(* IEC 61131-3 sources: volt/packages/volt-lsp-iec/test-corpus/lenze-mid/Device/Plc Logic/Application/Library Manager/(unresolved)/cmpopcuastack interfaces (part 2) *)

(* ---- OPCUA_NODEIDS.dut ---- *)
TYPE OPCUA_NODEIDS :
(
	OPCUAID_BASEDATATYPE := 24,
	OPCUAID_NUMBER := 26,
	OPCUAID_INTEGER := 27,
	OPCUAID_UINTEGER := 28,
	OPCUAID_ENUMERATION := 29,
	OPCUAID_BOOLEAN := 1,
	OPCUAID_SBYTE := 2,
	OPCUAID_BYTE := 3,
	OPCUAID_INT16 := 4,
	OPCUAID_UINT16 := 5,
	OPCUAID_INT32 := 6,
	OPCUAID_UINT32 := 7,
	OPCUAID_INT64 := 8,
	OPCUAID_UINT64 := 9,
	OPCUAID_FLOAT := 10,
	OPCUAID_DOUBLE := 11,
	OPCUAID_STRING := 12,
	OPCUAID_DATETIME := 13,
	OPCUAID_GUID := 14,
	OPCUAID_BYTESTRING := 15,
	OPCUAID_XMLELEMENT := 16,
	OPCUAID_NODEID := 17,
	OPCUAID_EXPANDEDNODEID := 18,
	OPCUAID_STATUSCODE := 19,
	OPCUAID_QUALIFIEDNAME := 20,
	OPCUAID_LOCALIZEDTEXT := 21,
	OPCUAID_STRUCTURE := 22,
	OPCUAID_DATAVALUE := 23,
	OPCUAID_DIAGNOSTICINFO := 25,
	OPCUAID_IMAGE := 30,
	OPCUAID_DECIMAL := 50,
	OPCUAID_NAMINGRULETYPE := 120,
	OPCUAID_IMAGEBMP := 2000,
	OPCUAID_IMAGEGIF := 2001,
	OPCUAID_IMAGEJPG := 2002,
	OPCUAID_IMAGEPNG := 2003,
	OPCUAID_AUDIODATATYPE := 16307,
	OPCUAID_BITFIELDMASKDATATYPE := 11737,
	OPCUAID_KEYVALUEPAIR := 14533,
	OPCUAID_ENDPOINTTYPE := 15528,
	OPCUAID_OPENFILEMODE := 11939,
	OPCUAID_IDENTITYCRITERIATYPE := 15632,
	OPCUAID_IDENTITYMAPPINGRULETYPE := 15634,
	OPCUAID_TRUSTLISTMASKS := 12552,
	OPCUAID_TRUSTLISTDATATYPE := 12554,
	OPCUAID_DECIMALDATATYPE := 17861,
	OPCUAID_DATATYPESCHEMAHEADER := 15534,
	OPCUAID_DATATYPEDESCRIPTION := 14525,
	OPCUAID_STRUCTUREDESCRIPTION := 15487,
	OPCUAID_ENUMDESCRIPTION := 15488,
	OPCUAID_SIMPLETYPEDESCRIPTION := 15005,
	OPCUAID_UABINARYFILEDATATYPE := 15006,
	OPCUAID_PUBSUBSTATE := 14647,
	OPCUAID_DATASETMETADATATYPE := 14523,
	OPCUAID_FIELDMETADATA := 14524,
	OPCUAID_DATASETFIELDFLAGS := 15904,
	OPCUAID_CONFIGURATIONVERSIONDATATYPE := 14593,
	OPCUAID_PUBLISHEDDATASETDATATYPE := 15578,
	OPCUAID_PUBLISHEDDATASETSOURCEDATATYPE := 15580,
	OPCUAID_PUBLISHEDVARIABLEDATATYPE := 14273,
	OPCUAID_PUBLISHEDDATAITEMSDATATYPE := 15581,
	OPCUAID_PUBLISHEDEVENTSDATATYPE := 15582,
	OPCUAID_DATASETFIELDCONTENTMASK := 15583,
	OPCUAID_DATASETWRITERDATATYPE := 15597,
	OPCUAID_DATASETWRITERTRANSPORTDATATYPE := 15598,
	OPCUAID_DATASETWRITERMESSAGEDATATYPE := 15605,
	OPCUAID_PUBSUBGROUPDATATYPE := 15609,
	OPCUAID_WRITERGROUPDATATYPE := 15480,
	OPCUAID_WRITERGROUPTRANSPORTDATATYPE := 15611,
	OPCUAID_WRITERGROUPMESSAGEDATATYPE := 15616,
	OPCUAID_PUBSUBCONNECTIONDATATYPE := 15617,
	OPCUAID_CONNECTIONTRANSPORTDATATYPE := 15618,
	OPCUAID_NETWORKADDRESSDATATYPE := 15502,
	OPCUAID_NETWORKADDRESSURLDATATYPE := 15510,
	OPCUAID_READERGROUPDATATYPE := 15520,
	OPCUAID_READERGROUPTRANSPORTDATATYPE := 15621,
	OPCUAID_READERGROUPMESSAGEDATATYPE := 15622,
	OPCUAID_DATASETREADERDATATYPE := 15623,
	OPCUAID_DATASETREADERTRANSPORTDATATYPE := 15628,
	OPCUAID_DATASETREADERMESSAGEDATATYPE := 15629,
	OPCUAID_SUBSCRIBEDDATASETDATATYPE := 15630,
	OPCUAID_TARGETVARIABLESDATATYPE := 15631,
	OPCUAID_FIELDTARGETDATATYPE := 14744,
	OPCUAID_OVERRIDEVALUEHANDLING := 15874,
	OPCUAID_SUBSCRIBEDDATASETMIRRORDATATYPE := 15635,
	OPCUAID_PUBSUBCONFIGURATIONDATATYPE := 15530,
	OPCUAID_DATASETORDERINGTYPE := 20408,
	OPCUAID_UADPNETWORKMESSAGECONTENTMASK := 15642,
	OPCUAID_UADPWRITERGROUPMESSAGEDATATYPE := 15645,
	OPCUAID_UADPDATASETMESSAGECONTENTMASK := 15646,
	OPCUAID_UADPDATASETWRITERMESSAGEDATATYPE := 15652,
	OPCUAID_UADPDATASETREADERMESSAGEDATATYPE := 15653,
	OPCUAID_JSONNETWORKMESSAGECONTENTMASK := 15654,
	OPCUAID_JSONWRITERGROUPMESSAGEDATATYPE := 15657,
	OPCUAID_JSONDATASETMESSAGECONTENTMASK := 15658,
	OPCUAID_JSONDATASETWRITERMESSAGEDATATYPE := 15664,
	OPCUAID_JSONDATASETREADERMESSAGEDATATYPE := 15665,
	OPCUAID_DATAGRAMCONNECTIONTRANSPORTDATATYPE := 17467,
	OPCUAID_DATAGRAMWRITERGROUPTRANSPORTDATATYPE := 15532,
	OPCUAID_BROKERCONNECTIONTRANSPORTDATATYPE := 15007,
	OPCUAID_BROKERTRANSPORTQUALITYOFSERVICE := 15008,
	OPCUAID_BROKERWRITERGROUPTRANSPORTDATATYPE := 15667,
	OPCUAID_BROKERDATASETWRITERTRANSPORTDATATYPE := 15669,
	OPCUAID_BROKERDATASETREADERTRANSPORTDATATYPE := 15670,
	OPCUAID_DIAGNOSTICSLEVEL := 19723,
	OPCUAID_PUBSUBDIAGNOSTICSCOUNTERCLASSIFICATION := 19730,
	OPCUAID_IDTYPE := 256,
	OPCUAID_NODECLASS := 257,
	OPCUAID_PERMISSIONTYPE := 94,
	OPCUAID_ACCESSLEVELTYPE := 15031,
	OPCUAID_ACCESSLEVELEXTYPE := 15406,
	OPCUAID_EVENTNOTIFIERTYPE := 15033,
	OPCUAID_ACCESSRESTRICTIONTYPE := 95,
	OPCUAID_ROLEPERMISSIONTYPE := 96,
	OPCUAID_DATATYPEDEFINITION := 97,
	OPCUAID_STRUCTURETYPE := 98,
	OPCUAID_STRUCTUREFIELD := 101,
	OPCUAID_STRUCTUREDEFINITION := 99,
	OPCUAID_ENUMDEFINITION := 100,
	OPCUAID_NODE := 258,
	OPCUAID_INSTANCENODE := 11879,
	OPCUAID_TYPENODE := 11880,
	OPCUAID_OBJECTNODE := 261,
	OPCUAID_OBJECTTYPENODE := 264,
	OPCUAID_VARIABLENODE := 267,
	OPCUAID_VARIABLETYPENODE := 270,
	OPCUAID_REFERENCETYPENODE := 273,
	OPCUAID_METHODNODE := 276,
	OPCUAID_VIEWNODE := 279,
	OPCUAID_DATATYPENODE := 282,
	OPCUAID_REFERENCENODE := 285,
	OPCUAID_ARGUMENT := 296,
	OPCUAID_ENUMVALUETYPE := 7594,
	OPCUAID_ENUMFIELD := 102,
	OPCUAID_OPTIONSET := 12755,
	OPCUAID_UNION := 12756,
	OPCUAID_NORMALIZEDSTRING := 12877,
	OPCUAID_DECIMALSTRING := 12878,
	OPCUAID_DURATIONSTRING := 12879,
	OPCUAID_TIMESTRING := 12880,
	OPCUAID_DATESTRING := 12881,
	OPCUAID_DURATION := 290,
	OPCUAID_UTCTIME := 294,
	OPCUAID_LOCALEID := 295,
	OPCUAID_TIMEZONEDATATYPE := 8912,
	OPCUAID_INTEGERID := 288,
	OPCUAID_APPLICATIONTYPE := 307,
	OPCUAID_APPLICATIONDESCRIPTION := 308,
	OPCUAID_REQUESTHEADER := 389,
	OPCUAID_RESPONSEHEADER := 392,
	OPCUAID_VERSIONTIME := 20998,
	OPCUAID_SERVICEFAULT := 395,
	OPCUAID_SESSIONLESSINVOKEREQUESTTYPE := 15901,
	OPCUAID_SESSIONLESSINVOKERESPONSETYPE := 20999,
	OPCUAID_FINDSERVERSREQUEST := 420,
	OPCUAID_FINDSERVERSRESPONSE := 423,
	OPCUAID_SERVERONNETWORK := 12189,
	OPCUAID_FINDSERVERSONNETWORKREQUEST := 12190,
	OPCUAID_FINDSERVERSONNETWORKRESPONSE := 12191,
	OPCUAID_APPLICATIONINSTANCECERTIFICATE := 311,
	OPCUAID_MESSAGESECURITYMODE := 302,
	OPCUAID_USERTOKENTYPE := 303,
	OPCUAID_USERTOKENPOLICY := 304,
	OPCUAID_ENDPOINTDESCRIPTION := 312,
	OPCUAID_GETENDPOINTSREQUEST := 426,
	OPCUAID_GETENDPOINTSRESPONSE := 429,
	OPCUAID_REGISTEREDSERVER := 432,
	OPCUAID_REGISTERSERVERREQUEST := 435,
	OPCUAID_REGISTERSERVERRESPONSE := 438,
	OPCUAID_DISCOVERYCONFIGURATION := 12890,
	OPCUAID_MDNSDISCOVERYCONFIGURATION := 12891,
	OPCUAID_REGISTERSERVER2REQUEST := 12193,
	OPCUAID_REGISTERSERVER2RESPONSE := 12194,
	OPCUAID_SECURITYTOKENREQUESTTYPE := 315,
	OPCUAID_CHANNELSECURITYTOKEN := 441,
	OPCUAID_OPENSECURECHANNELREQUEST := 444,
	OPCUAID_OPENSECURECHANNELRESPONSE := 447,
	OPCUAID_CLOSESECURECHANNELREQUEST := 450,
	OPCUAID_CLOSESECURECHANNELRESPONSE := 453,
	OPCUAID_SIGNEDSOFTWARECERTIFICATE := 344,
	OPCUAID_SESSIONAUTHENTICATIONTOKEN := 388,
	OPCUAID_SIGNATUREDATA := 456,
	OPCUAID_CREATESESSIONREQUEST := 459,
	OPCUAID_CREATESESSIONRESPONSE := 462,
	OPCUAID_USERIDENTITYTOKEN := 316,
	OPCUAID_ANONYMOUSIDENTITYTOKEN := 319,
	OPCUAID_USERNAMEIDENTITYTOKEN := 322,
	OPCUAID_X509IDENTITYTOKEN := 325,
	OPCUAID_ISSUEDIDENTITYTOKEN := 938,
	OPCUAID_ACTIVATESESSIONREQUEST := 465,
	OPCUAID_ACTIVATESESSIONRESPONSE := 468,
	OPCUAID_CLOSESESSIONREQUEST := 471,
	OPCUAID_CLOSESESSIONRESPONSE := 474,
	OPCUAID_CANCELREQUEST := 477,
	OPCUAID_CANCELRESPONSE := 480,
	OPCUAID_NODEATTRIBUTESMASK := 348,
	OPCUAID_NODEATTRIBUTES := 349,
	OPCUAID_OBJECTATTRIBUTES := 352,
	OPCUAID_VARIABLEATTRIBUTES := 355,
	OPCUAID_METHODATTRIBUTES := 358,
	OPCUAID_OBJECTTYPEATTRIBUTES := 361,
	OPCUAID_VARIABLETYPEATTRIBUTES := 364,
	OPCUAID_REFERENCETYPEATTRIBUTES := 367,
	OPCUAID_DATATYPEATTRIBUTES := 370,
	OPCUAID_VIEWATTRIBUTES := 373,
	OPCUAID_GENERICATTRIBUTEVALUE := 17606,
	OPCUAID_GENERICATTRIBUTES := 17607,
	OPCUAID_ADDNODESITEM := 376,
	OPCUAID_ADDNODESRESULT := 483,
	OPCUAID_ADDNODESREQUEST := 486,
	OPCUAID_ADDNODESRESPONSE := 489,
	OPCUAID_ADDREFERENCESITEM := 379,
	OPCUAID_ADDREFERENCESREQUEST := 492,
	OPCUAID_ADDREFERENCESRESPONSE := 495,
	OPCUAID_DELETENODESITEM := 382,
	OPCUAID_DELETENODESREQUEST := 498,
	OPCUAID_DELETENODESRESPONSE := 501,
	OPCUAID_DELETEREFERENCESITEM := 385,
	OPCUAID_DELETEREFERENCESREQUEST := 504,
	OPCUAID_DELETEREFERENCESRESPONSE := 507,
	OPCUAID_ATTRIBUTEWRITEMASK := 347,
	OPCUAID_BROWSEDIRECTION := 510,
	OPCUAID_VIEWDESCRIPTION := 511,
	OPCUAID_BROWSEDESCRIPTION := 514,
	OPCUAID_BROWSERESULTMASK := 517,
	OPCUAID_REFERENCEDESCRIPTION := 518,
	OPCUAID_CONTINUATIONPOINT := 521,
	OPCUAID_BROWSERESULT := 522,
	OPCUAID_BROWSEREQUEST := 525,
	OPCUAID_BROWSERESPONSE := 528,
	OPCUAID_BROWSENEXTREQUEST := 531,
	OPCUAID_BROWSENEXTRESPONSE := 534,
	OPCUAID_RELATIVEPATHELEMENT := 537,
	OPCUAID_RELATIVEPATH := 540,
	OPCUAID_BROWSEPATH := 543,
	OPCUAID_BROWSEPATHTARGET := 546,
	OPCUAID_BROWSEPATHRESULT := 549,
	OPCUAID_TRANSLATEBROWSEPATHSTONODEIDSREQUEST := 552,
	OPCUAID_TRANSLATEBROWSEPATHSTONODEIDSRESPONSE := 555,
	OPCUAID_REGISTERNODESREQUEST := 558,
	OPCUAID_REGISTERNODESRESPONSE := 561,
	OPCUAID_UNREGISTERNODESREQUEST := 564,
	OPCUAID_UNREGISTERNODESRESPONSE := 567,
	OPCUAID_COUNTER := 289,
	OPCUAID_NUMERICRANGE := 291,
	OPCUAID_TIME := 292,
	OPCUAID_DATE := 293,
	OPCUAID_ENDPOINTCONFIGURATION := 331,
	OPCUAID_QUERYDATADESCRIPTION := 570,
	OPCUAID_NODETYPEDESCRIPTION := 573,
	OPCUAID_FILTEROPERATOR := 576,
	OPCUAID_QUERYDATASET := 577,
	OPCUAID_NODEREFERENCE := 580,
	OPCUAID_CONTENTFILTERELEMENT := 583,
	OPCUAID_CONTENTFILTER := 586,
	OPCUAID_FILTEROPERAND := 589,
	OPCUAID_ELEMENTOPERAND := 592,
	OPCUAID_LITERALOPERAND := 595,
	OPCUAID_ATTRIBUTEOPERAND := 598,
	OPCUAID_SIMPLEATTRIBUTEOPERAND := 601,
	OPCUAID_CONTENTFILTERELEMENTRESULT := 604,
	OPCUAID_CONTENTFILTERRESULT := 607,
	OPCUAID_PARSINGRESULT := 610,
	OPCUAID_QUERYFIRSTREQUEST := 613,
	OPCUAID_QUERYFIRSTRESPONSE := 616,
	OPCUAID_QUERYNEXTREQUEST := 619,
	OPCUAID_QUERYNEXTRESPONSE := 622,
	OPCUAID_TIMESTAMPSTORETURN := 625,
	OPCUAID_READVALUEID := 626,
	OPCUAID_READREQUEST := 629,
	OPCUAID_READRESPONSE := 632,
	OPCUAID_HISTORYREADVALUEID := 635,
	OPCUAID_HISTORYREADRESULT := 638,
	OPCUAID_HISTORYREADDETAILS := 641,
	OPCUAID_READEVENTDETAILS := 644,
	OPCUAID_READRAWMODIFIEDDETAILS := 647,
	OPCUAID_READPROCESSEDDETAILS := 650,
	OPCUAID_READATTIMEDETAILS := 653,
	OPCUAID_HISTORYDATA := 656,
	OPCUAID_MODIFICATIONINFO := 11216,
	OPCUAID_HISTORYMODIFIEDDATA := 11217,
	OPCUAID_HISTORYEVENT := 659,
	OPCUAID_HISTORYREADREQUEST := 662,
	OPCUAID_HISTORYREADRESPONSE := 665,
	OPCUAID_WRITEVALUE := 668,
	OPCUAID_WRITEREQUEST := 671,
	OPCUAID_WRITERESPONSE := 674,
	OPCUAID_HISTORYUPDATEDETAILS := 677,
	OPCUAID_HISTORYUPDATETYPE := 11234,
	OPCUAID_PERFORMUPDATETYPE := 11293,
	OPCUAID_UPDATEDATADETAILS := 680,
	OPCUAID_UPDATESTRUCTUREDATADETAILS := 11295,
	OPCUAID_UPDATEEVENTDETAILS := 683,
	OPCUAID_DELETERAWMODIFIEDDETAILS := 686,
	OPCUAID_DELETEATTIMEDETAILS := 689,
	OPCUAID_DELETEEVENTDETAILS := 692,
	OPCUAID_HISTORYUPDATERESULT := 695,
	OPCUAID_HISTORYUPDATEREQUEST := 698,
	OPCUAID_HISTORYUPDATERESPONSE := 701,
	OPCUAID_CALLMETHODREQUEST := 704,
	OPCUAID_CALLMETHODRESULT := 707,
	OPCUAID_CALLREQUEST := 710,
	OPCUAID_CALLRESPONSE := 713,
	OPCUAID_MONITORINGMODE := 716,
	OPCUAID_DATACHANGETRIGGER := 717,
	OPCUAID_DEADBANDTYPE := 718,
	OPCUAID_MONITORINGFILTER := 719,
	OPCUAID_DATACHANGEFILTER := 722,
	OPCUAID_EVENTFILTER := 725,
	OPCUAID_AGGREGATECONFIGURATION := 948,
	OPCUAID_AGGREGATEFILTER := 728,
	OPCUAID_MONITORINGFILTERRESULT := 731,
	OPCUAID_EVENTFILTERRESULT := 734,
	OPCUAID_AGGREGATEFILTERRESULT := 737,
	OPCUAID_MONITORINGPARAMETERS := 740,
	OPCUAID_MONITOREDITEMCREATEREQUEST := 743,
	OPCUAID_MONITOREDITEMCREATERESULT := 746,
	OPCUAID_CREATEMONITOREDITEMSREQUEST := 749,
	OPCUAID_CREATEMONITOREDITEMSRESPONSE := 752,
	OPCUAID_MONITOREDITEMMODIFYREQUEST := 755,
	OPCUAID_MONITOREDITEMMODIFYRESULT := 758,
	OPCUAID_MODIFYMONITOREDITEMSREQUEST := 761,
	OPCUAID_MODIFYMONITOREDITEMSRESPONSE := 764,
	OPCUAID_SETMONITORINGMODEREQUEST := 767,
	OPCUAID_SETMONITORINGMODERESPONSE := 770,
	OPCUAID_SETTRIGGERINGREQUEST := 773,
	OPCUAID_SETTRIGGERINGRESPONSE := 776,
	OPCUAID_DELETEMONITOREDITEMSREQUEST := 779,
	OPCUAID_DELETEMONITOREDITEMSRESPONSE := 782,
	OPCUAID_CREATESUBSCRIPTIONREQUEST := 785,
	OPCUAID_CREATESUBSCRIPTIONRESPONSE := 788,
	OPCUAID_MODIFYSUBSCRIPTIONREQUEST := 791,
	OPCUAID_MODIFYSUBSCRIPTIONRESPONSE := 794,
	OPCUAID_SETPUBLISHINGMODEREQUEST := 797,
	OPCUAID_SETPUBLISHINGMODERESPONSE := 800,
	OPCUAID_NOTIFICATIONMESSAGE := 803,
	OPCUAID_NOTIFICATIONDATA := 945,
	OPCUAID_DATACHANGENOTIFICATION := 809,
	OPCUAID_MONITOREDITEMNOTIFICATION := 806,
	OPCUAID_EVENTNOTIFICATIONLIST := 914,
	OPCUAID_EVENTFIELDLIST := 917,
	OPCUAID_HISTORYEVENTFIELDLIST := 920,
	OPCUAID_STATUSCHANGENOTIFICATION := 818,
	OPCUAID_SUBSCRIPTIONACKNOWLEDGEMENT := 821,
	OPCUAID_PUBLISHREQUEST := 824,
	OPCUAID_PUBLISHRESPONSE := 827,
	OPCUAID_REPUBLISHREQUEST := 830,
	OPCUAID_REPUBLISHRESPONSE := 833,
	OPCUAID_TRANSFERRESULT := 836,
	OPCUAID_TRANSFERSUBSCRIPTIONSREQUEST := 839,
	OPCUAID_TRANSFERSUBSCRIPTIONSRESPONSE := 842,
	OPCUAID_DELETESUBSCRIPTIONSREQUEST := 845,
	OPCUAID_DELETESUBSCRIPTIONSRESPONSE := 848,
	OPCUAID_BUILDINFO := 338,
	OPCUAID_REDUNDANCYSUPPORT := 851,
	OPCUAID_SERVERSTATE := 852,
	OPCUAID_REDUNDANTSERVERDATATYPE := 853,
	OPCUAID_ENDPOINTURLLISTDATATYPE := 11943,
	OPCUAID_NETWORKGROUPDATATYPE := 11944,
	OPCUAID_SAMPLINGINTERVALDIAGNOSTICSDATATYPE := 856,
	OPCUAID_SERVERDIAGNOSTICSSUMMARYDATATYPE := 859,
	OPCUAID_SERVERSTATUSDATATYPE := 862,
	OPCUAID_SESSIONDIAGNOSTICSDATATYPE := 865,
	OPCUAID_SESSIONSECURITYDIAGNOSTICSDATATYPE := 868,
	OPCUAID_SERVICECOUNTERDATATYPE := 871,
	OPCUAID_STATUSRESULT := 299,
	OPCUAID_SUBSCRIPTIONDIAGNOSTICSDATATYPE := 874,
	OPCUAID_MODELCHANGESTRUCTUREVERBMASK := 11941,
	OPCUAID_MODELCHANGESTRUCTUREDATATYPE := 877,
	OPCUAID_SEMANTICCHANGESTRUCTUREDATATYPE := 897,
	OPCUAID_RANGE := 884,
	OPCUAID_EUINFORMATION := 887,
	OPCUAID_AXISSCALEENUMERATION := 12077,
	OPCUAID_COMPLEXNUMBERTYPE := 12171,
	OPCUAID_DOUBLECOMPLEXNUMBERTYPE := 12172,
	OPCUAID_AXISINFORMATION := 12079,
	OPCUAID_XVTYPE := 12080,
	OPCUAID_PROGRAMDIAGNOSTICDATATYPE := 894,
	OPCUAID_PROGRAMDIAGNOSTIC2DATATYPE := 15396,
	OPCUAID_ANNOTATION := 891,
	OPCUAID_EXCEPTIONDEVIATIONFORMAT := 890,
	OPCUAID_OPCUANAMESPACEMETADATA_NAMESPACEFILE_OPEN := 15971,
	OPCUAID_OPCUANAMESPACEMETADATA_NAMESPACEFILE_CLOSE := 15974,
	OPCUAID_OPCUANAMESPACEMETADATA_NAMESPACEFILE_READ := 15976,
	OPCUAID_OPCUANAMESPACEMETADATA_NAMESPACEFILE_WRITE := 15979,
	OPCUAID_OPCUANAMESPACEMETADATA_NAMESPACEFILE_GETPOSITION := 15981,
	OPCUAID_OPCUANAMESPACEMETADATA_NAMESPACEFILE_SETPOSITION := 15984,
	OPCUAID_SERVERTYPE_SERVERCAPABILITIES_ROLESET_ADDROLE := 16290,
	OPCUAID_SERVERTYPE_SERVERCAPABILITIES_ROLESET_REMOVEROLE := 16293,
	OPCUAID_SERVERTYPE_GETMONITOREDITEMS := 11489,
	OPCUAID_SERVERTYPE_RESENDDATA := 12871,
	OPCUAID_SERVERTYPE_SETSUBSCRIPTIONDURABLE := 12746,
	OPCUAID_SERVERTYPE_REQUESTSERVERSTATECHANGE := 12883,
	OPCUAID_SERVERCAPABILITIESTYPE_ROLESET_ADDROLE := 16296,
	OPCUAID_SERVERCAPABILITIESTYPE_ROLESET_REMOVEROLE := 16299,
	OPCUAID_FILETYPE_OPEN := 11580,
	OPCUAID_FILETYPE_CLOSE := 11583,
	OPCUAID_FILETYPE_READ := 11585,
	OPCUAID_FILETYPE_WRITE := 11588,
	OPCUAID_FILETYPE_GETPOSITION := 11590,
	OPCUAID_FILETYPE_SETPOSITION := 11593,
	OPCUAID_ADDRESSSPACEFILETYPE_EXPORTNAMESPACE := 11615,
	OPCUAID_NAMESPACEMETADATATYPE_NAMESPACEFILE_OPEN := 11629,
	OPCUAID_NAMESPACEMETADATATYPE_NAMESPACEFILE_CLOSE := 11632,
	OPCUAID_NAMESPACEMETADATATYPE_NAMESPACEFILE_READ := 11634,
	OPCUAID_NAMESPACEMETADATATYPE_NAMESPACEFILE_WRITE := 11637,
	OPCUAID_NAMESPACEMETADATATYPE_NAMESPACEFILE_GETPOSITION := 11639,
	OPCUAID_NAMESPACEMETADATATYPE_NAMESPACEFILE_SETPOSITION := 11642,
	OPCUAID_NAMESPACESTYPE_NAMESPACEIDENTIFIER_PLACEHOLDER_NAMESPACEFILE_OPEN := 11659,
	OPCUAID_NAMESPACESTYPE_NAMESPACEIDENTIFIER_PLACEHOLDER_NAMESPACEFILE_CLOSE := 11662,
	OPCUAID_NAMESPACESTYPE_NAMESPACEIDENTIFIER_PLACEHOLDER_NAMESPACEFILE_READ := 11664,
	OPCUAID_NAMESPACESTYPE_NAMESPACEIDENTIFIER_PLACEHOLDER_NAMESPACEFILE_WRITE := 11667,
	OPCUAID_NAMESPACESTYPE_NAMESPACEIDENTIFIER_PLACEHOLDER_NAMESPACEFILE_GETPOSITION := 11669,
	OPCUAID_NAMESPACESTYPE_NAMESPACEIDENTIFIER_PLACEHOLDER_NAMESPACEFILE_SETPOSITION := 11672,
	OPCUAID_SERVER_SERVERCAPABILITIES_ROLESET_ADDROLE := 16301,
	OPCUAID_SERVER_SERVERCAPABILITIES_ROLESET_REMOVEROLE := 16304,
	OPCUAID_SERVER_GETMONITOREDITEMS := 11492,
	OPCUAID_SERVER_RESENDDATA := 12873,
	OPCUAID_SERVER_SETSUBSCRIPTIONDURABLE := 12749,
	OPCUAID_SERVER_REQUESTSERVERSTATECHANGE := 12886,
	OPCUAID_FILEDIRECTORYTYPE_FILEDIRECTORYNAME_PLACEHOLDER_CREATEDIRECTORY := 13355,
	OPCUAID_FILEDIRECTORYTYPE_FILEDIRECTORYNAME_PLACEHOLDER_CREATEFILE := 13358,
	OPCUAID_FILEDIRECTORYTYPE_FILEDIRECTORYNAME_PLACEHOLDER_DELETEFILESYSTEMOBJECT := 17718,
	OPCUAID_FILEDIRECTORYTYPE_FILEDIRECTORYNAME_PLACEHOLDER_MOVEORCOPY := 13363,
	OPCUAID_FILEDIRECTORYTYPE_FILENAME_PLACEHOLDER_OPEN := 13372,
	OPCUAID_FILEDIRECTORYTYPE_FILENAME_PLACEHOLDER_CLOSE := 13375,
	OPCUAID_FILEDIRECTORYTYPE_FILENAME_PLACEHOLDER_READ := 13377,
	OPCUAID_FILEDIRECTORYTYPE_FILENAME_PLACEHOLDER_WRITE := 13380,
	OPCUAID_FILEDIRECTORYTYPE_FILENAME_PLACEHOLDER_GETPOSITION := 13382,
	OPCUAID_FILEDIRECTORYTYPE_FILENAME_PLACEHOLDER_SETPOSITION := 13385,
	OPCUAID_FILEDIRECTORYTYPE_CREATEDIRECTORY := 13387,
	OPCUAID_FILEDIRECTORYTYPE_CREATEFILE := 13390,
	OPCUAID_FILEDIRECTORYTYPE_DELETEFILESYSTEMOBJECT := 13393,
	OPCUAID_FILEDIRECTORYTYPE_MOVEORCOPY := 13395,
	OPCUAID_FILESYSTEM_FILEDIRECTORYNAME_PLACEHOLDER_CREATEDIRECTORY := 16316,
	OPCUAID_FILESYSTEM_FILEDIRECTORYNAME_PLACEHOLDER_CREATEFILE := 16319,
	OPCUAID_FILESYSTEM_FILEDIRECTORYNAME_PLACEHOLDER_DELETEFILESYSTEMOBJECT := 17722,
	OPCUAID_FILESYSTEM_FILEDIRECTORYNAME_PLACEHOLDER_MOVEORCOPY := 16324,
	OPCUAID_FILESYSTEM_FILENAME_PLACEHOLDER_OPEN := 16333,
	OPCUAID_FILESYSTEM_FILENAME_PLACEHOLDER_CLOSE := 16336,
	OPCUAID_FILESYSTEM_FILENAME_PLACEHOLDER_READ := 16338,
	OPCUAID_FILESYSTEM_FILENAME_PLACEHOLDER_WRITE := 16341,
	OPCUAID_FILESYSTEM_FILENAME_PLACEHOLDER_GETPOSITION := 16343,
	OPCUAID_FILESYSTEM_FILENAME_PLACEHOLDER_SETPOSITION := 16346,
	OPCUAID_FILESYSTEM_CREATEDIRECTORY := 16348,
	OPCUAID_FILESYSTEM_CREATEFILE := 16351,
	OPCUAID_FILESYSTEM_DELETEFILESYSTEMOBJECT := 16354,
	OPCUAID_FILESYSTEM_MOVEORCOPY := 16356,
	OPCUAID_TEMPORARYFILETRANSFERTYPE_GENERATEFILEFORREAD := 15746,
	OPCUAID_TEMPORARYFILETRANSFERTYPE_GENERATEFILEFORWRITE := 15749,
	OPCUAID_TEMPORARYFILETRANSFERTYPE_CLOSEANDCOMMIT := 15751,
	OPCUAID_TEMPORARYFILETRANSFERTYPE_TRANSFERSTATE_PLACEHOLDER_RESET := 15794,
	OPCUAID_FILETRANSFERSTATEMACHINETYPE_RESET := 15843,
	OPCUAID_ROLESETTYPE_ADDROLE := 15997,
	OPCUAID_ROLESETTYPE_REMOVEROLE := 16000,
	OPCUAID_ROLETYPE_ADDIDENTITY := 15624,
	OPCUAID_ROLETYPE_REMOVEIDENTITY := 15626,
	OPCUAID_ROLETYPE_ADDAPPLICATION := 16176,
	OPCUAID_ROLETYPE_REMOVEAPPLICATION := 16178,
	OPCUAID_ROLETYPE_ADDENDPOINT := 16180,
	OPCUAID_ROLETYPE_REMOVEENDPOINT := 16182,
	OPCUAID_WELLKNOWNROLE_ANONYMOUS_ADDIDENTITY := 15648,
	OPCUAID_WELLKNOWNROLE_ANONYMOUS_REMOVEIDENTITY := 15650,
	OPCUAID_WELLKNOWNROLE_ANONYMOUS_ADDAPPLICATION := 16195,
	OPCUAID_WELLKNOWNROLE_ANONYMOUS_REMOVEAPPLICATION := 16197,
	OPCUAID_WELLKNOWNROLE_ANONYMOUS_ADDENDPOINT := 16199,
	OPCUAID_WELLKNOWNROLE_ANONYMOUS_REMOVEENDPOINT := 16201,
	OPCUAID_WELLKNOWNROLE_AUTHENTICATEDUSER_ADDIDENTITY := 15660,
	OPCUAID_WELLKNOWNROLE_AUTHENTICATEDUSER_REMOVEIDENTITY := 15662,
	OPCUAID_WELLKNOWNROLE_AUTHENTICATEDUSER_ADDAPPLICATION := 16206,
	OPCUAID_WELLKNOWNROLE_AUTHENTICATEDUSER_REMOVEAPPLICATION := 16208,
	OPCUAID_WELLKNOWNROLE_AUTHENTICATEDUSER_ADDENDPOINT := 16210,
	OPCUAID_WELLKNOWNROLE_AUTHENTICATEDUSER_REMOVEENDPOINT := 16212,
	OPCUAID_WELLKNOWNROLE_OBSERVER_ADDIDENTITY := 15672,
	OPCUAID_WELLKNOWNROLE_OBSERVER_REMOVEIDENTITY := 15674,
	OPCUAID_WELLKNOWNROLE_OBSERVER_ADDAPPLICATION := 16217,
	OPCUAID_WELLKNOWNROLE_OBSERVER_REMOVEAPPLICATION := 16219,
	OPCUAID_WELLKNOWNROLE_OBSERVER_ADDENDPOINT := 16221,
	OPCUAID_WELLKNOWNROLE_OBSERVER_REMOVEENDPOINT := 16223,
	OPCUAID_WELLKNOWNROLE_OPERATOR_ADDIDENTITY := 15684,
	OPCUAID_WELLKNOWNROLE_OPERATOR_REMOVEIDENTITY := 15686,
	OPCUAID_WELLKNOWNROLE_OPERATOR_ADDAPPLICATION := 16228,
	OPCUAID_WELLKNOWNROLE_OPERATOR_REMOVEAPPLICATION := 16230,
	OPCUAID_WELLKNOWNROLE_OPERATOR_ADDENDPOINT := 16232,
	OPCUAID_WELLKNOWNROLE_OPERATOR_REMOVEENDPOINT := 16234,
	OPCUAID_WELLKNOWNROLE_ENGINEER_ADDIDENTITY := 16041,
	OPCUAID_WELLKNOWNROLE_ENGINEER_REMOVEIDENTITY := 16043,
	OPCUAID_WELLKNOWNROLE_ENGINEER_ADDAPPLICATION := 16239,
	OPCUAID_WELLKNOWNROLE_ENGINEER_REMOVEAPPLICATION := 16241,
	OPCUAID_WELLKNOWNROLE_ENGINEER_ADDENDPOINT := 16243,
	OPCUAID_WELLKNOWNROLE_ENGINEER_REMOVEENDPOINT := 16245,
	OPCUAID_WELLKNOWNROLE_SUPERVISOR_ADDIDENTITY := 15696,
	OPCUAID_WELLKNOWNROLE_SUPERVISOR_REMOVEIDENTITY := 15698,
	OPCUAID_WELLKNOWNROLE_SUPERVISOR_ADDAPPLICATION := 16250,
	OPCUAID_WELLKNOWNROLE_SUPERVISOR_REMOVEAPPLICATION := 16252,
	OPCUAID_WELLKNOWNROLE_SUPERVISOR_ADDENDPOINT := 16254,
	OPCUAID_WELLKNOWNROLE_SUPERVISOR_REMOVEENDPOINT := 16256,
	OPCUAID_WELLKNOWNROLE_CONFIGUREADMIN_ADDIDENTITY := 15720,
	OPCUAID_WELLKNOWNROLE_CONFIGUREADMIN_REMOVEIDENTITY := 15722,
	OPCUAID_WELLKNOWNROLE_CONFIGUREADMIN_ADDAPPLICATION := 16272,
	OPCUAID_WELLKNOWNROLE_CONFIGUREADMIN_REMOVEAPPLICATION := 16274,
	OPCUAID_WELLKNOWNROLE_CONFIGUREADMIN_ADDENDPOINT := 16276,
	OPCUAID_WELLKNOWNROLE_CONFIGUREADMIN_REMOVEENDPOINT := 16278,
	OPCUAID_WELLKNOWNROLE_SECURITYADMIN_ADDIDENTITY := 15708,
	OPCUAID_WELLKNOWNROLE_SECURITYADMIN_REMOVEIDENTITY := 15710,
	OPCUAID_WELLKNOWNROLE_SECURITYADMIN_ADDAPPLICATION := 16261,
	OPCUAID_WELLKNOWNROLE_SECURITYADMIN_REMOVEAPPLICATION := 16263,
	OPCUAID_WELLKNOWNROLE_SECURITYADMIN_ADDENDPOINT := 16265,
	OPCUAID_WELLKNOWNROLE_SECURITYADMIN_REMOVEENDPOINT := 16267,
	OPCUAID_CONDITIONTYPE_DISABLE := 9028,
	OPCUAID_CONDITIONTYPE_ENABLE := 9027,
	OPCUAID_CONDITIONTYPE_ADDCOMMENT := 9029,
	OPCUAID_CONDITIONTYPE_CONDITIONREFRESH := 3875,
	OPCUAID_CONDITIONTYPE_CONDITIONREFRESH2 := 12912,
	OPCUAID_DIALOGCONDITIONTYPE_RESPOND := 9069,
	OPCUAID_ACKNOWLEDGEABLECONDITIONTYPE_ACKNOWLEDGE := 9111,
	OPCUAID_ACKNOWLEDGEABLECONDITIONTYPE_CONFIRM := 9113,
	OPCUAID_ALARMCONDITIONTYPE_SHELVINGSTATE_TIMEDSHELVE := 9213,
	OPCUAID_ALARMCONDITIONTYPE_SHELVINGSTATE_UNSHELVE := 9211,
	OPCUAID_ALARMCONDITIONTYPE_SHELVINGSTATE_ONESHOTSHELVE := 9212,
	OPCUAID_ALARMCONDITIONTYPE_SILENCE := 16402,
	OPCUAID_ALARMCONDITIONTYPE_SUPPRESS := 16403,
	OPCUAID_ALARMCONDITIONTYPE_UNSUPPRESS := 17868,
	OPCUAID_ALARMCONDITIONTYPE_REMOVEFROMSERVICE := 17869,
	OPCUAID_ALARMCONDITIONTYPE_PLACEINSERVICE := 17870,
	OPCUAID_ALARMCONDITIONTYPE_RESET := 18199,
	OPCUAID_ALARMGROUPTYPE_ALARMCONDITIONINSTANCE_PLACEHOLDER_DISABLE := 16439,
	OPCUAID_ALARMGROUPTYPE_ALARMCONDITIONINSTANCE_PLACEHOLDER_ENABLE := 16440,
	OPCUAID_ALARMGROUPTYPE_ALARMCONDITIONINSTANCE_PLACEHOLDER_ADDCOMMENT := 16441,
	OPCUAID_ALARMGROUPTYPE_ALARMCONDITIONINSTANCE_PLACEHOLDER_ACKNOWLEDGE := 16461,
	OPCUAID_ALARMGROUPTYPE_ALARMCONDITIONINSTANCE_PLACEHOLDER_SHELVINGSTATE_TIMEDSHELVE := 16517,
	OPCUAID_ALARMGROUPTYPE_ALARMCONDITIONINSTANCE_PLACEHOLDER_SHELVINGSTATE_UNSHELVE := 16515,
	OPCUAID_ALARMGROUPTYPE_ALARMCONDITIONINSTANCE_PLACEHOLDER_SHELVINGSTATE_ONESHOTSHELVE := 16516,
	OPCUAID_SHELVEDSTATEMACHINETYPE_TIMEDSHELVE := 2949,
	OPCUAID_SHELVEDSTATEMACHINETYPE_UNSHELVE := 2947,
	OPCUAID_SHELVEDSTATEMACHINETYPE_ONESHOTSHELVE := 2948,
	OPCUAID_LIMITALARMTYPE_SHELVINGSTATE_TIMEDSHELVE := 9314,
	OPCUAID_LIMITALARMTYPE_SHELVINGSTATE_UNSHELVE := 9312,
	OPCUAID_LIMITALARMTYPE_SHELVINGSTATE_ONESHOTSHELVE := 9313,
	OPCUAID_EXCLUSIVELIMITALARMTYPE_SHELVINGSTATE_TIMEDSHELVE := 9451,
	OPCUAID_EXCLUSIVELIMITALARMTYPE_SHELVINGSTATE_UNSHELVE := 9449,
	OPCUAID_EXCLUSIVELIMITALARMTYPE_SHELVINGSTATE_ONESHOTSHELVE := 9450,
	OPCUAID_NONEXCLUSIVELIMITALARMTYPE_SHELVINGSTATE_TIMEDSHELVE := 10016,
	OPCUAID_NONEXCLUSIVELIMITALARMTYPE_SHELVINGSTATE_UNSHELVE := 10014,
	OPCUAID_NONEXCLUSIVELIMITALARMTYPE_SHELVINGSTATE_ONESHOTSHELVE := 10015,
	OPCUAID_NONEXCLUSIVELEVELALARMTYPE_SHELVINGSTATE_TIMEDSHELVE := 10170,
	OPCUAID_NONEXCLUSIVELEVELALARMTYPE_SHELVINGSTATE_UNSHELVE := 10168,
	OPCUAID_NONEXCLUSIVELEVELALARMTYPE_SHELVINGSTATE_ONESHOTSHELVE := 10169,
	OPCUAID_EXCLUSIVELEVELALARMTYPE_SHELVINGSTATE_TIMEDSHELVE := 9592,
	OPCUAID_EXCLUSIVELEVELALARMTYPE_SHELVINGSTATE_UNSHELVE := 9590,
	OPCUAID_EXCLUSIVELEVELALARMTYPE_SHELVINGSTATE_ONESHOTSHELVE := 9591,
	OPCUAID_NONEXCLUSIVEDEVIATIONALARMTYPE_SHELVINGSTATE_TIMEDSHELVE := 10478,
	OPCUAID_NONEXCLUSIVEDEVIATIONALARMTYPE_SHELVINGSTATE_UNSHELVE := 10476,
	OPCUAID_NONEXCLUSIVEDEVIATIONALARMTYPE_SHELVINGSTATE_ONESHOTSHELVE := 10477,
	OPCUAID_NONEXCLUSIVERATEOFCHANGEALARMTYPE_SHELVINGSTATE_TIMEDSHELVE := 10324,
	OPCUAID_NONEXCLUSIVERATEOFCHANGEALARMTYPE_SHELVINGSTATE_UNSHELVE := 10322,
	OPCUAID_NONEXCLUSIVERATEOFCHANGEALARMTYPE_SHELVINGSTATE_ONESHOTSHELVE := 10323,
	OPCUAID_EXCLUSIVEDEVIATIONALARMTYPE_SHELVINGSTATE_TIMEDSHELVE := 9874,
	OPCUAID_EXCLUSIVEDEVIATIONALARMTYPE_SHELVINGSTATE_UNSHELVE := 9872,
	OPCUAID_EXCLUSIVEDEVIATIONALARMTYPE_SHELVINGSTATE_ONESHOTSHELVE := 9873,
	OPCUAID_EXCLUSIVERATEOFCHANGEALARMTYPE_SHELVINGSTATE_TIMEDSHELVE := 9733,
	OPCUAID_EXCLUSIVERATEOFCHANGEALARMTYPE_SHELVINGSTATE_UNSHELVE := 9731,
	OPCUAID_EXCLUSIVERATEOFCHANGEALARMTYPE_SHELVINGSTATE_ONESHOTSHELVE := 9732,
	OPCUAID_DISCRETEALARMTYPE_SHELVINGSTATE_TIMEDSHELVE := 10633,
	OPCUAID_DISCRETEALARMTYPE_SHELVINGSTATE_UNSHELVE := 10631,
	OPCUAID_DISCRETEALARMTYPE_SHELVINGSTATE_ONESHOTSHELVE := 10632,
	OPCUAID_OFFNORMALALARMTYPE_SHELVINGSTATE_TIMEDSHELVE := 10747,
	OPCUAID_OFFNORMALALARMTYPE_SHELVINGSTATE_UNSHELVE := 10745,
	OPCUAID_OFFNORMALALARMTYPE_SHELVINGSTATE_ONESHOTSHELVE := 10746,
	OPCUAID_SYSTEMOFFNORMALALARMTYPE_SHELVINGSTATE_TIMEDSHELVE := 11846,
	OPCUAID_SYSTEMOFFNORMALALARMTYPE_SHELVINGSTATE_UNSHELVE := 11844,
	OPCUAID_SYSTEMOFFNORMALALARMTYPE_SHELVINGSTATE_ONESHOTSHELVE := 11845,
	OPCUAID_TRIPALARMTYPE_SHELVINGSTATE_TIMEDSHELVE := 10861,
	OPCUAID_TRIPALARMTYPE_SHELVINGSTATE_UNSHELVE := 10859,
	OPCUAID_TRIPALARMTYPE_SHELVINGSTATE_ONESHOTSHELVE := 10860,
	OPCUAID_INSTRUMENTDIAGNOSTICALARMTYPE_SHELVINGSTATE_TIMEDSHELVE := 18453,
	OPCUAID_INSTRUMENTDIAGNOSTICALARMTYPE_SHELVINGSTATE_UNSHELVE := 18455,
	OPCUAID_INSTRUMENTDIAGNOSTICALARMTYPE_SHELVINGSTATE_ONESHOTSHELVE := 18456,
	OPCUAID_SYSTEMDIAGNOSTICALARMTYPE_SHELVINGSTATE_TIMEDSHELVE := 18602,
	OPCUAID_SYSTEMDIAGNOSTICALARMTYPE_SHELVINGSTATE_UNSHELVE := 18604,
	OPCUAID_SYSTEMDIAGNOSTICALARMTYPE_SHELVINGSTATE_ONESHOTSHELVE := 18605,
	OPCUAID_CERTIFICATEEXPIRATIONALARMTYPE_SHELVINGSTATE_TIMEDSHELVE := 13320,
	OPCUAID_CERTIFICATEEXPIRATIONALARMTYPE_SHELVINGSTATE_UNSHELVE := 13318,
	OPCUAID_CERTIFICATEEXPIRATIONALARMTYPE_SHELVINGSTATE_ONESHOTSHELVE := 13319,
	OPCUAID_DISCREPANCYALARMTYPE_SHELVINGSTATE_TIMEDSHELVE := 17195,
	OPCUAID_DISCREPANCYALARMTYPE_SHELVINGSTATE_UNSHELVE := 17193,
	OPCUAID_DISCREPANCYALARMTYPE_SHELVINGSTATE_ONESHOTSHELVE := 17194,
	OPCUAID_ALARMMETRICSTYPE_RESET := 18666,
	OPCUAID_PROGRAMSTATEMACHINETYPE_START := 2426,
	OPCUAID_PROGRAMSTATEMACHINETYPE_SUSPEND := 2427,
	OPCUAID_PROGRAMSTATEMACHINETYPE_RESUME := 2428,
	OPCUAID_PROGRAMSTATEMACHINETYPE_HALT := 2429,
	OPCUAID_PROGRAMSTATEMACHINETYPE_RESET := 2430,
	OPCUAID_TRUSTLISTTYPE_OPENWITHMASKS := 12543,
	OPCUAID_TRUSTLISTTYPE_CLOSEANDUPDATE := 12546,
	OPCUAID_TRUSTLISTTYPE_ADDCERTIFICATE := 12548,
	OPCUAID_TRUSTLISTTYPE_REMOVECERTIFICATE := 12550,
	OPCUAID_CERTIFICATEGROUPTYPE_TRUSTLIST_OPEN := 13605,
	OPCUAID_CERTIFICATEGROUPTYPE_TRUSTLIST_CLOSE := 13608,
	OPCUAID_CERTIFICATEGROUPTYPE_TRUSTLIST_READ := 13610,
	OPCUAID_CERTIFICATEGROUPTYPE_TRUSTLIST_WRITE := 13613,
	OPCUAID_CERTIFICATEGROUPTYPE_TRUSTLIST_GETPOSITION := 13615,
	OPCUAID_CERTIFICATEGROUPTYPE_TRUSTLIST_SETPOSITION := 13618,
	OPCUAID_CERTIFICATEGROUPTYPE_TRUSTLIST_OPENWITHMASKS := 13621,
	OPCUAID_CERTIFICATEGROUPFOLDERTYPE_DEFAULTAPPLICATIONGROUP_TRUSTLIST_OPEN := 13821,
	OPCUAID_CERTIFICATEGROUPFOLDERTYPE_DEFAULTAPPLICATIONGROUP_TRUSTLIST_CLOSE := 13824,
	OPCUAID_CERTIFICATEGROUPFOLDERTYPE_DEFAULTAPPLICATIONGROUP_TRUSTLIST_READ := 13826,
	OPCUAID_CERTIFICATEGROUPFOLDERTYPE_DEFAULTAPPLICATIONGROUP_TRUSTLIST_WRITE := 13829,
	OPCUAID_CERTIFICATEGROUPFOLDERTYPE_DEFAULTAPPLICATIONGROUP_TRUSTLIST_GETPOSITION := 13831,
	OPCUAID_CERTIFICATEGROUPFOLDERTYPE_DEFAULTAPPLICATIONGROUP_TRUSTLIST_SETPOSITION := 13834,
	OPCUAID_CERTIFICATEGROUPFOLDERTYPE_DEFAULTAPPLICATIONGROUP_TRUSTLIST_OPENWITHMASKS := 13837,
	OPCUAID_CERTIFICATEGROUPFOLDERTYPE_DEFAULTHTTPSGROUP_TRUSTLIST_OPEN := 13855,
	OPCUAID_CERTIFICATEGROUPFOLDERTYPE_DEFAULTHTTPSGROUP_TRUSTLIST_CLOSE := 13858,
	OPCUAID_CERTIFICATEGROUPFOLDERTYPE_DEFAULTHTTPSGROUP_TRUSTLIST_READ := 13860,
	OPCUAID_CERTIFICATEGROUPFOLDERTYPE_DEFAULTHTTPSGROUP_TRUSTLIST_WRITE := 13863,
	OPCUAID_CERTIFICATEGROUPFOLDERTYPE_DEFAULTHTTPSGROUP_TRUSTLIST_GETPOSITION := 13865,
	OPCUAID_CERTIFICATEGROUPFOLDERTYPE_DEFAULTHTTPSGROUP_TRUSTLIST_SETPOSITION := 13868,
	OPCUAID_CERTIFICATEGROUPFOLDERTYPE_DEFAULTHTTPSGROUP_TRUSTLIST_OPENWITHMASKS := 13871,
	OPCUAID_CERTIFICATEGROUPFOLDERTYPE_DEFAULTUSERTOKENGROUP_TRUSTLIST_OPEN := 13889,
	OPCUAID_CERTIFICATEGROUPFOLDERTYPE_DEFAULTUSERTOKENGROUP_TRUSTLIST_CLOSE := 13892,
	OPCUAID_CERTIFICATEGROUPFOLDERTYPE_DEFAULTUSERTOKENGROUP_TRUSTLIST_READ := 13894,
	OPCUAID_CERTIFICATEGROUPFOLDERTYPE_DEFAULTUSERTOKENGROUP_TRUSTLIST_WRITE := 13897,
	OPCUAID_CERTIFICATEGROUPFOLDERTYPE_DEFAULTUSERTOKENGROUP_TRUSTLIST_GETPOSITION := 13899,
	OPCUAID_CERTIFICATEGROUPFOLDERTYPE_DEFAULTUSERTOKENGROUP_TRUSTLIST_SETPOSITION := 13902,
	OPCUAID_CERTIFICATEGROUPFOLDERTYPE_DEFAULTUSERTOKENGROUP_TRUSTLIST_OPENWITHMASKS := 13905,
	OPCUAID_CERTIFICATEGROUPFOLDERTYPE_ADDITIONALGROUP_PLACEHOLDER_TRUSTLIST_OPEN := 13923,
	OPCUAID_CERTIFICATEGROUPFOLDERTYPE_ADDITIONALGROUP_PLACEHOLDER_TRUSTLIST_CLOSE := 13926,
	OPCUAID_CERTIFICATEGROUPFOLDERTYPE_ADDITIONALGROUP_PLACEHOLDER_TRUSTLIST_READ := 13928,
	OPCUAID_CERTIFICATEGROUPFOLDERTYPE_ADDITIONALGROUP_PLACEHOLDER_TRUSTLIST_WRITE := 13931,
	OPCUAID_CERTIFICATEGROUPFOLDERTYPE_ADDITIONALGROUP_PLACEHOLDER_TRUSTLIST_GETPOSITION := 13933,
	OPCUAID_CERTIFICATEGROUPFOLDERTYPE_ADDITIONALGROUP_PLACEHOLDER_TRUSTLIST_SETPOSITION := 13936,
	OPCUAID_CERTIFICATEGROUPFOLDERTYPE_ADDITIONALGROUP_PLACEHOLDER_TRUSTLIST_OPENWITHMASKS := 13939,
	OPCUAID_SERVERCONFIGURATIONTYPE_CERTIFICATEGROUPS_DEFAULTAPPLICATIONGROUP_TRUSTLIST_OPEN := 13958,
	OPCUAID_SERVERCONFIGURATIONTYPE_CERTIFICATEGROUPS_DEFAULTAPPLICATIONGROUP_TRUSTLIST_CLOSE := 13961,
	OPCUAID_SERVERCONFIGURATIONTYPE_CERTIFICATEGROUPS_DEFAULTAPPLICATIONGROUP_TRUSTLIST_READ := 13963,
	OPCUAID_SERVERCONFIGURATIONTYPE_CERTIFICATEGROUPS_DEFAULTAPPLICATIONGROUP_TRUSTLIST_WRITE := 13966,
	OPCUAID_SERVERCONFIGURATIONTYPE_CERTIFICATEGROUPS_DEFAULTAPPLICATIONGROUP_TRUSTLIST_GETPOSITION := 13968,
	OPCUAID_SERVERCONFIGURATIONTYPE_CERTIFICATEGROUPS_DEFAULTAPPLICATIONGROUP_TRUSTLIST_SETPOSITION := 13971,
	OPCUAID_SERVERCONFIGURATIONTYPE_CERTIFICATEGROUPS_DEFAULTAPPLICATIONGROUP_TRUSTLIST_OPENWITHMASKS := 13974,
	OPCUAID_SERVERCONFIGURATIONTYPE_CERTIFICATEGROUPS_DEFAULTHTTPSGROUP_TRUSTLIST_OPEN := 13992,
	OPCUAID_SERVERCONFIGURATIONTYPE_CERTIFICATEGROUPS_DEFAULTHTTPSGROUP_TRUSTLIST_CLOSE := 13995,
	OPCUAID_SERVERCONFIGURATIONTYPE_CERTIFICATEGROUPS_DEFAULTHTTPSGROUP_TRUSTLIST_READ := 13997,
	OPCUAID_SERVERCONFIGURATIONTYPE_CERTIFICATEGROUPS_DEFAULTHTTPSGROUP_TRUSTLIST_WRITE := 14000,
	OPCUAID_SERVERCONFIGURATIONTYPE_CERTIFICATEGROUPS_DEFAULTHTTPSGROUP_TRUSTLIST_GETPOSITION := 14002,
	OPCUAID_SERVERCONFIGURATIONTYPE_CERTIFICATEGROUPS_DEFAULTHTTPSGROUP_TRUSTLIST_SETPOSITION := 14005,
	OPCUAID_SERVERCONFIGURATIONTYPE_CERTIFICATEGROUPS_DEFAULTHTTPSGROUP_TRUSTLIST_OPENWITHMASKS := 14008,
	OPCUAID_SERVERCONFIGURATIONTYPE_CERTIFICATEGROUPS_DEFAULTUSERTOKENGROUP_TRUSTLIST_OPEN := 14026,
	OPCUAID_SERVERCONFIGURATIONTYPE_CERTIFICATEGROUPS_DEFAULTUSERTOKENGROUP_TRUSTLIST_CLOSE := 14029,
	OPCUAID_SERVERCONFIGURATIONTYPE_CERTIFICATEGROUPS_DEFAULTUSERTOKENGROUP_TRUSTLIST_READ := 14031,
	OPCUAID_SERVERCONFIGURATIONTYPE_CERTIFICATEGROUPS_DEFAULTUSERTOKENGROUP_TRUSTLIST_WRITE := 14034,
	OPCUAID_SERVERCONFIGURATIONTYPE_CERTIFICATEGROUPS_DEFAULTUSERTOKENGROUP_TRUSTLIST_GETPOSITION := 14036,
	OPCUAID_SERVERCONFIGURATIONTYPE_CERTIFICATEGROUPS_DEFAULTUSERTOKENGROUP_TRUSTLIST_SETPOSITION := 14039,
	OPCUAID_SERVERCONFIGURATIONTYPE_CERTIFICATEGROUPS_DEFAULTUSERTOKENGROUP_TRUSTLIST_OPENWITHMASKS := 14042,
	OPCUAID_SERVERCONFIGURATIONTYPE_UPDATECERTIFICATE := 12616,
	OPCUAID_SERVERCONFIGURATIONTYPE_APPLYCHANGES := 12734,
	OPCUAID_SERVERCONFIGURATIONTYPE_CREATESIGNINGREQUEST := 12731,
	OPCUAID_SERVERCONFIGURATIONTYPE_GETREJECTEDLIST := 12775,
	OPCUAID_SERVERCONFIGURATION_CERTIFICATEGROUPS_DEFAULTAPPLICATIONGROUP_TRUSTLIST_OPEN := 12647,
	OPCUAID_SERVERCONFIGURATION_CERTIFICATEGROUPS_DEFAULTAPPLICATIONGROUP_TRUSTLIST_CLOSE := 12650,
	OPCUAID_SERVERCONFIGURATION_CERTIFICATEGROUPS_DEFAULTAPPLICATIONGROUP_TRUSTLIST_READ := 12652,
	OPCUAID_SERVERCONFIGURATION_CERTIFICATEGROUPS_DEFAULTAPPLICATIONGROUP_TRUSTLIST_WRITE := 12655,
	OPCUAID_SERVERCONFIGURATION_CERTIFICATEGROUPS_DEFAULTAPPLICATIONGROUP_TRUSTLIST_GETPOSITION := 12657,
	OPCUAID_SERVERCONFIGURATION_CERTIFICATEGROUPS_DEFAULTAPPLICATIONGROUP_TRUSTLIST_SETPOSITION := 12660,
	OPCUAID_SERVERCONFIGURATION_CERTIFICATEGROUPS_DEFAULTAPPLICATIONGROUP_TRUSTLIST_OPENWITHMASKS := 12663,
	OPCUAID_SERVERCONFIGURATION_CERTIFICATEGROUPS_DEFAULTAPPLICATIONGROUP_TRUSTLIST_CLOSEANDUPDATE := 12666,
	OPCUAID_SERVERCONFIGURATION_CERTIFICATEGROUPS_DEFAULTAPPLICATIONGROUP_TRUSTLIST_ADDCERTIFICATE := 12668,
	OPCUAID_SERVERCONFIGURATION_CERTIFICATEGROUPS_DEFAULTAPPLICATIONGROUP_TRUSTLIST_REMOVECERTIFICATE := 12670,
	OPCUAID_SERVERCONFIGURATION_CERTIFICATEGROUPS_DEFAULTHTTPSGROUP_TRUSTLIST_OPEN := 14095,
	OPCUAID_SERVERCONFIGURATION_CERTIFICATEGROUPS_DEFAULTHTTPSGROUP_TRUSTLIST_CLOSE := 14098,
	OPCUAID_SERVERCONFIGURATION_CERTIFICATEGROUPS_DEFAULTHTTPSGROUP_TRUSTLIST_READ := 14100,
	OPCUAID_SERVERCONFIGURATION_CERTIFICATEGROUPS_DEFAULTHTTPSGROUP_TRUSTLIST_WRITE := 14103,
	OPCUAID_SERVERCONFIGURATION_CERTIFICATEGROUPS_DEFAULTHTTPSGROUP_TRUSTLIST_GETPOSITION := 14105,
	OPCUAID_SERVERCONFIGURATION_CERTIFICATEGROUPS_DEFAULTHTTPSGROUP_TRUSTLIST_SETPOSITION := 14108,
	OPCUAID_SERVERCONFIGURATION_CERTIFICATEGROUPS_DEFAULTHTTPSGROUP_TRUSTLIST_OPENWITHMASKS := 14111,
	OPCUAID_SERVERCONFIGURATION_CERTIFICATEGROUPS_DEFAULTHTTPSGROUP_TRUSTLIST_CLOSEANDUPDATE := 14114,
	OPCUAID_SERVERCONFIGURATION_CERTIFICATEGROUPS_DEFAULTHTTPSGROUP_TRUSTLIST_ADDCERTIFICATE := 14117,
	OPCUAID_SERVERCONFIGURATION_CERTIFICATEGROUPS_DEFAULTHTTPSGROUP_TRUSTLIST_REMOVECERTIFICATE := 14119,
	OPCUAID_SERVERCONFIGURATION_CERTIFICATEGROUPS_DEFAULTUSERTOKENGROUP_TRUSTLIST_OPEN := 14129,
	OPCUAID_SERVERCONFIGURATION_CERTIFICATEGROUPS_DEFAULTUSERTOKENGROUP_TRUSTLIST_CLOSE := 14132,
	OPCUAID_SERVERCONFIGURATION_CERTIFICATEGROUPS_DEFAULTUSERTOKENGROUP_TRUSTLIST_READ := 14134,
	OPCUAID_SERVERCONFIGURATION_CERTIFICATEGROUPS_DEFAULTUSERTOKENGROUP_TRUSTLIST_WRITE := 14137,
	OPCUAID_SERVERCONFIGURATION_CERTIFICATEGROUPS_DEFAULTUSERTOKENGROUP_TRUSTLIST_GETPOSITION := 14139,
	OPCUAID_SERVERCONFIGURATION_CERTIFICATEGROUPS_DEFAULTUSERTOKENGROUP_TRUSTLIST_SETPOSITION := 14142,
	OPCUAID_SERVERCONFIGURATION_CERTIFICATEGROUPS_DEFAULTUSERTOKENGROUP_TRUSTLIST_OPENWITHMASKS := 14145,
	OPCUAID_SERVERCONFIGURATION_CERTIFICATEGROUPS_DEFAULTUSERTOKENGROUP_TRUSTLIST_CLOSEANDUPDATE := 14148,
	OPCUAID_SERVERCONFIGURATION_CERTIFICATEGROUPS_DEFAULTUSERTOKENGROUP_TRUSTLIST_ADDCERTIFICATE := 14151,
	OPCUAID_SERVERCONFIGURATION_CERTIFICATEGROUPS_DEFAULTUSERTOKENGROUP_TRUSTLIST_REMOVECERTIFICATE := 14153,
	OPCUAID_SERVERCONFIGURATION_UPDATECERTIFICATE := 13737,
	OPCUAID_SERVERCONFIGURATION_APPLYCHANGES := 12740,
	OPCUAID_SERVERCONFIGURATION_CREATESIGNINGREQUEST := 12737,
	OPCUAID_SERVERCONFIGURATION_GETREJECTEDLIST := 12777,
	OPCUAID_KEYCREDENTIALCONFIGURATIONFOLDERTYPE_CREATECREDENTIAL := 17522,
	OPCUAID_KEYCREDENTIALCONFIGURATIONTYPE_GETENCRYPTINGKEY := 17534,
	OPCUAID_KEYCREDENTIALCONFIGURATIONTYPE_UPDATECREDENTIAL := 18006,
	OPCUAID_KEYCREDENTIALCONFIGURATIONTYPE_DELETECREDENTIAL := 18008,
	OPCUAID_PUBSUBKEYSERVICETYPE_GETSECURITYKEYS := 15907,
	OPCUAID_PUBSUBKEYSERVICETYPE_GETSECURITYGROUP := 15910,
	OPCUAID_PUBSUBKEYSERVICETYPE_SECURITYGROUPS_ADDSECURITYGROUP := 15914,
	OPCUAID_PUBSUBKEYSERVICETYPE_SECURITYGROUPS_REMOVESECURITYGROUP := 15917,
	OPCUAID_SECURITYGROUPFOLDERTYPE_SECURITYGROUPFOLDERNAME_PLACEHOLDER_ADDSECURITYGROUP := 15454,
	OPCUAID_SECURITYGROUPFOLDERTYPE_SECURITYGROUPFOLDERNAME_PLACEHOLDER_REMOVESECURITYGROUP := 15457,
	OPCUAID_SECURITYGROUPFOLDERTYPE_ADDSECURITYGROUP := 15461,
	OPCUAID_SECURITYGROUPFOLDERTYPE_REMOVESECURITYGROUP := 15464,
	OPCUAID_PUBLISHSUBSCRIBETYPE_SECURITYGROUPS_ADDSECURITYGROUP := 15435,
	OPCUAID_PUBLISHSUBSCRIBETYPE_SECURITYGROUPS_REMOVESECURITYGROUP := 15438,
	OPCUAID_PUBLISHSUBSCRIBETYPE_CONNECTIONNAME_PLACEHOLDER_DIAGNOSTICS_RESET := 18679,
	OPCUAID_PUBLISHSUBSCRIBETYPE_SETSECURITYKEYS := 17296,
	OPCUAID_PUBLISHSUBSCRIBETYPE_ADDCONNECTION := 16598,
	OPCUAID_PUBLISHSUBSCRIBETYPE_REMOVECONNECTION := 14432,
	OPCUAID_PUBLISHSUBSCRIBETYPE_DIAGNOSTICS_RESET := 18727,
	OPCUAID_PUBLISHSUBSCRIBE_GETSECURITYKEYS := 15215,
	OPCUAID_PUBLISHSUBSCRIBE_GETSECURITYGROUP := 15440,
	OPCUAID_PUBLISHSUBSCRIBE_SECURITYGROUPS_ADDSECURITYGROUP := 15444,
	OPCUAID_PUBLISHSUBSCRIBE_SECURITYGROUPS_REMOVESECURITYGROUP := 15447,
	OPCUAID_PUBLISHSUBSCRIBE_CONNECTIONNAME_PLACEHOLDER_DIAGNOSTICS_RESET := 16076,
	OPCUAID_PUBLISHSUBSCRIBE_ADDCONNECTION := 17366,
	OPCUAID_PUBLISHSUBSCRIBE_REMOVECONNECTION := 17369,
	OPCUAID_PUBLISHSUBSCRIBE_DIAGNOSTICS_RESET := 17421,
	OPCUAID_PUBLISHEDDATASETTYPE_DATASETWRITERNAME_PLACEHOLDER_DIAGNOSTICS_RESET := 18883,
	OPCUAID_PUBLISHEDDATASETTYPE_EXTENSIONFIELDS_ADDEXTENSIONFIELD := 15482,
	OPCUAID_PUBLISHEDDATASETTYPE_EXTENSIONFIELDS_REMOVEEXTENSIONFIELD := 15485,
	OPCUAID_EXTENSIONFIELDSTYPE_ADDEXTENSIONFIELD := 15491,
	OPCUAID_EXTENSIONFIELDSTYPE_REMOVEEXTENSIONFIELD := 15494,
	OPCUAID_PUBLISHEDDATAITEMSTYPE_DATASETWRITERNAME_PLACEHOLDER_DIAGNOSTICS_RESET := 18942,
	OPCUAID_PUBLISHEDDATAITEMSTYPE_EXTENSIONFIELDS_ADDEXTENSIONFIELD := 15504,
	OPCUAID_PUBLISHEDDATAITEMSTYPE_EXTENSIONFIELDS_REMOVEEXTENSIONFIELD := 15507,
	OPCUAID_PUBLISHEDDATAITEMSTYPE_ADDVARIABLES := 14555,
	OPCUAID_PUBLISHEDDATAITEMSTYPE_REMOVEVARIABLES := 14558,
	OPCUAID_PUBLISHEDEVENTSTYPE_DATASETWRITERNAME_PLACEHOLDER_DIAGNOSTICS_RESET := 19001,
	OPCUAID_PUBLISHEDEVENTSTYPE_EXTENSIONFIELDS_ADDEXTENSIONFIELD := 15512,
	OPCUAID_PUBLISHEDEVENTSTYPE_EXTENSIONFIELDS_REMOVEEXTENSIONFIELD := 15515,
	OPCUAID_PUBLISHEDEVENTSTYPE_MODIFYFIELDSELECTION := 15052,
	OPCUAID_DATASETFOLDERTYPE_DATASETFOLDERNAME_PLACEHOLDER_ADDPUBLISHEDDATAITEMS := 14479,
	OPCUAID_DATASETFOLDERTYPE_DATASETFOLDERNAME_PLACEHOLDER_ADDPUBLISHEDEVENTS := 14482,
	OPCUAID_DATASETFOLDERTYPE_DATASETFOLDERNAME_PLACEHOLDER_ADDPUBLISHEDDATAITEMSTEMPLATE := 16842,
	OPCUAID_DATASETFOLDERTYPE_DATASETFOLDERNAME_PLACEHOLDER_ADDPUBLISHEDEVENTSTEMPLATE := 16881,
	OPCUAID_DATASETFOLDERTYPE_DATASETFOLDERNAME_PLACEHOLDER_REMOVEPUBLISHEDDATASET := 14485,
	OPCUAID_DATASETFOLDERTYPE_DATASETFOLDERNAME_PLACEHOLDER_ADDDATASETFOLDER := 16884,
	OPCUAID_DATASETFOLDERTYPE_DATASETFOLDERNAME_PLACEHOLDER_REMOVEDATASETFOLDER := 16923,
	OPCUAID_DATASETFOLDERTYPE_PUBLISHEDDATASETNAME_PLACEHOLDER_EXTENSIONFIELDS_ADDEXTENSIONFIELD := 15474,
	OPCUAID_DATASETFOLDERTYPE_PUBLISHEDDATASETNAME_PLACEHOLDER_EXTENSIONFIELDS_REMOVEEXTENSIONFIELD := 15477,
	OPCUAID_DATASETFOLDERTYPE_ADDPUBLISHEDDATAITEMS := 14493,
	OPCUAID_DATASETFOLDERTYPE_ADDPUBLISHEDEVENTS := 14496,
	OPCUAID_DATASETFOLDERTYPE_ADDPUBLISHEDDATAITEMSTEMPLATE := 16935,
	OPCUAID_DATASETFOLDERTYPE_ADDPUBLISHEDEVENTSTEMPLATE := 16960,
	OPCUAID_DATASETFOLDERTYPE_REMOVEPUBLISHEDDATASET := 14499,
	OPCUAID_DATASETFOLDERTYPE_ADDDATASETFOLDER := 16994,
	OPCUAID_DATASETFOLDERTYPE_REMOVEDATASETFOLDER := 16997,
	OPCUAID_PUBSUBCONNECTIONTYPE_WRITERGROUPNAME_PLACEHOLDER_DIAGNOSTICS_RESET := 19119,
	OPCUAID_PUBSUBCONNECTIONTYPE_READERGROUPNAME_PLACEHOLDER_DIAGNOSTICS_RESET := 19188,
	OPCUAID_PUBSUBCONNECTIONTYPE_DIAGNOSTICS_RESET := 19253,
	OPCUAID_PUBSUBCONNECTIONTYPE_ADDWRITERGROUP := 17427,
	OPCUAID_PUBSUBCONNECTIONTYPE_ADDREADERGROUP := 17465,
	OPCUAID_PUBSUBCONNECTIONTYPE_REMOVEGROUP := 14225,
	OPCUAID_WRITERGROUPTYPE_DATASETWRITERNAME_PLACEHOLDER_DIAGNOSTICS_RESET := 17765,
	OPCUAID_WRITERGROUPTYPE_DIAGNOSTICS_RESET := 17824,
	OPCUAID_WRITERGROUPTYPE_ADDDATASETWRITER := 17969,
	OPCUAID_WRITERGROUPTYPE_REMOVEDATASETWRITER := 17992,
	OPCUAID_READERGROUPTYPE_DATASETREADERNAME_PLACEHOLDER_DIAGNOSTICS_RESET := 18104,
	OPCUAID_READERGROUPTYPE_DIAGNOSTICS_RESET := 21027,
	OPCUAID_READERGROUPTYPE_ADDDATASETREADER := 21082,
	OPCUAID_READERGROUPTYPE_REMOVEDATASETREADER := 21085,
	OPCUAID_DATASETWRITERTYPE_DIAGNOSTICS_RESET := 19562,
	OPCUAID_DATASETREADERTYPE_DIAGNOSTICS_RESET := 19621,
	OPCUAID_DATASETREADERTYPE_CREATETARGETVARIABLES := 17386,
	OPCUAID_DATASETREADERTYPE_CREATEDATASETMIRROR := 17389,
	OPCUAID_TARGETVARIABLESTYPE_ADDTARGETVARIABLES := 15115,
	OPCUAID_TARGETVARIABLESTYPE_REMOVETARGETVARIABLES := 15118,
	OPCUAID_PUBSUBSTATUSTYPE_ENABLE := 14645,
	OPCUAID_PUBSUBSTATUSTYPE_DISABLE := 14646,
	OPCUAID_PUBSUBDIAGNOSTICSTYPE_RESET := 19689,
	OPCUAID_DEFAULTBINARY := 3062,
	OPCUAID_DEFAULTXML := 3063,
	OPCUAID_MODELLINGRULE_MANDATORY := 78,
	OPCUAID_MODELLINGRULE_OPTIONAL := 80,
	OPCUAID_MODELLINGRULE_EXPOSESITSARRAY := 83,
	OPCUAID_MODELLINGRULE_MANDATORYSHARED := 79,
	OPCUAID_MODELLINGRULE_OPTIONALPLACEHOLDER := 11508,
	OPCUAID_MODELLINGRULE_MANDATORYPLACEHOLDER := 11510,
	OPCUAID_ROOTFOLDER := 84,
	OPCUAID_OBJECTSFOLDER := 85,
	OPCUAID_TYPESFOLDER := 86,
	OPCUAID_VIEWSFOLDER := 87,
	OPCUAID_OBJECTTYPESFOLDER := 88,
	OPCUAID_VARIABLETYPESFOLDER := 89,
	OPCUAID_DATATYPESFOLDER := 90,
	OPCUAID_REFERENCETYPESFOLDER := 91,
	OPCUAID_XMLSCHEMA_TYPESYSTEM := 92,
	OPCUAID_OPCBINARYSCHEMA_TYPESYSTEM := 93,
	OPCUAID_OPCUANAMESPACEMETADATA := 15957,
	OPCUAID_SERVERTYPE_SERVERCAPABILITIES := 2009,
	OPCUAID_SERVERTYPE_SERVERCAPABILITIES_MODELLINGRULES := 3093,
	OPCUAID_SERVERTYPE_SERVERCAPABILITIES_AGGREGATEFUNCTIONS := 3094,
	OPCUAID_SERVERTYPE_SERVERDIAGNOSTICS := 2010,
	OPCUAID_SERVERTYPE_SERVERDIAGNOSTICS_SESSIONSDIAGNOSTICSSUMMARY := 3111,
	OPCUAID_SERVERTYPE_VENDORSERVERINFO := 2011,
	OPCUAID_SERVERTYPE_SERVERREDUNDANCY := 2012,
	OPCUAID_SERVERTYPE_NAMESPACES := 11527,
	OPCUAID_SERVERCAPABILITIESTYPE_OPERATIONLIMITS := 11551,
	OPCUAID_SERVERCAPABILITIESTYPE_MODELLINGRULES := 2019,
	OPCUAID_SERVERCAPABILITIESTYPE_AGGREGATEFUNCTIONS := 2754,
	OPCUAID_SERVERCAPABILITIESTYPE_ROLESET := 16295,
	OPCUAID_SERVERDIAGNOSTICSTYPE_SESSIONSDIAGNOSTICSSUMMARY := 2744,
	OPCUAID_SESSIONSDIAGNOSTICSSUMMARYTYPE_CLIENTNAME_PLACEHOLDER := 12097,
	OPCUAID_NAMESPACEMETADATATYPE_NAMESPACEFILE := 11624,
	OPCUAID_NAMESPACESTYPE_NAMESPACEIDENTIFIER_PLACEHOLDER := 11646,
	OPCUAID_EVENTTYPESFOLDER := 3048,
	OPCUAID_SERVER := 2253,
	OPCUAID_SERVER_SERVERCAPABILITIES := 2268,
	OPCUAID_SERVER_SERVERCAPABILITIES_OPERATIONLIMITS := 11704,
	OPCUAID_SERVER_SERVERCAPABILITIES_MODELLINGRULES := 2996,
	OPCUAID_SERVER_SERVERCAPABILITIES_AGGREGATEFUNCTIONS := 2997,
	OPCUAID_SERVER_SERVERCAPABILITIES_ROLESET := 15606,
	OPCUAID_SERVER_SERVERDIAGNOSTICS := 2274,
	OPCUAID_SERVER_SERVERDIAGNOSTICS_SESSIONSDIAGNOSTICSSUMMARY := 3706,
	OPCUAID_SERVER_VENDORSERVERINFO := 2295,
	OPCUAID_SERVER_SERVERREDUNDANCY := 2296,
	OPCUAID_SERVER_NAMESPACES := 11715,
	OPCUAID_HISTORYSERVERCAPABILITIES := 11192,
	OPCUAID_HISTORYSERVERCAPABILITIES_AGGREGATEFUNCTIONS := 11201,
	OPCUAID_FILEDIRECTORYTYPE_FILEDIRECTORYNAME_PLACEHOLDER := 13354,
	OPCUAID_FILEDIRECTORYTYPE_FILENAME_PLACEHOLDER := 13366,
	OPCUAID_FILESYSTEM := 16314,
	OPCUAID_TEMPORARYFILETRANSFERTYPE_TRANSFERSTATE_PLACEHOLDER := 15754,
	OPCUAID_FILETRANSFERSTATEMACHINETYPE_IDLE := 15815,
	OPCUAID_FILETRANSFERSTATEMACHINETYPE_READPREPARE := 15817,
	OPCUAID_FILETRANSFERSTATEMACHINETYPE_READTRANSFER := 15819,
	OPCUAID_FILETRANSFERSTATEMACHINETYPE_APPLYWRITE := 15821,
	OPCUAID_FILETRANSFERSTATEMACHINETYPE_ERROR := 15823,
	OPCUAID_FILETRANSFERSTATEMACHINETYPE_IDLETOREADPREPARE := 15825,
	OPCUAID_FILETRANSFERSTATEMACHINETYPE_READPREPARETOREADTRANSFER := 15827,
	OPCUAID_FILETRANSFERSTATEMACHINETYPE_READTRANSFERTOIDLE := 15829,
	OPCUAID_FILETRANSFERSTATEMACHINETYPE_IDLETOAPPLYWRITE := 15831,
	OPCUAID_FILETRANSFERSTATEMACHINETYPE_APPLYWRITETOIDLE := 15833,
	OPCUAID_FILETRANSFERSTATEMACHINETYPE_READPREPARETOERROR := 15835,
	OPCUAID_FILETRANSFERSTATEMACHINETYPE_READTRANSFERTOERROR := 15837,
	OPCUAID_FILETRANSFERSTATEMACHINETYPE_APPLYWRITETOERROR := 15839,
	OPCUAID_FILETRANSFERSTATEMACHINETYPE_ERRORTOIDLE := 15841,
	OPCUAID_ROLESETTYPE_ROLENAME_PLACEHOLDER := 15608,
	OPCUAID_WELLKNOWNROLE_ANONYMOUS := 15644,
	OPCUAID_WELLKNOWNROLE_AUTHENTICATEDUSER := 15656,
	OPCUAID_WELLKNOWNROLE_OBSERVER := 15668,
	OPCUAID_WELLKNOWNROLE_OPERATOR := 15680,
	OPCUAID_WELLKNOWNROLE_ENGINEER := 16036,
	OPCUAID_WELLKNOWNROLE_SUPERVISOR := 15692,
	OPCUAID_WELLKNOWNROLE_CONFIGUREADMIN := 15716,
	OPCUAID_WELLKNOWNROLE_SECURITYADMIN := 15704,
	OPCUAID_ALARMCONDITIONTYPE_SHELVINGSTATE := 9178,
	OPCUAID_ALARMCONDITIONTYPE_FIRSTINGROUP := 16398,
	OPCUAID_ALARMCONDITIONTYPE_ALARMGROUP_PLACEHOLDER := 16399,
	OPCUAID_ALARMGROUPTYPE_ALARMCONDITIONINSTANCE_PLACEHOLDER := 16406,
	OPCUAID_SHELVEDSTATEMACHINETYPE_UNSHELVED := 2930,
	OPCUAID_SHELVEDSTATEMACHINETYPE_TIMEDSHELVED := 2932,
	OPCUAID_SHELVEDSTATEMACHINETYPE_ONESHOTSHELVED := 2933,
	OPCUAID_SHELVEDSTATEMACHINETYPE_UNSHELVEDTOTIMEDSHELVED := 2935,
	OPCUAID_SHELVEDSTATEMACHINETYPE_UNSHELVEDTOONESHOTSHELVED := 2936,
	OPCUAID_SHELVEDSTATEMACHINETYPE_TIMEDSHELVEDTOUNSHELVED := 2940,
	OPCUAID_SHELVEDSTATEMACHINETYPE_TIMEDSHELVEDTOONESHOTSHELVED := 2942,
	OPCUAID_SHELVEDSTATEMACHINETYPE_ONESHOTSHELVEDTOUNSHELVED := 2943,
	OPCUAID_SHELVEDSTATEMACHINETYPE_ONESHOTSHELVEDTOTIMEDSHELVED := 2945,
	OPCUAID_EXCLUSIVELIMITSTATEMACHINETYPE_HIGHHIGH := 9329,
	OPCUAID_EXCLUSIVELIMITSTATEMACHINETYPE_HIGH := 9331,
	OPCUAID_EXCLUSIVELIMITSTATEMACHINETYPE_LOW := 9333,
	OPCUAID_EXCLUSIVELIMITSTATEMACHINETYPE_LOWLOW := 9335,
	OPCUAID_EXCLUSIVELIMITSTATEMACHINETYPE_LOWLOWTOLOW := 9337,
	OPCUAID_EXCLUSIVELIMITSTATEMACHINETYPE_LOWTOLOWLOW := 9338,
	OPCUAID_EXCLUSIVELIMITSTATEMACHINETYPE_HIGHHIGHTOHIGH := 9339,
	OPCUAID_EXCLUSIVELIMITSTATEMACHINETYPE_HIGHTOHIGHHIGH := 9340,
	OPCUAID_EXCLUSIVELIMITALARMTYPE_LIMITSTATE := 9455,
	OPCUAID_PROGRAMSTATEMACHINETYPE_FINALRESULTDATA := 3850,
	OPCUAID_PROGRAMSTATEMACHINETYPE_HALTED := 2406,
	OPCUAID_PROGRAMSTATEMACHINETYPE_READY := 2400,
	OPCUAID_PROGRAMSTATEMACHINETYPE_RUNNING := 2402,
	OPCUAID_PROGRAMSTATEMACHINETYPE_SUSPENDED := 2404,
	OPCUAID_PROGRAMSTATEMACHINETYPE_HALTEDTOREADY := 2408,
	OPCUAID_PROGRAMSTATEMACHINETYPE_READYTORUNNING := 2410,
	OPCUAID_PROGRAMSTATEMACHINETYPE_RUNNINGTOHALTED := 2412,
	OPCUAID_PROGRAMSTATEMACHINETYPE_RUNNINGTOREADY := 2414,
	OPCUAID_PROGRAMSTATEMACHINETYPE_RUNNINGTOSUSPENDED := 2416,
	OPCUAID_PROGRAMSTATEMACHINETYPE_SUSPENDEDTORUNNING := 2418,
	OPCUAID_PROGRAMSTATEMACHINETYPE_SUSPENDEDTOHALTED := 2420,
	OPCUAID_PROGRAMSTATEMACHINETYPE_SUSPENDEDTOREADY := 2422,
	OPCUAID_PROGRAMSTATEMACHINETYPE_READYTOHALTED := 2424,
	OPCUAID_HISTORICALDATACONFIGURATIONTYPE_AGGREGATECONFIGURATION := 3059,
	OPCUAID_HISTORICALDATACONFIGURATIONTYPE_AGGREGATEFUNCTIONS := 11876,
	OPCUAID_HACONFIGURATION := 11202,
	OPCUAID_HACONFIGURATION_AGGREGATECONFIGURATION := 11203,
	OPCUAID_HISTORYSERVERCAPABILITIESTYPE_AGGREGATEFUNCTIONS := 11172,
	OPCUAID_CERTIFICATEGROUPTYPE_TRUSTLIST := 13599,
	OPCUAID_CERTIFICATEGROUPFOLDERTYPE_DEFAULTAPPLICATIONGROUP := 13814,
	OPCUAID_CERTIFICATEGROUPFOLDERTYPE_DEFAULTAPPLICATIONGROUP_TRUSTLIST := 13815,
	OPCUAID_CERTIFICATEGROUPFOLDERTYPE_DEFAULTHTTPSGROUP := 13848,
	OPCUAID_CERTIFICATEGROUPFOLDERTYPE_DEFAULTHTTPSGROUP_TRUSTLIST := 13849,
	OPCUAID_CERTIFICATEGROUPFOLDERTYPE_DEFAULTUSERTOKENGROUP := 13882,
	OPCUAID_CERTIFICATEGROUPFOLDERTYPE_DEFAULTUSERTOKENGROUP_TRUSTLIST := 13883,
	OPCUAID_CERTIFICATEGROUPFOLDERTYPE_ADDITIONALGROUP_PLACEHOLDER := 13916,
	OPCUAID_CERTIFICATEGROUPFOLDERTYPE_ADDITIONALGROUP_PLACEHOLDER_TRUSTLIST := 13917,
	OPCUAID_SERVERCONFIGURATIONTYPE_CERTIFICATEGROUPS := 13950,
	OPCUAID_SERVERCONFIGURATIONTYPE_CERTIFICATEGROUPS_DEFAULTAPPLICATIONGROUP := 13951,
	OPCUAID_SERVERCONFIGURATIONTYPE_CERTIFICATEGROUPS_DEFAULTAPPLICATIONGROUP_TRUSTLIST := 13952,
	OPCUAID_SERVERCONFIGURATIONTYPE_CERTIFICATEGROUPS_DEFAULTHTTPSGROUP_TRUSTLIST := 13986,
	OPCUAID_SERVERCONFIGURATIONTYPE_CERTIFICATEGROUPS_DEFAULTUSERTOKENGROUP_TRUSTLIST := 14020,
	OPCUAID_SERVERCONFIGURATION := 12637,
	OPCUAID_SERVERCONFIGURATION_CERTIFICATEGROUPS := 14053,
	OPCUAID_SERVERCONFIGURATION_CERTIFICATEGROUPS_DEFAULTAPPLICATIONGROUP := 14156,
	OPCUAID_SERVERCONFIGURATION_CERTIFICATEGROUPS_DEFAULTAPPLICATIONGROUP_TRUSTLIST := 12642,
	OPCUAID_SERVERCONFIGURATION_CERTIFICATEGROUPS_DEFAULTHTTPSGROUP := 14088,
	OPCUAID_SERVERCONFIGURATION_CERTIFICATEGROUPS_DEFAULTHTTPSGROUP_TRUSTLIST := 14089,
	OPCUAID_SERVERCONFIGURATION_CERTIFICATEGROUPS_DEFAULTUSERTOKENGROUP := 14122,
	OPCUAID_SERVERCONFIGURATION_CERTIFICATEGROUPS_DEFAULTUSERTOKENGROUP_TRUSTLIST := 14123,
	OPCUAID_KEYCREDENTIALCONFIGURATIONFOLDERTYPE_SERVICENAME_PLACEHOLDER := 17511,
	OPCUAID_KEYCREDENTIALCONFIGURATION := 18155,
	OPCUAID_AUTHORIZATIONSERVICES := 17732,
	OPCUAID_AGGREGATEFUNCTION_INTERPOLATIVE := 2341,
	OPCUAID_AGGREGATEFUNCTION_AVERAGE := 2342,
	OPCUAID_AGGREGATEFUNCTION_TIMEAVERAGE := 2343,
	OPCUAID_AGGREGATEFUNCTION_TIMEAVERAGE2 := 11285,
	OPCUAID_AGGREGATEFUNCTION_TOTAL := 2344,
	OPCUAID_AGGREGATEFUNCTION_TOTAL2 := 11304,
	OPCUAID_AGGREGATEFUNCTION_MINIMUM := 2346,
	OPCUAID_AGGREGATEFUNCTION_MAXIMUM := 2347,
	OPCUAID_AGGREGATEFUNCTION_MINIMUMACTUALTIME := 2348,
	OPCUAID_AGGREGATEFUNCTION_MAXIMUMACTUALTIME := 2349,
	OPCUAID_AGGREGATEFUNCTION_RANGE := 2350,
	OPCUAID_AGGREGATEFUNCTION_MINIMUM2 := 11286,
	OPCUAID_AGGREGATEFUNCTION_MAXIMUM2 := 11287,
	OPCUAID_AGGREGATEFUNCTION_MINIMUMACTUALTIME2 := 11305,
	OPCUAID_AGGREGATEFUNCTION_MAXIMUMACTUALTIME2 := 11306,
	OPCUAID_AGGREGATEFUNCTION_RANGE2 := 11288,
	OPCUAID_AGGREGATEFUNCTION_ANNOTATIONCOUNT := 2351,
	OPCUAID_AGGREGATEFUNCTION_COUNT := 2352,
	OPCUAID_AGGREGATEFUNCTION_DURATIONINSTATEZERO := 11307,
	OPCUAID_AGGREGATEFUNCTION_DURATIONINSTATENONZERO := 11308,
	OPCUAID_AGGREGATEFUNCTION_NUMBEROFTRANSITIONS := 2355,
	OPCUAID_AGGREGATEFUNCTION_START := 2357,
	OPCUAID_AGGREGATEFUNCTION_END := 2358,
	OPCUAID_AGGREGATEFUNCTION_DELTA := 2359,
	OPCUAID_AGGREGATEFUNCTION_STARTBOUND := 11505,
	OPCUAID_AGGREGATEFUNCTION_ENDBOUND := 11506,
	OPCUAID_AGGREGATEFUNCTION_DELTABOUNDS := 11507,
	OPCUAID_AGGREGATEFUNCTION_DURATIONGOOD := 2360,
	OPCUAID_AGGREGATEFUNCTION_DURATIONBAD := 2361,
	OPCUAID_AGGREGATEFUNCTION_PERCENTGOOD := 2362,
	OPCUAID_AGGREGATEFUNCTION_PERCENTBAD := 2363,
	OPCUAID_AGGREGATEFUNCTION_WORSTQUALITY := 2364,
	OPCUAID_AGGREGATEFUNCTION_WORSTQUALITY2 := 11292,
	OPCUAID_AGGREGATEFUNCTION_STANDARDDEVIATIONSAMPLE := 11426,
	OPCUAID_AGGREGATEFUNCTION_STANDARDDEVIATIONPOPULATION := 11427,
	OPCUAID_AGGREGATEFUNCTION_VARIANCESAMPLE := 11428,
	OPCUAID_AGGREGATEFUNCTION_VARIANCEPOPULATION := 11429,
	OPCUAID_PUBSUBKEYSERVICETYPE_SECURITYGROUPS := 15913,
	OPCUAID_SECURITYGROUPFOLDERTYPE_SECURITYGROUPFOLDERNAME_PLACEHOLDER := 15453,
	OPCUAID_SECURITYGROUPFOLDERTYPE_SECURITYGROUPNAME_PLACEHOLDER := 15459,
	OPCUAID_PUBLISHSUBSCRIBETYPE_CONNECTIONNAME_PLACEHOLDER := 14417,
	OPCUAID_PUBLISHSUBSCRIBETYPE_CONNECTIONNAME_PLACEHOLDER_ADDRESS := 14423,
	OPCUAID_PUBLISHSUBSCRIBETYPE_CONNECTIONNAME_PLACEHOLDER_STATUS := 14419,
	OPCUAID_PUBLISHSUBSCRIBETYPE_CONNECTIONNAME_PLACEHOLDER_DIAGNOSTICS_COUNTERS := 18681,
	OPCUAID_PUBLISHSUBSCRIBETYPE_CONNECTIONNAME_PLACEHOLDER_DIAGNOSTICS_LIVEVALUES := 18712,
	OPCUAID_PUBLISHSUBSCRIBETYPE_PUBLISHEDDATASETS := 14434,
	OPCUAID_PUBLISHSUBSCRIBETYPE_STATUS := 15844,
	OPCUAID_PUBLISHSUBSCRIBETYPE_DIAGNOSTICS := 18715,
	OPCUAID_PUBLISHSUBSCRIBETYPE_DIAGNOSTICS_COUNTERS := 18729,
	OPCUAID_PUBLISHSUBSCRIBETYPE_DIAGNOSTICS_LIVEVALUES := 18760,
	OPCUAID_PUBLISHSUBSCRIBE := 14443,
	OPCUAID_PUBLISHSUBSCRIBE_SECURITYGROUPS := 15443,
	OPCUAID_PUBLISHSUBSCRIBE_CONNECTIONNAME_PLACEHOLDER_ADDRESS := 15851,
	OPCUAID_PUBLISHSUBSCRIBE_CONNECTIONNAME_PLACEHOLDER_STATUS := 15865,
	OPCUAID_PUBLISHSUBSCRIBE_CONNECTIONNAME_PLACEHOLDER_DIAGNOSTICS_COUNTERS := 16102,
	OPCUAID_PUBLISHSUBSCRIBE_CONNECTIONNAME_PLACEHOLDER_DIAGNOSTICS_LIVEVALUES := 17352,
	OPCUAID_PUBLISHSUBSCRIBE_PUBLISHEDDATASETS := 17371,
	OPCUAID_PUBLISHSUBSCRIBE_STATUS := 17405,
	OPCUAID_PUBLISHSUBSCRIBE_DIAGNOSTICS := 17409,
	OPCUAID_PUBLISHSUBSCRIBE_DIAGNOSTICS_COUNTERS := 17423,
	OPCUAID_PUBLISHSUBSCRIBE_DIAGNOSTICS_LIVEVALUES := 17457,
	OPCUAID_PUBLISHEDDATASETTYPE_DATASETWRITERNAME_PLACEHOLDER := 15222,
	OPCUAID_PUBLISHEDDATASETTYPE_DATASETWRITERNAME_PLACEHOLDER_STATUS := 15223,
	OPCUAID_PUBLISHEDDATASETTYPE_DATASETWRITERNAME_PLACEHOLDER_DIAGNOSTICS_COUNTERS := 18885,
	OPCUAID_PUBLISHEDDATASETTYPE_DATASETWRITERNAME_PLACEHOLDER_DIAGNOSTICS_LIVEVALUES := 18916,
	OPCUAID_PUBLISHEDDATASETTYPE_EXTENSIONFIELDS := 15481,
	OPCUAID_PUBLISHEDDATAITEMSTYPE_DATASETWRITERNAME_PLACEHOLDER_STATUS := 15231,
	OPCUAID_PUBLISHEDDATAITEMSTYPE_DATASETWRITERNAME_PLACEHOLDER_DIAGNOSTICS_COUNTERS := 18944,
	OPCUAID_PUBLISHEDDATAITEMSTYPE_DATASETWRITERNAME_PLACEHOLDER_DIAGNOSTICS_LIVEVALUES := 18975,
	OPCUAID_PUBLISHEDEVENTSTYPE_DATASETWRITERNAME_PLACEHOLDER_STATUS := 15239,
	OPCUAID_PUBLISHEDEVENTSTYPE_DATASETWRITERNAME_PLACEHOLDER_DIAGNOSTICS_COUNTERS := 19003,
	OPCUAID_PUBLISHEDEVENTSTYPE_DATASETWRITERNAME_PLACEHOLDER_DIAGNOSTICS_LIVEVALUES := 19034,
	OPCUAID_DATASETFOLDERTYPE_DATASETFOLDERNAME_PLACEHOLDER := 14478,
	OPCUAID_DATASETFOLDERTYPE_PUBLISHEDDATASETNAME_PLACEHOLDER := 14487,
	OPCUAID_PUBSUBCONNECTIONTYPE_ADDRESS := 14221,
	OPCUAID_PUBSUBCONNECTIONTYPE_TRANSPORTSETTINGS := 17203,
	OPCUAID_PUBSUBCONNECTIONTYPE_WRITERGROUPNAME_PLACEHOLDER := 17310,
	OPCUAID_PUBSUBCONNECTIONTYPE_WRITERGROUPNAME_PLACEHOLDER_STATUS := 17314,
	OPCUAID_PUBSUBCONNECTIONTYPE_WRITERGROUPNAME_PLACEHOLDER_DIAGNOSTICS_COUNTERS := 19121,
	OPCUAID_PUBSUBCONNECTIONTYPE_WRITERGROUPNAME_PLACEHOLDER_DIAGNOSTICS_LIVEVALUES := 19152,
	OPCUAID_PUBSUBCONNECTIONTYPE_READERGROUPNAME_PLACEHOLDER := 17325,
	OPCUAID_PUBSUBCONNECTIONTYPE_READERGROUPNAME_PLACEHOLDER_STATUS := 17329,
	OPCUAID_PUBSUBCONNECTIONTYPE_READERGROUPNAME_PLACEHOLDER_DIAGNOSTICS_COUNTERS := 19190,
	OPCUAID_PUBSUBCONNECTIONTYPE_READERGROUPNAME_PLACEHOLDER_DIAGNOSTICS_LIVEVALUES := 19221,
	OPCUAID_PUBSUBCONNECTIONTYPE_STATUS := 14600,
	OPCUAID_PUBSUBCONNECTIONTYPE_DIAGNOSTICS := 19241,
	OPCUAID_PUBSUBCONNECTIONTYPE_DIAGNOSTICS_COUNTERS := 19255,
	OPCUAID_PUBSUBCONNECTIONTYPE_DIAGNOSTICS_LIVEVALUES := 19286,
	OPCUAID_PUBSUBGROUPTYPE_STATUS := 15265,
	OPCUAID_WRITERGROUPTYPE_TRANSPORTSETTINGS := 17741,
	OPCUAID_WRITERGROUPTYPE_MESSAGESETTINGS := 17742,
	OPCUAID_WRITERGROUPTYPE_DATASETWRITERNAME_PLACEHOLDER := 17743,
	OPCUAID_WRITERGROUPTYPE_DATASETWRITERNAME_PLACEHOLDER_STATUS := 17749,
	OPCUAID_WRITERGROUPTYPE_DATASETWRITERNAME_PLACEHOLDER_DIAGNOSTICS_COUNTERS := 17767,
	OPCUAID_WRITERGROUPTYPE_DATASETWRITERNAME_PLACEHOLDER_DIAGNOSTICS_LIVEVALUES := 17798,
	OPCUAID_WRITERGROUPTYPE_DIAGNOSTICS := 17812,
	OPCUAID_WRITERGROUPTYPE_DIAGNOSTICS_COUNTERS := 17826,
	OPCUAID_WRITERGROUPTYPE_DIAGNOSTICS_LIVEVALUES := 17858,
	OPCUAID_READERGROUPTYPE_DATASETREADERNAME_PLACEHOLDER := 18076,
	OPCUAID_READERGROUPTYPE_DATASETREADERNAME_PLACEHOLDER_STATUS := 18088,
	OPCUAID_READERGROUPTYPE_DATASETREADERNAME_PLACEHOLDER_DIAGNOSTICS_COUNTERS := 18106,
	OPCUAID_READERGROUPTYPE_DATASETREADERNAME_PLACEHOLDER_DIAGNOSTICS_LIVEVALUES := 18137,
	OPCUAID_READERGROUPTYPE_DATASETREADERNAME_PLACEHOLDER_SUBSCRIBEDDATASET := 21006,
	OPCUAID_READERGROUPTYPE_DIAGNOSTICS := 21015,
	OPCUAID_READERGROUPTYPE_DIAGNOSTICS_COUNTERS := 21029,
	OPCUAID_READERGROUPTYPE_DIAGNOSTICS_LIVEVALUES := 21060,
	OPCUAID_READERGROUPTYPE_TRANSPORTSETTINGS := 21080,
	OPCUAID_READERGROUPTYPE_MESSAGESETTINGS := 21081,
	OPCUAID_DATASETWRITERTYPE_TRANSPORTSETTINGS := 15303,
	OPCUAID_DATASETWRITERTYPE_MESSAGESETTINGS := 21095,
	OPCUAID_DATASETWRITERTYPE_STATUS := 15299,
	OPCUAID_DATASETWRITERTYPE_DIAGNOSTICS := 19550,
	OPCUAID_DATASETWRITERTYPE_DIAGNOSTICS_COUNTERS := 19564,
	OPCUAID_DATASETWRITERTYPE_DIAGNOSTICS_LIVEVALUES := 19595,
	OPCUAID_DATASETREADERTYPE_TRANSPORTSETTINGS := 15311,
	OPCUAID_DATASETREADERTYPE_MESSAGESETTINGS := 21103,
	OPCUAID_DATASETREADERTYPE_STATUS := 15307,
	OPCUAID_DATASETREADERTYPE_DIAGNOSTICS := 19609,
	OPCUAID_DATASETREADERTYPE_DIAGNOSTICS_COUNTERS := 19623,
	OPCUAID_DATASETREADERTYPE_DIAGNOSTICS_LIVEVALUES := 19654,
	OPCUAID_DATASETREADERTYPE_SUBSCRIBEDDATASET := 15316,
	OPCUAID_PUBSUBDIAGNOSTICSTYPE_COUNTERS := 19691,
	OPCUAID_PUBSUBDIAGNOSTICSTYPE_LIVEVALUES := 19722,
	OPCUAID_PUBSUBDIAGNOSTICSROOTTYPE_LIVEVALUES := 19777,
	OPCUAID_PUBSUBDIAGNOSTICSCONNECTIONTYPE_LIVEVALUES := 19831,
	OPCUAID_PUBSUBDIAGNOSTICSWRITERGROUPTYPE_COUNTERS := 19848,
	OPCUAID_PUBSUBDIAGNOSTICSWRITERGROUPTYPE_LIVEVALUES := 19879,
	OPCUAID_PUBSUBDIAGNOSTICSREADERGROUPTYPE_COUNTERS := 19917,
	OPCUAID_PUBSUBDIAGNOSTICSREADERGROUPTYPE_LIVEVALUES := 19948,
	OPCUAID_PUBSUBDIAGNOSTICSDATASETWRITERTYPE_COUNTERS := 19982,
	OPCUAID_PUBSUBDIAGNOSTICSDATASETWRITERTYPE_LIVEVALUES := 20013,
	OPCUAID_PUBSUBDIAGNOSTICSDATASETREADERTYPE_COUNTERS := 20041,
	OPCUAID_PUBSUBDIAGNOSTICSDATASETREADERTYPE_LIVEVALUES := 20072,
	OPCUAID_DATAGRAMCONNECTIONTRANSPORTTYPE_DISCOVERYADDRESS := 15072,
	OPCUAID_KEYVALUEPAIR_ENCODING_DEFAULTBINARY := 14846,
	OPCUAID_ENDPOINTTYPE_ENCODING_DEFAULTBINARY := 15671,
	OPCUAID_IDENTITYMAPPINGRULETYPE_ENCODING_DEFAULTBINARY := 15736,
	OPCUAID_TRUSTLISTDATATYPE_ENCODING_DEFAULTBINARY := 12680,
	OPCUAID_DECIMALDATATYPE_ENCODING_DEFAULTBINARY := 17863,
	OPCUAID_DATATYPESCHEMAHEADER_ENCODING_DEFAULTBINARY := 15676,
	OPCUAID_DATATYPEDESCRIPTION_ENCODING_DEFAULTBINARY := 125,
	OPCUAID_STRUCTUREDESCRIPTION_ENCODING_DEFAULTBINARY := 126,
	OPCUAID_ENUMDESCRIPTION_ENCODING_DEFAULTBINARY := 127,
	OPCUAID_SIMPLETYPEDESCRIPTION_ENCODING_DEFAULTBINARY := 15421,
	OPCUAID_UABINARYFILEDATATYPE_ENCODING_DEFAULTBINARY := 15422,
	OPCUAID_DATASETMETADATATYPE_ENCODING_DEFAULTBINARY := 124,
	OPCUAID_FIELDMETADATA_ENCODING_DEFAULTBINARY := 14839,
	OPCUAID_CONFIGURATIONVERSIONDATATYPE_ENCODING_DEFAULTBINARY := 14847,
	OPCUAID_PUBLISHEDDATASETDATATYPE_ENCODING_DEFAULTBINARY := 15677,
	OPCUAID_PUBLISHEDDATASETSOURCEDATATYPE_ENCODING_DEFAULTBINARY := 15678,
	OPCUAID_PUBLISHEDVARIABLEDATATYPE_ENCODING_DEFAULTBINARY := 14323,
	OPCUAID_PUBLISHEDDATAITEMSDATATYPE_ENCODING_DEFAULTBINARY := 15679,
	OPCUAID_PUBLISHEDEVENTSDATATYPE_ENCODING_DEFAULTBINARY := 15681,
	OPCUAID_DATASETWRITERDATATYPE_ENCODING_DEFAULTBINARY := 15682,
	OPCUAID_DATASETWRITERTRANSPORTDATATYPE_ENCODING_DEFAULTBINARY := 15683,
	OPCUAID_DATASETWRITERMESSAGEDATATYPE_ENCODING_DEFAULTBINARY := 15688,
	OPCUAID_PUBSUBGROUPDATATYPE_ENCODING_DEFAULTBINARY := 15689,
	OPCUAID_WRITERGROUPDATATYPE_ENCODING_DEFAULTBINARY := 21150,
	OPCUAID_WRITERGROUPTRANSPORTDATATYPE_ENCODING_DEFAULTBINARY := 15691,
	OPCUAID_WRITERGROUPMESSAGEDATATYPE_ENCODING_DEFAULTBINARY := 15693,
	OPCUAID_PUBSUBCONNECTIONDATATYPE_ENCODING_DEFAULTBINARY := 15694,
	OPCUAID_CONNECTIONTRANSPORTDATATYPE_ENCODING_DEFAULTBINARY := 15695,
	OPCUAID_NETWORKADDRESSDATATYPE_ENCODING_DEFAULTBINARY := 21151,
	OPCUAID_NETWORKADDRESSURLDATATYPE_ENCODING_DEFAULTBINARY := 21152,
	OPCUAID_READERGROUPDATATYPE_ENCODING_DEFAULTBINARY := 21153,
	OPCUAID_READERGROUPTRANSPORTDATATYPE_ENCODING_DEFAULTBINARY := 15701,
	OPCUAID_READERGROUPMESSAGEDATATYPE_ENCODING_DEFAULTBINARY := 15702,
	OPCUAID_DATASETREADERDATATYPE_ENCODING_DEFAULTBINARY := 15703,
	OPCUAID_DATASETREADERTRANSPORTDATATYPE_ENCODING_DEFAULTBINARY := 15705,
	OPCUAID_DATASETREADERMESSAGEDATATYPE_ENCODING_DEFAULTBINARY := 15706,
	OPCUAID_SUBSCRIBEDDATASETDATATYPE_ENCODING_DEFAULTBINARY := 15707,
	OPCUAID_TARGETVARIABLESDATATYPE_ENCODING_DEFAULTBINARY := 15712,
	OPCUAID_FIELDTARGETDATATYPE_ENCODING_DEFAULTBINARY := 14848,
	OPCUAID_SUBSCRIBEDDATASETMIRRORDATATYPE_ENCODING_DEFAULTBINARY := 15713,
	OPCUAID_PUBSUBCONFIGURATIONDATATYPE_ENCODING_DEFAULTBINARY := 21154,
	OPCUAID_UADPWRITERGROUPMESSAGEDATATYPE_ENCODING_DEFAULTBINARY := 15715,
	OPCUAID_UADPDATASETWRITERMESSAGEDATATYPE_ENCODING_DEFAULTBINARY := 15717,
	OPCUAID_UADPDATASETREADERMESSAGEDATATYPE_ENCODING_DEFAULTBINARY := 15718,
	OPCUAID_JSONWRITERGROUPMESSAGEDATATYPE_ENCODING_DEFAULTBINARY := 15719,
	OPCUAID_JSONDATASETWRITERMESSAGEDATATYPE_ENCODING_DEFAULTBINARY := 15724,
	OPCUAID_JSONDATASETREADERMESSAGEDATATYPE_ENCODING_DEFAULTBINARY := 15725,
	OPCUAID_DATAGRAMCONNECTIONTRANSPORTDATATYPE_ENCODING_DEFAULTBINARY := 17468,
	OPCUAID_DATAGRAMWRITERGROUPTRANSPORTDATATYPE_ENCODING_DEFAULTBINARY := 21155,
	OPCUAID_BROKERCONNECTIONTRANSPORTDATATYPE_ENCODING_DEFAULTBINARY := 15479,
	OPCUAID_BROKERWRITERGROUPTRANSPORTDATATYPE_ENCODING_DEFAULTBINARY := 15727,
	OPCUAID_BROKERDATASETWRITERTRANSPORTDATATYPE_ENCODING_DEFAULTBINARY := 15729,
	OPCUAID_BROKERDATASETREADERTRANSPORTDATATYPE_ENCODING_DEFAULTBINARY := 15733,
	OPCUAID_ROLEPERMISSIONTYPE_ENCODING_DEFAULTBINARY := 128,
	OPCUAID_DATATYPEDEFINITION_ENCODING_DEFAULTBINARY := 121,
	OPCUAID_STRUCTUREFIELD_ENCODING_DEFAULTBINARY := 14844,
	OPCUAID_STRUCTUREDEFINITION_ENCODING_DEFAULTBINARY := 122,
	OPCUAID_ENUMDEFINITION_ENCODING_DEFAULTBINARY := 123,
	OPCUAID_NODE_ENCODING_DEFAULTBINARY := 260,
	OPCUAID_INSTANCENODE_ENCODING_DEFAULTBINARY := 11889,
	OPCUAID_TYPENODE_ENCODING_DEFAULTBINARY := 11890,
	OPCUAID_OBJECTNODE_ENCODING_DEFAULTBINARY := 263,
	OPCUAID_OBJECTTYPENODE_ENCODING_DEFAULTBINARY := 266,
	OPCUAID_VARIABLENODE_ENCODING_DEFAULTBINARY := 269,
	OPCUAID_VARIABLETYPENODE_ENCODING_DEFAULTBINARY := 272,
	OPCUAID_REFERENCETYPENODE_ENCODING_DEFAULTBINARY := 275,
	OPCUAID_METHODNODE_ENCODING_DEFAULTBINARY := 278,
	OPCUAID_VIEWNODE_ENCODING_DEFAULTBINARY := 281,
	OPCUAID_DATATYPENODE_ENCODING_DEFAULTBINARY := 284,
	OPCUAID_REFERENCENODE_ENCODING_DEFAULTBINARY := 287,
	OPCUAID_ARGUMENT_ENCODING_DEFAULTBINARY := 298,
	OPCUAID_ENUMVALUETYPE_ENCODING_DEFAULTBINARY := 8251,
	OPCUAID_ENUMFIELD_ENCODING_DEFAULTBINARY := 14845,
	OPCUAID_OPTIONSET_ENCODING_DEFAULTBINARY := 12765,
	OPCUAID_UNION_ENCODING_DEFAULTBINARY := 12766,
	OPCUAID_TIMEZONEDATATYPE_ENCODING_DEFAULTBINARY := 8917,
	OPCUAID_APPLICATIONDESCRIPTION_ENCODING_DEFAULTBINARY := 310,
	OPCUAID_REQUESTHEADER_ENCODING_DEFAULTBINARY := 391,
	OPCUAID_RESPONSEHEADER_ENCODING_DEFAULTBINARY := 394,
	OPCUAID_SERVICEFAULT_ENCODING_DEFAULTBINARY := 397,
	OPCUAID_SESSIONLESSINVOKEREQUESTTYPE_ENCODING_DEFAULTBINARY := 15903,
	OPCUAID_SESSIONLESSINVOKERESPONSETYPE_ENCODING_DEFAULTBINARY := 21001,
	OPCUAID_FINDSERVERSREQUEST_ENCODING_DEFAULTBINARY := 422,
	OPCUAID_FINDSERVERSRESPONSE_ENCODING_DEFAULTBINARY := 425,
	OPCUAID_SERVERONNETWORK_ENCODING_DEFAULTBINARY := 12207,
	OPCUAID_FINDSERVERSONNETWORKREQUEST_ENCODING_DEFAULTBINARY := 12208,
	OPCUAID_FINDSERVERSONNETWORKRESPONSE_ENCODING_DEFAULTBINARY := 12209,
	OPCUAID_USERTOKENPOLICY_ENCODING_DEFAULTBINARY := 306,
	OPCUAID_ENDPOINTDESCRIPTION_ENCODING_DEFAULTBINARY := 314,
	OPCUAID_GETENDPOINTSREQUEST_ENCODING_DEFAULTBINARY := 428,
	OPCUAID_GETENDPOINTSRESPONSE_ENCODING_DEFAULTBINARY := 431,
	OPCUAID_REGISTEREDSERVER_ENCODING_DEFAULTBINARY := 434,
	OPCUAID_REGISTERSERVERREQUEST_ENCODING_DEFAULTBINARY := 437,
	OPCUAID_REGISTERSERVERRESPONSE_ENCODING_DEFAULTBINARY := 440,
	OPCUAID_DISCOVERYCONFIGURATION_ENCODING_DEFAULTBINARY := 12900,
	OPCUAID_MDNSDISCOVERYCONFIGURATION_ENCODING_DEFAULTBINARY := 12901,
	OPCUAID_REGISTERSERVER2REQUEST_ENCODING_DEFAULTBINARY := 12211,
	OPCUAID_REGISTERSERVER2RESPONSE_ENCODING_DEFAULTBINARY := 12212,
	OPCUAID_CHANNELSECURITYTOKEN_ENCODING_DEFAULTBINARY := 443,
	OPCUAID_OPENSECURECHANNELREQUEST_ENCODING_DEFAULTBINARY := 446,
	OPCUAID_OPENSECURECHANNELRESPONSE_ENCODING_DEFAULTBINARY := 449,
	OPCUAID_CLOSESECURECHANNELREQUEST_ENCODING_DEFAULTBINARY := 452,
	OPCUAID_CLOSESECURECHANNELRESPONSE_ENCODING_DEFAULTBINARY := 455,
	OPCUAID_SIGNEDSOFTWARECERTIFICATE_ENCODING_DEFAULTBINARY := 346,
	OPCUAID_SIGNATUREDATA_ENCODING_DEFAULTBINARY := 458,
	OPCUAID_CREATESESSIONREQUEST_ENCODING_DEFAULTBINARY := 461,
	OPCUAID_CREATESESSIONRESPONSE_ENCODING_DEFAULTBINARY := 464,
	OPCUAID_USERIDENTITYTOKEN_ENCODING_DEFAULTBINARY := 318,
	OPCUAID_ANONYMOUSIDENTITYTOKEN_ENCODING_DEFAULTBINARY := 321,
	OPCUAID_USERNAMEIDENTITYTOKEN_ENCODING_DEFAULTBINARY := 324,
	OPCUAID_X509IDENTITYTOKEN_ENCODING_DEFAULTBINARY := 327,
	OPCUAID_ISSUEDIDENTITYTOKEN_ENCODING_DEFAULTBINARY := 940,
	OPCUAID_ACTIVATESESSIONREQUEST_ENCODING_DEFAULTBINARY := 467,
	OPCUAID_ACTIVATESESSIONRESPONSE_ENCODING_DEFAULTBINARY := 470,
	OPCUAID_CLOSESESSIONREQUEST_ENCODING_DEFAULTBINARY := 473,
	OPCUAID_CLOSESESSIONRESPONSE_ENCODING_DEFAULTBINARY := 476,
	OPCUAID_CANCELREQUEST_ENCODING_DEFAULTBINARY := 479,
	OPCUAID_CANCELRESPONSE_ENCODING_DEFAULTBINARY := 482,
	OPCUAID_NODEATTRIBUTES_ENCODING_DEFAULTBINARY := 351,
	OPCUAID_OBJECTATTRIBUTES_ENCODING_DEFAULTBINARY := 354,
	OPCUAID_VARIABLEATTRIBUTES_ENCODING_DEFAULTBINARY := 357,
	OPCUAID_METHODATTRIBUTES_ENCODING_DEFAULTBINARY := 360,
	OPCUAID_OBJECTTYPEATTRIBUTES_ENCODING_DEFAULTBINARY := 363,
	OPCUAID_VARIABLETYPEATTRIBUTES_ENCODING_DEFAULTBINARY := 366,
	OPCUAID_REFERENCETYPEATTRIBUTES_ENCODING_DEFAULTBINARY := 369,
	OPCUAID_DATATYPEATTRIBUTES_ENCODING_DEFAULTBINARY := 372,
	OPCUAID_VIEWATTRIBUTES_ENCODING_DEFAULTBINARY := 375,
	OPCUAID_GENERICATTRIBUTEVALUE_ENCODING_DEFAULTBINARY := 17610,
	OPCUAID_GENERICATTRIBUTES_ENCODING_DEFAULTBINARY := 17611,
	OPCUAID_ADDNODESITEM_ENCODING_DEFAULTBINARY := 378,
	OPCUAID_ADDNODESRESULT_ENCODING_DEFAULTBINARY := 485,
	OPCUAID_ADDNODESREQUEST_ENCODING_DEFAULTBINARY := 488,
	OPCUAID_ADDNODESRESPONSE_ENCODING_DEFAULTBINARY := 491,
	OPCUAID_ADDREFERENCESITEM_ENCODING_DEFAULTBINARY := 381,
	OPCUAID_ADDREFERENCESREQUEST_ENCODING_DEFAULTBINARY := 494,
	OPCUAID_ADDREFERENCESRESPONSE_ENCODING_DEFAULTBINARY := 497,
	OPCUAID_DELETENODESITEM_ENCODING_DEFAULTBINARY := 384,
	OPCUAID_DELETENODESREQUEST_ENCODING_DEFAULTBINARY := 500,
	OPCUAID_DELETENODESRESPONSE_ENCODING_DEFAULTBINARY := 503,
	OPCUAID_DELETEREFERENCESITEM_ENCODING_DEFAULTBINARY := 387,
	OPCUAID_DELETEREFERENCESREQUEST_ENCODING_DEFAULTBINARY := 506,
	OPCUAID_DELETEREFERENCESRESPONSE_ENCODING_DEFAULTBINARY := 509,
	OPCUAID_VIEWDESCRIPTION_ENCODING_DEFAULTBINARY := 513,
	OPCUAID_BROWSEDESCRIPTION_ENCODING_DEFAULTBINARY := 516,
	OPCUAID_REFERENCEDESCRIPTION_ENCODING_DEFAULTBINARY := 520,
	OPCUAID_BROWSERESULT_ENCODING_DEFAULTBINARY := 524,
	OPCUAID_BROWSEREQUEST_ENCODING_DEFAULTBINARY := 527,
	OPCUAID_BROWSERESPONSE_ENCODING_DEFAULTBINARY := 530,
	OPCUAID_BROWSENEXTREQUEST_ENCODING_DEFAULTBINARY := 533,
	OPCUAID_BROWSENEXTRESPONSE_ENCODING_DEFAULTBINARY := 536,
	OPCUAID_RELATIVEPATHELEMENT_ENCODING_DEFAULTBINARY := 539,
	OPCUAID_RELATIVEPATH_ENCODING_DEFAULTBINARY := 542,
	OPCUAID_BROWSEPATH_ENCODING_DEFAULTBINARY := 545,
	OPCUAID_BROWSEPATHTARGET_ENCODING_DEFAULTBINARY := 548,
	OPCUAID_BROWSEPATHRESULT_ENCODING_DEFAULTBINARY := 551,
	OPCUAID_TRANSLATEBROWSEPATHSTONODEIDSREQUEST_ENCODING_DEFAULTBINARY := 554,
	OPCUAID_TRANSLATEBROWSEPATHSTONODEIDSRESPONSE_ENCODING_DEFAULTBINARY := 557,
	OPCUAID_REGISTERNODESREQUEST_ENCODING_DEFAULTBINARY := 560,
	OPCUAID_REGISTERNODESRESPONSE_ENCODING_DEFAULTBINARY := 563,
	OPCUAID_UNREGISTERNODESREQUEST_ENCODING_DEFAULTBINARY := 566,
	OPCUAID_UNREGISTERNODESRESPONSE_ENCODING_DEFAULTBINARY := 569,
	OPCUAID_ENDPOINTCONFIGURATION_ENCODING_DEFAULTBINARY := 333,
	OPCUAID_QUERYDATADESCRIPTION_ENCODING_DEFAULTBINARY := 572,
	OPCUAID_NODETYPEDESCRIPTION_ENCODING_DEFAULTBINARY := 575,
	OPCUAID_QUERYDATASET_ENCODING_DEFAULTBINARY := 579,
	OPCUAID_NODEREFERENCE_ENCODING_DEFAULTBINARY := 582,
	OPCUAID_CONTENTFILTERELEMENT_ENCODING_DEFAULTBINARY := 585,
	OPCUAID_CONTENTFILTER_ENCODING_DEFAULTBINARY := 588,
	OPCUAID_FILTEROPERAND_ENCODING_DEFAULTBINARY := 591,
	OPCUAID_ELEMENTOPERAND_ENCODING_DEFAULTBINARY := 594,
	OPCUAID_LITERALOPERAND_ENCODING_DEFAULTBINARY := 597,
	OPCUAID_ATTRIBUTEOPERAND_ENCODING_DEFAULTBINARY := 600,
	OPCUAID_SIMPLEATTRIBUTEOPERAND_ENCODING_DEFAULTBINARY := 603,
	OPCUAID_CONTENTFILTERELEMENTRESULT_ENCODING_DEFAULTBINARY := 606,
	OPCUAID_CONTENTFILTERRESULT_ENCODING_DEFAULTBINARY := 609,
	OPCUAID_PARSINGRESULT_ENCODING_DEFAULTBINARY := 612,
	OPCUAID_QUERYFIRSTREQUEST_ENCODING_DEFAULTBINARY := 615,
	OPCUAID_QUERYFIRSTRESPONSE_ENCODING_DEFAULTBINARY := 618,
	OPCUAID_QUERYNEXTREQUEST_ENCODING_DEFAULTBINARY := 621,
	OPCUAID_QUERYNEXTRESPONSE_ENCODING_DEFAULTBINARY := 624,
	OPCUAID_READVALUEID_ENCODING_DEFAULTBINARY := 628,
	OPCUAID_READREQUEST_ENCODING_DEFAULTBINARY := 631,
	OPCUAID_READRESPONSE_ENCODING_DEFAULTBINARY := 634,
	OPCUAID_HISTORYREADVALUEID_ENCODING_DEFAULTBINARY := 637,
	OPCUAID_HISTORYREADRESULT_ENCODING_DEFAULTBINARY := 640,
	OPCUAID_HISTORYREADDETAILS_ENCODING_DEFAULTBINARY := 643,
	OPCUAID_READEVENTDETAILS_ENCODING_DEFAULTBINARY := 646,
	OPCUAID_READRAWMODIFIEDDETAILS_ENCODING_DEFAULTBINARY := 649,
	OPCUAID_READPROCESSEDDETAILS_ENCODING_DEFAULTBINARY := 652,
	OPCUAID_READATTIMEDETAILS_ENCODING_DEFAULTBINARY := 655,
	OPCUAID_HISTORYDATA_ENCODING_DEFAULTBINARY := 658,
	OPCUAID_MODIFICATIONINFO_ENCODING_DEFAULTBINARY := 11226,
	OPCUAID_HISTORYMODIFIEDDATA_ENCODING_DEFAULTBINARY := 11227,
	OPCUAID_HISTORYEVENT_ENCODING_DEFAULTBINARY := 661,
	OPCUAID_HISTORYREADREQUEST_ENCODING_DEFAULTBINARY := 664,
	OPCUAID_HISTORYREADRESPONSE_ENCODING_DEFAULTBINARY := 667,
	OPCUAID_WRITEVALUE_ENCODING_DEFAULTBINARY := 670,
	OPCUAID_WRITEREQUEST_ENCODING_DEFAULTBINARY := 673,
	OPCUAID_WRITERESPONSE_ENCODING_DEFAULTBINARY := 676,
	OPCUAID_HISTORYUPDATEDETAILS_ENCODING_DEFAULTBINARY := 679,
	OPCUAID_UPDATEDATADETAILS_ENCODING_DEFAULTBINARY := 682,
	OPCUAID_UPDATESTRUCTUREDATADETAILS_ENCODING_DEFAULTBINARY := 11300,
	OPCUAID_UPDATEEVENTDETAILS_ENCODING_DEFAULTBINARY := 685,
	OPCUAID_DELETERAWMODIFIEDDETAILS_ENCODING_DEFAULTBINARY := 688,
	OPCUAID_DELETEATTIMEDETAILS_ENCODING_DEFAULTBINARY := 691,
	OPCUAID_DELETEEVENTDETAILS_ENCODING_DEFAULTBINARY := 694,
	OPCUAID_HISTORYUPDATERESULT_ENCODING_DEFAULTBINARY := 697,
	OPCUAID_HISTORYUPDATEREQUEST_ENCODING_DEFAULTBINARY := 700,
	OPCUAID_HISTORYUPDATERESPONSE_ENCODING_DEFAULTBINARY := 703,
	OPCUAID_CALLMETHODREQUEST_ENCODING_DEFAULTBINARY := 706,
	OPCUAID_CALLMETHODRESULT_ENCODING_DEFAULTBINARY := 709,
	OPCUAID_CALLREQUEST_ENCODING_DEFAULTBINARY := 712,
	OPCUAID_CALLRESPONSE_ENCODING_DEFAULTBINARY := 715,
	OPCUAID_MONITORINGFILTER_ENCODING_DEFAULTBINARY := 721,
	OPCUAID_DATACHANGEFILTER_ENCODING_DEFAULTBINARY := 724,
	OPCUAID_EVENTFILTER_ENCODING_DEFAULTBINARY := 727,
	OPCUAID_AGGREGATECONFIGURATION_ENCODING_DEFAULTBINARY := 950,
	OPCUAID_AGGREGATEFILTER_ENCODING_DEFAULTBINARY := 730,
	OPCUAID_MONITORINGFILTERRESULT_ENCODING_DEFAULTBINARY := 733,
	OPCUAID_EVENTFILTERRESULT_ENCODING_DEFAULTBINARY := 736,
	OPCUAID_AGGREGATEFILTERRESULT_ENCODING_DEFAULTBINARY := 739,
	OPCUAID_MONITORINGPARAMETERS_ENCODING_DEFAULTBINARY := 742,
	OPCUAID_MONITOREDITEMCREATEREQUEST_ENCODING_DEFAULTBINARY := 745,
	OPCUAID_MONITOREDITEMCREATERESULT_ENCODING_DEFAULTBINARY := 748,
	OPCUAID_CREATEMONITOREDITEMSREQUEST_ENCODING_DEFAULTBINARY := 751,
	OPCUAID_CREATEMONITOREDITEMSRESPONSE_ENCODING_DEFAULTBINARY := 754,
	OPCUAID_MONITOREDITEMMODIFYREQUEST_ENCODING_DEFAULTBINARY := 757,
	OPCUAID_MONITOREDITEMMODIFYRESULT_ENCODING_DEFAULTBINARY := 760,
	OPCUAID_MODIFYMONITOREDITEMSREQUEST_ENCODING_DEFAULTBINARY := 763,
	OPCUAID_MODIFYMONITOREDITEMSRESPONSE_ENCODING_DEFAULTBINARY := 766,
	OPCUAID_SETMONITORINGMODEREQUEST_ENCODING_DEFAULTBINARY := 769,
	OPCUAID_SETMONITORINGMODERESPONSE_ENCODING_DEFAULTBINARY := 772,
	OPCUAID_SETTRIGGERINGREQUEST_ENCODING_DEFAULTBINARY := 775,
	OPCUAID_SETTRIGGERINGRESPONSE_ENCODING_DEFAULTBINARY := 778,
	OPCUAID_DELETEMONITOREDITEMSREQUEST_ENCODING_DEFAULTBINARY := 781,
	OPCUAID_DELETEMONITOREDITEMSRESPONSE_ENCODING_DEFAULTBINARY := 784,
	OPCUAID_CREATESUBSCRIPTIONREQUEST_ENCODING_DEFAULTBINARY := 787,
	OPCUAID_CREATESUBSCRIPTIONRESPONSE_ENCODING_DEFAULTBINARY := 790,
	OPCUAID_MODIFYSUBSCRIPTIONREQUEST_ENCODING_DEFAULTBINARY := 793,
	OPCUAID_MODIFYSUBSCRIPTIONRESPONSE_ENCODING_DEFAULTBINARY := 796,
	OPCUAID_SETPUBLISHINGMODEREQUEST_ENCODING_DEFAULTBINARY := 799,
	OPCUAID_SETPUBLISHINGMODERESPONSE_ENCODING_DEFAULTBINARY := 802,
	OPCUAID_NOTIFICATIONMESSAGE_ENCODING_DEFAULTBINARY := 805,
	OPCUAID_NOTIFICATIONDATA_ENCODING_DEFAULTBINARY := 947,
	OPCUAID_DATACHANGENOTIFICATION_ENCODING_DEFAULTBINARY := 811,
	OPCUAID_MONITOREDITEMNOTIFICATION_ENCODING_DEFAULTBINARY := 808,
	OPCUAID_EVENTNOTIFICATIONLIST_ENCODING_DEFAULTBINARY := 916,
	OPCUAID_EVENTFIELDLIST_ENCODING_DEFAULTBINARY := 919,
	OPCUAID_HISTORYEVENTFIELDLIST_ENCODING_DEFAULTBINARY := 922,
	OPCUAID_STATUSCHANGENOTIFICATION_ENCODING_DEFAULTBINARY := 820,
	OPCUAID_SUBSCRIPTIONACKNOWLEDGEMENT_ENCODING_DEFAULTBINARY := 823,
	OPCUAID_PUBLISHREQUEST_ENCODING_DEFAULTBINARY := 826,
	OPCUAID_PUBLISHRESPONSE_ENCODING_DEFAULTBINARY := 829,
	OPCUAID_REPUBLISHREQUEST_ENCODING_DEFAULTBINARY := 832,
	OPCUAID_REPUBLISHRESPONSE_ENCODING_DEFAULTBINARY := 835,
	OPCUAID_TRANSFERRESULT_ENCODING_DEFAULTBINARY := 838,
	OPCUAID_TRANSFERSUBSCRIPTIONSREQUEST_ENCODING_DEFAULTBINARY := 841,
	OPCUAID_TRANSFERSUBSCRIPTIONSRESPONSE_ENCODING_DEFAULTBINARY := 844,
	OPCUAID_DELETESUBSCRIPTIONSREQUEST_ENCODING_DEFAULTBINARY := 847,
	OPCUAID_DELETESUBSCRIPTIONSRESPONSE_ENCODING_DEFAULTBINARY := 850,
	OPCUAID_BUILDINFO_ENCODING_DEFAULTBINARY := 340,
	OPCUAID_REDUNDANTSERVERDATATYPE_ENCODING_DEFAULTBINARY := 855,
	OPCUAID_ENDPOINTURLLISTDATATYPE_ENCODING_DEFAULTBINARY := 11957,
	OPCUAID_NETWORKGROUPDATATYPE_ENCODING_DEFAULTBINARY := 11958,
	OPCUAID_SAMPLINGINTERVALDIAGNOSTICSDATATYPE_ENCODING_DEFAULTBINARY := 858,
	OPCUAID_SERVERDIAGNOSTICSSUMMARYDATATYPE_ENCODING_DEFAULTBINARY := 861,
	OPCUAID_SERVERSTATUSDATATYPE_ENCODING_DEFAULTBINARY := 864,
	OPCUAID_SESSIONDIAGNOSTICSDATATYPE_ENCODING_DEFAULTBINARY := 867,
	OPCUAID_SESSIONSECURITYDIAGNOSTICSDATATYPE_ENCODING_DEFAULTBINARY := 870,
	OPCUAID_SERVICECOUNTERDATATYPE_ENCODING_DEFAULTBINARY := 873,
	OPCUAID_STATUSRESULT_ENCODING_DEFAULTBINARY := 301,
	OPCUAID_SUBSCRIPTIONDIAGNOSTICSDATATYPE_ENCODING_DEFAULTBINARY := 876,
	OPCUAID_MODELCHANGESTRUCTUREDATATYPE_ENCODING_DEFAULTBINARY := 879,
	OPCUAID_SEMANTICCHANGESTRUCTUREDATATYPE_ENCODING_DEFAULTBINARY := 899,
	OPCUAID_RANGE_ENCODING_DEFAULTBINARY := 886,
	OPCUAID_EUINFORMATION_ENCODING_DEFAULTBINARY := 889,
	OPCUAID_COMPLEXNUMBERTYPE_ENCODING_DEFAULTBINARY := 12181,
	OPCUAID_DOUBLECOMPLEXNUMBERTYPE_ENCODING_DEFAULTBINARY := 12182,
	OPCUAID_AXISINFORMATION_ENCODING_DEFAULTBINARY := 12089,
	OPCUAID_XVTYPE_ENCODING_DEFAULTBINARY := 12090,
	OPCUAID_PROGRAMDIAGNOSTICDATATYPE_ENCODING_DEFAULTBINARY := 896,
	OPCUAID_PROGRAMDIAGNOSTIC2DATATYPE_ENCODING_DEFAULTBINARY := 15397,
	OPCUAID_ANNOTATION_ENCODING_DEFAULTBINARY := 893,
	OPCUAID_KEYVALUEPAIR_ENCODING_DEFAULTXML := 14802,
	OPCUAID_ENDPOINTTYPE_ENCODING_DEFAULTXML := 15949,
	OPCUAID_IDENTITYMAPPINGRULETYPE_ENCODING_DEFAULTXML := 15728,
	OPCUAID_TRUSTLISTDATATYPE_ENCODING_DEFAULTXML := 12676,
	OPCUAID_DECIMALDATATYPE_ENCODING_DEFAULTXML := 17862,
	OPCUAID_DATATYPESCHEMAHEADER_ENCODING_DEFAULTXML := 15950,
	OPCUAID_DATATYPEDESCRIPTION_ENCODING_DEFAULTXML := 14796,
	OPCUAID_STRUCTUREDESCRIPTION_ENCODING_DEFAULTXML := 15589,
	OPCUAID_ENUMDESCRIPTION_ENCODING_DEFAULTXML := 15590,
	OPCUAID_SIMPLETYPEDESCRIPTION_ENCODING_DEFAULTXML := 15529,
	OPCUAID_UABINARYFILEDATATYPE_ENCODING_DEFAULTXML := 15531,
	OPCUAID_DATASETMETADATATYPE_ENCODING_DEFAULTXML := 14794,
	OPCUAID_FIELDMETADATA_ENCODING_DEFAULTXML := 14795,
	OPCUAID_CONFIGURATIONVERSIONDATATYPE_ENCODING_DEFAULTXML := 14803,
	OPCUAID_PUBLISHEDDATASETDATATYPE_ENCODING_DEFAULTXML := 15951,
	OPCUAID_PUBLISHEDDATASETSOURCEDATATYPE_ENCODING_DEFAULTXML := 15952,
	OPCUAID_PUBLISHEDVARIABLEDATATYPE_ENCODING_DEFAULTXML := 14319,
	OPCUAID_PUBLISHEDDATAITEMSDATATYPE_ENCODING_DEFAULTXML := 15953,
	OPCUAID_PUBLISHEDEVENTSDATATYPE_ENCODING_DEFAULTXML := 15954,
	OPCUAID_DATASETWRITERDATATYPE_ENCODING_DEFAULTXML := 15955,
	OPCUAID_DATASETWRITERTRANSPORTDATATYPE_ENCODING_DEFAULTXML := 15956,
	OPCUAID_DATASETWRITERMESSAGEDATATYPE_ENCODING_DEFAULTXML := 15987,
	OPCUAID_PUBSUBGROUPDATATYPE_ENCODING_DEFAULTXML := 15988,
	OPCUAID_WRITERGROUPDATATYPE_ENCODING_DEFAULTXML := 21174,
	OPCUAID_WRITERGROUPTRANSPORTDATATYPE_ENCODING_DEFAULTXML := 15990,
	OPCUAID_WRITERGROUPMESSAGEDATATYPE_ENCODING_DEFAULTXML := 15991,
	OPCUAID_PUBSUBCONNECTIONDATATYPE_ENCODING_DEFAULTXML := 15992,
	OPCUAID_CONNECTIONTRANSPORTDATATYPE_ENCODING_DEFAULTXML := 15993,
	OPCUAID_NETWORKADDRESSDATATYPE_ENCODING_DEFAULTXML := 21175,
	OPCUAID_NETWORKADDRESSURLDATATYPE_ENCODING_DEFAULTXML := 21176,
	OPCUAID_READERGROUPDATATYPE_ENCODING_DEFAULTXML := 21177,
	OPCUAID_READERGROUPTRANSPORTDATATYPE_ENCODING_DEFAULTXML := 15995,
	OPCUAID_READERGROUPMESSAGEDATATYPE_ENCODING_DEFAULTXML := 15996,
	OPCUAID_DATASETREADERDATATYPE_ENCODING_DEFAULTXML := 16007,
	OPCUAID_DATASETREADERTRANSPORTDATATYPE_ENCODING_DEFAULTXML := 16008,
	OPCUAID_DATASETREADERMESSAGEDATATYPE_ENCODING_DEFAULTXML := 16009,
	OPCUAID_SUBSCRIBEDDATASETDATATYPE_ENCODING_DEFAULTXML := 16010,
	OPCUAID_TARGETVARIABLESDATATYPE_ENCODING_DEFAULTXML := 16011,
	OPCUAID_FIELDTARGETDATATYPE_ENCODING_DEFAULTXML := 14804,
	OPCUAID_SUBSCRIBEDDATASETMIRRORDATATYPE_ENCODING_DEFAULTXML := 16012,
	OPCUAID_PUBSUBCONFIGURATIONDATATYPE_ENCODING_DEFAULTXML := 21178,
	OPCUAID_UADPWRITERGROUPMESSAGEDATATYPE_ENCODING_DEFAULTXML := 16014,
	OPCUAID_UADPDATASETWRITERMESSAGEDATATYPE_ENCODING_DEFAULTXML := 16015,
	OPCUAID_UADPDATASETREADERMESSAGEDATATYPE_ENCODING_DEFAULTXML := 16016,
	OPCUAID_JSONWRITERGROUPMESSAGEDATATYPE_ENCODING_DEFAULTXML := 16017,
	OPCUAID_JSONDATASETWRITERMESSAGEDATATYPE_ENCODING_DEFAULTXML := 16018,
	OPCUAID_JSONDATASETREADERMESSAGEDATATYPE_ENCODING_DEFAULTXML := 16019,
	OPCUAID_DATAGRAMCONNECTIONTRANSPORTDATATYPE_ENCODING_DEFAULTXML := 17472,
	OPCUAID_DATAGRAMWRITERGROUPTRANSPORTDATATYPE_ENCODING_DEFAULTXML := 21179,
	OPCUAID_BROKERCONNECTIONTRANSPORTDATATYPE_ENCODING_DEFAULTXML := 15579,
	OPCUAID_BROKERWRITERGROUPTRANSPORTDATATYPE_ENCODING_DEFAULTXML := 16021,
	OPCUAID_BROKERDATASETWRITERTRANSPORTDATATYPE_ENCODING_DEFAULTXML := 16022,
	OPCUAID_BROKERDATASETREADERTRANSPORTDATATYPE_ENCODING_DEFAULTXML := 16023,
	OPCUAID_ROLEPERMISSIONTYPE_ENCODING_DEFAULTXML := 16126,
	OPCUAID_DATATYPEDEFINITION_ENCODING_DEFAULTXML := 14797,
	OPCUAID_STRUCTUREFIELD_ENCODING_DEFAULTXML := 14800,
	OPCUAID_STRUCTUREDEFINITION_ENCODING_DEFAULTXML := 14798,
	OPCUAID_ENUMDEFINITION_ENCODING_DEFAULTXML := 14799,
	OPCUAID_NODE_ENCODING_DEFAULTXML := 259,
	OPCUAID_INSTANCENODE_ENCODING_DEFAULTXML := 11887,
	OPCUAID_TYPENODE_ENCODING_DEFAULTXML := 11888,
	OPCUAID_OBJECTNODE_ENCODING_DEFAULTXML := 262,
	OPCUAID_OBJECTTYPENODE_ENCODING_DEFAULTXML := 265,
	OPCUAID_VARIABLENODE_ENCODING_DEFAULTXML := 268,
	OPCUAID_VARIABLETYPENODE_ENCODING_DEFAULTXML := 271,
	OPCUAID_REFERENCETYPENODE_ENCODING_DEFAULTXML := 274,
	OPCUAID_METHODNODE_ENCODING_DEFAULTXML := 277,
	OPCUAID_VIEWNODE_ENCODING_DEFAULTXML := 280,
	OPCUAID_DATATYPENODE_ENCODING_DEFAULTXML := 283,
	OPCUAID_REFERENCENODE_ENCODING_DEFAULTXML := 286,
	OPCUAID_ARGUMENT_ENCODING_DEFAULTXML := 297,
	OPCUAID_ENUMVALUETYPE_ENCODING_DEFAULTXML := 7616,
	OPCUAID_ENUMFIELD_ENCODING_DEFAULTXML := 14801,
	OPCUAID_OPTIONSET_ENCODING_DEFAULTXML := 12757,
	OPCUAID_UNION_ENCODING_DEFAULTXML := 12758,
	OPCUAID_TIMEZONEDATATYPE_ENCODING_DEFAULTXML := 8913,
	OPCUAID_APPLICATIONDESCRIPTION_ENCODING_DEFAULTXML := 309,
	OPCUAID_REQUESTHEADER_ENCODING_DEFAULTXML := 390,
	OPCUAID_RESPONSEHEADER_ENCODING_DEFAULTXML := 393,
	OPCUAID_SERVICEFAULT_ENCODING_DEFAULTXML := 396,
	OPCUAID_SESSIONLESSINVOKEREQUESTTYPE_ENCODING_DEFAULTXML := 15902,
	OPCUAID_SESSIONLESSINVOKERESPONSETYPE_ENCODING_DEFAULTXML := 21000,
	OPCUAID_FINDSERVERSREQUEST_ENCODING_DEFAULTXML := 421,
	OPCUAID_FINDSERVERSRESPONSE_ENCODING_DEFAULTXML := 424,
	OPCUAID_SERVERONNETWORK_ENCODING_DEFAULTXML := 12195,
	OPCUAID_FINDSERVERSONNETWORKREQUEST_ENCODING_DEFAULTXML := 12196,
	OPCUAID_FINDSERVERSONNETWORKRESPONSE_ENCODING_DEFAULTXML := 12197,
	OPCUAID_USERTOKENPOLICY_ENCODING_DEFAULTXML := 305,
	OPCUAID_ENDPOINTDESCRIPTION_ENCODING_DEFAULTXML := 313,
	OPCUAID_GETENDPOINTSREQUEST_ENCODING_DEFAULTXML := 427,
	OPCUAID_GETENDPOINTSRESPONSE_ENCODING_DEFAULTXML := 430,
	OPCUAID_REGISTEREDSERVER_ENCODING_DEFAULTXML := 433,
	OPCUAID_REGISTERSERVERREQUEST_ENCODING_DEFAULTXML := 436,
	OPCUAID_REGISTERSERVERRESPONSE_ENCODING_DEFAULTXML := 439,
	OPCUAID_DISCOVERYCONFIGURATION_ENCODING_DEFAULTXML := 12892,
	OPCUAID_MDNSDISCOVERYCONFIGURATION_ENCODING_DEFAULTXML := 12893,
	OPCUAID_REGISTERSERVER2REQUEST_ENCODING_DEFAULTXML := 12199,
	OPCUAID_REGISTERSERVER2RESPONSE_ENCODING_DEFAULTXML := 12200,
	OPCUAID_CHANNELSECURITYTOKEN_ENCODING_DEFAULTXML := 442,
	OPCUAID_OPENSECURECHANNELREQUEST_ENCODING_DEFAULTXML := 445,
	OPCUAID_OPENSECURECHANNELRESPONSE_ENCODING_DEFAULTXML := 448,
	OPCUAID_CLOSESECURECHANNELREQUEST_ENCODING_DEFAULTXML := 451,
	OPCUAID_CLOSESECURECHANNELRESPONSE_ENCODING_DEFAULTXML := 454,
	OPCUAID_SIGNEDSOFTWARECERTIFICATE_ENCODING_DEFAULTXML := 345,
	OPCUAID_SIGNATUREDATA_ENCODING_DEFAULTXML := 457,
	OPCUAID_CREATESESSIONREQUEST_ENCODING_DEFAULTXML := 460,
	OPCUAID_CREATESESSIONRESPONSE_ENCODING_DEFAULTXML := 463,
	OPCUAID_USERIDENTITYTOKEN_ENCODING_DEFAULTXML := 317,
	OPCUAID_ANONYMOUSIDENTITYTOKEN_ENCODING_DEFAULTXML := 320,
	OPCUAID_USERNAMEIDENTITYTOKEN_ENCODING_DEFAULTXML := 323,
	OPCUAID_X509IDENTITYTOKEN_ENCODING_DEFAULTXML := 326,
	OPCUAID_ISSUEDIDENTITYTOKEN_ENCODING_DEFAULTXML := 939,
	OPCUAID_ACTIVATESESSIONREQUEST_ENCODING_DEFAULTXML := 466,
	OPCUAID_ACTIVATESESSIONRESPONSE_ENCODING_DEFAULTXML := 469,
	OPCUAID_CLOSESESSIONREQUEST_ENCODING_DEFAULTXML := 472,
	OPCUAID_CLOSESESSIONRESPONSE_ENCODING_DEFAULTXML := 475,
	OPCUAID_CANCELREQUEST_ENCODING_DEFAULTXML := 478,
	OPCUAID_CANCELRESPONSE_ENCODING_DEFAULTXML := 481,
	OPCUAID_NODEATTRIBUTES_ENCODING_DEFAULTXML := 350,
	OPCUAID_OBJECTATTRIBUTES_ENCODING_DEFAULTXML := 353,
	OPCUAID_VARIABLEATTRIBUTES_ENCODING_DEFAULTXML := 356,
	OPCUAID_METHODATTRIBUTES_ENCODING_DEFAULTXML := 359,
	OPCUAID_OBJECTTYPEATTRIBUTES_ENCODING_DEFAULTXML := 362,
	OPCUAID_VARIABLETYPEATTRIBUTES_ENCODING_DEFAULTXML := 365,
	OPCUAID_REFERENCETYPEATTRIBUTES_ENCODING_DEFAULTXML := 368,
	OPCUAID_DATATYPEATTRIBUTES_ENCODING_DEFAULTXML := 371,
	OPCUAID_VIEWATTRIBUTES_ENCODING_DEFAULTXML := 374,
	OPCUAID_GENERICATTRIBUTEVALUE_ENCODING_DEFAULTXML := 17608,
	OPCUAID_GENERICATTRIBUTES_ENCODING_DEFAULTXML := 17609,
	OPCUAID_ADDNODESITEM_ENCODING_DEFAULTXML := 377,
	OPCUAID_ADDNODESRESULT_ENCODING_DEFAULTXML := 484,
	OPCUAID_ADDNODESREQUEST_ENCODING_DEFAULTXML := 487,
	OPCUAID_ADDNODESRESPONSE_ENCODING_DEFAULTXML := 490,
	OPCUAID_ADDREFERENCESITEM_ENCODING_DEFAULTXML := 380,
	OPCUAID_ADDREFERENCESREQUEST_ENCODING_DEFAULTXML := 493,
	OPCUAID_ADDREFERENCESRESPONSE_ENCODING_DEFAULTXML := 496,
	OPCUAID_DELETENODESITEM_ENCODING_DEFAULTXML := 383,
	OPCUAID_DELETENODESREQUEST_ENCODING_DEFAULTXML := 499,
	OPCUAID_DELETENODESRESPONSE_ENCODING_DEFAULTXML := 502,
	OPCUAID_DELETEREFERENCESITEM_ENCODING_DEFAULTXML := 386,
	OPCUAID_DELETEREFERENCESREQUEST_ENCODING_DEFAULTXML := 505,
	OPCUAID_DELETEREFERENCESRESPONSE_ENCODING_DEFAULTXML := 508,
	OPCUAID_VIEWDESCRIPTION_ENCODING_DEFAULTXML := 512,
	OPCUAID_BROWSEDESCRIPTION_ENCODING_DEFAULTXML := 515,
	OPCUAID_REFERENCEDESCRIPTION_ENCODING_DEFAULTXML := 519,
	OPCUAID_BROWSERESULT_ENCODING_DEFAULTXML := 523,
	OPCUAID_BROWSEREQUEST_ENCODING_DEFAULTXML := 526,
	OPCUAID_BROWSERESPONSE_ENCODING_DEFAULTXML := 529,
	OPCUAID_BROWSENEXTREQUEST_ENCODING_DEFAULTXML := 532,
	OPCUAID_BROWSENEXTRESPONSE_ENCODING_DEFAULTXML := 535,
	OPCUAID_RELATIVEPATHELEMENT_ENCODING_DEFAULTXML := 538,
	OPCUAID_RELATIVEPATH_ENCODING_DEFAULTXML := 541,
	OPCUAID_BROWSEPATH_ENCODING_DEFAULTXML := 544,
	OPCUAID_BROWSEPATHTARGET_ENCODING_DEFAULTXML := 547,
	OPCUAID_BROWSEPATHRESULT_ENCODING_DEFAULTXML := 550,
	OPCUAID_TRANSLATEBROWSEPATHSTONODEIDSREQUEST_ENCODING_DEFAULTXML := 553,
	OPCUAID_TRANSLATEBROWSEPATHSTONODEIDSRESPONSE_ENCODING_DEFAULTXML := 556,
	OPCUAID_REGISTERNODESREQUEST_ENCODING_DEFAULTXML := 559,
	OPCUAID_REGISTERNODESRESPONSE_ENCODING_DEFAULTXML := 562,
	OPCUAID_UNREGISTERNODESREQUEST_ENCODING_DEFAULTXML := 565,
	OPCUAID_UNREGISTERNODESRESPONSE_ENCODING_DEFAULTXML := 568,
	OPCUAID_ENDPOINTCONFIGURATION_ENCODING_DEFAULTXML := 332,
	OPCUAID_QUERYDATADESCRIPTION_ENCODING_DEFAULTXML := 571,
	OPCUAID_NODETYPEDESCRIPTION_ENCODING_DEFAULTXML := 574,
	OPCUAID_QUERYDATASET_ENCODING_DEFAULTXML := 578,
	OPCUAID_NODEREFERENCE_ENCODING_DEFAULTXML := 581,
	OPCUAID_CONTENTFILTERELEMENT_ENCODING_DEFAULTXML := 584,
	OPCUAID_CONTENTFILTER_ENCODING_DEFAULTXML := 587,
	OPCUAID_FILTEROPERAND_ENCODING_DEFAULTXML := 590,
	OPCUAID_ELEMENTOPERAND_ENCODING_DEFAULTXML := 593,
	OPCUAID_LITERALOPERAND_ENCODING_DEFAULTXML := 596,
	OPCUAID_ATTRIBUTEOPERAND_ENCODING_DEFAULTXML := 599,
	OPCUAID_SIMPLEATTRIBUTEOPERAND_ENCODING_DEFAULTXML := 602,
	OPCUAID_CONTENTFILTERELEMENTRESULT_ENCODING_DEFAULTXML := 605,
	OPCUAID_CONTENTFILTERRESULT_ENCODING_DEFAULTXML := 608,
	OPCUAID_PARSINGRESULT_ENCODING_DEFAULTXML := 611,
	OPCUAID_QUERYFIRSTREQUEST_ENCODING_DEFAULTXML := 614,
	OPCUAID_QUERYFIRSTRESPONSE_ENCODING_DEFAULTXML := 617,
	OPCUAID_QUERYNEXTREQUEST_ENCODING_DEFAULTXML := 620,
	OPCUAID_QUERYNEXTRESPONSE_ENCODING_DEFAULTXML := 623,
	OPCUAID_READVALUEID_ENCODING_DEFAULTXML := 627,
	OPCUAID_READREQUEST_ENCODING_DEFAULTXML := 630,
	OPCUAID_READRESPONSE_ENCODING_DEFAULTXML := 633,
	OPCUAID_HISTORYREADVALUEID_ENCODING_DEFAULTXML := 636,
	OPCUAID_HISTORYREADRESULT_ENCODING_DEFAULTXML := 639,
	OPCUAID_HISTORYREADDETAILS_ENCODING_DEFAULTXML := 642,
	OPCUAID_READEVENTDETAILS_ENCODING_DEFAULTXML := 645,
	OPCUAID_READRAWMODIFIEDDETAILS_ENCODING_DEFAULTXML := 648,
	OPCUAID_READPROCESSEDDETAILS_ENCODING_DEFAULTXML := 651,
	OPCUAID_READATTIMEDETAILS_ENCODING_DEFAULTXML := 654,
	OPCUAID_HISTORYDATA_ENCODING_DEFAULTXML := 657,
	OPCUAID_MODIFICATIONINFO_ENCODING_DEFAULTXML := 11218,
	OPCUAID_HISTORYMODIFIEDDATA_ENCODING_DEFAULTXML := 11219,
	OPCUAID_HISTORYEVENT_ENCODING_DEFAULTXML := 660,
	OPCUAID_HISTORYREADREQUEST_ENCODING_DEFAULTXML := 663,
	OPCUAID_HISTORYREADRESPONSE_ENCODING_DEFAULTXML := 666,
	OPCUAID_WRITEVALUE_ENCODING_DEFAULTXML := 669,
	OPCUAID_WRITEREQUEST_ENCODING_DEFAULTXML := 672,
	OPCUAID_WRITERESPONSE_ENCODING_DEFAULTXML := 675,
	OPCUAID_HISTORYUPDATEDETAILS_ENCODING_DEFAULTXML := 678,
	OPCUAID_UPDATEDATADETAILS_ENCODING_DEFAULTXML := 681,
	OPCUAID_UPDATESTRUCTUREDATADETAILS_ENCODING_DEFAULTXML := 11296,
	OPCUAID_UPDATEEVENTDETAILS_ENCODING_DEFAULTXML := 684,
	OPCUAID_DELETERAWMODIFIEDDETAILS_ENCODING_DEFAULTXML := 687,
	OPCUAID_DELETEATTIMEDETAILS_ENCODING_DEFAULTXML := 690,
	OPCUAID_DELETEEVENTDETAILS_ENCODING_DEFAULTXML := 693,
	OPCUAID_HISTORYUPDATERESULT_ENCODING_DEFAULTXML := 696,
	OPCUAID_HISTORYUPDATEREQUEST_ENCODING_DEFAULTXML := 699,
	OPCUAID_HISTORYUPDATERESPONSE_ENCODING_DEFAULTXML := 702,
	OPCUAID_CALLMETHODREQUEST_ENCODING_DEFAULTXML := 705,
	OPCUAID_CALLMETHODRESULT_ENCODING_DEFAULTXML := 708,
	OPCUAID_CALLREQUEST_ENCODING_DEFAULTXML := 711,
	OPCUAID_CALLRESPONSE_ENCODING_DEFAULTXML := 714,
	OPCUAID_MONITORINGFILTER_ENCODING_DEFAULTXML := 720,
	OPCUAID_DATACHANGEFILTER_ENCODING_DEFAULTXML := 723,
	OPCUAID_EVENTFILTER_ENCODING_DEFAULTXML := 726,
	OPCUAID_AGGREGATECONFIGURATION_ENCODING_DEFAULTXML := 949,
	OPCUAID_AGGREGATEFILTER_ENCODING_DEFAULTXML := 729,
	OPCUAID_MONITORINGFILTERRESULT_ENCODING_DEFAULTXML := 732,
	OPCUAID_EVENTFILTERRESULT_ENCODING_DEFAULTXML := 735,
	OPCUAID_AGGREGATEFILTERRESULT_ENCODING_DEFAULTXML := 738,
	OPCUAID_MONITORINGPARAMETERS_ENCODING_DEFAULTXML := 741,
	OPCUAID_MONITOREDITEMCREATEREQUEST_ENCODING_DEFAULTXML := 744,
	OPCUAID_MONITOREDITEMCREATERESULT_ENCODING_DEFAULTXML := 747,
	OPCUAID_CREATEMONITOREDITEMSREQUEST_ENCODING_DEFAULTXML := 750,
	OPCUAID_CREATEMONITOREDITEMSRESPONSE_ENCODING_DEFAULTXML := 753,
	OPCUAID_MONITOREDITEMMODIFYREQUEST_ENCODING_DEFAULTXML := 756,
	OPCUAID_MONITOREDITEMMODIFYRESULT_ENCODING_DEFAULTXML := 759,
	OPCUAID_MODIFYMONITOREDITEMSREQUEST_ENCODING_DEFAULTXML := 762,
	OPCUAID_MODIFYMONITOREDITEMSRESPONSE_ENCODING_DEFAULTXML := 765,
	OPCUAID_SETMONITORINGMODEREQUEST_ENCODING_DEFAULTXML := 768,
	OPCUAID_SETMONITORINGMODERESPONSE_ENCODING_DEFAULTXML := 771,
	OPCUAID_SETTRIGGERINGREQUEST_ENCODING_DEFAULTXML := 774,
	OPCUAID_SETTRIGGERINGRESPONSE_ENCODING_DEFAULTXML := 777,
	OPCUAID_DELETEMONITOREDITEMSREQUEST_ENCODING_DEFAULTXML := 780,
	OPCUAID_DELETEMONITOREDITEMSRESPONSE_ENCODING_DEFAULTXML := 783,
	OPCUAID_CREATESUBSCRIPTIONREQUEST_ENCODING_DEFAULTXML := 786,
	OPCUAID_CREATESUBSCRIPTIONRESPONSE_ENCODING_DEFAULTXML := 789,
	OPCUAID_MODIFYSUBSCRIPTIONREQUEST_ENCODING_DEFAULTXML := 792,
	OPCUAID_MODIFYSUBSCRIPTIONRESPONSE_ENCODING_DEFAULTXML := 795,
	OPCUAID_SETPUBLISHINGMODEREQUEST_ENCODING_DEFAULTXML := 798,
	OPCUAID_SETPUBLISHINGMODERESPONSE_ENCODING_DEFAULTXML := 801,
	OPCUAID_NOTIFICATIONMESSAGE_ENCODING_DEFAULTXML := 804,
	OPCUAID_NOTIFICATIONDATA_ENCODING_DEFAULTXML := 946,
	OPCUAID_DATACHANGENOTIFICATION_ENCODING_DEFAULTXML := 810,
	OPCUAID_MONITOREDITEMNOTIFICATION_ENCODING_DEFAULTXML := 807,
	OPCUAID_EVENTNOTIFICATIONLIST_ENCODING_DEFAULTXML := 915,
	OPCUAID_EVENTFIELDLIST_ENCODING_DEFAULTXML := 918,
	OPCUAID_HISTORYEVENTFIELDLIST_ENCODING_DEFAULTXML := 921,
	OPCUAID_STATUSCHANGENOTIFICATION_ENCODING_DEFAULTXML := 819,
	OPCUAID_SUBSCRIPTIONACKNOWLEDGEMENT_ENCODING_DEFAULTXML := 822,
	OPCUAID_PUBLISHREQUEST_ENCODING_DEFAULTXML := 825,
	OPCUAID_PUBLISHRESPONSE_ENCODING_DEFAULTXML := 828,
	OPCUAID_REPUBLISHREQUEST_ENCODING_DEFAULTXML := 831,
	OPCUAID_REPUBLISHRESPONSE_ENCODING_DEFAULTXML := 834,
	OPCUAID_TRANSFERRESULT_ENCODING_DEFAULTXML := 837,
	OPCUAID_TRANSFERSUBSCRIPTIONSREQUEST_ENCODING_DEFAULTXML := 840,
	OPCUAID_TRANSFERSUBSCRIPTIONSRESPONSE_ENCODING_DEFAULTXML := 843,
	OPCUAID_DELETESUBSCRIPTIONSREQUEST_ENCODING_DEFAULTXML := 846,
	OPCUAID_DELETESUBSCRIPTIONSRESPONSE_ENCODING_DEFAULTXML := 849,
	OPCUAID_BUILDINFO_ENCODING_DEFAULTXML := 339,
	OPCUAID_REDUNDANTSERVERDATATYPE_ENCODING_DEFAULTXML := 854,
	OPCUAID_ENDPOINTURLLISTDATATYPE_ENCODING_DEFAULTXML := 11949,
	OPCUAID_NETWORKGROUPDATATYPE_ENCODING_DEFAULTXML := 11950,
	OPCUAID_SAMPLINGINTERVALDIAGNOSTICSDATATYPE_ENCODING_DEFAULTXML := 857,
	OPCUAID_SERVERDIAGNOSTICSSUMMARYDATATYPE_ENCODING_DEFAULTXML := 860,
	OPCUAID_SERVERSTATUSDATATYPE_ENCODING_DEFAULTXML := 863,
	OPCUAID_SESSIONDIAGNOSTICSDATATYPE_ENCODING_DEFAULTXML := 866,
	OPCUAID_SESSIONSECURITYDIAGNOSTICSDATATYPE_ENCODING_DEFAULTXML := 869,
	OPCUAID_SERVICECOUNTERDATATYPE_ENCODING_DEFAULTXML := 872,
	OPCUAID_STATUSRESULT_ENCODING_DEFAULTXML := 300,
	OPCUAID_SUBSCRIPTIONDIAGNOSTICSDATATYPE_ENCODING_DEFAULTXML := 875,
	OPCUAID_MODELCHANGESTRUCTUREDATATYPE_ENCODING_DEFAULTXML := 878,
	OPCUAID_SEMANTICCHANGESTRUCTUREDATATYPE_ENCODING_DEFAULTXML := 898,
	OPCUAID_RANGE_ENCODING_DEFAULTXML := 885,
	OPCUAID_EUINFORMATION_ENCODING_DEFAULTXML := 888,
	OPCUAID_COMPLEXNUMBERTYPE_ENCODING_DEFAULTXML := 12173,
	OPCUAID_DOUBLECOMPLEXNUMBERTYPE_ENCODING_DEFAULTXML := 12174,
	OPCUAID_AXISINFORMATION_ENCODING_DEFAULTXML := 12081,
	OPCUAID_XVTYPE_ENCODING_DEFAULTXML := 12082,
	OPCUAID_PROGRAMDIAGNOSTICDATATYPE_ENCODING_DEFAULTXML := 895,
	OPCUAID_PROGRAMDIAGNOSTIC2DATATYPE_ENCODING_DEFAULTXML := 15401,
	OPCUAID_ANNOTATION_ENCODING_DEFAULTXML := 892,
	OPCUAID_KEYVALUEPAIR_ENCODING_DEFAULTJSON := 15041,
	OPCUAID_ENDPOINTTYPE_ENCODING_DEFAULTJSON := 16150,
	OPCUAID_IDENTITYMAPPINGRULETYPE_ENCODING_DEFAULTJSON := 15042,
	OPCUAID_TRUSTLISTDATATYPE_ENCODING_DEFAULTJSON := 15044,
	OPCUAID_DECIMALDATATYPE_ENCODING_DEFAULTJSON := 15045,
	OPCUAID_DATATYPESCHEMAHEADER_ENCODING_DEFAULTJSON := 16151,
	OPCUAID_DATATYPEDESCRIPTION_ENCODING_DEFAULTJSON := 15057,
	OPCUAID_STRUCTUREDESCRIPTION_ENCODING_DEFAULTJSON := 15058,
	OPCUAID_ENUMDESCRIPTION_ENCODING_DEFAULTJSON := 15059,
	OPCUAID_SIMPLETYPEDESCRIPTION_ENCODING_DEFAULTJSON := 15700,
	OPCUAID_UABINARYFILEDATATYPE_ENCODING_DEFAULTJSON := 15714,
	OPCUAID_DATASETMETADATATYPE_ENCODING_DEFAULTJSON := 15050,
	OPCUAID_FIELDMETADATA_ENCODING_DEFAULTJSON := 15051,
	OPCUAID_CONFIGURATIONVERSIONDATATYPE_ENCODING_DEFAULTJSON := 15049,
	OPCUAID_PUBLISHEDDATASETDATATYPE_ENCODING_DEFAULTJSON := 16152,
	OPCUAID_PUBLISHEDDATASETSOURCEDATATYPE_ENCODING_DEFAULTJSON := 16153,
	OPCUAID_PUBLISHEDVARIABLEDATATYPE_ENCODING_DEFAULTJSON := 15060,
	OPCUAID_PUBLISHEDDATAITEMSDATATYPE_ENCODING_DEFAULTJSON := 16154,
	OPCUAID_PUBLISHEDEVENTSDATATYPE_ENCODING_DEFAULTJSON := 16155,
	OPCUAID_DATASETWRITERDATATYPE_ENCODING_DEFAULTJSON := 16156,
	OPCUAID_DATASETWRITERTRANSPORTDATATYPE_ENCODING_DEFAULTJSON := 16157,
	OPCUAID_DATASETWRITERMESSAGEDATATYPE_ENCODING_DEFAULTJSON := 16158,
	OPCUAID_PUBSUBGROUPDATATYPE_ENCODING_DEFAULTJSON := 16159,
	OPCUAID_WRITERGROUPDATATYPE_ENCODING_DEFAULTJSON := 21198,
	OPCUAID_WRITERGROUPTRANSPORTDATATYPE_ENCODING_DEFAULTJSON := 16161,
	OPCUAID_WRITERGROUPMESSAGEDATATYPE_ENCODING_DEFAULTJSON := 16280,
	OPCUAID_PUBSUBCONNECTIONDATATYPE_ENCODING_DEFAULTJSON := 16281,
	OPCUAID_CONNECTIONTRANSPORTDATATYPE_ENCODING_DEFAULTJSON := 16282,
	OPCUAID_NETWORKADDRESSDATATYPE_ENCODING_DEFAULTJSON := 21199,
	OPCUAID_NETWORKADDRESSURLDATATYPE_ENCODING_DEFAULTJSON := 21200,
	OPCUAID_READERGROUPDATATYPE_ENCODING_DEFAULTJSON := 21201,
	OPCUAID_READERGROUPTRANSPORTDATATYPE_ENCODING_DEFAULTJSON := 16284,
	OPCUAID_READERGROUPMESSAGEDATATYPE_ENCODING_DEFAULTJSON := 16285,
	OPCUAID_DATASETREADERDATATYPE_ENCODING_DEFAULTJSON := 16286,
	OPCUAID_DATASETREADERTRANSPORTDATATYPE_ENCODING_DEFAULTJSON := 16287,
	OPCUAID_DATASETREADERMESSAGEDATATYPE_ENCODING_DEFAULTJSON := 16288,
	OPCUAID_SUBSCRIBEDDATASETDATATYPE_ENCODING_DEFAULTJSON := 16308,
	OPCUAID_TARGETVARIABLESDATATYPE_ENCODING_DEFAULTJSON := 16310,
	OPCUAID_FIELDTARGETDATATYPE_ENCODING_DEFAULTJSON := 15061,
	OPCUAID_SUBSCRIBEDDATASETMIRRORDATATYPE_ENCODING_DEFAULTJSON := 16311,
	OPCUAID_PUBSUBCONFIGURATIONDATATYPE_ENCODING_DEFAULTJSON := 21202,
	OPCUAID_UADPWRITERGROUPMESSAGEDATATYPE_ENCODING_DEFAULTJSON := 16323,
	OPCUAID_UADPDATASETWRITERMESSAGEDATATYPE_ENCODING_DEFAULTJSON := 16391,
	OPCUAID_UADPDATASETREADERMESSAGEDATATYPE_ENCODING_DEFAULTJSON := 16392,
	OPCUAID_JSONWRITERGROUPMESSAGEDATATYPE_ENCODING_DEFAULTJSON := 16393,
	OPCUAID_JSONDATASETWRITERMESSAGEDATATYPE_ENCODING_DEFAULTJSON := 16394,
	OPCUAID_JSONDATASETREADERMESSAGEDATATYPE_ENCODING_DEFAULTJSON := 16404,
	OPCUAID_DATAGRAMCONNECTIONTRANSPORTDATATYPE_ENCODING_DEFAULTJSON := 17476,
	OPCUAID_DATAGRAMWRITERGROUPTRANSPORTDATATYPE_ENCODING_DEFAULTJSON := 21203,
	OPCUAID_BROKERCONNECTIONTRANSPORTDATATYPE_ENCODING_DEFAULTJSON := 15726,
	OPCUAID_BROKERWRITERGROUPTRANSPORTDATATYPE_ENCODING_DEFAULTJSON := 16524,
	OPCUAID_BROKERDATASETWRITERTRANSPORTDATATYPE_ENCODING_DEFAULTJSON := 16525,
	OPCUAID_BROKERDATASETREADERTRANSPORTDATATYPE_ENCODING_DEFAULTJSON := 16526,
	OPCUAID_ROLEPERMISSIONTYPE_ENCODING_DEFAULTJSON := 15062,
	OPCUAID_DATATYPEDEFINITION_ENCODING_DEFAULTJSON := 15063,
	OPCUAID_STRUCTUREFIELD_ENCODING_DEFAULTJSON := 15065,
	OPCUAID_STRUCTUREDEFINITION_ENCODING_DEFAULTJSON := 15066,
	OPCUAID_ENUMDEFINITION_ENCODING_DEFAULTJSON := 15067,
	OPCUAID_NODE_ENCODING_DEFAULTJSON := 15068,
	OPCUAID_INSTANCENODE_ENCODING_DEFAULTJSON := 15069,
	OPCUAID_TYPENODE_ENCODING_DEFAULTJSON := 15070,
	OPCUAID_OBJECTNODE_ENCODING_DEFAULTJSON := 15071,
	OPCUAID_OBJECTTYPENODE_ENCODING_DEFAULTJSON := 15073,
	OPCUAID_VARIABLENODE_ENCODING_DEFAULTJSON := 15074,
	OPCUAID_VARIABLETYPENODE_ENCODING_DEFAULTJSON := 15075,
	OPCUAID_REFERENCETYPENODE_ENCODING_DEFAULTJSON := 15076,
	OPCUAID_METHODNODE_ENCODING_DEFAULTJSON := 15077,
	OPCUAID_VIEWNODE_ENCODING_DEFAULTJSON := 15078,
	OPCUAID_DATATYPENODE_ENCODING_DEFAULTJSON := 15079,
	OPCUAID_REFERENCENODE_ENCODING_DEFAULTJSON := 15080,
	OPCUAID_ARGUMENT_ENCODING_DEFAULTJSON := 15081,
	OPCUAID_ENUMVALUETYPE_ENCODING_DEFAULTJSON := 15082,
	OPCUAID_ENUMFIELD_ENCODING_DEFAULTJSON := 15083,
	OPCUAID_OPTIONSET_ENCODING_DEFAULTJSON := 15084,
	OPCUAID_UNION_ENCODING_DEFAULTJSON := 15085,
	OPCUAID_TIMEZONEDATATYPE_ENCODING_DEFAULTJSON := 15086,
	OPCUAID_APPLICATIONDESCRIPTION_ENCODING_DEFAULTJSON := 15087,
	OPCUAID_REQUESTHEADER_ENCODING_DEFAULTJSON := 15088,
	OPCUAID_RESPONSEHEADER_ENCODING_DEFAULTJSON := 15089,
	OPCUAID_SERVICEFAULT_ENCODING_DEFAULTJSON := 15090,
	OPCUAID_SESSIONLESSINVOKEREQUESTTYPE_ENCODING_DEFAULTJSON := 15091,
	OPCUAID_SESSIONLESSINVOKERESPONSETYPE_ENCODING_DEFAULTJSON := 15092,
	OPCUAID_FINDSERVERSREQUEST_ENCODING_DEFAULTJSON := 15093,
	OPCUAID_FINDSERVERSRESPONSE_ENCODING_DEFAULTJSON := 15094,
	OPCUAID_SERVERONNETWORK_ENCODING_DEFAULTJSON := 15095,
	OPCUAID_FINDSERVERSONNETWORKREQUEST_ENCODING_DEFAULTJSON := 15096,
	OPCUAID_FINDSERVERSONNETWORKRESPONSE_ENCODING_DEFAULTJSON := 15097,
	OPCUAID_USERTOKENPOLICY_ENCODING_DEFAULTJSON := 15098,
	OPCUAID_ENDPOINTDESCRIPTION_ENCODING_DEFAULTJSON := 15099,
	OPCUAID_GETENDPOINTSREQUEST_ENCODING_DEFAULTJSON := 15100,
	OPCUAID_GETENDPOINTSRESPONSE_ENCODING_DEFAULTJSON := 15101,
	OPCUAID_REGISTEREDSERVER_ENCODING_DEFAULTJSON := 15102,
	OPCUAID_REGISTERSERVERREQUEST_ENCODING_DEFAULTJSON := 15103,
	OPCUAID_REGISTERSERVERRESPONSE_ENCODING_DEFAULTJSON := 15104,
	OPCUAID_DISCOVERYCONFIGURATION_ENCODING_DEFAULTJSON := 15105,
	OPCUAID_MDNSDISCOVERYCONFIGURATION_ENCODING_DEFAULTJSON := 15106,
	OPCUAID_REGISTERSERVER2REQUEST_ENCODING_DEFAULTJSON := 15107,
	OPCUAID_REGISTERSERVER2RESPONSE_ENCODING_DEFAULTJSON := 15130,
	OPCUAID_CHANNELSECURITYTOKEN_ENCODING_DEFAULTJSON := 15131,
	OPCUAID_OPENSECURECHANNELREQUEST_ENCODING_DEFAULTJSON := 15132,
	OPCUAID_OPENSECURECHANNELRESPONSE_ENCODING_DEFAULTJSON := 15133,
	OPCUAID_CLOSESECURECHANNELREQUEST_ENCODING_DEFAULTJSON := 15134,
	OPCUAID_CLOSESECURECHANNELRESPONSE_ENCODING_DEFAULTJSON := 15135,
	OPCUAID_SIGNEDSOFTWARECERTIFICATE_ENCODING_DEFAULTJSON := 15136,
	OPCUAID_SIGNATUREDATA_ENCODING_DEFAULTJSON := 15137,
	OPCUAID_CREATESESSIONREQUEST_ENCODING_DEFAULTJSON := 15138,
	OPCUAID_CREATESESSIONRESPONSE_ENCODING_DEFAULTJSON := 15139,
	OPCUAID_USERIDENTITYTOKEN_ENCODING_DEFAULTJSON := 15140,
	OPCUAID_ANONYMOUSIDENTITYTOKEN_ENCODING_DEFAULTJSON := 15141,
	OPCUAID_USERNAMEIDENTITYTOKEN_ENCODING_DEFAULTJSON := 15142,
	OPCUAID_X509IDENTITYTOKEN_ENCODING_DEFAULTJSON := 15143,
	OPCUAID_ISSUEDIDENTITYTOKEN_ENCODING_DEFAULTJSON := 15144,
	OPCUAID_ACTIVATESESSIONREQUEST_ENCODING_DEFAULTJSON := 15145,
	OPCUAID_ACTIVATESESSIONRESPONSE_ENCODING_DEFAULTJSON := 15146,
	OPCUAID_CLOSESESSIONREQUEST_ENCODING_DEFAULTJSON := 15147,
	OPCUAID_CLOSESESSIONRESPONSE_ENCODING_DEFAULTJSON := 15148,
	OPCUAID_CANCELREQUEST_ENCODING_DEFAULTJSON := 15149,
	OPCUAID_CANCELRESPONSE_ENCODING_DEFAULTJSON := 15150,
	OPCUAID_NODEATTRIBUTES_ENCODING_DEFAULTJSON := 15151,
	OPCUAID_OBJECTATTRIBUTES_ENCODING_DEFAULTJSON := 15152,
	OPCUAID_VARIABLEATTRIBUTES_ENCODING_DEFAULTJSON := 15153,
	OPCUAID_METHODATTRIBUTES_ENCODING_DEFAULTJSON := 15157,
	OPCUAID_OBJECTTYPEATTRIBUTES_ENCODING_DEFAULTJSON := 15158,
	OPCUAID_VARIABLETYPEATTRIBUTES_ENCODING_DEFAULTJSON := 15159,
	OPCUAID_REFERENCETYPEATTRIBUTES_ENCODING_DEFAULTJSON := 15160,
	OPCUAID_DATATYPEATTRIBUTES_ENCODING_DEFAULTJSON := 15161,
	OPCUAID_VIEWATTRIBUTES_ENCODING_DEFAULTJSON := 15162,
	OPCUAID_GENERICATTRIBUTEVALUE_ENCODING_DEFAULTJSON := 15163,
	OPCUAID_GENERICATTRIBUTES_ENCODING_DEFAULTJSON := 15164,
	OPCUAID_ADDNODESITEM_ENCODING_DEFAULTJSON := 15165,
	OPCUAID_ADDNODESRESULT_ENCODING_DEFAULTJSON := 15166,
	OPCUAID_ADDNODESREQUEST_ENCODING_DEFAULTJSON := 15167,
	OPCUAID_ADDNODESRESPONSE_ENCODING_DEFAULTJSON := 15168,
	OPCUAID_ADDREFERENCESITEM_ENCODING_DEFAULTJSON := 15169,
	OPCUAID_ADDREFERENCESREQUEST_ENCODING_DEFAULTJSON := 15170,
	OPCUAID_ADDREFERENCESRESPONSE_ENCODING_DEFAULTJSON := 15171,
	OPCUAID_DELETENODESITEM_ENCODING_DEFAULTJSON := 15172,
	OPCUAID_DELETENODESREQUEST_ENCODING_DEFAULTJSON := 15173,
	OPCUAID_DELETENODESRESPONSE_ENCODING_DEFAULTJSON := 15174,
	OPCUAID_DELETEREFERENCESITEM_ENCODING_DEFAULTJSON := 15175,
	OPCUAID_DELETEREFERENCESREQUEST_ENCODING_DEFAULTJSON := 15176,
	OPCUAID_DELETEREFERENCESRESPONSE_ENCODING_DEFAULTJSON := 15177,
	OPCUAID_VIEWDESCRIPTION_ENCODING_DEFAULTJSON := 15179,
	OPCUAID_BROWSEDESCRIPTION_ENCODING_DEFAULTJSON := 15180,
	OPCUAID_REFERENCEDESCRIPTION_ENCODING_DEFAULTJSON := 15182,
	OPCUAID_BROWSERESULT_ENCODING_DEFAULTJSON := 15183,
	OPCUAID_BROWSEREQUEST_ENCODING_DEFAULTJSON := 15184,
	OPCUAID_BROWSERESPONSE_ENCODING_DEFAULTJSON := 15185,
	OPCUAID_BROWSENEXTREQUEST_ENCODING_DEFAULTJSON := 15186,
	OPCUAID_BROWSENEXTRESPONSE_ENCODING_DEFAULTJSON := 15187,
	OPCUAID_RELATIVEPATHELEMENT_ENCODING_DEFAULTJSON := 15188,
	OPCUAID_RELATIVEPATH_ENCODING_DEFAULTJSON := 15189,
	OPCUAID_BROWSEPATH_ENCODING_DEFAULTJSON := 15190,
	OPCUAID_BROWSEPATHTARGET_ENCODING_DEFAULTJSON := 15191,
	OPCUAID_BROWSEPATHRESULT_ENCODING_DEFAULTJSON := 15192,
	OPCUAID_TRANSLATEBROWSEPATHSTONODEIDSREQUEST_ENCODING_DEFAULTJSON := 15193,
	OPCUAID_TRANSLATEBROWSEPATHSTONODEIDSRESPONSE_ENCODING_DEFAULTJSON := 15194,
	OPCUAID_REGISTERNODESREQUEST_ENCODING_DEFAULTJSON := 15195,
	OPCUAID_REGISTERNODESRESPONSE_ENCODING_DEFAULTJSON := 15196,
	OPCUAID_UNREGISTERNODESREQUEST_ENCODING_DEFAULTJSON := 15197,
	OPCUAID_UNREGISTERNODESRESPONSE_ENCODING_DEFAULTJSON := 15198,
	OPCUAID_ENDPOINTCONFIGURATION_ENCODING_DEFAULTJSON := 15199,
	OPCUAID_QUERYDATADESCRIPTION_ENCODING_DEFAULTJSON := 15200,
	OPCUAID_NODETYPEDESCRIPTION_ENCODING_DEFAULTJSON := 15201,
	OPCUAID_QUERYDATASET_ENCODING_DEFAULTJSON := 15202,
	OPCUAID_NODEREFERENCE_ENCODING_DEFAULTJSON := 15203,
	OPCUAID_CONTENTFILTERELEMENT_ENCODING_DEFAULTJSON := 15204,
	OPCUAID_CONTENTFILTER_ENCODING_DEFAULTJSON := 15205,
	OPCUAID_FILTEROPERAND_ENCODING_DEFAULTJSON := 15206,
	OPCUAID_ELEMENTOPERAND_ENCODING_DEFAULTJSON := 15207,
	OPCUAID_LITERALOPERAND_ENCODING_DEFAULTJSON := 15208,
	OPCUAID_ATTRIBUTEOPERAND_ENCODING_DEFAULTJSON := 15209,
	OPCUAID_SIMPLEATTRIBUTEOPERAND_ENCODING_DEFAULTJSON := 15210,
	OPCUAID_CONTENTFILTERELEMENTRESULT_ENCODING_DEFAULTJSON := 15211,
	OPCUAID_CONTENTFILTERRESULT_ENCODING_DEFAULTJSON := 15228,
	OPCUAID_PARSINGRESULT_ENCODING_DEFAULTJSON := 15236,
	OPCUAID_QUERYFIRSTREQUEST_ENCODING_DEFAULTJSON := 15244,
	OPCUAID_QUERYFIRSTRESPONSE_ENCODING_DEFAULTJSON := 15252,
	OPCUAID_QUERYNEXTREQUEST_ENCODING_DEFAULTJSON := 15254,
	OPCUAID_QUERYNEXTRESPONSE_ENCODING_DEFAULTJSON := 15255,
	OPCUAID_READVALUEID_ENCODING_DEFAULTJSON := 15256,
	OPCUAID_READREQUEST_ENCODING_DEFAULTJSON := 15257,
	OPCUAID_READRESPONSE_ENCODING_DEFAULTJSON := 15258,
	OPCUAID_HISTORYREADVALUEID_ENCODING_DEFAULTJSON := 15259,
	OPCUAID_HISTORYREADRESULT_ENCODING_DEFAULTJSON := 15260,
	OPCUAID_HISTORYREADDETAILS_ENCODING_DEFAULTJSON := 15261,
	OPCUAID_READEVENTDETAILS_ENCODING_DEFAULTJSON := 15262,
	OPCUAID_READRAWMODIFIEDDETAILS_ENCODING_DEFAULTJSON := 15263,
	OPCUAID_READPROCESSEDDETAILS_ENCODING_DEFAULTJSON := 15264,
	OPCUAID_READATTIMEDETAILS_ENCODING_DEFAULTJSON := 15269,
	OPCUAID_HISTORYDATA_ENCODING_DEFAULTJSON := 15270,
	OPCUAID_MODIFICATIONINFO_ENCODING_DEFAULTJSON := 15271,
	OPCUAID_HISTORYMODIFIEDDATA_ENCODING_DEFAULTJSON := 15272,
	OPCUAID_HISTORYEVENT_ENCODING_DEFAULTJSON := 15273,
	OPCUAID_HISTORYREADREQUEST_ENCODING_DEFAULTJSON := 15274,
	OPCUAID_HISTORYREADRESPONSE_ENCODING_DEFAULTJSON := 15275,
	OPCUAID_WRITEVALUE_ENCODING_DEFAULTJSON := 15276,
	OPCUAID_WRITEREQUEST_ENCODING_DEFAULTJSON := 15277,
	OPCUAID_WRITERESPONSE_ENCODING_DEFAULTJSON := 15278,
	OPCUAID_HISTORYUPDATEDETAILS_ENCODING_DEFAULTJSON := 15279,
	OPCUAID_UPDATEDATADETAILS_ENCODING_DEFAULTJSON := 15280,
	OPCUAID_UPDATESTRUCTUREDATADETAILS_ENCODING_DEFAULTJSON := 15281,
	OPCUAID_UPDATEEVENTDETAILS_ENCODING_DEFAULTJSON := 15282,
	OPCUAID_DELETERAWMODIFIEDDETAILS_ENCODING_DEFAULTJSON := 15283,
	OPCUAID_DELETEATTIMEDETAILS_ENCODING_DEFAULTJSON := 15284,
	OPCUAID_DELETEEVENTDETAILS_ENCODING_DEFAULTJSON := 15285,
	OPCUAID_HISTORYUPDATERESULT_ENCODING_DEFAULTJSON := 15286,
	OPCUAID_HISTORYUPDATEREQUEST_ENCODING_DEFAULTJSON := 15287,
	OPCUAID_HISTORYUPDATERESPONSE_ENCODING_DEFAULTJSON := 15288,
	OPCUAID_CALLMETHODREQUEST_ENCODING_DEFAULTJSON := 15289,
	OPCUAID_CALLMETHODRESULT_ENCODING_DEFAULTJSON := 15290,
	OPCUAID_CALLREQUEST_ENCODING_DEFAULTJSON := 15291,
	OPCUAID_CALLRESPONSE_ENCODING_DEFAULTJSON := 15292,
	OPCUAID_MONITORINGFILTER_ENCODING_DEFAULTJSON := 15293,
	OPCUAID_DATACHANGEFILTER_ENCODING_DEFAULTJSON := 15294,
	OPCUAID_EVENTFILTER_ENCODING_DEFAULTJSON := 15295,
	OPCUAID_AGGREGATECONFIGURATION_ENCODING_DEFAULTJSON := 15304,
	OPCUAID_AGGREGATEFILTER_ENCODING_DEFAULTJSON := 15312,
	OPCUAID_MONITORINGFILTERRESULT_ENCODING_DEFAULTJSON := 15313,
	OPCUAID_EVENTFILTERRESULT_ENCODING_DEFAULTJSON := 15314,
	OPCUAID_AGGREGATEFILTERRESULT_ENCODING_DEFAULTJSON := 15315,
	OPCUAID_MONITORINGPARAMETERS_ENCODING_DEFAULTJSON := 15320,
	OPCUAID_MONITOREDITEMCREATEREQUEST_ENCODING_DEFAULTJSON := 15321,
	OPCUAID_MONITOREDITEMCREATERESULT_ENCODING_DEFAULTJSON := 15322,
	OPCUAID_CREATEMONITOREDITEMSREQUEST_ENCODING_DEFAULTJSON := 15323,
	OPCUAID_CREATEMONITOREDITEMSRESPONSE_ENCODING_DEFAULTJSON := 15324,
	OPCUAID_MONITOREDITEMMODIFYREQUEST_ENCODING_DEFAULTJSON := 15325,
	OPCUAID_MONITOREDITEMMODIFYRESULT_ENCODING_DEFAULTJSON := 15326,
	OPCUAID_MODIFYMONITOREDITEMSREQUEST_ENCODING_DEFAULTJSON := 15327,
	OPCUAID_MODIFYMONITOREDITEMSRESPONSE_ENCODING_DEFAULTJSON := 15328,
	OPCUAID_SETMONITORINGMODEREQUEST_ENCODING_DEFAULTJSON := 15329,
	OPCUAID_SETMONITORINGMODERESPONSE_ENCODING_DEFAULTJSON := 15331,
	OPCUAID_SETTRIGGERINGREQUEST_ENCODING_DEFAULTJSON := 15332,
	OPCUAID_SETTRIGGERINGRESPONSE_ENCODING_DEFAULTJSON := 15333,
	OPCUAID_DELETEMONITOREDITEMSREQUEST_ENCODING_DEFAULTJSON := 15335,
	OPCUAID_DELETEMONITOREDITEMSRESPONSE_ENCODING_DEFAULTJSON := 15336,
	OPCUAID_CREATESUBSCRIPTIONREQUEST_ENCODING_DEFAULTJSON := 15337,
	OPCUAID_CREATESUBSCRIPTIONRESPONSE_ENCODING_DEFAULTJSON := 15338,
	OPCUAID_MODIFYSUBSCRIPTIONREQUEST_ENCODING_DEFAULTJSON := 15339,
	OPCUAID_MODIFYSUBSCRIPTIONRESPONSE_ENCODING_DEFAULTJSON := 15340,
	OPCUAID_SETPUBLISHINGMODEREQUEST_ENCODING_DEFAULTJSON := 15341,
	OPCUAID_SETPUBLISHINGMODERESPONSE_ENCODING_DEFAULTJSON := 15342,
	OPCUAID_NOTIFICATIONMESSAGE_ENCODING_DEFAULTJSON := 15343,
	OPCUAID_NOTIFICATIONDATA_ENCODING_DEFAULTJSON := 15344,
	OPCUAID_DATACHANGENOTIFICATION_ENCODING_DEFAULTJSON := 15345,
	OPCUAID_MONITOREDITEMNOTIFICATION_ENCODING_DEFAULTJSON := 15346,
	OPCUAID_EVENTNOTIFICATIONLIST_ENCODING_DEFAULTJSON := 15347,
	OPCUAID_EVENTFIELDLIST_ENCODING_DEFAULTJSON := 15348,
	OPCUAID_HISTORYEVENTFIELDLIST_ENCODING_DEFAULTJSON := 15349,
	OPCUAID_STATUSCHANGENOTIFICATION_ENCODING_DEFAULTJSON := 15350,
	OPCUAID_SUBSCRIPTIONACKNOWLEDGEMENT_ENCODING_DEFAULTJSON := 15351,
	OPCUAID_PUBLISHREQUEST_ENCODING_DEFAULTJSON := 15352,
	OPCUAID_PUBLISHRESPONSE_ENCODING_DEFAULTJSON := 15353,
	OPCUAID_REPUBLISHREQUEST_ENCODING_DEFAULTJSON := 15354,
	OPCUAID_REPUBLISHRESPONSE_ENCODING_DEFAULTJSON := 15355,
	OPCUAID_TRANSFERRESULT_ENCODING_DEFAULTJSON := 15356,
	OPCUAID_TRANSFERSUBSCRIPTIONSREQUEST_ENCODING_DEFAULTJSON := 15357,
	OPCUAID_TRANSFERSUBSCRIPTIONSRESPONSE_ENCODING_DEFAULTJSON := 15358,
	OPCUAID_DELETESUBSCRIPTIONSREQUEST_ENCODING_DEFAULTJSON := 15359,
	OPCUAID_DELETESUBSCRIPTIONSRESPONSE_ENCODING_DEFAULTJSON := 15360,
	OPCUAID_BUILDINFO_ENCODING_DEFAULTJSON := 15361,
	OPCUAID_REDUNDANTSERVERDATATYPE_ENCODING_DEFAULTJSON := 15362,
	OPCUAID_ENDPOINTURLLISTDATATYPE_ENCODING_DEFAULTJSON := 15363,
	OPCUAID_NETWORKGROUPDATATYPE_ENCODING_DEFAULTJSON := 15364,
	OPCUAID_SAMPLINGINTERVALDIAGNOSTICSDATATYPE_ENCODING_DEFAULTJSON := 15365,
	OPCUAID_SERVERDIAGNOSTICSSUMMARYDATATYPE_ENCODING_DEFAULTJSON := 15366,
	OPCUAID_SERVERSTATUSDATATYPE_ENCODING_DEFAULTJSON := 15367,
	OPCUAID_SESSIONDIAGNOSTICSDATATYPE_ENCODING_DEFAULTJSON := 15368,
	OPCUAID_SESSIONSECURITYDIAGNOSTICSDATATYPE_ENCODING_DEFAULTJSON := 15369,
	OPCUAID_SERVICECOUNTERDATATYPE_ENCODING_DEFAULTJSON := 15370,
	OPCUAID_STATUSRESULT_ENCODING_DEFAULTJSON := 15371,
	OPCUAID_SUBSCRIPTIONDIAGNOSTICSDATATYPE_ENCODING_DEFAULTJSON := 15372,
	OPCUAID_MODELCHANGESTRUCTUREDATATYPE_ENCODING_DEFAULTJSON := 15373,
	OPCUAID_SEMANTICCHANGESTRUCTUREDATATYPE_ENCODING_DEFAULTJSON := 15374,
	OPCUAID_RANGE_ENCODING_DEFAULTJSON := 15375,
	OPCUAID_EUINFORMATION_ENCODING_DEFAULTJSON := 15376,
	OPCUAID_COMPLEXNUMBERTYPE_ENCODING_DEFAULTJSON := 15377,
	OPCUAID_DOUBLECOMPLEXNUMBERTYPE_ENCODING_DEFAULTJSON := 15378,
	OPCUAID_AXISINFORMATION_ENCODING_DEFAULTJSON := 15379,
	OPCUAID_XVTYPE_ENCODING_DEFAULTJSON := 15380,
	OPCUAID_PROGRAMDIAGNOSTICDATATYPE_ENCODING_DEFAULTJSON := 15381,
	OPCUAID_PROGRAMDIAGNOSTIC2DATATYPE_ENCODING_DEFAULTJSON := 15405,
	OPCUAID_ANNOTATION_ENCODING_DEFAULTJSON := 15382,
	OPCUAID_BASEOBJECTTYPE := 58,
	OPCUAID_FOLDERTYPE := 61,
	OPCUAID_DATATYPESYSTEMTYPE := 75,
	OPCUAID_DATATYPEENCODINGTYPE := 76,
	OPCUAID_MODELLINGRULETYPE := 77,
	OPCUAID_SERVERTYPE := 2004,
	OPCUAID_SERVERCAPABILITIESTYPE := 2013,
	OPCUAID_SERVERDIAGNOSTICSTYPE := 2020,
	OPCUAID_SESSIONSDIAGNOSTICSSUMMARYTYPE := 2026,
	OPCUAID_SESSIONDIAGNOSTICSOBJECTTYPE := 2029,
	OPCUAID_VENDORSERVERINFOTYPE := 2033,
	OPCUAID_SERVERREDUNDANCYTYPE := 2034,
	OPCUAID_TRANSPARENTREDUNDANCYTYPE := 2036,
	OPCUAID_NONTRANSPARENTREDUNDANCYTYPE := 2039,
	OPCUAID_NONTRANSPARENTNETWORKREDUNDANCYTYPE := 11945,
	OPCUAID_OPERATIONLIMITSTYPE := 11564,
	OPCUAID_FILETYPE := 11575,
	OPCUAID_ADDRESSSPACEFILETYPE := 11595,
	OPCUAID_NAMESPACEMETADATATYPE := 11616,
	OPCUAID_NAMESPACESTYPE := 11645,
	OPCUAID_BASEEVENTTYPE := 2041,
	OPCUAID_AUDITEVENTTYPE := 2052,
	OPCUAID_AUDITSECURITYEVENTTYPE := 2058,
	OPCUAID_AUDITCHANNELEVENTTYPE := 2059,
	OPCUAID_AUDITOPENSECURECHANNELEVENTTYPE := 2060,
	OPCUAID_AUDITSESSIONEVENTTYPE := 2069,
	OPCUAID_AUDITCREATESESSIONEVENTTYPE := 2071,
	OPCUAID_AUDITURLMISMATCHEVENTTYPE := 2748,
	OPCUAID_AUDITACTIVATESESSIONEVENTTYPE := 2075,
	OPCUAID_AUDITCANCELEVENTTYPE := 2078,
	OPCUAID_AUDITCERTIFICATEEVENTTYPE := 2080,
	OPCUAID_AUDITCERTIFICATEDATAMISMATCHEVENTTYPE := 2082,
	OPCUAID_AUDITCERTIFICATEEXPIREDEVENTTYPE := 2085,
	OPCUAID_AUDITCERTIFICATEINVALIDEVENTTYPE := 2086,
	OPCUAID_AUDITCERTIFICATEUNTRUSTEDEVENTTYPE := 2087,
	OPCUAID_AUDITCERTIFICATEREVOKEDEVENTTYPE := 2088,
	OPCUAID_AUDITCERTIFICATEMISMATCHEVENTTYPE := 2089,
	OPCUAID_AUDITNODEMANAGEMENTEVENTTYPE := 2090,
	OPCUAID_AUDITADDNODESEVENTTYPE := 2091,
	OPCUAID_AUDITDELETENODESEVENTTYPE := 2093,
	OPCUAID_AUDITADDREFERENCESEVENTTYPE := 2095,
	OPCUAID_AUDITDELETEREFERENCESEVENTTYPE := 2097,
	OPCUAID_AUDITUPDATEEVENTTYPE := 2099,
	OPCUAID_AUDITWRITEUPDATEEVENTTYPE := 2100,
	OPCUAID_AUDITHISTORYUPDATEEVENTTYPE := 2104,
	OPCUAID_AUDITUPDATEMETHODEVENTTYPE := 2127,
	OPCUAID_SYSTEMEVENTTYPE := 2130,
	OPCUAID_DEVICEFAILUREEVENTTYPE := 2131,
	OPCUAID_SYSTEMSTATUSCHANGEEVENTTYPE := 11446,
	OPCUAID_BASEMODELCHANGEEVENTTYPE := 2132,
	OPCUAID_GENERALMODELCHANGEEVENTTYPE := 2133,
	OPCUAID_SEMANTICCHANGEEVENTTYPE := 2738,
	OPCUAID_EVENTQUEUEOVERFLOWEVENTTYPE := 3035,
	OPCUAID_PROGRESSEVENTTYPE := 11436,
	OPCUAID_AGGREGATEFUNCTIONTYPE := 2340,
	OPCUAID_STATEMACHINETYPE := 2299,
	OPCUAID_FINITESTATEMACHINETYPE := 2771,
	OPCUAID_STATETYPE := 2307,
	OPCUAID_INITIALSTATETYPE := 2309,
	OPCUAID_TRANSITIONTYPE := 2310,
	OPCUAID_TRANSITIONEVENTTYPE := 2311,
	OPCUAID_AUDITUPDATESTATEEVENTTYPE := 2315,
	OPCUAID_FILEDIRECTORYTYPE := 13353,
	OPCUAID_TEMPORARYFILETRANSFERTYPE := 15744,
	OPCUAID_FILETRANSFERSTATEMACHINETYPE := 15803,
	OPCUAID_ROLESETTYPE := 15607,
	OPCUAID_ROLETYPE := 15620,
	OPCUAID_ROLEMAPPINGRULECHANGEDAUDITEVENTTYPE := 17641,
	OPCUAID_CONDITIONTYPE := 2782,
	OPCUAID_DIALOGCONDITIONTYPE := 2830,
	OPCUAID_ACKNOWLEDGEABLECONDITIONTYPE := 2881,
	OPCUAID_ALARMCONDITIONTYPE := 2915,
	OPCUAID_ALARMGROUPTYPE := 16405,
	OPCUAID_SHELVEDSTATEMACHINETYPE := 2929,
	OPCUAID_LIMITALARMTYPE := 2955,
	OPCUAID_EXCLUSIVELIMITSTATEMACHINETYPE := 9318,
	OPCUAID_EXCLUSIVELIMITALARMTYPE := 9341,
	OPCUAID_NONEXCLUSIVELIMITALARMTYPE := 9906,
	OPCUAID_NONEXCLUSIVELEVELALARMTYPE := 10060,
	OPCUAID_EXCLUSIVELEVELALARMTYPE := 9482,
	OPCUAID_NONEXCLUSIVEDEVIATIONALARMTYPE := 10368,
	OPCUAID_NONEXCLUSIVERATEOFCHANGEALARMTYPE := 10214,
	OPCUAID_EXCLUSIVEDEVIATIONALARMTYPE := 9764,
	OPCUAID_EXCLUSIVERATEOFCHANGEALARMTYPE := 9623,
	OPCUAID_DISCRETEALARMTYPE := 10523,
	OPCUAID_OFFNORMALALARMTYPE := 10637,
	OPCUAID_SYSTEMOFFNORMALALARMTYPE := 11753,
	OPCUAID_TRIPALARMTYPE := 10751,
	OPCUAID_INSTRUMENTDIAGNOSTICALARMTYPE := 18347,
	OPCUAID_SYSTEMDIAGNOSTICALARMTYPE := 18496,
	OPCUAID_CERTIFICATEEXPIRATIONALARMTYPE := 13225,
	OPCUAID_DISCREPANCYALARMTYPE := 17080,
	OPCUAID_BASECONDITIONCLASSTYPE := 11163,
	OPCUAID_PROCESSCONDITIONCLASSTYPE := 11164,
	OPCUAID_MAINTENANCECONDITIONCLASSTYPE := 11165,
	OPCUAID_SYSTEMCONDITIONCLASSTYPE := 11166,
	OPCUAID_SAFETYCONDITIONCLASSTYPE := 17218,
	OPCUAID_HIGHLYMANAGEDALARMCONDITIONCLASSTYPE := 17219,
	OPCUAID_TRAININGCONDITIONCLASSTYPE := 17220,
	OPCUAID_STATISTICALCONDITIONCLASSTYPE := 18665,
	OPCUAID_TESTINGCONDITIONCLASSTYPE := 17221,
	OPCUAID_AUDITCONDITIONEVENTTYPE := 2790,
	OPCUAID_AUDITCONDITIONENABLEEVENTTYPE := 2803,
	OPCUAID_AUDITCONDITIONCOMMENTEVENTTYPE := 2829,
	OPCUAID_AUDITCONDITIONRESPONDEVENTTYPE := 8927,
	OPCUAID_AUDITCONDITIONACKNOWLEDGEEVENTTYPE := 8944,
	OPCUAID_AUDITCONDITIONCONFIRMEVENTTYPE := 8961,
	OPCUAID_AUDITCONDITIONSHELVINGEVENTTYPE := 11093,
	OPCUAID_AUDITCONDITIONSUPPRESSEVENTTYPE := 17225,
	OPCUAID_AUDITCONDITIONSILENCEEVENTTYPE := 17242,
	OPCUAID_AUDITCONDITIONRESETEVENTTYPE := 15013,
	OPCUAID_AUDITCONDITIONOUTOFSERVICEEVENTTYPE := 17259,
	OPCUAID_REFRESHSTARTEVENTTYPE := 2787,
	OPCUAID_REFRESHENDEVENTTYPE := 2788,
	OPCUAID_REFRESHREQUIREDEVENTTYPE := 2789,
	OPCUAID_ALARMMETRICSTYPE := 17279,
	OPCUAID_PROGRAMSTATEMACHINETYPE := 2391,
	OPCUAID_PROGRAMTRANSITIONEVENTTYPE := 2378,
	OPCUAID_AUDITPROGRAMTRANSITIONEVENTTYPE := 11856,
	OPCUAID_PROGRAMTRANSITIONAUDITEVENTTYPE := 3806,
	OPCUAID_HISTORICALDATACONFIGURATIONTYPE := 2318,
	OPCUAID_HISTORYSERVERCAPABILITIESTYPE := 2330,
	OPCUAID_AUDITHISTORYEVENTUPDATEEVENTTYPE := 2999,
	OPCUAID_AUDITHISTORYVALUEUPDATEEVENTTYPE := 3006,
	OPCUAID_AUDITHISTORYDELETEEVENTTYPE := 3012,
	OPCUAID_AUDITHISTORYRAWMODIFYDELETEEVENTTYPE := 3014,
	OPCUAID_AUDITHISTORYATTIMEDELETEEVENTTYPE := 3019,
	OPCUAID_AUDITHISTORYEVENTDELETEEVENTTYPE := 3022,
	OPCUAID_TRUSTLISTTYPE := 12522,
	OPCUAID_CERTIFICATEGROUPTYPE := 12555,
	OPCUAID_CERTIFICATEGROUPFOLDERTYPE := 13813,
	OPCUAID_CERTIFICATETYPE := 12556,
	OPCUAID_APPLICATIONCERTIFICATETYPE := 12557,
	OPCUAID_HTTPSCERTIFICATETYPE := 12558,
	OPCUAID_USERCREDENTIALCERTIFICATETYPE := 15181,
	OPCUAID_RSAMINAPPLICATIONCERTIFICATETYPE := 12559,
	OPCUAID_RSASHA256APPLICATIONCERTIFICATETYPE := 12560,
	OPCUAID_TRUSTLISTUPDATEDAUDITEVENTTYPE := 12561,
	OPCUAID_SERVERCONFIGURATIONTYPE := 12581,
	OPCUAID_CERTIFICATEUPDATEDAUDITEVENTTYPE := 12620,
	OPCUAID_KEYCREDENTIALCONFIGURATIONFOLDERTYPE := 17496,
	OPCUAID_KEYCREDENTIALCONFIGURATIONTYPE := 18001,
	OPCUAID_KEYCREDENTIALAUDITEVENTTYPE := 18011,
	OPCUAID_KEYCREDENTIALUPDATEDAUDITEVENTTYPE := 18029,
	OPCUAID_KEYCREDENTIALDELETEDAUDITEVENTTYPE := 18047,
	OPCUAID_AUTHORIZATIONSERVICECONFIGURATIONTYPE := 17852,
	OPCUAID_AGGREGATECONFIGURATIONTYPE := 11187,
	OPCUAID_PUBSUBKEYSERVICETYPE := 15906,
	OPCUAID_SECURITYGROUPFOLDERTYPE := 15452,
	OPCUAID_SECURITYGROUPTYPE := 15471,
	OPCUAID_PUBLISHSUBSCRIBETYPE := 14416,
	OPCUAID_PUBLISHEDDATASETTYPE := 14509,
	OPCUAID_EXTENSIONFIELDSTYPE := 15489,
	OPCUAID_PUBLISHEDDATAITEMSTYPE := 14534,
	OPCUAID_PUBLISHEDEVENTSTYPE := 14572,
	OPCUAID_DATASETFOLDERTYPE := 14477,
	OPCUAID_PUBSUBCONNECTIONTYPE := 14209,
	OPCUAID_CONNECTIONTRANSPORTTYPE := 17721,
	OPCUAID_PUBSUBGROUPTYPE := 14232,
	OPCUAID_WRITERGROUPTYPE := 17725,
	OPCUAID_WRITERGROUPTRANSPORTTYPE := 17997,
	OPCUAID_WRITERGROUPMESSAGETYPE := 17998,
	OPCUAID_READERGROUPTYPE := 17999,
	OPCUAID_READERGROUPTRANSPORTTYPE := 21090,
	OPCUAID_READERGROUPMESSAGETYPE := 21091,
	OPCUAID_DATASETWRITERTYPE := 15298,
	OPCUAID_DATASETWRITERTRANSPORTTYPE := 15305,
	OPCUAID_DATASETWRITERMESSAGETYPE := 21096,
	OPCUAID_DATASETREADERTYPE := 15306,
	OPCUAID_DATASETREADERTRANSPORTTYPE := 15319,
	OPCUAID_DATASETREADERMESSAGETYPE := 21104,
	OPCUAID_SUBSCRIBEDDATASETTYPE := 15108,
	OPCUAID_TARGETVARIABLESTYPE := 15111,
	OPCUAID_SUBSCRIBEDDATASETMIRRORTYPE := 15127,
	OPCUAID_PUBSUBSTATUSTYPE := 14643,
	OPCUAID_PUBSUBDIAGNOSTICSTYPE := 19677,
	OPCUAID_PUBSUBDIAGNOSTICSROOTTYPE := 19732,
	OPCUAID_PUBSUBDIAGNOSTICSCONNECTIONTYPE := 19786,
	OPCUAID_PUBSUBDIAGNOSTICSWRITERGROUPTYPE := 19834,
	OPCUAID_PUBSUBDIAGNOSTICSREADERGROUPTYPE := 19903,
	OPCUAID_PUBSUBDIAGNOSTICSDATASETWRITERTYPE := 19968,
	OPCUAID_PUBSUBDIAGNOSTICSDATASETREADERTYPE := 20027,
	OPCUAID_PUBSUBSTATUSEVENTTYPE := 15535,
	OPCUAID_PUBSUBTRANSPORTLIMITSEXCEEDEVENTTYPE := 15548,
	OPCUAID_PUBSUBCOMMUNICATIONFAILUREEVENTTYPE := 15563,
	OPCUAID_UADPWRITERGROUPMESSAGETYPE := 21105,
	OPCUAID_UADPDATASETWRITERMESSAGETYPE := 21111,
	OPCUAID_UADPDATASETREADERMESSAGETYPE := 21116,
	OPCUAID_JSONWRITERGROUPMESSAGETYPE := 21126,
	OPCUAID_JSONDATASETWRITERMESSAGETYPE := 21128,
	OPCUAID_JSONDATASETREADERMESSAGETYPE := 21130,
	OPCUAID_DATAGRAMCONNECTIONTRANSPORTTYPE := 15064,
	OPCUAID_DATAGRAMWRITERGROUPTRANSPORTTYPE := 21133,
	OPCUAID_BROKERCONNECTIONTRANSPORTTYPE := 15155,
	OPCUAID_BROKERWRITERGROUPTRANSPORTTYPE := 21136,
	OPCUAID_BROKERDATASETWRITERTRANSPORTTYPE := 21138,
	OPCUAID_BROKERDATASETREADERTRANSPORTTYPE := 21142,
	OPCUAID_NETWORKADDRESSTYPE := 21145,
	OPCUAID_NETWORKADDRESSURLTYPE := 21147,
	OPCUAID_REFERENCES := 31,
	OPCUAID_NONHIERARCHICALREFERENCES := 32,
	OPCUAID_HIERARCHICALREFERENCES := 33,
	OPCUAID_HASCHILD := 34,
	OPCUAID_ORGANIZES := 35,
	OPCUAID_HASEVENTSOURCE := 36,
	OPCUAID_HASMODELLINGRULE := 37,
	OPCUAID_HASENCODING := 38,
	OPCUAID_HASDESCRIPTION := 39,
	OPCUAID_HASTYPEDEFINITION := 40,
	OPCUAID_GENERATESEVENT := 41,
	OPCUAID_ALWAYSGENERATESEVENT := 3065,
	OPCUAID_AGGREGATES := 44,
	OPCUAID_HASSUBTYPE := 45,
	OPCUAID_HASPROPERTY := 46,
	OPCUAID_HASCOMPONENT := 47,
	OPCUAID_HASNOTIFIER := 48,
	OPCUAID_HASORDEREDCOMPONENT := 49,
	OPCUAID_FROMSTATE := 51,
	OPCUAID_TOSTATE := 52,
	OPCUAID_HASCAUSE := 53,
	OPCUAID_HASEFFECT := 54,
	OPCUAID_HASSUBSTATEMACHINE := 117,
	OPCUAID_HASHISTORICALCONFIGURATION := 56,
	OPCUAID_DESCRIBESARGUMENT := 129,
	OPCUAID_DESCRIBESINPUTARGUMENT := 130,
	OPCUAID_DESCRIBESOPTIONALINPUTARGUMENT := 131,
	OPCUAID_DESCRIBESOUTPUTARGUMENT := 132,
	OPCUAID_HASTRUESUBSTATE := 9004,
	OPCUAID_HASFALSESUBSTATE := 9005,
	OPCUAID_HASALARMSUPPRESSIONGROUP := 16361,
	OPCUAID_ALARMGROUPMEMBER := 16362,
	OPCUAID_HASCONDITION := 9006,
	OPCUAID_HASEFFECTDISABLE := 17276,
	OPCUAID_HASEFFECTENABLE := 17983,
	OPCUAID_HASEFFECTSUPPRESSED := 17984,
	OPCUAID_HASEFFECTUNSUPPRESSED := 17985,
	OPCUAID_HASPUBSUBCONNECTION := 14476,
	OPCUAID_DATASETTOWRITER := 14936,
	OPCUAID_HASDATASETWRITER := 15296,
	OPCUAID_HASDATASETREADER := 15297,
	OPCUAID_DATATYPEDESCRIPTIONTYPE_DATATYPEVERSION := 104,
	OPCUAID_DATATYPEDESCRIPTIONTYPE_DICTIONARYFRAGMENT := 105,
	OPCUAID_DATATYPEDICTIONARYTYPE_DATATYPEVERSION := 106,
	OPCUAID_DATATYPEDICTIONARYTYPE_NAMESPACEURI := 107,
	OPCUAID_DATATYPEDICTIONARYTYPE_DEPRECATED := 15001,
	OPCUAID_NAMINGRULETYPE_ENUMVALUES := 12169,
	OPCUAID_MODELLINGRULETYPE_NAMINGRULE := 111,
	OPCUAID_MODELLINGRULE_MANDATORY_NAMINGRULE := 112,
	OPCUAID_MODELLINGRULE_OPTIONAL_NAMINGRULE := 113,
	OPCUAID_MODELLINGRULE_EXPOSESITSARRAY_NAMINGRULE := 114,
	OPCUAID_MODELLINGRULE_MANDATORYSHARED_NAMINGRULE := 116,
	OPCUAID_MODELLINGRULE_OPTIONALPLACEHOLDER_NAMINGRULE := 11509,
	OPCUAID_MODELLINGRULE_MANDATORYPLACEHOLDER_NAMINGRULE := 11511,
	OPCUAID_OPCUANAMESPACEMETADATA_NAMESPACEURI := 15958,
	OPCUAID_OPCUANAMESPACEMETADATA_NAMESPACEVERSION := 15959,
	OPCUAID_OPCUANAMESPACEMETADATA_NAMESPACEPUBLICATIONDATE := 15960,
	OPCUAID_OPCUANAMESPACEMETADATA_ISNAMESPACESUBSET := 15961,
	OPCUAID_OPCUANAMESPACEMETADATA_STATICNODEIDTYPES := 15962,
	OPCUAID_OPCUANAMESPACEMETADATA_STATICNUMERICNODEIDRANGE := 15963,
	OPCUAID_OPCUANAMESPACEMETADATA_STATICSTRINGNODEIDPATTERN := 15964,
	OPCUAID_OPCUANAMESPACEMETADATA_NAMESPACEFILE_SIZE := 15966,
	OPCUAID_OPCUANAMESPACEMETADATA_NAMESPACEFILE_WRITABLE := 15967,
	OPCUAID_OPCUANAMESPACEMETADATA_NAMESPACEFILE_USERWRITABLE := 15968,
	OPCUAID_OPCUANAMESPACEMETADATA_NAMESPACEFILE_OPENCOUNT := 15969,
	OPCUAID_OPCUANAMESPACEMETADATA_NAMESPACEFILE_OPEN_INPUTARGUMENTS := 15972,
	OPCUAID_OPCUANAMESPACEMETADATA_NAMESPACEFILE_OPEN_OUTPUTARGUMENTS := 15973,
	OPCUAID_OPCUANAMESPACEMETADATA_NAMESPACEFILE_CLOSE_INPUTARGUMENTS := 15975,
	OPCUAID_OPCUANAMESPACEMETADATA_NAMESPACEFILE_READ_INPUTARGUMENTS := 15977,
	OPCUAID_OPCUANAMESPACEMETADATA_NAMESPACEFILE_READ_OUTPUTARGUMENTS := 15978,
	OPCUAID_OPCUANAMESPACEMETADATA_NAMESPACEFILE_WRITE_INPUTARGUMENTS := 15980,
	OPCUAID_OPCUANAMESPACEMETADATA_NAMESPACEFILE_GETPOSITION_INPUTARGUMENTS := 15982,
	OPCUAID_OPCUANAMESPACEMETADATA_NAMESPACEFILE_GETPOSITION_OUTPUTARGUMENTS := 15983,
	OPCUAID_OPCUANAMESPACEMETADATA_NAMESPACEFILE_SETPOSITION_INPUTARGUMENTS := 15985,
	OPCUAID_OPCUANAMESPACEMETADATA_DEFAULTROLEPERMISSIONS := 16134,
	OPCUAID_OPCUANAMESPACEMETADATA_DEFAULTUSERROLEPERMISSIONS := 16135,
	OPCUAID_OPCUANAMESPACEMETADATA_DEFAULTACCESSRESTRICTIONS := 16136,
	OPCUAID_NODEVERSION := 3068,
	OPCUAID_VIEWVERSION := 12170,
	OPCUAID_ICON := 3067,
	OPCUAID_LOCALTIME := 3069,
	OPCUAID_ALLOWNULLS := 3070,
	OPCUAID_VALUEASTEXT := 11433,
	OPCUAID_MAXSTRINGLENGTH := 11498,
	OPCUAID_MAXCHARACTERS := 15002,
	OPCUAID_MAXBYTESTRINGLENGTH := 12908,
	OPCUAID_MAXARRAYLENGTH := 11512,
	OPCUAID_ENGINEERINGUNITS := 11513,
	OPCUAID_ENUMSTRINGS := 11432,
	OPCUAID_ENUMVALUES := 3071,
	OPCUAID_OPTIONSETVALUES := 12745,
	OPCUAID_INPUTARGUMENTS := 3072,
	OPCUAID_OUTPUTARGUMENTS := 3073,
	OPCUAID_DEFAULTINPUTVALUES := 16306,
	OPCUAID_SERVERTYPE_SERVERARRAY := 2005,
	OPCUAID_SERVERTYPE_NAMESPACEARRAY := 2006,
	OPCUAID_SERVERTYPE_URISVERSION := 15003,
	OPCUAID_SERVERTYPE_SERVERSTATUS := 2007,
	OPCUAID_SERVERTYPE_SERVERSTATUS_STARTTIME := 3074,
	OPCUAID_SERVERTYPE_SERVERSTATUS_CURRENTTIME := 3075,
	OPCUAID_SERVERTYPE_SERVERSTATUS_STATE := 3076,
	OPCUAID_SERVERTYPE_SERVERSTATUS_BUILDINFO := 3077,
	OPCUAID_SERVERTYPE_SERVERSTATUS_BUILDINFO_PRODUCTURI := 3078,
	OPCUAID_SERVERTYPE_SERVERSTATUS_BUILDINFO_MANUFACTURERNAME := 3079,
	OPCUAID_SERVERTYPE_SERVERSTATUS_BUILDINFO_PRODUCTNAME := 3080,
	OPCUAID_SERVERTYPE_SERVERSTATUS_BUILDINFO_SOFTWAREVERSION := 3081,
	OPCUAID_SERVERTYPE_SERVERSTATUS_BUILDINFO_BUILDNUMBER := 3082,
	OPCUAID_SERVERTYPE_SERVERSTATUS_BUILDINFO_BUILDDATE := 3083,
	OPCUAID_SERVERTYPE_SERVERSTATUS_SECONDSTILLSHUTDOWN := 3084,
	OPCUAID_SERVERTYPE_SERVERSTATUS_SHUTDOWNREASON := 3085,
	OPCUAID_SERVERTYPE_SERVICELEVEL := 2008,
	OPCUAID_SERVERTYPE_AUDITING := 2742,
	OPCUAID_SERVERTYPE_ESTIMATEDRETURNTIME := 12882,
	OPCUAID_SERVERTYPE_LOCALTIME := 17612,
	OPCUAID_SERVERTYPE_SERVERCAPABILITIES_SERVERPROFILEARRAY := 3086,
	OPCUAID_SERVERTYPE_SERVERCAPABILITIES_LOCALEIDARRAY := 3087,
	OPCUAID_SERVERTYPE_SERVERCAPABILITIES_MINSUPPORTEDSAMPLERATE := 3088,
	OPCUAID_SERVERTYPE_SERVERCAPABILITIES_MAXBROWSECONTINUATIONPOINTS := 3089,
	OPCUAID_SERVERTYPE_SERVERCAPABILITIES_MAXQUERYCONTINUATIONPOINTS := 3090,
	OPCUAID_SERVERTYPE_SERVERCAPABILITIES_MAXHISTORYCONTINUATIONPOINTS := 3091,
	OPCUAID_SERVERTYPE_SERVERCAPABILITIES_SOFTWARECERTIFICATES := 3092,
	OPCUAID_SERVERTYPE_SERVERCAPABILITIES_ROLESET_ADDROLE_INPUTARGUMENTS := 16291,
	OPCUAID_SERVERTYPE_SERVERCAPABILITIES_ROLESET_ADDROLE_OUTPUTARGUMENTS := 16292,
	OPCUAID_SERVERTYPE_SERVERCAPABILITIES_ROLESET_REMOVEROLE_INPUTARGUMENTS := 16294,
	OPCUAID_SERVERTYPE_SERVERDIAGNOSTICS_SERVERDIAGNOSTICSSUMMARY := 3095,
	OPCUAID_SERVERTYPE_SERVERDIAGNOSTICS_SERVERDIAGNOSTICSSUMMARY_SERVERVIEWCOUNT := 3096,
	OPCUAID_SERVERTYPE_SERVERDIAGNOSTICS_SERVERDIAGNOSTICSSUMMARY_CURRENTSESSIONCOUNT := 3097,
	OPCUAID_SERVERTYPE_SERVERDIAGNOSTICS_SERVERDIAGNOSTICSSUMMARY_CUMULATEDSESSIONCOUNT := 3098,
	OPCUAID_SERVERTYPE_SERVERDIAGNOSTICS_SERVERDIAGNOSTICSSUMMARY_SECURITYREJECTEDSESSIONCOUNT := 3099,
	OPCUAID_SERVERTYPE_SERVERDIAGNOSTICS_SERVERDIAGNOSTICSSUMMARY_REJECTEDSESSIONCOUNT := 3100,
	OPCUAID_SERVERTYPE_SERVERDIAGNOSTICS_SERVERDIAGNOSTICSSUMMARY_SESSIONTIMEOUTCOUNT := 3101,
	OPCUAID_SERVERTYPE_SERVERDIAGNOSTICS_SERVERDIAGNOSTICSSUMMARY_SESSIONABORTCOUNT := 3102,
	OPCUAID_SERVERTYPE_SERVERDIAGNOSTICS_SERVERDIAGNOSTICSSUMMARY_PUBLISHINGINTERVALCOUNT := 3104,
	OPCUAID_SERVERTYPE_SERVERDIAGNOSTICS_SERVERDIAGNOSTICSSUMMARY_CURRENTSUBSCRIPTIONCOUNT := 3105,
	OPCUAID_SERVERTYPE_SERVERDIAGNOSTICS_SERVERDIAGNOSTICSSUMMARY_CUMULATEDSUBSCRIPTIONCOUNT := 3106,
	OPCUAID_SERVERTYPE_SERVERDIAGNOSTICS_SERVERDIAGNOSTICSSUMMARY_SECURITYREJECTEDREQUESTSCOUNT := 3107,
	OPCUAID_SERVERTYPE_SERVERDIAGNOSTICS_SERVERDIAGNOSTICSSUMMARY_REJECTEDREQUESTSCOUNT := 3108,
	OPCUAID_SERVERTYPE_SERVERDIAGNOSTICS_SUBSCRIPTIONDIAGNOSTICSARRAY := 3110,
	OPCUAID_SERVERTYPE_SERVERDIAGNOSTICS_SESSIONSDIAGNOSTICSSUMMARY_SESSIONDIAGNOSTICSARRAY := 3112,
	OPCUAID_SERVERTYPE_SERVERDIAGNOSTICS_SESSIONSDIAGNOSTICSSUMMARY_SESSIONSECURITYDIAGNOSTICSARRAY := 3113,
	OPCUAID_SERVERTYPE_SERVERDIAGNOSTICS_ENABLEDFLAG := 3114,
	OPCUAID_SERVERTYPE_SERVERREDUNDANCY_REDUNDANCYSUPPORT := 3115,
	OPCUAID_SERVERTYPE_GETMONITOREDITEMS_INPUTARGUMENTS := 11490,
	OPCUAID_SERVERTYPE_GETMONITOREDITEMS_OUTPUTARGUMENTS := 11491,
	OPCUAID_SERVERTYPE_RESENDDATA_INPUTARGUMENTS := 12872,
	OPCUAID_SERVERTYPE_SETSUBSCRIPTIONDURABLE_INPUTARGUMENTS := 12747,
	OPCUAID_SERVERTYPE_SETSUBSCRIPTIONDURABLE_OUTPUTARGUMENTS := 12748,
	OPCUAID_SERVERTYPE_REQUESTSERVERSTATECHANGE_INPUTARGUMENTS := 12884,
	OPCUAID_SERVERCAPABILITIESTYPE_SERVERPROFILEARRAY := 2014,
	OPCUAID_SERVERCAPABILITIESTYPE_LOCALEIDARRAY := 2016,
	OPCUAID_SERVERCAPABILITIESTYPE_MINSUPPORTEDSAMPLERATE := 2017,
	OPCUAID_SERVERCAPABILITIESTYPE_MAXBROWSECONTINUATIONPOINTS := 2732,
	OPCUAID_SERVERCAPABILITIESTYPE_MAXQUERYCONTINUATIONPOINTS := 2733,
	OPCUAID_SERVERCAPABILITIESTYPE_MAXHISTORYCONTINUATIONPOINTS := 2734,
	OPCUAID_SERVERCAPABILITIESTYPE_SOFTWARECERTIFICATES := 3049,
	OPCUAID_SERVERCAPABILITIESTYPE_MAXARRAYLENGTH := 11549,
	OPCUAID_SERVERCAPABILITIESTYPE_MAXSTRINGLENGTH := 11550,
	OPCUAID_SERVERCAPABILITIESTYPE_MAXBYTESTRINGLENGTH := 12910,
	OPCUAID_SERVERCAPABILITIESTYPE_VENDORCAPABILITY_PLACEHOLDER := 11562,
	OPCUAID_SERVERCAPABILITIESTYPE_ROLESET_ADDROLE_INPUTARGUMENTS := 16297,
	OPCUAID_SERVERCAPABILITIESTYPE_ROLESET_ADDROLE_OUTPUTARGUMENTS := 16298,
	OPCUAID_SERVERCAPABILITIESTYPE_ROLESET_REMOVEROLE_INPUTARGUMENTS := 16300,
	OPCUAID_SERVERDIAGNOSTICSTYPE_SERVERDIAGNOSTICSSUMMARY := 2021,
	OPCUAID_SERVERDIAGNOSTICSTYPE_SERVERDIAGNOSTICSSUMMARY_SERVERVIEWCOUNT := 3116,
	OPCUAID_SERVERDIAGNOSTICSTYPE_SERVERDIAGNOSTICSSUMMARY_CURRENTSESSIONCOUNT := 3117,
	OPCUAID_SERVERDIAGNOSTICSTYPE_SERVERDIAGNOSTICSSUMMARY_CUMULATEDSESSIONCOUNT := 3118,
	OPCUAID_SERVERDIAGNOSTICSTYPE_SERVERDIAGNOSTICSSUMMARY_SECURITYREJECTEDSESSIONCOUNT := 3119,
	OPCUAID_SERVERDIAGNOSTICSTYPE_SERVERDIAGNOSTICSSUMMARY_REJECTEDSESSIONCOUNT := 3120,
	OPCUAID_SERVERDIAGNOSTICSTYPE_SERVERDIAGNOSTICSSUMMARY_SESSIONTIMEOUTCOUNT := 3121,
	OPCUAID_SERVERDIAGNOSTICSTYPE_SERVERDIAGNOSTICSSUMMARY_SESSIONABORTCOUNT := 3122,
	OPCUAID_SERVERDIAGNOSTICSTYPE_SERVERDIAGNOSTICSSUMMARY_PUBLISHINGINTERVALCOUNT := 3124,
	OPCUAID_SERVERDIAGNOSTICSTYPE_SERVERDIAGNOSTICSSUMMARY_CURRENTSUBSCRIPTIONCOUNT := 3125,
	OPCUAID_SERVERDIAGNOSTICSTYPE_SERVERDIAGNOSTICSSUMMARY_CUMULATEDSUBSCRIPTIONCOUNT := 3126,
	OPCUAID_SERVERDIAGNOSTICSTYPE_SERVERDIAGNOSTICSSUMMARY_SECURITYREJECTEDREQUESTSCOUNT := 3127,
	OPCUAID_SERVERDIAGNOSTICSTYPE_SERVERDIAGNOSTICSSUMMARY_REJECTEDREQUESTSCOUNT := 3128,
	OPCUAID_SERVERDIAGNOSTICSTYPE_SAMPLINGINTERVALDIAGNOSTICSARRAY := 2022,
	OPCUAID_SERVERDIAGNOSTICSTYPE_SUBSCRIPTIONDIAGNOSTICSARRAY := 2023,
	OPCUAID_SERVERDIAGNOSTICSTYPE_SESSIONSDIAGNOSTICSSUMMARY_SESSIONDIAGNOSTICSARRAY := 3129,
	OPCUAID_SERVERDIAGNOSTICSTYPE_SESSIONSDIAGNOSTICSSUMMARY_SESSIONSECURITYDIAGNOSTICSARRAY := 3130,
	OPCUAID_SERVERDIAGNOSTICSTYPE_ENABLEDFLAG := 2025,
	OPCUAID_SESSIONSDIAGNOSTICSSUMMARYTYPE_SESSIONDIAGNOSTICSARRAY := 2027,
	OPCUAID_SESSIONSDIAGNOSTICSSUMMARYTYPE_SESSIONSECURITYDIAGNOSTICSARRAY := 2028,
	OPCUAID_SESSIONSDIAGNOSTICSSUMMARYTYPE_CLIENTNAME_PLACEHOLDER_SESSIONDIAGNOSTICS := 12098,
	OPCUAID_SESSIONSDIAGNOSTICSSUMMARYTYPE_CLIENTNAME_PLACEHOLDER_SESSIONDIAGNOSTICS_SESSIONID := 12099,
	OPCUAID_SESSIONSDIAGNOSTICSSUMMARYTYPE_CLIENTNAME_PLACEHOLDER_SESSIONDIAGNOSTICS_SESSIONNAME := 12100,
	OPCUAID_SESSIONSDIAGNOSTICSSUMMARYTYPE_CLIENTNAME_PLACEHOLDER_SESSIONDIAGNOSTICS_CLIENTDESCRIPTION := 12101,
	OPCUAID_SESSIONSDIAGNOSTICSSUMMARYTYPE_CLIENTNAME_PLACEHOLDER_SESSIONDIAGNOSTICS_SERVERURI := 12102,
	OPCUAID_SESSIONSDIAGNOSTICSSUMMARYTYPE_CLIENTNAME_PLACEHOLDER_SESSIONDIAGNOSTICS_ENDPOINTURL := 12103,
	OPCUAID_SESSIONSDIAGNOSTICSSUMMARYTYPE_CLIENTNAME_PLACEHOLDER_SESSIONDIAGNOSTICS_LOCALEIDS := 12104,
	OPCUAID_SESSIONSDIAGNOSTICSSUMMARYTYPE_CLIENTNAME_PLACEHOLDER_SESSIONDIAGNOSTICS_ACTUALSESSIONTIMEOUT := 12105,
	OPCUAID_SESSIONSDIAGNOSTICSSUMMARYTYPE_CLIENTNAME_PLACEHOLDER_SESSIONDIAGNOSTICS_MAXRESPONSEMESSAGESIZE := 12106,
	OPCUAID_SESSIONSDIAGNOSTICSSUMMARYTYPE_CLIENTNAME_PLACEHOLDER_SESSIONDIAGNOSTICS_CLIENTCONNECTIONTIME := 12107,
	OPCUAID_SESSIONSDIAGNOSTICSSUMMARYTYPE_CLIENTNAME_PLACEHOLDER_SESSIONDIAGNOSTICS_CLIENTLASTCONTACTTIME := 12108,
	OPCUAID_SESSIONSDIAGNOSTICSSUMMARYTYPE_CLIENTNAME_PLACEHOLDER_SESSIONDIAGNOSTICS_CURRENTSUBSCRIPTIONSCOUNT := 12109,
	OPCUAID_SESSIONSDIAGNOSTICSSUMMARYTYPE_CLIENTNAME_PLACEHOLDER_SESSIONDIAGNOSTICS_CURRENTMONITOREDITEMSCOUNT := 12110,
	OPCUAID_SESSIONSDIAGNOSTICSSUMMARYTYPE_CLIENTNAME_PLACEHOLDER_SESSIONDIAGNOSTICS_CURRENTPUBLISHREQUESTSINQUEUE := 12111,
	OPCUAID_SESSIONSDIAGNOSTICSSUMMARYTYPE_CLIENTNAME_PLACEHOLDER_SESSIONDIAGNOSTICS_TOTALREQUESTCOUNT := 12112,
	OPCUAID_SESSIONSDIAGNOSTICSSUMMARYTYPE_CLIENTNAME_PLACEHOLDER_SESSIONDIAGNOSTICS_UNAUTHORIZEDREQUESTCOUNT := 12113,
	OPCUAID_SESSIONSDIAGNOSTICSSUMMARYTYPE_CLIENTNAME_PLACEHOLDER_SESSIONDIAGNOSTICS_READCOUNT := 12114,
	OPCUAID_SESSIONSDIAGNOSTICSSUMMARYTYPE_CLIENTNAME_PLACEHOLDER_SESSIONDIAGNOSTICS_HISTORYREADCOUNT := 12115,
	OPCUAID_SESSIONSDIAGNOSTICSSUMMARYTYPE_CLIENTNAME_PLACEHOLDER_SESSIONDIAGNOSTICS_WRITECOUNT := 12116,
	OPCUAID_SESSIONSDIAGNOSTICSSUMMARYTYPE_CLIENTNAME_PLACEHOLDER_SESSIONDIAGNOSTICS_HISTORYUPDATECOUNT := 12117,
	OPCUAID_SESSIONSDIAGNOSTICSSUMMARYTYPE_CLIENTNAME_PLACEHOLDER_SESSIONDIAGNOSTICS_CALLCOUNT := 12118,
	OPCUAID_SESSIONSDIAGNOSTICSSUMMARYTYPE_CLIENTNAME_PLACEHOLDER_SESSIONDIAGNOSTICS_CREATEMONITOREDITEMSCOUNT := 12119,
	OPCUAID_SESSIONSDIAGNOSTICSSUMMARYTYPE_CLIENTNAME_PLACEHOLDER_SESSIONDIAGNOSTICS_MODIFYMONITOREDITEMSCOUNT := 12120,
	OPCUAID_SESSIONSDIAGNOSTICSSUMMARYTYPE_CLIENTNAME_PLACEHOLDER_SESSIONDIAGNOSTICS_SETMONITORINGMODECOUNT := 12121,
	OPCUAID_SESSIONSDIAGNOSTICSSUMMARYTYPE_CLIENTNAME_PLACEHOLDER_SESSIONDIAGNOSTICS_SETTRIGGERINGCOUNT := 12122,
	OPCUAID_SESSIONSDIAGNOSTICSSUMMARYTYPE_CLIENTNAME_PLACEHOLDER_SESSIONDIAGNOSTICS_DELETEMONITOREDITEMSCOUNT := 12123,
	OPCUAID_SESSIONSDIAGNOSTICSSUMMARYTYPE_CLIENTNAME_PLACEHOLDER_SESSIONDIAGNOSTICS_CREATESUBSCRIPTIONCOUNT := 12124,
	OPCUAID_SESSIONSDIAGNOSTICSSUMMARYTYPE_CLIENTNAME_PLACEHOLDER_SESSIONDIAGNOSTICS_MODIFYSUBSCRIPTIONCOUNT := 12125,
	OPCUAID_SESSIONSDIAGNOSTICSSUMMARYTYPE_CLIENTNAME_PLACEHOLDER_SESSIONDIAGNOSTICS_SETPUBLISHINGMODECOUNT := 12126,
	OPCUAID_SESSIONSDIAGNOSTICSSUMMARYTYPE_CLIENTNAME_PLACEHOLDER_SESSIONDIAGNOSTICS_PUBLISHCOUNT := 12127,
	OPCUAID_SESSIONSDIAGNOSTICSSUMMARYTYPE_CLIENTNAME_PLACEHOLDER_SESSIONDIAGNOSTICS_REPUBLISHCOUNT := 12128,
	OPCUAID_SESSIONSDIAGNOSTICSSUMMARYTYPE_CLIENTNAME_PLACEHOLDER_SESSIONDIAGNOSTICS_TRANSFERSUBSCRIPTIONSCOUNT := 12129,
	OPCUAID_SESSIONSDIAGNOSTICSSUMMARYTYPE_CLIENTNAME_PLACEHOLDER_SESSIONDIAGNOSTICS_DELETESUBSCRIPTIONSCOUNT := 12130,
	OPCUAID_SESSIONSDIAGNOSTICSSUMMARYTYPE_CLIENTNAME_PLACEHOLDER_SESSIONDIAGNOSTICS_ADDNODESCOUNT := 12131,
	OPCUAID_SESSIONSDIAGNOSTICSSUMMARYTYPE_CLIENTNAME_PLACEHOLDER_SESSIONDIAGNOSTICS_ADDREFERENCESCOUNT := 12132,
	OPCUAID_SESSIONSDIAGNOSTICSSUMMARYTYPE_CLIENTNAME_PLACEHOLDER_SESSIONDIAGNOSTICS_DELETENODESCOUNT := 12133,
	OPCUAID_SESSIONSDIAGNOSTICSSUMMARYTYPE_CLIENTNAME_PLACEHOLDER_SESSIONDIAGNOSTICS_DELETEREFERENCESCOUNT := 12134,
	OPCUAID_SESSIONSDIAGNOSTICSSUMMARYTYPE_CLIENTNAME_PLACEHOLDER_SESSIONDIAGNOSTICS_BROWSECOUNT := 12135,
	OPCUAID_SESSIONSDIAGNOSTICSSUMMARYTYPE_CLIENTNAME_PLACEHOLDER_SESSIONDIAGNOSTICS_BROWSENEXTCOUNT := 12136,
	OPCUAID_SESSIONSDIAGNOSTICSSUMMARYTYPE_CLIENTNAME_PLACEHOLDER_SESSIONDIAGNOSTICS_TRANSLATEBROWSEPATHSTONODEIDSCOUNT := 12137,
	OPCUAID_SESSIONSDIAGNOSTICSSUMMARYTYPE_CLIENTNAME_PLACEHOLDER_SESSIONDIAGNOSTICS_QUERYFIRSTCOUNT := 12138,
	OPCUAID_SESSIONSDIAGNOSTICSSUMMARYTYPE_CLIENTNAME_PLACEHOLDER_SESSIONDIAGNOSTICS_QUERYNEXTCOUNT := 12139,
	OPCUAID_SESSIONSDIAGNOSTICSSUMMARYTYPE_CLIENTNAME_PLACEHOLDER_SESSIONDIAGNOSTICS_REGISTERNODESCOUNT := 12140,
	OPCUAID_SESSIONSDIAGNOSTICSSUMMARYTYPE_CLIENTNAME_PLACEHOLDER_SESSIONDIAGNOSTICS_UNREGISTERNODESCOUNT := 12141,
	OPCUAID_SESSIONSDIAGNOSTICSSUMMARYTYPE_CLIENTNAME_PLACEHOLDER_SESSIONSECURITYDIAGNOSTICS := 12142,
	OPCUAID_SESSIONSDIAGNOSTICSSUMMARYTYPE_CLIENTNAME_PLACEHOLDER_SESSIONSECURITYDIAGNOSTICS_SESSIONID := 12143,
	OPCUAID_SESSIONSDIAGNOSTICSSUMMARYTYPE_CLIENTNAME_PLACEHOLDER_SESSIONSECURITYDIAGNOSTICS_CLIENTUSERIDOFSESSION := 12144,
	OPCUAID_SESSIONSDIAGNOSTICSSUMMARYTYPE_CLIENTNAME_PLACEHOLDER_SESSIONSECURITYDIAGNOSTICS_CLIENTUSERIDHISTORY := 12145,
	OPCUAID_SESSIONSDIAGNOSTICSSUMMARYTYPE_CLIENTNAME_PLACEHOLDER_SESSIONSECURITYDIAGNOSTICS_AUTHENTICATIONMECHANISM := 12146,
	OPCUAID_SESSIONSDIAGNOSTICSSUMMARYTYPE_CLIENTNAME_PLACEHOLDER_SESSIONSECURITYDIAGNOSTICS_ENCODING := 12147,
	OPCUAID_SESSIONSDIAGNOSTICSSUMMARYTYPE_CLIENTNAME_PLACEHOLDER_SESSIONSECURITYDIAGNOSTICS_TRANSPORTPROTOCOL := 12148,
	OPCUAID_SESSIONSDIAGNOSTICSSUMMARYTYPE_CLIENTNAME_PLACEHOLDER_SESSIONSECURITYDIAGNOSTICS_SECURITYMODE := 12149,
	OPCUAID_SESSIONSDIAGNOSTICSSUMMARYTYPE_CLIENTNAME_PLACEHOLDER_SESSIONSECURITYDIAGNOSTICS_SECURITYPOLICYURI := 12150,
	OPCUAID_SESSIONSDIAGNOSTICSSUMMARYTYPE_CLIENTNAME_PLACEHOLDER_SESSIONSECURITYDIAGNOSTICS_CLIENTCERTIFICATE := 12151,
	OPCUAID_SESSIONSDIAGNOSTICSSUMMARYTYPE_CLIENTNAME_PLACEHOLDER_SUBSCRIPTIONDIAGNOSTICSARRAY := 12152,
	OPCUAID_SESSIONDIAGNOSTICSOBJECTTYPE_SESSIONDIAGNOSTICS := 2030,
	OPCUAID_SESSIONDIAGNOSTICSOBJECTTYPE_SESSIONDIAGNOSTICS_SESSIONID := 3131,
	OPCUAID_SESSIONDIAGNOSTICSOBJECTTYPE_SESSIONDIAGNOSTICS_SESSIONNAME := 3132,
	OPCUAID_SESSIONDIAGNOSTICSOBJECTTYPE_SESSIONDIAGNOSTICS_CLIENTDESCRIPTION := 3133,
	OPCUAID_SESSIONDIAGNOSTICSOBJECTTYPE_SESSIONDIAGNOSTICS_SERVERURI := 3134,
	OPCUAID_SESSIONDIAGNOSTICSOBJECTTYPE_SESSIONDIAGNOSTICS_ENDPOINTURL := 3135,
	OPCUAID_SESSIONDIAGNOSTICSOBJECTTYPE_SESSIONDIAGNOSTICS_LOCALEIDS := 3136,
	OPCUAID_SESSIONDIAGNOSTICSOBJECTTYPE_SESSIONDIAGNOSTICS_ACTUALSESSIONTIMEOUT := 3137,
	OPCUAID_SESSIONDIAGNOSTICSOBJECTTYPE_SESSIONDIAGNOSTICS_MAXRESPONSEMESSAGESIZE := 3138,
	OPCUAID_SESSIONDIAGNOSTICSOBJECTTYPE_SESSIONDIAGNOSTICS_CLIENTCONNECTIONTIME := 3139,
	OPCUAID_SESSIONDIAGNOSTICSOBJECTTYPE_SESSIONDIAGNOSTICS_CLIENTLASTCONTACTTIME := 3140,
	OPCUAID_SESSIONDIAGNOSTICSOBJECTTYPE_SESSIONDIAGNOSTICS_CURRENTSUBSCRIPTIONSCOUNT := 3141,
	OPCUAID_SESSIONDIAGNOSTICSOBJECTTYPE_SESSIONDIAGNOSTICS_CURRENTMONITOREDITEMSCOUNT := 3142,
	OPCUAID_SESSIONDIAGNOSTICSOBJECTTYPE_SESSIONDIAGNOSTICS_CURRENTPUBLISHREQUESTSINQUEUE := 3143,
	OPCUAID_SESSIONDIAGNOSTICSOBJECTTYPE_SESSIONDIAGNOSTICS_TOTALREQUESTCOUNT := 8898,
	OPCUAID_SESSIONDIAGNOSTICSOBJECTTYPE_SESSIONDIAGNOSTICS_UNAUTHORIZEDREQUESTCOUNT := 11891,
	OPCUAID_SESSIONDIAGNOSTICSOBJECTTYPE_SESSIONDIAGNOSTICS_READCOUNT := 3151,
	OPCUAID_SESSIONDIAGNOSTICSOBJECTTYPE_SESSIONDIAGNOSTICS_HISTORYREADCOUNT := 3152,
	OPCUAID_SESSIONDIAGNOSTICSOBJECTTYPE_SESSIONDIAGNOSTICS_WRITECOUNT := 3153,
	OPCUAID_SESSIONDIAGNOSTICSOBJECTTYPE_SESSIONDIAGNOSTICS_HISTORYUPDATECOUNT := 3154,
	OPCUAID_SESSIONDIAGNOSTICSOBJECTTYPE_SESSIONDIAGNOSTICS_CALLCOUNT := 3155,
	OPCUAID_SESSIONDIAGNOSTICSOBJECTTYPE_SESSIONDIAGNOSTICS_CREATEMONITOREDITEMSCOUNT := 3156,
	OPCUAID_SESSIONDIAGNOSTICSOBJECTTYPE_SESSIONDIAGNOSTICS_MODIFYMONITOREDITEMSCOUNT := 3157,
	OPCUAID_SESSIONDIAGNOSTICSOBJECTTYPE_SESSIONDIAGNOSTICS_SETMONITORINGMODECOUNT := 3158,
	OPCUAID_SESSIONDIAGNOSTICSOBJECTTYPE_SESSIONDIAGNOSTICS_SETTRIGGERINGCOUNT := 3159,
	OPCUAID_SESSIONDIAGNOSTICSOBJECTTYPE_SESSIONDIAGNOSTICS_DELETEMONITOREDITEMSCOUNT := 3160,
	OPCUAID_SESSIONDIAGNOSTICSOBJECTTYPE_SESSIONDIAGNOSTICS_CREATESUBSCRIPTIONCOUNT := 3161,
	OPCUAID_SESSIONDIAGNOSTICSOBJECTTYPE_SESSIONDIAGNOSTICS_MODIFYSUBSCRIPTIONCOUNT := 3162,
	OPCUAID_SESSIONDIAGNOSTICSOBJECTTYPE_SESSIONDIAGNOSTICS_SETPUBLISHINGMODECOUNT := 3163,
	OPCUAID_SESSIONDIAGNOSTICSOBJECTTYPE_SESSIONDIAGNOSTICS_PUBLISHCOUNT := 3164,
	OPCUAID_SESSIONDIAGNOSTICSOBJECTTYPE_SESSIONDIAGNOSTICS_REPUBLISHCOUNT := 3165,
	OPCUAID_SESSIONDIAGNOSTICSOBJECTTYPE_SESSIONDIAGNOSTICS_TRANSFERSUBSCRIPTIONSCOUNT := 3166,
	OPCUAID_SESSIONDIAGNOSTICSOBJECTTYPE_SESSIONDIAGNOSTICS_DELETESUBSCRIPTIONSCOUNT := 3167,
	OPCUAID_SESSIONDIAGNOSTICSOBJECTTYPE_SESSIONDIAGNOSTICS_ADDNODESCOUNT := 3168,
	OPCUAID_SESSIONDIAGNOSTICSOBJECTTYPE_SESSIONDIAGNOSTICS_ADDREFERENCESCOUNT := 3169,
	OPCUAID_SESSIONDIAGNOSTICSOBJECTTYPE_SESSIONDIAGNOSTICS_DELETENODESCOUNT := 3170,
	OPCUAID_SESSIONDIAGNOSTICSOBJECTTYPE_SESSIONDIAGNOSTICS_DELETEREFERENCESCOUNT := 3171,
	OPCUAID_SESSIONDIAGNOSTICSOBJECTTYPE_SESSIONDIAGNOSTICS_BROWSECOUNT := 3172,
	OPCUAID_SESSIONDIAGNOSTICSOBJECTTYPE_SESSIONDIAGNOSTICS_BROWSENEXTCOUNT := 3173,
	OPCUAID_SESSIONDIAGNOSTICSOBJECTTYPE_SESSIONDIAGNOSTICS_TRANSLATEBROWSEPATHSTONODEIDSCOUNT := 3174,
	OPCUAID_SESSIONDIAGNOSTICSOBJECTTYPE_SESSIONDIAGNOSTICS_QUERYFIRSTCOUNT := 3175,
	OPCUAID_SESSIONDIAGNOSTICSOBJECTTYPE_SESSIONDIAGNOSTICS_QUERYNEXTCOUNT := 3176,
	OPCUAID_SESSIONDIAGNOSTICSOBJECTTYPE_SESSIONDIAGNOSTICS_REGISTERNODESCOUNT := 3177,
	OPCUAID_SESSIONDIAGNOSTICSOBJECTTYPE_SESSIONDIAGNOSTICS_UNREGISTERNODESCOUNT := 3178,
	OPCUAID_SESSIONDIAGNOSTICSOBJECTTYPE_SESSIONSECURITYDIAGNOSTICS := 2031,
	OPCUAID_SESSIONDIAGNOSTICSOBJECTTYPE_SESSIONSECURITYDIAGNOSTICS_SESSIONID := 3179,
	OPCUAID_SESSIONDIAGNOSTICSOBJECTTYPE_SESSIONSECURITYDIAGNOSTICS_CLIENTUSERIDOFSESSION := 3180,
	OPCUAID_SESSIONDIAGNOSTICSOBJECTTYPE_SESSIONSECURITYDIAGNOSTICS_CLIENTUSERIDHISTORY := 3181,
	OPCUAID_SESSIONDIAGNOSTICSOBJECTTYPE_SESSIONSECURITYDIAGNOSTICS_AUTHENTICATIONMECHANISM := 3182,
	OPCUAID_SESSIONDIAGNOSTICSOBJECTTYPE_SESSIONSECURITYDIAGNOSTICS_ENCODING := 3183,
	OPCUAID_SESSIONDIAGNOSTICSOBJECTTYPE_SESSIONSECURITYDIAGNOSTICS_TRANSPORTPROTOCOL := 3184,
	OPCUAID_SESSIONDIAGNOSTICSOBJECTTYPE_SESSIONSECURITYDIAGNOSTICS_SECURITYMODE := 3185,
	OPCUAID_SESSIONDIAGNOSTICSOBJECTTYPE_SESSIONSECURITYDIAGNOSTICS_SECURITYPOLICYURI := 3186,
	OPCUAID_SESSIONDIAGNOSTICSOBJECTTYPE_SESSIONSECURITYDIAGNOSTICS_CLIENTCERTIFICATE := 3187,
	OPCUAID_SESSIONDIAGNOSTICSOBJECTTYPE_SUBSCRIPTIONDIAGNOSTICSARRAY := 2032,
	OPCUAID_SERVERREDUNDANCYTYPE_REDUNDANCYSUPPORT := 2035,
	OPCUAID_TRANSPARENTREDUNDANCYTYPE_CURRENTSERVERID := 2037,
	OPCUAID_TRANSPARENTREDUNDANCYTYPE_REDUNDANTSERVERARRAY := 2038,
	OPCUAID_NONTRANSPARENTREDUNDANCYTYPE_SERVERURIARRAY := 2040,
	OPCUAID_NONTRANSPARENTNETWORKREDUNDANCYTYPE_SERVERNETWORKGROUPS := 11948,
	OPCUAID_OPERATIONLIMITSTYPE_MAXNODESPERREAD := 11565,
	OPCUAID_OPERATIONLIMITSTYPE_MAXNODESPERHISTORYREADDATA := 12161,
	OPCUAID_OPERATIONLIMITSTYPE_MAXNODESPERHISTORYREADEVENTS := 12162,
	OPCUAID_OPERATIONLIMITSTYPE_MAXNODESPERWRITE := 11567,
	OPCUAID_OPERATIONLIMITSTYPE_MAXNODESPERHISTORYUPDATEDATA := 12163,
	OPCUAID_OPERATIONLIMITSTYPE_MAXNODESPERHISTORYUPDATEEVENTS := 12164,
	OPCUAID_OPERATIONLIMITSTYPE_MAXNODESPERMETHODCALL := 11569,
	OPCUAID_OPERATIONLIMITSTYPE_MAXNODESPERBROWSE := 11570,
	OPCUAID_OPERATIONLIMITSTYPE_MAXNODESPERREGISTERNODES := 11571,
	OPCUAID_OPERATIONLIMITSTYPE_MAXNODESPERTRANSLATEBROWSEPATHSTONODEIDS := 11572,
	OPCUAID_OPERATIONLIMITSTYPE_MAXNODESPERNODEMANAGEMENT := 11573,
	OPCUAID_OPERATIONLIMITSTYPE_MAXMONITOREDITEMSPERCALL := 11574,
	OPCUAID_FILETYPE_SIZE := 11576,
	OPCUAID_FILETYPE_WRITABLE := 12686,
	OPCUAID_FILETYPE_USERWRITABLE := 12687,
	OPCUAID_FILETYPE_OPENCOUNT := 11579,
	OPCUAID_FILETYPE_MIMETYPE := 13341,
	OPCUAID_FILETYPE_OPEN_INPUTARGUMENTS := 11581,
	OPCUAID_FILETYPE_OPEN_OUTPUTARGUMENTS := 11582,
	OPCUAID_FILETYPE_CLOSE_INPUTARGUMENTS := 11584,
	OPCUAID_FILETYPE_READ_INPUTARGUMENTS := 11586,
	OPCUAID_FILETYPE_READ_OUTPUTARGUMENTS := 11587,
	OPCUAID_FILETYPE_WRITE_INPUTARGUMENTS := 11589,
	OPCUAID_FILETYPE_GETPOSITION_INPUTARGUMENTS := 11591,
	OPCUAID_FILETYPE_GETPOSITION_OUTPUTARGUMENTS := 11592,
	OPCUAID_FILETYPE_SETPOSITION_INPUTARGUMENTS := 11594,
	OPCUAID_ADDRESSSPACEFILETYPE_OPEN_INPUTARGUMENTS := 11601,
	OPCUAID_ADDRESSSPACEFILETYPE_OPEN_OUTPUTARGUMENTS := 11602,
	OPCUAID_ADDRESSSPACEFILETYPE_CLOSE_INPUTARGUMENTS := 11604,
	OPCUAID_ADDRESSSPACEFILETYPE_READ_INPUTARGUMENTS := 11606,
	OPCUAID_ADDRESSSPACEFILETYPE_READ_OUTPUTARGUMENTS := 11607,
	OPCUAID_ADDRESSSPACEFILETYPE_WRITE_INPUTARGUMENTS := 11609,
	OPCUAID_ADDRESSSPACEFILETYPE_GETPOSITION_INPUTARGUMENTS := 11611,
	OPCUAID_ADDRESSSPACEFILETYPE_GETPOSITION_OUTPUTARGUMENTS := 11612,
	OPCUAID_ADDRESSSPACEFILETYPE_SETPOSITION_INPUTARGUMENTS := 11614,
	OPCUAID_NAMESPACEMETADATATYPE_NAMESPACEURI := 11617,
	OPCUAID_NAMESPACEMETADATATYPE_NAMESPACEVERSION := 11618,
	OPCUAID_NAMESPACEMETADATATYPE_NAMESPACEPUBLICATIONDATE := 11619,
	OPCUAID_NAMESPACEMETADATATYPE_ISNAMESPACESUBSET := 11620,
	OPCUAID_NAMESPACEMETADATATYPE_STATICNODEIDTYPES := 11621,
	OPCUAID_NAMESPACEMETADATATYPE_STATICNUMERICNODEIDRANGE := 11622,
	OPCUAID_NAMESPACEMETADATATYPE_STATICSTRINGNODEIDPATTERN := 11623,
	OPCUAID_NAMESPACEMETADATATYPE_NAMESPACEFILE_SIZE := 11625,
	OPCUAID_NAMESPACEMETADATATYPE_NAMESPACEFILE_WRITABLE := 12690,
	OPCUAID_NAMESPACEMETADATATYPE_NAMESPACEFILE_USERWRITABLE := 12691,
	OPCUAID_NAMESPACEMETADATATYPE_NAMESPACEFILE_OPENCOUNT := 11628,
	OPCUAID_NAMESPACEMETADATATYPE_NAMESPACEFILE_OPEN_INPUTARGUMENTS := 11630,
	OPCUAID_NAMESPACEMETADATATYPE_NAMESPACEFILE_OPEN_OUTPUTARGUMENTS := 11631,
	OPCUAID_NAMESPACEMETADATATYPE_NAMESPACEFILE_CLOSE_INPUTARGUMENTS := 11633,
	OPCUAID_NAMESPACEMETADATATYPE_NAMESPACEFILE_READ_INPUTARGUMENTS := 11635,
	OPCUAID_NAMESPACEMETADATATYPE_NAMESPACEFILE_READ_OUTPUTARGUMENTS := 11636,
	OPCUAID_NAMESPACEMETADATATYPE_NAMESPACEFILE_WRITE_INPUTARGUMENTS := 11638,
	OPCUAID_NAMESPACEMETADATATYPE_NAMESPACEFILE_GETPOSITION_INPUTARGUMENTS := 11640,
	OPCUAID_NAMESPACEMETADATATYPE_NAMESPACEFILE_GETPOSITION_OUTPUTARGUMENTS := 11641,
	OPCUAID_NAMESPACEMETADATATYPE_NAMESPACEFILE_SETPOSITION_INPUTARGUMENTS := 11643,
	OPCUAID_NAMESPACEMETADATATYPE_DEFAULTROLEPERMISSIONS := 16137,
	OPCUAID_NAMESPACEMETADATATYPE_DEFAULTUSERROLEPERMISSIONS := 16138,
	OPCUAID_NAMESPACEMETADATATYPE_DEFAULTACCESSRESTRICTIONS := 16139,
	OPCUAID_NAMESPACESTYPE_NAMESPACEIDENTIFIER_PLACEHOLDER_NAMESPACEURI := 11647,
	OPCUAID_NAMESPACESTYPE_NAMESPACEIDENTIFIER_PLACEHOLDER_NAMESPACEVERSION := 11648,
	OPCUAID_NAMESPACESTYPE_NAMESPACEIDENTIFIER_PLACEHOLDER_NAMESPACEPUBLICATIONDATE := 11649,
	OPCUAID_NAMESPACESTYPE_NAMESPACEIDENTIFIER_PLACEHOLDER_ISNAMESPACESUBSET := 11650,
	OPCUAID_NAMESPACESTYPE_NAMESPACEIDENTIFIER_PLACEHOLDER_STATICNODEIDTYPES := 11651,
	OPCUAID_NAMESPACESTYPE_NAMESPACEIDENTIFIER_PLACEHOLDER_STATICNUMERICNODEIDRANGE := 11652,
	OPCUAID_NAMESPACESTYPE_NAMESPACEIDENTIFIER_PLACEHOLDER_STATICSTRINGNODEIDPATTERN := 11653,
	OPCUAID_NAMESPACESTYPE_NAMESPACEIDENTIFIER_PLACEHOLDER_NAMESPACEFILE_SIZE := 11655,
	OPCUAID_NAMESPACESTYPE_NAMESPACEIDENTIFIER_PLACEHOLDER_NAMESPACEFILE_WRITABLE := 12692,
	OPCUAID_NAMESPACESTYPE_NAMESPACEIDENTIFIER_PLACEHOLDER_NAMESPACEFILE_USERWRITABLE := 12693,
	OPCUAID_NAMESPACESTYPE_NAMESPACEIDENTIFIER_PLACEHOLDER_NAMESPACEFILE_OPENCOUNT := 11658,
	OPCUAID_NAMESPACESTYPE_NAMESPACEIDENTIFIER_PLACEHOLDER_NAMESPACEFILE_OPEN_INPUTARGUMENTS := 11660,
	OPCUAID_NAMESPACESTYPE_NAMESPACEIDENTIFIER_PLACEHOLDER_NAMESPACEFILE_OPEN_OUTPUTARGUMENTS := 11661,
	OPCUAID_NAMESPACESTYPE_NAMESPACEIDENTIFIER_PLACEHOLDER_NAMESPACEFILE_CLOSE_INPUTARGUMENTS := 11663,
	OPCUAID_NAMESPACESTYPE_NAMESPACEIDENTIFIER_PLACEHOLDER_NAMESPACEFILE_READ_INPUTARGUMENTS := 11665,
	OPCUAID_NAMESPACESTYPE_NAMESPACEIDENTIFIER_PLACEHOLDER_NAMESPACEFILE_READ_OUTPUTARGUMENTS := 11666,
	OPCUAID_NAMESPACESTYPE_NAMESPACEIDENTIFIER_PLACEHOLDER_NAMESPACEFILE_WRITE_INPUTARGUMENTS := 11668,
	OPCUAID_NAMESPACESTYPE_NAMESPACEIDENTIFIER_PLACEHOLDER_NAMESPACEFILE_GETPOSITION_INPUTARGUMENTS := 11670,
	OPCUAID_NAMESPACESTYPE_NAMESPACEIDENTIFIER_PLACEHOLDER_NAMESPACEFILE_GETPOSITION_OUTPUTARGUMENTS := 11671,
	OPCUAID_NAMESPACESTYPE_NAMESPACEIDENTIFIER_PLACEHOLDER_NAMESPACEFILE_SETPOSITION_INPUTARGUMENTS := 11673,
	OPCUAID_BASEEVENTTYPE_EVENTID := 2042,
	OPCUAID_BASEEVENTTYPE_EVENTTYPE := 2043,
	OPCUAID_BASEEVENTTYPE_SOURCENODE := 2044,
	OPCUAID_BASEEVENTTYPE_SOURCENAME := 2045,
	OPCUAID_BASEEVENTTYPE_TIME := 2046,
	OPCUAID_BASEEVENTTYPE_RECEIVETIME := 2047,
	OPCUAID_BASEEVENTTYPE_LOCALTIME := 3190,
	OPCUAID_BASEEVENTTYPE_MESSAGE := 2050,
	OPCUAID_BASEEVENTTYPE_SEVERITY := 2051,
	OPCUAID_AUDITEVENTTYPE_ACTIONTIMESTAMP := 2053,
	OPCUAID_AUDITEVENTTYPE_STATUS := 2054,
	OPCUAID_AUDITEVENTTYPE_SERVERID := 2055,
	OPCUAID_AUDITEVENTTYPE_CLIENTAUDITENTRYID := 2056,
	OPCUAID_AUDITEVENTTYPE_CLIENTUSERID := 2057,
	OPCUAID_AUDITSECURITYEVENTTYPE_STATUSCODEID := 17615,
	OPCUAID_AUDITCHANNELEVENTTYPE_SECURECHANNELID := 2745,
	OPCUAID_AUDITOPENSECURECHANNELEVENTTYPE_CLIENTCERTIFICATE := 2061,
	OPCUAID_AUDITOPENSECURECHANNELEVENTTYPE_CLIENTCERTIFICATETHUMBPRINT := 2746,
	OPCUAID_AUDITOPENSECURECHANNELEVENTTYPE_REQUESTTYPE := 2062,
	OPCUAID_AUDITOPENSECURECHANNELEVENTTYPE_SECURITYPOLICYURI := 2063,
	OPCUAID_AUDITOPENSECURECHANNELEVENTTYPE_SECURITYMODE := 2065,
	OPCUAID_AUDITOPENSECURECHANNELEVENTTYPE_REQUESTEDLIFETIME := 2066,
	OPCUAID_AUDITSESSIONEVENTTYPE_SESSIONID := 2070,
	OPCUAID_AUDITCREATESESSIONEVENTTYPE_SECURECHANNELID := 2072,
	OPCUAID_AUDITCREATESESSIONEVENTTYPE_CLIENTCERTIFICATE := 2073,
	OPCUAID_AUDITCREATESESSIONEVENTTYPE_CLIENTCERTIFICATETHUMBPRINT := 2747,
	OPCUAID_AUDITCREATESESSIONEVENTTYPE_REVISEDSESSIONTIMEOUT := 2074,
	OPCUAID_AUDITURLMISMATCHEVENTTYPE_ENDPOINTURL := 2749,
	OPCUAID_AUDITACTIVATESESSIONEVENTTYPE_CLIENTSOFTWARECERTIFICATES := 2076,
	OPCUAID_AUDITACTIVATESESSIONEVENTTYPE_USERIDENTITYTOKEN := 2077,
	OPCUAID_AUDITACTIVATESESSIONEVENTTYPE_SECURECHANNELID := 11485,
	OPCUAID_AUDITCANCELEVENTTYPE_REQUESTHANDLE := 2079,
	OPCUAID_AUDITCERTIFICATEEVENTTYPE_CERTIFICATE := 2081,
	OPCUAID_AUDITCERTIFICATEDATAMISMATCHEVENTTYPE_INVALIDHOSTNAME := 2083,
	OPCUAID_AUDITCERTIFICATEDATAMISMATCHEVENTTYPE_INVALIDURI := 2084,
	OPCUAID_AUDITADDNODESEVENTTYPE_NODESTOADD := 2092,
	OPCUAID_AUDITDELETENODESEVENTTYPE_NODESTODELETE := 2094,
	OPCUAID_AUDITADDREFERENCESEVENTTYPE_REFERENCESTOADD := 2096,
	OPCUAID_AUDITDELETEREFERENCESEVENTTYPE_REFERENCESTODELETE := 2098,
	OPCUAID_AUDITWRITEUPDATEEVENTTYPE_ATTRIBUTEID := 2750,
	OPCUAID_AUDITWRITEUPDATEEVENTTYPE_INDEXRANGE := 2101,
	OPCUAID_AUDITWRITEUPDATEEVENTTYPE_OLDVALUE := 2102,
	OPCUAID_AUDITWRITEUPDATEEVENTTYPE_NEWVALUE := 2103,
	OPCUAID_AUDITHISTORYUPDATEEVENTTYPE_PARAMETERDATATYPEID := 2751,
	OPCUAID_AUDITUPDATEMETHODEVENTTYPE_METHODID := 2128,
	OPCUAID_AUDITUPDATEMETHODEVENTTYPE_INPUTARGUMENTS := 2129,
	OPCUAID_SYSTEMSTATUSCHANGEEVENTTYPE_SYSTEMSTATE := 11696,
	OPCUAID_GENERALMODELCHANGEEVENTTYPE_CHANGES := 2134,
	OPCUAID_SEMANTICCHANGEEVENTTYPE_CHANGES := 2739,
	OPCUAID_PROGRESSEVENTTYPE_CONTEXT := 12502,
	OPCUAID_PROGRESSEVENTTYPE_PROGRESS := 12503,
	OPCUAID_SERVERSTATUSTYPE_STARTTIME := 2139,
	OPCUAID_SERVERSTATUSTYPE_CURRENTTIME := 2140,
	OPCUAID_SERVERSTATUSTYPE_STATE := 2141,
	OPCUAID_SERVERSTATUSTYPE_BUILDINFO := 2142,
	OPCUAID_SERVERSTATUSTYPE_BUILDINFO_PRODUCTURI := 3698,
	OPCUAID_SERVERSTATUSTYPE_BUILDINFO_MANUFACTURERNAME := 3699,
	OPCUAID_SERVERSTATUSTYPE_BUILDINFO_PRODUCTNAME := 3700,
	OPCUAID_SERVERSTATUSTYPE_BUILDINFO_SOFTWAREVERSION := 3701,
	OPCUAID_SERVERSTATUSTYPE_BUILDINFO_BUILDNUMBER := 3702,
	OPCUAID_SERVERSTATUSTYPE_BUILDINFO_BUILDDATE := 3703,
	OPCUAID_SERVERSTATUSTYPE_SECONDSTILLSHUTDOWN := 2752,
	OPCUAID_SERVERSTATUSTYPE_SHUTDOWNREASON := 2753,
	OPCUAID_BUILDINFOTYPE_PRODUCTURI := 3052,
	OPCUAID_BUILDINFOTYPE_MANUFACTURERNAME := 3053,
	OPCUAID_BUILDINFOTYPE_PRODUCTNAME := 3054,
	OPCUAID_BUILDINFOTYPE_SOFTWAREVERSION := 3055,
	OPCUAID_BUILDINFOTYPE_BUILDNUMBER := 3056,
	OPCUAID_BUILDINFOTYPE_BUILDDATE := 3057,
	OPCUAID_SERVERDIAGNOSTICSSUMMARYTYPE_SERVERVIEWCOUNT := 2151,
	OPCUAID_SERVERDIAGNOSTICSSUMMARYTYPE_CURRENTSESSIONCOUNT := 2152,
	OPCUAID_SERVERDIAGNOSTICSSUMMARYTYPE_CUMULATEDSESSIONCOUNT := 2153,
	OPCUAID_SERVERDIAGNOSTICSSUMMARYTYPE_SECURITYREJECTEDSESSIONCOUNT := 2154,
	OPCUAID_SERVERDIAGNOSTICSSUMMARYTYPE_REJECTEDSESSIONCOUNT := 2155,
	OPCUAID_SERVERDIAGNOSTICSSUMMARYTYPE_SESSIONTIMEOUTCOUNT := 2156,
	OPCUAID_SERVERDIAGNOSTICSSUMMARYTYPE_SESSIONABORTCOUNT := 2157,
	OPCUAID_SERVERDIAGNOSTICSSUMMARYTYPE_PUBLISHINGINTERVALCOUNT := 2159,
	OPCUAID_SERVERDIAGNOSTICSSUMMARYTYPE_CURRENTSUBSCRIPTIONCOUNT := 2160,
	OPCUAID_SERVERDIAGNOSTICSSUMMARYTYPE_CUMULATEDSUBSCRIPTIONCOUNT := 2161,
	OPCUAID_SERVERDIAGNOSTICSSUMMARYTYPE_SECURITYREJECTEDREQUESTSCOUNT := 2162,
	OPCUAID_SERVERDIAGNOSTICSSUMMARYTYPE_REJECTEDREQUESTSCOUNT := 2163,
	OPCUAID_SAMPLINGINTERVALDIAGNOSTICSARRAYTYPE_SAMPLINGINTERVALDIAGNOSTICS := 12779,
	OPCUAID_SAMPLINGINTERVALDIAGNOSTICSARRAYTYPE_SAMPLINGINTERVALDIAGNOSTICS_SAMPLINGINTERVAL := 12780,
	OPCUAID_SAMPLINGINTERVALDIAGNOSTICSARRAYTYPE_SAMPLINGINTERVALDIAGNOSTICS_SAMPLEDMONITOREDITEMSCOUNT := 12781,
	OPCUAID_SAMPLINGINTERVALDIAGNOSTICSARRAYTYPE_SAMPLINGINTERVALDIAGNOSTICS_MAXSAMPLEDMONITOREDITEMSCOUNT := 12782,
	OPCUAID_SAMPLINGINTERVALDIAGNOSTICSARRAYTYPE_SAMPLINGINTERVALDIAGNOSTICS_DISABLEDMONITOREDITEMSSAMPLINGCOUNT := 12783,
	OPCUAID_SAMPLINGINTERVALDIAGNOSTICSTYPE_SAMPLINGINTERVAL := 2166,
	OPCUAID_SAMPLINGINTERVALDIAGNOSTICSTYPE_SAMPLEDMONITOREDITEMSCOUNT := 11697,
	OPCUAID_SAMPLINGINTERVALDIAGNOSTICSTYPE_MAXSAMPLEDMONITOREDITEMSCOUNT := 11698,
	OPCUAID_SAMPLINGINTERVALDIAGNOSTICSTYPE_DISABLEDMONITOREDITEMSSAMPLINGCOUNT := 11699,
	OPCUAID_SUBSCRIPTIONDIAGNOSTICSARRAYTYPE_SUBSCRIPTIONDIAGNOSTICS := 12784,
	OPCUAID_SUBSCRIPTIONDIAGNOSTICSARRAYTYPE_SUBSCRIPTIONDIAGNOSTICS_SESSIONID := 12785,
	OPCUAID_SUBSCRIPTIONDIAGNOSTICSARRAYTYPE_SUBSCRIPTIONDIAGNOSTICS_SUBSCRIPTIONID := 12786,
	OPCUAID_SUBSCRIPTIONDIAGNOSTICSARRAYTYPE_SUBSCRIPTIONDIAGNOSTICS_PRIORITY := 12787,
	OPCUAID_SUBSCRIPTIONDIAGNOSTICSARRAYTYPE_SUBSCRIPTIONDIAGNOSTICS_PUBLISHINGINTERVAL := 12788,
	OPCUAID_SUBSCRIPTIONDIAGNOSTICSARRAYTYPE_SUBSCRIPTIONDIAGNOSTICS_MAXKEEPALIVECOUNT := 12789,
	OPCUAID_SUBSCRIPTIONDIAGNOSTICSARRAYTYPE_SUBSCRIPTIONDIAGNOSTICS_MAXLIFETIMECOUNT := 12790,
	OPCUAID_SUBSCRIPTIONDIAGNOSTICSARRAYTYPE_SUBSCRIPTIONDIAGNOSTICS_MAXNOTIFICATIONSPERPUBLISH := 12791,
	OPCUAID_SUBSCRIPTIONDIAGNOSTICSARRAYTYPE_SUBSCRIPTIONDIAGNOSTICS_PUBLISHINGENABLED := 12792,
	OPCUAID_SUBSCRIPTIONDIAGNOSTICSARRAYTYPE_SUBSCRIPTIONDIAGNOSTICS_MODIFYCOUNT := 12793,
	OPCUAID_SUBSCRIPTIONDIAGNOSTICSARRAYTYPE_SUBSCRIPTIONDIAGNOSTICS_ENABLECOUNT := 12794,
	OPCUAID_SUBSCRIPTIONDIAGNOSTICSARRAYTYPE_SUBSCRIPTIONDIAGNOSTICS_DISABLECOUNT := 12795,
	OPCUAID_SUBSCRIPTIONDIAGNOSTICSARRAYTYPE_SUBSCRIPTIONDIAGNOSTICS_REPUBLISHREQUESTCOUNT := 12796,
	OPCUAID_SUBSCRIPTIONDIAGNOSTICSARRAYTYPE_SUBSCRIPTIONDIAGNOSTICS_REPUBLISHMESSAGEREQUESTCOUNT := 12797,
	OPCUAID_SUBSCRIPTIONDIAGNOSTICSARRAYTYPE_SUBSCRIPTIONDIAGNOSTICS_REPUBLISHMESSAGECOUNT := 12798,
	OPCUAID_SUBSCRIPTIONDIAGNOSTICSARRAYTYPE_SUBSCRIPTIONDIAGNOSTICS_TRANSFERREQUESTCOUNT := 12799,
	OPCUAID_SUBSCRIPTIONDIAGNOSTICSARRAYTYPE_SUBSCRIPTIONDIAGNOSTICS_TRANSFERREDTOALTCLIENTCOUNT := 12800,
	OPCUAID_SUBSCRIPTIONDIAGNOSTICSARRAYTYPE_SUBSCRIPTIONDIAGNOSTICS_TRANSFERREDTOSAMECLIENTCOUNT := 12801,
	OPCUAID_SUBSCRIPTIONDIAGNOSTICSARRAYTYPE_SUBSCRIPTIONDIAGNOSTICS_PUBLISHREQUESTCOUNT := 12802,
	OPCUAID_SUBSCRIPTIONDIAGNOSTICSARRAYTYPE_SUBSCRIPTIONDIAGNOSTICS_DATACHANGENOTIFICATIONSCOUNT := 12803,
	OPCUAID_SUBSCRIPTIONDIAGNOSTICSARRAYTYPE_SUBSCRIPTIONDIAGNOSTICS_EVENTNOTIFICATIONSCOUNT := 12804,
	OPCUAID_SUBSCRIPTIONDIAGNOSTICSARRAYTYPE_SUBSCRIPTIONDIAGNOSTICS_NOTIFICATIONSCOUNT := 12805,
	OPCUAID_SUBSCRIPTIONDIAGNOSTICSARRAYTYPE_SUBSCRIPTIONDIAGNOSTICS_LATEPUBLISHREQUESTCOUNT := 12806,
	OPCUAID_SUBSCRIPTIONDIAGNOSTICSARRAYTYPE_SUBSCRIPTIONDIAGNOSTICS_CURRENTKEEPALIVECOUNT := 12807,
	OPCUAID_SUBSCRIPTIONDIAGNOSTICSARRAYTYPE_SUBSCRIPTIONDIAGNOSTICS_CURRENTLIFETIMECOUNT := 12808,
	OPCUAID_SUBSCRIPTIONDIAGNOSTICSARRAYTYPE_SUBSCRIPTIONDIAGNOSTICS_UNACKNOWLEDGEDMESSAGECOUNT := 12809,
	OPCUAID_SUBSCRIPTIONDIAGNOSTICSARRAYTYPE_SUBSCRIPTIONDIAGNOSTICS_DISCARDEDMESSAGECOUNT := 12810,
	OPCUAID_SUBSCRIPTIONDIAGNOSTICSARRAYTYPE_SUBSCRIPTIONDIAGNOSTICS_MONITOREDITEMCOUNT := 12811,
	OPCUAID_SUBSCRIPTIONDIAGNOSTICSARRAYTYPE_SUBSCRIPTIONDIAGNOSTICS_DISABLEDMONITOREDITEMCOUNT := 12812,
	OPCUAID_SUBSCRIPTIONDIAGNOSTICSARRAYTYPE_SUBSCRIPTIONDIAGNOSTICS_MONITORINGQUEUEOVERFLOWCOUNT := 12813,
	OPCUAID_SUBSCRIPTIONDIAGNOSTICSARRAYTYPE_SUBSCRIPTIONDIAGNOSTICS_NEXTSEQUENCENUMBER := 12814,
	OPCUAID_SUBSCRIPTIONDIAGNOSTICSARRAYTYPE_SUBSCRIPTIONDIAGNOSTICS_EVENTQUEUEOVERFLOWCOUNT := 12815,
	OPCUAID_SUBSCRIPTIONDIAGNOSTICSTYPE_SESSIONID := 2173,
	OPCUAID_SUBSCRIPTIONDIAGNOSTICSTYPE_SUBSCRIPTIONID := 2174,
	OPCUAID_SUBSCRIPTIONDIAGNOSTICSTYPE_PRIORITY := 2175,
	OPCUAID_SUBSCRIPTIONDIAGNOSTICSTYPE_PUBLISHINGINTERVAL := 2176,
	OPCUAID_SUBSCRIPTIONDIAGNOSTICSTYPE_MAXKEEPALIVECOUNT := 2177,
	OPCUAID_SUBSCRIPTIONDIAGNOSTICSTYPE_MAXLIFETIMECOUNT := 8888,
	OPCUAID_SUBSCRIPTIONDIAGNOSTICSTYPE_MAXNOTIFICATIONSPERPUBLISH := 2179,
	OPCUAID_SUBSCRIPTIONDIAGNOSTICSTYPE_PUBLISHINGENABLED := 2180,
	OPCUAID_SUBSCRIPTIONDIAGNOSTICSTYPE_MODIFYCOUNT := 2181,
	OPCUAID_SUBSCRIPTIONDIAGNOSTICSTYPE_ENABLECOUNT := 2182,
	OPCUAID_SUBSCRIPTIONDIAGNOSTICSTYPE_DISABLECOUNT := 2183,
	OPCUAID_SUBSCRIPTIONDIAGNOSTICSTYPE_REPUBLISHREQUESTCOUNT := 2184,
	OPCUAID_SUBSCRIPTIONDIAGNOSTICSTYPE_REPUBLISHMESSAGEREQUESTCOUNT := 2185,
	OPCUAID_SUBSCRIPTIONDIAGNOSTICSTYPE_REPUBLISHMESSAGECOUNT := 2186,
	OPCUAID_SUBSCRIPTIONDIAGNOSTICSTYPE_TRANSFERREQUESTCOUNT := 2187,
	OPCUAID_SUBSCRIPTIONDIAGNOSTICSTYPE_TRANSFERREDTOALTCLIENTCOUNT := 2188,
	OPCUAID_SUBSCRIPTIONDIAGNOSTICSTYPE_TRANSFERREDTOSAMECLIENTCOUNT := 2189,
	OPCUAID_SUBSCRIPTIONDIAGNOSTICSTYPE_PUBLISHREQUESTCOUNT := 2190,
	OPCUAID_SUBSCRIPTIONDIAGNOSTICSTYPE_DATACHANGENOTIFICATIONSCOUNT := 2191,
	OPCUAID_SUBSCRIPTIONDIAGNOSTICSTYPE_EVENTNOTIFICATIONSCOUNT := 2998,
	OPCUAID_SUBSCRIPTIONDIAGNOSTICSTYPE_NOTIFICATIONSCOUNT := 2193,
	OPCUAID_SUBSCRIPTIONDIAGNOSTICSTYPE_LATEPUBLISHREQUESTCOUNT := 8889,
	OPCUAID_SUBSCRIPTIONDIAGNOSTICSTYPE_CURRENTKEEPALIVECOUNT := 8890,
	OPCUAID_SUBSCRIPTIONDIAGNOSTICSTYPE_CURRENTLIFETIMECOUNT := 8891,
	OPCUAID_SUBSCRIPTIONDIAGNOSTICSTYPE_UNACKNOWLEDGEDMESSAGECOUNT := 8892,
	OPCUAID_SUBSCRIPTIONDIAGNOSTICSTYPE_DISCARDEDMESSAGECOUNT := 8893,
	OPCUAID_SUBSCRIPTIONDIAGNOSTICSTYPE_MONITOREDITEMCOUNT := 8894,
	OPCUAID_SUBSCRIPTIONDIAGNOSTICSTYPE_DISABLEDMONITOREDITEMCOUNT := 8895,
	OPCUAID_SUBSCRIPTIONDIAGNOSTICSTYPE_MONITORINGQUEUEOVERFLOWCOUNT := 8896,
	OPCUAID_SUBSCRIPTIONDIAGNOSTICSTYPE_NEXTSEQUENCENUMBER := 8897,
	OPCUAID_SUBSCRIPTIONDIAGNOSTICSTYPE_EVENTQUEUEOVERFLOWCOUNT := 8902,
	OPCUAID_SESSIONDIAGNOSTICSARRAYTYPE_SESSIONDIAGNOSTICS := 12816,
	OPCUAID_SESSIONDIAGNOSTICSARRAYTYPE_SESSIONDIAGNOSTICS_SESSIONID := 12817,
	OPCUAID_SESSIONDIAGNOSTICSARRAYTYPE_SESSIONDIAGNOSTICS_SESSIONNAME := 12818,
	OPCUAID_SESSIONDIAGNOSTICSARRAYTYPE_SESSIONDIAGNOSTICS_CLIENTDESCRIPTION := 12819,
	OPCUAID_SESSIONDIAGNOSTICSARRAYTYPE_SESSIONDIAGNOSTICS_SERVERURI := 12820,
	OPCUAID_SESSIONDIAGNOSTICSARRAYTYPE_SESSIONDIAGNOSTICS_ENDPOINTURL := 12821,
	OPCUAID_SESSIONDIAGNOSTICSARRAYTYPE_SESSIONDIAGNOSTICS_LOCALEIDS := 12822,
	OPCUAID_SESSIONDIAGNOSTICSARRAYTYPE_SESSIONDIAGNOSTICS_ACTUALSESSIONTIMEOUT := 12823,
	OPCUAID_SESSIONDIAGNOSTICSARRAYTYPE_SESSIONDIAGNOSTICS_MAXRESPONSEMESSAGESIZE := 12824,
	OPCUAID_SESSIONDIAGNOSTICSARRAYTYPE_SESSIONDIAGNOSTICS_CLIENTCONNECTIONTIME := 12825,
	OPCUAID_SESSIONDIAGNOSTICSARRAYTYPE_SESSIONDIAGNOSTICS_CLIENTLASTCONTACTTIME := 12826,
	OPCUAID_SESSIONDIAGNOSTICSARRAYTYPE_SESSIONDIAGNOSTICS_CURRENTSUBSCRIPTIONSCOUNT := 12827,
	OPCUAID_SESSIONDIAGNOSTICSARRAYTYPE_SESSIONDIAGNOSTICS_CURRENTMONITOREDITEMSCOUNT := 12828,
	OPCUAID_SESSIONDIAGNOSTICSARRAYTYPE_SESSIONDIAGNOSTICS_CURRENTPUBLISHREQUESTSINQUEUE := 12829,
	OPCUAID_SESSIONDIAGNOSTICSARRAYTYPE_SESSIONDIAGNOSTICS_TOTALREQUESTCOUNT := 12830,
	OPCUAID_SESSIONDIAGNOSTICSARRAYTYPE_SESSIONDIAGNOSTICS_UNAUTHORIZEDREQUESTCOUNT := 12831,
	OPCUAID_SESSIONDIAGNOSTICSARRAYTYPE_SESSIONDIAGNOSTICS_READCOUNT := 12832,
	OPCUAID_SESSIONDIAGNOSTICSARRAYTYPE_SESSIONDIAGNOSTICS_HISTORYREADCOUNT := 12833,
	OPCUAID_SESSIONDIAGNOSTICSARRAYTYPE_SESSIONDIAGNOSTICS_WRITECOUNT := 12834,
	OPCUAID_SESSIONDIAGNOSTICSARRAYTYPE_SESSIONDIAGNOSTICS_HISTORYUPDATECOUNT := 12835,
	OPCUAID_SESSIONDIAGNOSTICSARRAYTYPE_SESSIONDIAGNOSTICS_CALLCOUNT := 12836,
	OPCUAID_SESSIONDIAGNOSTICSARRAYTYPE_SESSIONDIAGNOSTICS_CREATEMONITOREDITEMSCOUNT := 12837,
	OPCUAID_SESSIONDIAGNOSTICSARRAYTYPE_SESSIONDIAGNOSTICS_MODIFYMONITOREDITEMSCOUNT := 12838,
	OPCUAID_SESSIONDIAGNOSTICSARRAYTYPE_SESSIONDIAGNOSTICS_SETMONITORINGMODECOUNT := 12839,
	OPCUAID_SESSIONDIAGNOSTICSARRAYTYPE_SESSIONDIAGNOSTICS_SETTRIGGERINGCOUNT := 12840,
	OPCUAID_SESSIONDIAGNOSTICSARRAYTYPE_SESSIONDIAGNOSTICS_DELETEMONITOREDITEMSCOUNT := 12841,
	OPCUAID_SESSIONDIAGNOSTICSARRAYTYPE_SESSIONDIAGNOSTICS_CREATESUBSCRIPTIONCOUNT := 12842,
	OPCUAID_SESSIONDIAGNOSTICSARRAYTYPE_SESSIONDIAGNOSTICS_MODIFYSUBSCRIPTIONCOUNT := 12843,
	OPCUAID_SESSIONDIAGNOSTICSARRAYTYPE_SESSIONDIAGNOSTICS_SETPUBLISHINGMODECOUNT := 12844,
	OPCUAID_SESSIONDIAGNOSTICSARRAYTYPE_SESSIONDIAGNOSTICS_PUBLISHCOUNT := 12845,
	OPCUAID_SESSIONDIAGNOSTICSARRAYTYPE_SESSIONDIAGNOSTICS_REPUBLISHCOUNT := 12846,
	OPCUAID_SESSIONDIAGNOSTICSARRAYTYPE_SESSIONDIAGNOSTICS_TRANSFERSUBSCRIPTIONSCOUNT := 12847,
	OPCUAID_SESSIONDIAGNOSTICSARRAYTYPE_SESSIONDIAGNOSTICS_DELETESUBSCRIPTIONSCOUNT := 12848,
	OPCUAID_SESSIONDIAGNOSTICSARRAYTYPE_SESSIONDIAGNOSTICS_ADDNODESCOUNT := 12849,
	OPCUAID_SESSIONDIAGNOSTICSARRAYTYPE_SESSIONDIAGNOSTICS_ADDREFERENCESCOUNT := 12850,
	OPCUAID_SESSIONDIAGNOSTICSARRAYTYPE_SESSIONDIAGNOSTICS_DELETENODESCOUNT := 12851,
	OPCUAID_SESSIONDIAGNOSTICSARRAYTYPE_SESSIONDIAGNOSTICS_DELETEREFERENCESCOUNT := 12852,
	OPCUAID_SESSIONDIAGNOSTICSARRAYTYPE_SESSIONDIAGNOSTICS_BROWSECOUNT := 12853,
	OPCUAID_SESSIONDIAGNOSTICSARRAYTYPE_SESSIONDIAGNOSTICS_BROWSENEXTCOUNT := 12854,
	OPCUAID_SESSIONDIAGNOSTICSARRAYTYPE_SESSIONDIAGNOSTICS_TRANSLATEBROWSEPATHSTONODEIDSCOUNT := 12855,
	OPCUAID_SESSIONDIAGNOSTICSARRAYTYPE_SESSIONDIAGNOSTICS_QUERYFIRSTCOUNT := 12856,
	OPCUAID_SESSIONDIAGNOSTICSARRAYTYPE_SESSIONDIAGNOSTICS_QUERYNEXTCOUNT := 12857,
	OPCUAID_SESSIONDIAGNOSTICSARRAYTYPE_SESSIONDIAGNOSTICS_REGISTERNODESCOUNT := 12858,
	OPCUAID_SESSIONDIAGNOSTICSARRAYTYPE_SESSIONDIAGNOSTICS_UNREGISTERNODESCOUNT := 12859,
	OPCUAID_SESSIONDIAGNOSTICSVARIABLETYPE_SESSIONID := 2198,
	OPCUAID_SESSIONDIAGNOSTICSVARIABLETYPE_SESSIONNAME := 2199,
	OPCUAID_SESSIONDIAGNOSTICSVARIABLETYPE_CLIENTDESCRIPTION := 2200,
	OPCUAID_SESSIONDIAGNOSTICSVARIABLETYPE_SERVERURI := 2201,
	OPCUAID_SESSIONDIAGNOSTICSVARIABLETYPE_ENDPOINTURL := 2202,
	OPCUAID_SESSIONDIAGNOSTICSVARIABLETYPE_LOCALEIDS := 2203,
	OPCUAID_SESSIONDIAGNOSTICSVARIABLETYPE_ACTUALSESSIONTIMEOUT := 2204,
	OPCUAID_SESSIONDIAGNOSTICSVARIABLETYPE_MAXRESPONSEMESSAGESIZE := 3050,
	OPCUAID_SESSIONDIAGNOSTICSVARIABLETYPE_CLIENTCONNECTIONTIME := 2205,
	OPCUAID_SESSIONDIAGNOSTICSVARIABLETYPE_CLIENTLASTCONTACTTIME := 2206,
	OPCUAID_SESSIONDIAGNOSTICSVARIABLETYPE_CURRENTSUBSCRIPTIONSCOUNT := 2207,
	OPCUAID_SESSIONDIAGNOSTICSVARIABLETYPE_CURRENTMONITOREDITEMSCOUNT := 2208,
	OPCUAID_SESSIONDIAGNOSTICSVARIABLETYPE_CURRENTPUBLISHREQUESTSINQUEUE := 2209,
	OPCUAID_SESSIONDIAGNOSTICSVARIABLETYPE_TOTALREQUESTCOUNT := 8900,
	OPCUAID_SESSIONDIAGNOSTICSVARIABLETYPE_UNAUTHORIZEDREQUESTCOUNT := 11892,
	OPCUAID_SESSIONDIAGNOSTICSVARIABLETYPE_READCOUNT := 2217,
	OPCUAID_SESSIONDIAGNOSTICSVARIABLETYPE_HISTORYREADCOUNT := 2218,
	OPCUAID_SESSIONDIAGNOSTICSVARIABLETYPE_WRITECOUNT := 2219,
	OPCUAID_SESSIONDIAGNOSTICSVARIABLETYPE_HISTORYUPDATECOUNT := 2220,
	OPCUAID_SESSIONDIAGNOSTICSVARIABLETYPE_CALLCOUNT := 2221,
	OPCUAID_SESSIONDIAGNOSTICSVARIABLETYPE_CREATEMONITOREDITEMSCOUNT := 2222,
	OPCUAID_SESSIONDIAGNOSTICSVARIABLETYPE_MODIFYMONITOREDITEMSCOUNT := 2223,
	OPCUAID_SESSIONDIAGNOSTICSVARIABLETYPE_SETMONITORINGMODECOUNT := 2224,
	OPCUAID_SESSIONDIAGNOSTICSVARIABLETYPE_SETTRIGGERINGCOUNT := 2225,
	OPCUAID_SESSIONDIAGNOSTICSVARIABLETYPE_DELETEMONITOREDITEMSCOUNT := 2226,
	OPCUAID_SESSIONDIAGNOSTICSVARIABLETYPE_CREATESUBSCRIPTIONCOUNT := 2227,
	OPCUAID_SESSIONDIAGNOSTICSVARIABLETYPE_MODIFYSUBSCRIPTIONCOUNT := 2228,
	OPCUAID_SESSIONDIAGNOSTICSVARIABLETYPE_SETPUBLISHINGMODECOUNT := 2229,
	OPCUAID_SESSIONDIAGNOSTICSVARIABLETYPE_PUBLISHCOUNT := 2230,
	OPCUAID_SESSIONDIAGNOSTICSVARIABLETYPE_REPUBLISHCOUNT := 2231,
	OPCUAID_SESSIONDIAGNOSTICSVARIABLETYPE_TRANSFERSUBSCRIPTIONSCOUNT := 2232,
	OPCUAID_SESSIONDIAGNOSTICSVARIABLETYPE_DELETESUBSCRIPTIONSCOUNT := 2233,
	OPCUAID_SESSIONDIAGNOSTICSVARIABLETYPE_ADDNODESCOUNT := 2234,
	OPCUAID_SESSIONDIAGNOSTICSVARIABLETYPE_ADDREFERENCESCOUNT := 2235,
	OPCUAID_SESSIONDIAGNOSTICSVARIABLETYPE_DELETENODESCOUNT := 2236,
	OPCUAID_SESSIONDIAGNOSTICSVARIABLETYPE_DELETEREFERENCESCOUNT := 2237,
	OPCUAID_SESSIONDIAGNOSTICSVARIABLETYPE_BROWSECOUNT := 2238,
	OPCUAID_SESSIONDIAGNOSTICSVARIABLETYPE_BROWSENEXTCOUNT := 2239,
	OPCUAID_SESSIONDIAGNOSTICSVARIABLETYPE_TRANSLATEBROWSEPATHSTONODEIDSCOUNT := 2240,
	OPCUAID_SESSIONDIAGNOSTICSVARIABLETYPE_QUERYFIRSTCOUNT := 2241,
	OPCUAID_SESSIONDIAGNOSTICSVARIABLETYPE_QUERYNEXTCOUNT := 2242,
	OPCUAID_SESSIONDIAGNOSTICSVARIABLETYPE_REGISTERNODESCOUNT := 2730,
	OPCUAID_SESSIONDIAGNOSTICSVARIABLETYPE_UNREGISTERNODESCOUNT := 2731,
	OPCUAID_SESSIONSECURITYDIAGNOSTICSARRAYTYPE_SESSIONSECURITYDIAGNOSTICS := 12860,
	OPCUAID_SESSIONSECURITYDIAGNOSTICSARRAYTYPE_SESSIONSECURITYDIAGNOSTICS_SESSIONID := 12861,
	OPCUAID_SESSIONSECURITYDIAGNOSTICSARRAYTYPE_SESSIONSECURITYDIAGNOSTICS_CLIENTUSERIDOFSESSION := 12862,
	OPCUAID_SESSIONSECURITYDIAGNOSTICSARRAYTYPE_SESSIONSECURITYDIAGNOSTICS_CLIENTUSERIDHISTORY := 12863,
	OPCUAID_SESSIONSECURITYDIAGNOSTICSARRAYTYPE_SESSIONSECURITYDIAGNOSTICS_AUTHENTICATIONMECHANISM := 12864,
	OPCUAID_SESSIONSECURITYDIAGNOSTICSARRAYTYPE_SESSIONSECURITYDIAGNOSTICS_ENCODING := 12865,
	OPCUAID_SESSIONSECURITYDIAGNOSTICSARRAYTYPE_SESSIONSECURITYDIAGNOSTICS_TRANSPORTPROTOCOL := 12866,
	OPCUAID_SESSIONSECURITYDIAGNOSTICSARRAYTYPE_SESSIONSECURITYDIAGNOSTICS_SECURITYMODE := 12867,
	OPCUAID_SESSIONSECURITYDIAGNOSTICSARRAYTYPE_SESSIONSECURITYDIAGNOSTICS_SECURITYPOLICYURI := 12868,
	OPCUAID_SESSIONSECURITYDIAGNOSTICSARRAYTYPE_SESSIONSECURITYDIAGNOSTICS_CLIENTCERTIFICATE := 12869,
	OPCUAID_SESSIONSECURITYDIAGNOSTICSTYPE_SESSIONID := 2245,
	OPCUAID_SESSIONSECURITYDIAGNOSTICSTYPE_CLIENTUSERIDOFSESSION := 2246,
	OPCUAID_SESSIONSECURITYDIAGNOSTICSTYPE_CLIENTUSERIDHISTORY := 2247,
	OPCUAID_SESSIONSECURITYDIAGNOSTICSTYPE_AUTHENTICATIONMECHANISM := 2248,
	OPCUAID_SESSIONSECURITYDIAGNOSTICSTYPE_ENCODING := 2249,
	OPCUAID_SESSIONSECURITYDIAGNOSTICSTYPE_TRANSPORTPROTOCOL := 2250,
	OPCUAID_SESSIONSECURITYDIAGNOSTICSTYPE_SECURITYMODE := 2251,
	OPCUAID_SESSIONSECURITYDIAGNOSTICSTYPE_SECURITYPOLICYURI := 2252,
	OPCUAID_SESSIONSECURITYDIAGNOSTICSTYPE_CLIENTCERTIFICATE := 3058,
	OPCUAID_OPTIONSETTYPE_OPTIONSETVALUES := 11488,
	OPCUAID_OPTIONSETTYPE_BITMASK := 11701,
	OPCUAID_SELECTIONLISTTYPE_SELECTIONS := 17632,
	OPCUAID_SELECTIONLISTTYPE_SELECTIONDESCRIPTIONS := 17633,
	OPCUAID_SELECTIONLISTTYPE_RESTRICTTOLIST := 16312,
	OPCUAID_AUDIOVARIABLETYPE_LISTID := 17988,
	OPCUAID_AUDIOVARIABLETYPE_AGENCYID := 17989,
	OPCUAID_AUDIOVARIABLETYPE_VERSIONID := 17990,
	OPCUAID_SERVER_SERVERARRAY := 2254,
	OPCUAID_SERVER_NAMESPACEARRAY := 2255,
	OPCUAID_SERVER_SERVERSTATUS := 2256,
	OPCUAID_SERVER_SERVERSTATUS_STARTTIME := 2257,
	OPCUAID_SERVER_SERVERSTATUS_CURRENTTIME := 2258,
	OPCUAID_SERVER_SERVERSTATUS_STATE := 2259,
	OPCUAID_SERVER_SERVERSTATUS_BUILDINFO := 2260,
	OPCUAID_SERVER_SERVERSTATUS_BUILDINFO_PRODUCTURI := 2262,
	OPCUAID_SERVER_SERVERSTATUS_BUILDINFO_MANUFACTURERNAME := 2263,
	OPCUAID_SERVER_SERVERSTATUS_BUILDINFO_PRODUCTNAME := 2261,
	OPCUAID_SERVER_SERVERSTATUS_BUILDINFO_SOFTWAREVERSION := 2264,
	OPCUAID_SERVER_SERVERSTATUS_BUILDINFO_BUILDNUMBER := 2265,
	OPCUAID_SERVER_SERVERSTATUS_BUILDINFO_BUILDDATE := 2266,
	OPCUAID_SERVER_SERVERSTATUS_SECONDSTILLSHUTDOWN := 2992,
	OPCUAID_SERVER_SERVERSTATUS_SHUTDOWNREASON := 2993,
	OPCUAID_SERVER_SERVICELEVEL := 2267,
	OPCUAID_SERVER_AUDITING := 2994,
	OPCUAID_SERVER_ESTIMATEDRETURNTIME := 12885,
	OPCUAID_SERVER_SERVERCAPABILITIES_SERVERPROFILEARRAY := 2269,
	OPCUAID_SERVER_SERVERCAPABILITIES_LOCALEIDARRAY := 2271,
	OPCUAID_SERVER_SERVERCAPABILITIES_MINSUPPORTEDSAMPLERATE := 2272,
	OPCUAID_SERVER_SERVERCAPABILITIES_MAXBROWSECONTINUATIONPOINTS := 2735,
	OPCUAID_SERVER_SERVERCAPABILITIES_MAXQUERYCONTINUATIONPOINTS := 2736,
	OPCUAID_SERVER_SERVERCAPABILITIES_MAXHISTORYCONTINUATIONPOINTS := 2737,
	OPCUAID_SERVER_SERVERCAPABILITIES_SOFTWARECERTIFICATES := 3704,
	OPCUAID_SERVER_SERVERCAPABILITIES_MAXARRAYLENGTH := 11702,
	OPCUAID_SERVER_SERVERCAPABILITIES_MAXSTRINGLENGTH := 11703,
	OPCUAID_SERVER_SERVERCAPABILITIES_MAXBYTESTRINGLENGTH := 12911,
	OPCUAID_SERVER_SERVERCAPABILITIES_OPERATIONLIMITS_MAXNODESPERREAD := 11705,
	OPCUAID_SERVER_SERVERCAPABILITIES_OPERATIONLIMITS_MAXNODESPERHISTORYREADDATA := 12165,
	OPCUAID_SERVER_SERVERCAPABILITIES_OPERATIONLIMITS_MAXNODESPERHISTORYREADEVENTS := 12166,
	OPCUAID_SERVER_SERVERCAPABILITIES_OPERATIONLIMITS_MAXNODESPERWRITE := 11707,
	OPCUAID_SERVER_SERVERCAPABILITIES_OPERATIONLIMITS_MAXNODESPERHISTORYUPDATEDATA := 12167,
	OPCUAID_SERVER_SERVERCAPABILITIES_OPERATIONLIMITS_MAXNODESPERHISTORYUPDATEEVENTS := 12168,
	OPCUAID_SERVER_SERVERCAPABILITIES_OPERATIONLIMITS_MAXNODESPERMETHODCALL := 11709,
	OPCUAID_SERVER_SERVERCAPABILITIES_OPERATIONLIMITS_MAXNODESPERBROWSE := 11710,
	OPCUAID_SERVER_SERVERCAPABILITIES_OPERATIONLIMITS_MAXNODESPERREGISTERNODES := 11711,
	OPCUAID_SERVER_SERVERCAPABILITIES_OPERATIONLIMITS_MAXNODESPERTRANSLATEBROWSEPATHSTONODEIDS := 11712,
	OPCUAID_SERVER_SERVERCAPABILITIES_OPERATIONLIMITS_MAXNODESPERNODEMANAGEMENT := 11713,
	OPCUAID_SERVER_SERVERCAPABILITIES_OPERATIONLIMITS_MAXMONITOREDITEMSPERCALL := 11714,
	OPCUAID_SERVER_SERVERCAPABILITIES_ROLESET_ADDROLE_INPUTARGUMENTS := 16302,
	OPCUAID_SERVER_SERVERCAPABILITIES_ROLESET_ADDROLE_OUTPUTARGUMENTS := 16303,
	OPCUAID_SERVER_SERVERCAPABILITIES_ROLESET_REMOVEROLE_INPUTARGUMENTS := 16305,
	OPCUAID_SERVER_SERVERDIAGNOSTICS_SERVERDIAGNOSTICSSUMMARY := 2275,
	OPCUAID_SERVER_SERVERDIAGNOSTICS_SERVERDIAGNOSTICSSUMMARY_SERVERVIEWCOUNT := 2276,
	OPCUAID_SERVER_SERVERDIAGNOSTICS_SERVERDIAGNOSTICSSUMMARY_CURRENTSESSIONCOUNT := 2277,
	OPCUAID_SERVER_SERVERDIAGNOSTICS_SERVERDIAGNOSTICSSUMMARY_CUMULATEDSESSIONCOUNT := 2278,
	OPCUAID_SERVER_SERVERDIAGNOSTICS_SERVERDIAGNOSTICSSUMMARY_SECURITYREJECTEDSESSIONCOUNT := 2279,
	OPCUAID_SERVER_SERVERDIAGNOSTICS_SERVERDIAGNOSTICSSUMMARY_REJECTEDSESSIONCOUNT := 3705,
	OPCUAID_SERVER_SERVERDIAGNOSTICS_SERVERDIAGNOSTICSSUMMARY_SESSIONTIMEOUTCOUNT := 2281,
	OPCUAID_SERVER_SERVERDIAGNOSTICS_SERVERDIAGNOSTICSSUMMARY_SESSIONABORTCOUNT := 2282,
	OPCUAID_SERVER_SERVERDIAGNOSTICS_SERVERDIAGNOSTICSSUMMARY_PUBLISHINGINTERVALCOUNT := 2284,
	OPCUAID_SERVER_SERVERDIAGNOSTICS_SERVERDIAGNOSTICSSUMMARY_CURRENTSUBSCRIPTIONCOUNT := 2285,
	OPCUAID_SERVER_SERVERDIAGNOSTICS_SERVERDIAGNOSTICSSUMMARY_CUMULATEDSUBSCRIPTIONCOUNT := 2286,
	OPCUAID_SERVER_SERVERDIAGNOSTICS_SERVERDIAGNOSTICSSUMMARY_SECURITYREJECTEDREQUESTSCOUNT := 2287,
	OPCUAID_SERVER_SERVERDIAGNOSTICS_SERVERDIAGNOSTICSSUMMARY_REJECTEDREQUESTSCOUNT := 2288,
	OPCUAID_SERVER_SERVERDIAGNOSTICS_SAMPLINGINTERVALDIAGNOSTICSARRAY := 2289,
	OPCUAID_SERVER_SERVERDIAGNOSTICS_SUBSCRIPTIONDIAGNOSTICSARRAY := 2290,
	OPCUAID_SERVER_SERVERDIAGNOSTICS_SESSIONSDIAGNOSTICSSUMMARY_SESSIONDIAGNOSTICSARRAY := 3707,
	OPCUAID_SERVER_SERVERDIAGNOSTICS_SESSIONSDIAGNOSTICSSUMMARY_SESSIONSECURITYDIAGNOSTICSARRAY := 3708,
	OPCUAID_SERVER_SERVERDIAGNOSTICS_ENABLEDFLAG := 2294,
	OPCUAID_SERVER_SERVERREDUNDANCY_REDUNDANCYSUPPORT := 3709,
	OPCUAID_SERVER_GETMONITOREDITEMS_INPUTARGUMENTS := 11493,
	OPCUAID_SERVER_GETMONITOREDITEMS_OUTPUTARGUMENTS := 11494,
	OPCUAID_SERVER_RESENDDATA_INPUTARGUMENTS := 12874,
	OPCUAID_SERVER_SETSUBSCRIPTIONDURABLE_INPUTARGUMENTS := 12750,
	OPCUAID_SERVER_SETSUBSCRIPTIONDURABLE_OUTPUTARGUMENTS := 12751,
	OPCUAID_SERVER_REQUESTSERVERSTATECHANGE_INPUTARGUMENTS := 12887,
	OPCUAID_SERVER_CURRENTTIMEZONE := 16313,
	OPCUAID_SERVER_SERVERREDUNDANCY_CURRENTSERVERID := 11312,
	OPCUAID_SERVER_SERVERREDUNDANCY_REDUNDANTSERVERARRAY := 11313,
	OPCUAID_SERVER_SERVERREDUNDANCY_SERVERURIARRAY := 11314,
	OPCUAID_SERVER_SERVERREDUNDANCY_SERVERNETWORKGROUPS := 14415,
	OPCUAID_HISTORYSERVERCAPABILITIES_ACCESSHISTORYDATACAPABILITY := 11193,
	OPCUAID_HISTORYSERVERCAPABILITIES_ACCESSHISTORYEVENTSCAPABILITY := 11242,
	OPCUAID_HISTORYSERVERCAPABILITIES_MAXRETURNDATAVALUES := 11273,
	OPCUAID_HISTORYSERVERCAPABILITIES_MAXRETURNEVENTVALUES := 11274,
	OPCUAID_HISTORYSERVERCAPABILITIES_INSERTDATACAPABILITY := 11196,
	OPCUAID_HISTORYSERVERCAPABILITIES_REPLACEDATACAPABILITY := 11197,
	OPCUAID_HISTORYSERVERCAPABILITIES_UPDATEDATACAPABILITY := 11198,
	OPCUAID_HISTORYSERVERCAPABILITIES_DELETERAWCAPABILITY := 11199,
	OPCUAID_HISTORYSERVERCAPABILITIES_DELETEATTIMECAPABILITY := 11200,
	OPCUAID_HISTORYSERVERCAPABILITIES_INSERTEVENTCAPABILITY := 11281,
	OPCUAID_HISTORYSERVERCAPABILITIES_REPLACEEVENTCAPABILITY := 11282,
	OPCUAID_HISTORYSERVERCAPABILITIES_UPDATEEVENTCAPABILITY := 11283,
	OPCUAID_HISTORYSERVERCAPABILITIES_DELETEEVENTCAPABILITY := 11502,
	OPCUAID_HISTORYSERVERCAPABILITIES_INSERTANNOTATIONCAPABILITY := 11275,
	OPCUAID_STATEMACHINETYPE_CURRENTSTATE := 2769,
	OPCUAID_STATEMACHINETYPE_CURRENTSTATE_ID := 3720,
	OPCUAID_STATEMACHINETYPE_LASTTRANSITION := 2770,
	OPCUAID_STATEMACHINETYPE_LASTTRANSITION_ID := 3724,
	OPCUAID_STATEVARIABLETYPE_ID := 2756,
	OPCUAID_STATEVARIABLETYPE_NAME := 2757,
	OPCUAID_STATEVARIABLETYPE_NUMBER := 2758,
	OPCUAID_STATEVARIABLETYPE_EFFECTIVEDISPLAYNAME := 2759,
	OPCUAID_TRANSITIONVARIABLETYPE_ID := 2763,
	OPCUAID_TRANSITIONVARIABLETYPE_NAME := 2764,
	OPCUAID_TRANSITIONVARIABLETYPE_NUMBER := 2765,
	OPCUAID_TRANSITIONVARIABLETYPE_TRANSITIONTIME := 2766,
	OPCUAID_TRANSITIONVARIABLETYPE_EFFECTIVETRANSITIONTIME := 11456,
	OPCUAID_FINITESTATEMACHINETYPE_CURRENTSTATE := 2772,
	OPCUAID_FINITESTATEMACHINETYPE_CURRENTSTATE_ID := 3728,
	OPCUAID_FINITESTATEMACHINETYPE_LASTTRANSITION := 2773,
	OPCUAID_FINITESTATEMACHINETYPE_LASTTRANSITION_ID := 3732,
	OPCUAID_FINITESTATEMACHINETYPE_AVAILABLESTATES := 17635,
	OPCUAID_FINITESTATEMACHINETYPE_AVAILABLETRANSITIONS := 17636,
	OPCUAID_FINITESTATEVARIABLETYPE_ID := 2761,
	OPCUAID_FINITETRANSITIONVARIABLETYPE_ID := 2768,
	OPCUAID_STATETYPE_STATENUMBER := 2308,
	OPCUAID_TRANSITIONTYPE_TRANSITIONNUMBER := 2312,
	OPCUAID_TRANSITIONEVENTTYPE_TRANSITION := 2774,
	OPCUAID_TRANSITIONEVENTTYPE_TRANSITION_ID := 3754,
	OPCUAID_TRANSITIONEVENTTYPE_FROMSTATE := 2775,
	OPCUAID_TRANSITIONEVENTTYPE_FROMSTATE_ID := 3746,
	OPCUAID_TRANSITIONEVENTTYPE_TOSTATE := 2776,
	OPCUAID_TRANSITIONEVENTTYPE_TOSTATE_ID := 3750,
	OPCUAID_AUDITUPDATESTATEEVENTTYPE_OLDSTATEID := 2777,
	OPCUAID_AUDITUPDATESTATEEVENTTYPE_NEWSTATEID := 2778,
	OPCUAID_OPENFILEMODE_ENUMVALUES := 11940,
	OPCUAID_FILEDIRECTORYTYPE_FILEDIRECTORYNAME_PLACEHOLDER_CREATEDIRECTORY_INPUTARGUMENTS := 13356,
	OPCUAID_FILEDIRECTORYTYPE_FILEDIRECTORYNAME_PLACEHOLDER_CREATEDIRECTORY_OUTPUTARGUMENTS := 13357,
	OPCUAID_FILEDIRECTORYTYPE_FILEDIRECTORYNAME_PLACEHOLDER_CREATEFILE_INPUTARGUMENTS := 13359,
	OPCUAID_FILEDIRECTORYTYPE_FILEDIRECTORYNAME_PLACEHOLDER_CREATEFILE_OUTPUTARGUMENTS := 13360,
	OPCUAID_FILEDIRECTORYTYPE_FILEDIRECTORYNAME_PLACEHOLDER_DELETEFILESYSTEMOBJECT_INPUTARGUMENTS := 17719,
	OPCUAID_FILEDIRECTORYTYPE_FILEDIRECTORYNAME_PLACEHOLDER_MOVEORCOPY_INPUTARGUMENTS := 13364,
	OPCUAID_FILEDIRECTORYTYPE_FILEDIRECTORYNAME_PLACEHOLDER_MOVEORCOPY_OUTPUTARGUMENTS := 13365,
	OPCUAID_FILEDIRECTORYTYPE_FILENAME_PLACEHOLDER_SIZE := 13367,
	OPCUAID_FILEDIRECTORYTYPE_FILENAME_PLACEHOLDER_WRITABLE := 13368,
	OPCUAID_FILEDIRECTORYTYPE_FILENAME_PLACEHOLDER_USERWRITABLE := 13369,
	OPCUAID_FILEDIRECTORYTYPE_FILENAME_PLACEHOLDER_OPENCOUNT := 13370,
	OPCUAID_FILEDIRECTORYTYPE_FILENAME_PLACEHOLDER_OPEN_INPUTARGUMENTS := 13373,
	OPCUAID_FILEDIRECTORYTYPE_FILENAME_PLACEHOLDER_OPEN_OUTPUTARGUMENTS := 13374,
	OPCUAID_FILEDIRECTORYTYPE_FILENAME_PLACEHOLDER_CLOSE_INPUTARGUMENTS := 13376,
	OPCUAID_FILEDIRECTORYTYPE_FILENAME_PLACEHOLDER_READ_INPUTARGUMENTS := 13378,
	OPCUAID_FILEDIRECTORYTYPE_FILENAME_PLACEHOLDER_READ_OUTPUTARGUMENTS := 13379,
	OPCUAID_FILEDIRECTORYTYPE_FILENAME_PLACEHOLDER_WRITE_INPUTARGUMENTS := 13381,
	OPCUAID_FILEDIRECTORYTYPE_FILENAME_PLACEHOLDER_GETPOSITION_INPUTARGUMENTS := 13383,
	OPCUAID_FILEDIRECTORYTYPE_FILENAME_PLACEHOLDER_GETPOSITION_OUTPUTARGUMENTS := 13384,
	OPCUAID_FILEDIRECTORYTYPE_FILENAME_PLACEHOLDER_SETPOSITION_INPUTARGUMENTS := 13386,
	OPCUAID_FILEDIRECTORYTYPE_CREATEDIRECTORY_INPUTARGUMENTS := 13388,
	OPCUAID_FILEDIRECTORYTYPE_CREATEDIRECTORY_OUTPUTARGUMENTS := 13389,
	OPCUAID_FILEDIRECTORYTYPE_CREATEFILE_INPUTARGUMENTS := 13391,
	OPCUAID_FILEDIRECTORYTYPE_CREATEFILE_OUTPUTARGUMENTS := 13392,
	OPCUAID_FILEDIRECTORYTYPE_DELETEFILESYSTEMOBJECT_INPUTARGUMENTS := 13394,
	OPCUAID_FILEDIRECTORYTYPE_MOVEORCOPY_INPUTARGUMENTS := 13396,
	OPCUAID_FILEDIRECTORYTYPE_MOVEORCOPY_OUTPUTARGUMENTS := 13397,
	OPCUAID_FILESYSTEM_FILEDIRECTORYNAME_PLACEHOLDER_CREATEDIRECTORY_INPUTARGUMENTS := 16317,
	OPCUAID_FILESYSTEM_FILEDIRECTORYNAME_PLACEHOLDER_CREATEDIRECTORY_OUTPUTARGUMENTS := 16318,
	OPCUAID_FILESYSTEM_FILEDIRECTORYNAME_PLACEHOLDER_CREATEFILE_INPUTARGUMENTS := 16320,
	OPCUAID_FILESYSTEM_FILEDIRECTORYNAME_PLACEHOLDER_CREATEFILE_OUTPUTARGUMENTS := 16321,
	OPCUAID_FILESYSTEM_FILEDIRECTORYNAME_PLACEHOLDER_DELETEFILESYSTEMOBJECT_INPUTARGUMENTS := 17723,
	OPCUAID_FILESYSTEM_FILEDIRECTORYNAME_PLACEHOLDER_MOVEORCOPY_INPUTARGUMENTS := 16325,
	OPCUAID_FILESYSTEM_FILEDIRECTORYNAME_PLACEHOLDER_MOVEORCOPY_OUTPUTARGUMENTS := 16326,
	OPCUAID_FILESYSTEM_FILENAME_PLACEHOLDER_SIZE := 16328,
	OPCUAID_FILESYSTEM_FILENAME_PLACEHOLDER_WRITABLE := 16329,
	OPCUAID_FILESYSTEM_FILENAME_PLACEHOLDER_USERWRITABLE := 16330,
	OPCUAID_FILESYSTEM_FILENAME_PLACEHOLDER_OPENCOUNT := 16331,
	OPCUAID_FILESYSTEM_FILENAME_PLACEHOLDER_OPEN_INPUTARGUMENTS := 16334,
	OPCUAID_FILESYSTEM_FILENAME_PLACEHOLDER_OPEN_OUTPUTARGUMENTS := 16335,
	OPCUAID_FILESYSTEM_FILENAME_PLACEHOLDER_CLOSE_INPUTARGUMENTS := 16337,
	OPCUAID_FILESYSTEM_FILENAME_PLACEHOLDER_READ_INPUTARGUMENTS := 16339,
	OPCUAID_FILESYSTEM_FILENAME_PLACEHOLDER_READ_OUTPUTARGUMENTS := 16340,
	OPCUAID_FILESYSTEM_FILENAME_PLACEHOLDER_WRITE_INPUTARGUMENTS := 16342,
	OPCUAID_FILESYSTEM_FILENAME_PLACEHOLDER_GETPOSITION_INPUTARGUMENTS := 16344,
	OPCUAID_FILESYSTEM_FILENAME_PLACEHOLDER_GETPOSITION_OUTPUTARGUMENTS := 16345,
	OPCUAID_FILESYSTEM_FILENAME_PLACEHOLDER_SETPOSITION_INPUTARGUMENTS := 16347,
	OPCUAID_FILESYSTEM_CREATEDIRECTORY_INPUTARGUMENTS := 16349,
	OPCUAID_FILESYSTEM_CREATEDIRECTORY_OUTPUTARGUMENTS := 16350,
	OPCUAID_FILESYSTEM_CREATEFILE_INPUTARGUMENTS := 16352,
	OPCUAID_FILESYSTEM_CREATEFILE_OUTPUTARGUMENTS := 16353,
	OPCUAID_FILESYSTEM_DELETEFILESYSTEMOBJECT_INPUTARGUMENTS := 16355,
	OPCUAID_FILESYSTEM_MOVEORCOPY_INPUTARGUMENTS := 16357,
	OPCUAID_FILESYSTEM_MOVEORCOPY_OUTPUTARGUMENTS := 16358,
	OPCUAID_TEMPORARYFILETRANSFERTYPE_CLIENTPROCESSINGTIMEOUT := 15745,
	OPCUAID_TEMPORARYFILETRANSFERTYPE_GENERATEFILEFORREAD_INPUTARGUMENTS := 15747,
	OPCUAID_TEMPORARYFILETRANSFERTYPE_GENERATEFILEFORREAD_OUTPUTARGUMENTS := 15748,
	OPCUAID_TEMPORARYFILETRANSFERTYPE_GENERATEFILEFORWRITE_INPUTARGUMENTS := 16359,
	OPCUAID_TEMPORARYFILETRANSFERTYPE_GENERATEFILEFORWRITE_OUTPUTARGUMENTS := 15750,
	OPCUAID_TEMPORARYFILETRANSFERTYPE_CLOSEANDCOMMIT_INPUTARGUMENTS := 15752,
	OPCUAID_TEMPORARYFILETRANSFERTYPE_CLOSEANDCOMMIT_OUTPUTARGUMENTS := 15753,
	OPCUAID_TEMPORARYFILETRANSFERTYPE_TRANSFERSTATE_PLACEHOLDER_CURRENTSTATE := 15755,
	OPCUAID_TEMPORARYFILETRANSFERTYPE_TRANSFERSTATE_PLACEHOLDER_CURRENTSTATE_ID := 15756,
	OPCUAID_TEMPORARYFILETRANSFERTYPE_TRANSFERSTATE_PLACEHOLDER_LASTTRANSITION_ID := 15761,
	OPCUAID_FILETRANSFERSTATEMACHINETYPE_CURRENTSTATE_ID := 15805,
	OPCUAID_FILETRANSFERSTATEMACHINETYPE_LASTTRANSITION_ID := 15810,
	OPCUAID_FILETRANSFERSTATEMACHINETYPE_IDLE_STATENUMBER := 15816,
	OPCUAID_FILETRANSFERSTATEMACHINETYPE_READPREPARE_STATENUMBER := 15818,
	OPCUAID_FILETRANSFERSTATEMACHINETYPE_READTRANSFER_STATENUMBER := 15820,
	OPCUAID_FILETRANSFERSTATEMACHINETYPE_APPLYWRITE_STATENUMBER := 15822,
	OPCUAID_FILETRANSFERSTATEMACHINETYPE_ERROR_STATENUMBER := 15824,
	OPCUAID_FILETRANSFERSTATEMACHINETYPE_IDLETOREADPREPARE_TRANSITIONNUMBER := 15826,
	OPCUAID_FILETRANSFERSTATEMACHINETYPE_READPREPARETOREADTRANSFER_TRANSITIONNUMBER := 15828,
	OPCUAID_FILETRANSFERSTATEMACHINETYPE_READTRANSFERTOIDLE_TRANSITIONNUMBER := 15830,
	OPCUAID_FILETRANSFERSTATEMACHINETYPE_IDLETOAPPLYWRITE_TRANSITIONNUMBER := 15832,
	OPCUAID_FILETRANSFERSTATEMACHINETYPE_APPLYWRITETOIDLE_TRANSITIONNUMBER := 15834,
	OPCUAID_FILETRANSFERSTATEMACHINETYPE_READPREPARETOERROR_TRANSITIONNUMBER := 15836,
	OPCUAID_FILETRANSFERSTATEMACHINETYPE_READTRANSFERTOERROR_TRANSITIONNUMBER := 15838,
	OPCUAID_FILETRANSFERSTATEMACHINETYPE_APPLYWRITETOERROR_TRANSITIONNUMBER := 15840,
	OPCUAID_FILETRANSFERSTATEMACHINETYPE_ERRORTOIDLE_TRANSITIONNUMBER := 15842,
	OPCUAID_ROLESETTYPE_ROLENAME_PLACEHOLDER_IDENTITIES := 16162,
	OPCUAID_ROLESETTYPE_ROLENAME_PLACEHOLDER_ADDIDENTITY_INPUTARGUMENTS := 15613,
	OPCUAID_ROLESETTYPE_ROLENAME_PLACEHOLDER_REMOVEIDENTITY_INPUTARGUMENTS := 15615,
	OPCUAID_ROLESETTYPE_ROLENAME_PLACEHOLDER_ADDAPPLICATION_INPUTARGUMENTS := 16166,
	OPCUAID_ROLESETTYPE_ROLENAME_PLACEHOLDER_REMOVEAPPLICATION_INPUTARGUMENTS := 16168,
	OPCUAID_ROLESETTYPE_ROLENAME_PLACEHOLDER_ADDENDPOINT_INPUTARGUMENTS := 16170,
	OPCUAID_ROLESETTYPE_ROLENAME_PLACEHOLDER_REMOVEENDPOINT_INPUTARGUMENTS := 16172,
	OPCUAID_ROLESETTYPE_ADDROLE_INPUTARGUMENTS := 15998,
	OPCUAID_ROLESETTYPE_ADDROLE_OUTPUTARGUMENTS := 15999,
	OPCUAID_ROLESETTYPE_REMOVEROLE_INPUTARGUMENTS := 16001,
	OPCUAID_ROLETYPE_IDENTITIES := 16173,
	OPCUAID_ROLETYPE_APPLICATIONS := 16174,
	OPCUAID_ROLETYPE_APPLICATIONSEXCLUDE := 15410,
	OPCUAID_ROLETYPE_ENDPOINTS := 16175,
	OPCUAID_ROLETYPE_ENDPOINTSEXCLUDE := 15411,
	OPCUAID_ROLETYPE_ADDIDENTITY_INPUTARGUMENTS := 15625,
	OPCUAID_ROLETYPE_REMOVEIDENTITY_INPUTARGUMENTS := 15627,
	OPCUAID_ROLETYPE_ADDAPPLICATION_INPUTARGUMENTS := 16177,
	OPCUAID_ROLETYPE_REMOVEAPPLICATION_INPUTARGUMENTS := 16179,
	OPCUAID_ROLETYPE_ADDENDPOINT_INPUTARGUMENTS := 16181,
	OPCUAID_ROLETYPE_REMOVEENDPOINT_INPUTARGUMENTS := 16183,
	OPCUAID_IDENTITYCRITERIATYPE_ENUMVALUES := 15633,
	OPCUAID_WELLKNOWNROLE_ANONYMOUS_IDENTITIES := 16192,
	OPCUAID_WELLKNOWNROLE_ANONYMOUS_APPLICATIONS := 16193,
	OPCUAID_WELLKNOWNROLE_ANONYMOUS_APPLICATIONSEXCLUDE := 15412,
	OPCUAID_WELLKNOWNROLE_ANONYMOUS_ENDPOINTS := 16194,
	OPCUAID_WELLKNOWNROLE_ANONYMOUS_ENDPOINTSEXCLUDE := 15413,
	OPCUAID_WELLKNOWNROLE_ANONYMOUS_ADDIDENTITY_INPUTARGUMENTS := 15649,
	OPCUAID_WELLKNOWNROLE_ANONYMOUS_REMOVEIDENTITY_INPUTARGUMENTS := 15651,
	OPCUAID_WELLKNOWNROLE_ANONYMOUS_ADDAPPLICATION_INPUTARGUMENTS := 16196,
	OPCUAID_WELLKNOWNROLE_ANONYMOUS_REMOVEAPPLICATION_INPUTARGUMENTS := 16198,
	OPCUAID_WELLKNOWNROLE_ANONYMOUS_ADDENDPOINT_INPUTARGUMENTS := 16200,
	OPCUAID_WELLKNOWNROLE_ANONYMOUS_REMOVEENDPOINT_INPUTARGUMENTS := 16202,
	OPCUAID_WELLKNOWNROLE_AUTHENTICATEDUSER_IDENTITIES := 16203,
	OPCUAID_WELLKNOWNROLE_AUTHENTICATEDUSER_APPLICATIONS := 16204,
	OPCUAID_WELLKNOWNROLE_AUTHENTICATEDUSER_APPLICATIONSEXCLUDE := 15414,
	OPCUAID_WELLKNOWNROLE_AUTHENTICATEDUSER_ENDPOINTS := 16205,
	OPCUAID_WELLKNOWNROLE_AUTHENTICATEDUSER_ENDPOINTSEXCLUDE := 15415,
	OPCUAID_WELLKNOWNROLE_AUTHENTICATEDUSER_ADDIDENTITY_INPUTARGUMENTS := 15661,
	OPCUAID_WELLKNOWNROLE_AUTHENTICATEDUSER_REMOVEIDENTITY_INPUTARGUMENTS := 15663,
	OPCUAID_WELLKNOWNROLE_AUTHENTICATEDUSER_ADDAPPLICATION_INPUTARGUMENTS := 16207,
	OPCUAID_WELLKNOWNROLE_AUTHENTICATEDUSER_REMOVEAPPLICATION_INPUTARGUMENTS := 16209,
	OPCUAID_WELLKNOWNROLE_AUTHENTICATEDUSER_ADDENDPOINT_INPUTARGUMENTS := 16211,
	OPCUAID_WELLKNOWNROLE_AUTHENTICATEDUSER_REMOVEENDPOINT_INPUTARGUMENTS := 16213,
	OPCUAID_WELLKNOWNROLE_OBSERVER_IDENTITIES := 16214,
	OPCUAID_WELLKNOWNROLE_OBSERVER_APPLICATIONS := 16215,
	OPCUAID_WELLKNOWNROLE_OBSERVER_APPLICATIONSEXCLUDE := 15416,
	OPCUAID_WELLKNOWNROLE_OBSERVER_ENDPOINTS := 16216,
	OPCUAID_WELLKNOWNROLE_OBSERVER_ENDPOINTSEXCLUDE := 15417,
	OPCUAID_WELLKNOWNROLE_OBSERVER_ADDIDENTITY_INPUTARGUMENTS := 15673,
	OPCUAID_WELLKNOWNROLE_OBSERVER_REMOVEIDENTITY_INPUTARGUMENTS := 15675,
	OPCUAID_WELLKNOWNROLE_OBSERVER_ADDAPPLICATION_INPUTARGUMENTS := 16218,
	OPCUAID_WELLKNOWNROLE_OBSERVER_REMOVEAPPLICATION_INPUTARGUMENTS := 16220,
	OPCUAID_WELLKNOWNROLE_OBSERVER_ADDENDPOINT_INPUTARGUMENTS := 16222,
	OPCUAID_WELLKNOWNROLE_OBSERVER_REMOVEENDPOINT_INPUTARGUMENTS := 16224,
	OPCUAID_WELLKNOWNROLE_OPERATOR_IDENTITIES := 16225,
	OPCUAID_WELLKNOWNROLE_OPERATOR_APPLICATIONS := 16226,
	OPCUAID_WELLKNOWNROLE_OPERATOR_APPLICATIONSEXCLUDE := 15418,
	OPCUAID_WELLKNOWNROLE_OPERATOR_ENDPOINTS := 16227,
	OPCUAID_WELLKNOWNROLE_OPERATOR_ENDPOINTSEXCLUDE := 15423,
	OPCUAID_WELLKNOWNROLE_OPERATOR_ADDIDENTITY_INPUTARGUMENTS := 15685,
	OPCUAID_WELLKNOWNROLE_OPERATOR_REMOVEIDENTITY_INPUTARGUMENTS := 15687,
	OPCUAID_WELLKNOWNROLE_OPERATOR_ADDAPPLICATION_INPUTARGUMENTS := 16229,
	OPCUAID_WELLKNOWNROLE_OPERATOR_REMOVEAPPLICATION_INPUTARGUMENTS := 16231,
	OPCUAID_WELLKNOWNROLE_OPERATOR_ADDENDPOINT_INPUTARGUMENTS := 16233,
	OPCUAID_WELLKNOWNROLE_OPERATOR_REMOVEENDPOINT_INPUTARGUMENTS := 16235,
	OPCUAID_WELLKNOWNROLE_ENGINEER_IDENTITIES := 16236,
	OPCUAID_WELLKNOWNROLE_ENGINEER_APPLICATIONS := 16237,
	OPCUAID_WELLKNOWNROLE_ENGINEER_APPLICATIONSEXCLUDE := 15424,
	OPCUAID_WELLKNOWNROLE_ENGINEER_ENDPOINTS := 16238,
	OPCUAID_WELLKNOWNROLE_ENGINEER_ENDPOINTSEXCLUDE := 15425,
	OPCUAID_WELLKNOWNROLE_ENGINEER_ADDIDENTITY_INPUTARGUMENTS := 16042,
	OPCUAID_WELLKNOWNROLE_ENGINEER_REMOVEIDENTITY_INPUTARGUMENTS := 16044,
	OPCUAID_WELLKNOWNROLE_ENGINEER_ADDAPPLICATION_INPUTARGUMENTS := 16240,
	OPCUAID_WELLKNOWNROLE_ENGINEER_REMOVEAPPLICATION_INPUTARGUMENTS := 16242,
	OPCUAID_WELLKNOWNROLE_ENGINEER_ADDENDPOINT_INPUTARGUMENTS := 16244,
	OPCUAID_WELLKNOWNROLE_ENGINEER_REMOVEENDPOINT_INPUTARGUMENTS := 16246,
	OPCUAID_WELLKNOWNROLE_SUPERVISOR_IDENTITIES := 16247,
	OPCUAID_WELLKNOWNROLE_SUPERVISOR_APPLICATIONS := 16248,
	OPCUAID_WELLKNOWNROLE_SUPERVISOR_APPLICATIONSEXCLUDE := 15426,
	OPCUAID_WELLKNOWNROLE_SUPERVISOR_ENDPOINTS := 16249,
	OPCUAID_WELLKNOWNROLE_SUPERVISOR_ENDPOINTSEXCLUDE := 15427,
	OPCUAID_WELLKNOWNROLE_SUPERVISOR_ADDIDENTITY_INPUTARGUMENTS := 15697,
	OPCUAID_WELLKNOWNROLE_SUPERVISOR_REMOVEIDENTITY_INPUTARGUMENTS := 15699,
	OPCUAID_WELLKNOWNROLE_SUPERVISOR_ADDAPPLICATION_INPUTARGUMENTS := 16251,
	OPCUAID_WELLKNOWNROLE_SUPERVISOR_REMOVEAPPLICATION_INPUTARGUMENTS := 16253,
	OPCUAID_WELLKNOWNROLE_SUPERVISOR_ADDENDPOINT_INPUTARGUMENTS := 16255,
	OPCUAID_WELLKNOWNROLE_SUPERVISOR_REMOVEENDPOINT_INPUTARGUMENTS := 16257,
	OPCUAID_WELLKNOWNROLE_CONFIGUREADMIN_IDENTITIES := 16269,
	OPCUAID_WELLKNOWNROLE_CONFIGUREADMIN_APPLICATIONS := 16270,
	OPCUAID_WELLKNOWNROLE_CONFIGUREADMIN_APPLICATIONSEXCLUDE := 15428,
	OPCUAID_WELLKNOWNROLE_CONFIGUREADMIN_ENDPOINTS := 16271,
	OPCUAID_WELLKNOWNROLE_CONFIGUREADMIN_ENDPOINTSEXCLUDE := 15429,
	OPCUAID_WELLKNOWNROLE_CONFIGUREADMIN_ADDIDENTITY_INPUTARGUMENTS := 15721,
	OPCUAID_WELLKNOWNROLE_CONFIGUREADMIN_REMOVEIDENTITY_INPUTARGUMENTS := 15723,
	OPCUAID_WELLKNOWNROLE_CONFIGUREADMIN_ADDAPPLICATION_INPUTARGUMENTS := 16273,
	OPCUAID_WELLKNOWNROLE_CONFIGUREADMIN_REMOVEAPPLICATION_INPUTARGUMENTS := 16275,
	OPCUAID_WELLKNOWNROLE_CONFIGUREADMIN_ADDENDPOINT_INPUTARGUMENTS := 16277,
	OPCUAID_WELLKNOWNROLE_CONFIGUREADMIN_REMOVEENDPOINT_INPUTARGUMENTS := 16279,
	OPCUAID_WELLKNOWNROLE_SECURITYADMIN_IDENTITIES := 16258,
	OPCUAID_WELLKNOWNROLE_SECURITYADMIN_APPLICATIONS := 16259,
	OPCUAID_WELLKNOWNROLE_SECURITYADMIN_APPLICATIONSEXCLUDE := 15430,
	OPCUAID_WELLKNOWNROLE_SECURITYADMIN_ENDPOINTS := 16260,
	OPCUAID_WELLKNOWNROLE_SECURITYADMIN_ENDPOINTSEXCLUDE := 15527,
	OPCUAID_WELLKNOWNROLE_SECURITYADMIN_ADDIDENTITY_INPUTARGUMENTS := 15709,
	OPCUAID_WELLKNOWNROLE_SECURITYADMIN_REMOVEIDENTITY_INPUTARGUMENTS := 15711,
	OPCUAID_WELLKNOWNROLE_SECURITYADMIN_ADDAPPLICATION_INPUTARGUMENTS := 16262,
	OPCUAID_WELLKNOWNROLE_SECURITYADMIN_REMOVEAPPLICATION_INPUTARGUMENTS := 16264,
	OPCUAID_WELLKNOWNROLE_SECURITYADMIN_ADDENDPOINT_INPUTARGUMENTS := 16266,
	OPCUAID_WELLKNOWNROLE_SECURITYADMIN_REMOVEENDPOINT_INPUTARGUMENTS := 16268,
	OPCUAID_DATAITEMTYPE_DEFINITION := 2366,
	OPCUAID_DATAITEMTYPE_VALUEPRECISION := 2367,
	OPCUAID_ANALOGITEMTYPE_INSTRUMENTRANGE := 2370,
	OPCUAID_ANALOGITEMTYPE_EURANGE := 2369,
	OPCUAID_ANALOGITEMTYPE_ENGINEERINGUNITS := 2371,
	OPCUAID_EUITEMTYPE_INSTRUMENTRANGE := 17500,
	OPCUAID_EUITEMTYPE_EURANGE := 17501,
	OPCUAID_EUITEMTYPE_ENGINEERINGUNITS := 17502,
	OPCUAID_ANALOGUNITITEMTYPE_INSTRUMENTRANGE := 17506,
	OPCUAID_ANALOGUNITITEMTYPE_EURANGE := 17509,
	OPCUAID_ANALOGUNITITEMTYPE_ENGINEERINGUNITS := 17510,
	OPCUAID_TWOSTATEDISCRETETYPE_FALSESTATE := 2374,
	OPCUAID_TWOSTATEDISCRETETYPE_TRUESTATE := 2375,
	OPCUAID_MULTISTATEDISCRETETYPE_ENUMSTRINGS := 2377,
	OPCUAID_MULTISTATEVALUEDISCRETETYPE_ENUMVALUES := 11241,
	OPCUAID_MULTISTATEVALUEDISCRETETYPE_VALUEASTEXT := 11461,
	OPCUAID_ARRAYITEMTYPE_INSTRUMENTRANGE := 12024,
	OPCUAID_ARRAYITEMTYPE_EURANGE := 12025,
	OPCUAID_ARRAYITEMTYPE_ENGINEERINGUNITS := 12026,
	OPCUAID_ARRAYITEMTYPE_TITLE := 12027,
	OPCUAID_ARRAYITEMTYPE_AXISSCALETYPE := 12028,
	OPCUAID_YARRAYITEMTYPE_XAXISDEFINITION := 12037,
	OPCUAID_XYARRAYITEMTYPE_XAXISDEFINITION := 12046,
	OPCUAID_IMAGEITEMTYPE_XAXISDEFINITION := 12055,
	OPCUAID_IMAGEITEMTYPE_YAXISDEFINITION := 12056,
	OPCUAID_CUBEITEMTYPE_XAXISDEFINITION := 12065,
	OPCUAID_CUBEITEMTYPE_YAXISDEFINITION := 12066,
	OPCUAID_CUBEITEMTYPE_ZAXISDEFINITION := 12067,
	OPCUAID_NDIMENSIONARRAYITEMTYPE_AXISDEFINITION := 12076,
	OPCUAID_TWOSTATEVARIABLETYPE_ID := 8996,
	OPCUAID_TWOSTATEVARIABLETYPE_TRANSITIONTIME := 9000,
	OPCUAID_TWOSTATEVARIABLETYPE_EFFECTIVETRANSITIONTIME := 9001,
	OPCUAID_TWOSTATEVARIABLETYPE_TRUESTATE := 11110,
	OPCUAID_TWOSTATEVARIABLETYPE_FALSESTATE := 11111,
	OPCUAID_CONDITIONVARIABLETYPE_SOURCETIMESTAMP := 9003,
	OPCUAID_CONDITIONTYPE_CONDITIONCLASSID := 11112,
	OPCUAID_CONDITIONTYPE_CONDITIONCLASSNAME := 11113,
	OPCUAID_CONDITIONTYPE_CONDITIONSUBCLASSID := 16363,
	OPCUAID_CONDITIONTYPE_CONDITIONSUBCLASSNAME := 16364,
	OPCUAID_CONDITIONTYPE_CONDITIONNAME := 9009,
	OPCUAID_CONDITIONTYPE_BRANCHID := 9010,
	OPCUAID_CONDITIONTYPE_RETAIN := 3874,
	OPCUAID_CONDITIONTYPE_ENABLEDSTATE := 9011,
	OPCUAID_CONDITIONTYPE_ENABLEDSTATE_ID := 9012,
	OPCUAID_CONDITIONTYPE_ENABLEDSTATE_EFFECTIVEDISPLAYNAME := 9015,
	OPCUAID_CONDITIONTYPE_ENABLEDSTATE_TRANSITIONTIME := 9016,
	OPCUAID_CONDITIONTYPE_ENABLEDSTATE_EFFECTIVETRANSITIONTIME := 9017,
	OPCUAID_CONDITIONTYPE_ENABLEDSTATE_TRUESTATE := 9018,
	OPCUAID_CONDITIONTYPE_ENABLEDSTATE_FALSESTATE := 9019,
	OPCUAID_CONDITIONTYPE_QUALITY := 9020,
	OPCUAID_CONDITIONTYPE_QUALITY_SOURCETIMESTAMP := 9021,
	OPCUAID_CONDITIONTYPE_LASTSEVERITY := 9022,
	OPCUAID_CONDITIONTYPE_LASTSEVERITY_SOURCETIMESTAMP := 9023,
	OPCUAID_CONDITIONTYPE_COMMENT := 9024,
	OPCUAID_CONDITIONTYPE_COMMENT_SOURCETIMESTAMP := 9025,
	OPCUAID_CONDITIONTYPE_CLIENTUSERID := 9026,
	OPCUAID_CONDITIONTYPE_ADDCOMMENT_INPUTARGUMENTS := 9030,
	OPCUAID_CONDITIONTYPE_CONDITIONREFRESH_INPUTARGUMENTS := 3876,
	OPCUAID_CONDITIONTYPE_CONDITIONREFRESH2_INPUTARGUMENTS := 12913,
	OPCUAID_DIALOGCONDITIONTYPE_ENABLEDSTATE := 9035,
	OPCUAID_DIALOGCONDITIONTYPE_ENABLEDSTATE_ID := 9036,
	OPCUAID_DIALOGCONDITIONTYPE_QUALITY_SOURCETIMESTAMP := 9045,
	OPCUAID_DIALOGCONDITIONTYPE_LASTSEVERITY_SOURCETIMESTAMP := 9047,
	OPCUAID_DIALOGCONDITIONTYPE_COMMENT_SOURCETIMESTAMP := 9049,
	OPCUAID_DIALOGCONDITIONTYPE_ADDCOMMENT_INPUTARGUMENTS := 9054,
	OPCUAID_DIALOGCONDITIONTYPE_CONDITIONREFRESH_INPUTARGUMENTS := 4199,
	OPCUAID_DIALOGCONDITIONTYPE_CONDITIONREFRESH2_INPUTARGUMENTS := 12917,
	OPCUAID_DIALOGCONDITIONTYPE_DIALOGSTATE := 9055,
	OPCUAID_DIALOGCONDITIONTYPE_DIALOGSTATE_ID := 9056,
	OPCUAID_DIALOGCONDITIONTYPE_DIALOGSTATE_TRANSITIONTIME := 9060,
	OPCUAID_DIALOGCONDITIONTYPE_DIALOGSTATE_TRUESTATE := 9062,
	OPCUAID_DIALOGCONDITIONTYPE_DIALOGSTATE_FALSESTATE := 9063,
	OPCUAID_DIALOGCONDITIONTYPE_PROMPT := 2831,
	OPCUAID_DIALOGCONDITIONTYPE_RESPONSEOPTIONSET := 9064,
	OPCUAID_DIALOGCONDITIONTYPE_DEFAULTRESPONSE := 9065,
	OPCUAID_DIALOGCONDITIONTYPE_OKRESPONSE := 9066,
	OPCUAID_DIALOGCONDITIONTYPE_CANCELRESPONSE := 9067,
	OPCUAID_DIALOGCONDITIONTYPE_LASTRESPONSE := 9068,
	OPCUAID_DIALOGCONDITIONTYPE_RESPOND_INPUTARGUMENTS := 9070,
	OPCUAID_ACKNOWLEDGEABLECONDITIONTYPE_ENABLEDSTATE := 9073,
	OPCUAID_ACKNOWLEDGEABLECONDITIONTYPE_ENABLEDSTATE_ID := 9074,
	OPCUAID_ACKNOWLEDGEABLECONDITIONTYPE_QUALITY_SOURCETIMESTAMP := 9083,
	OPCUAID_ACKNOWLEDGEABLECONDITIONTYPE_LASTSEVERITY_SOURCETIMESTAMP := 9085,
	OPCUAID_ACKNOWLEDGEABLECONDITIONTYPE_COMMENT_SOURCETIMESTAMP := 9087,
	OPCUAID_ACKNOWLEDGEABLECONDITIONTYPE_ADDCOMMENT_INPUTARGUMENTS := 9092,
	OPCUAID_ACKNOWLEDGEABLECONDITIONTYPE_CONDITIONREFRESH_INPUTARGUMENTS := 5124,
	OPCUAID_ACKNOWLEDGEABLECONDITIONTYPE_CONDITIONREFRESH2_INPUTARGUMENTS := 12919,
	OPCUAID_ACKNOWLEDGEABLECONDITIONTYPE_ACKEDSTATE := 9093,
	OPCUAID_ACKNOWLEDGEABLECONDITIONTYPE_ACKEDSTATE_ID := 9094,
	OPCUAID_ACKNOWLEDGEABLECONDITIONTYPE_ACKEDSTATE_TRANSITIONTIME := 9098,
	OPCUAID_ACKNOWLEDGEABLECONDITIONTYPE_ACKEDSTATE_TRUESTATE := 9100,
	OPCUAID_ACKNOWLEDGEABLECONDITIONTYPE_ACKEDSTATE_FALSESTATE := 9101,
	OPCUAID_ACKNOWLEDGEABLECONDITIONTYPE_CONFIRMEDSTATE := 9102,
	OPCUAID_ACKNOWLEDGEABLECONDITIONTYPE_CONFIRMEDSTATE_ID := 9103,
	OPCUAID_ACKNOWLEDGEABLECONDITIONTYPE_CONFIRMEDSTATE_TRANSITIONTIME := 9107,
	OPCUAID_ACKNOWLEDGEABLECONDITIONTYPE_CONFIRMEDSTATE_TRUESTATE := 9109,
	OPCUAID_ACKNOWLEDGEABLECONDITIONTYPE_CONFIRMEDSTATE_FALSESTATE := 9110,
	OPCUAID_ACKNOWLEDGEABLECONDITIONTYPE_ACKNOWLEDGE_INPUTARGUMENTS := 9112,
	OPCUAID_ACKNOWLEDGEABLECONDITIONTYPE_CONFIRM_INPUTARGUMENTS := 9114,
	OPCUAID_ALARMCONDITIONTYPE_ENABLEDSTATE := 9118,
	OPCUAID_ALARMCONDITIONTYPE_ENABLEDSTATE_ID := 9119,
	OPCUAID_ALARMCONDITIONTYPE_QUALITY_SOURCETIMESTAMP := 9128,
	OPCUAID_ALARMCONDITIONTYPE_LASTSEVERITY_SOURCETIMESTAMP := 9130,
	OPCUAID_ALARMCONDITIONTYPE_COMMENT_SOURCETIMESTAMP := 9132,
	OPCUAID_ALARMCONDITIONTYPE_ADDCOMMENT_INPUTARGUMENTS := 9137,
	OPCUAID_ALARMCONDITIONTYPE_CONDITIONREFRESH_INPUTARGUMENTS := 5551,
	OPCUAID_ALARMCONDITIONTYPE_CONDITIONREFRESH2_INPUTARGUMENTS := 12985,
	OPCUAID_ALARMCONDITIONTYPE_ACKEDSTATE_ID := 9139,
	OPCUAID_ALARMCONDITIONTYPE_CONFIRMEDSTATE_ID := 9148,
	OPCUAID_ALARMCONDITIONTYPE_ACKNOWLEDGE_INPUTARGUMENTS := 9157,
	OPCUAID_ALARMCONDITIONTYPE_CONFIRM_INPUTARGUMENTS := 9159,
	OPCUAID_ALARMCONDITIONTYPE_ACTIVESTATE := 9160,
	OPCUAID_ALARMCONDITIONTYPE_ACTIVESTATE_ID := 9161,
	OPCUAID_ALARMCONDITIONTYPE_ACTIVESTATE_EFFECTIVEDISPLAYNAME := 9164,
	OPCUAID_ALARMCONDITIONTYPE_ACTIVESTATE_TRANSITIONTIME := 9165,
	OPCUAID_ALARMCONDITIONTYPE_ACTIVESTATE_EFFECTIVETRANSITIONTIME := 9166,
	OPCUAID_ALARMCONDITIONTYPE_ACTIVESTATE_TRUESTATE := 9167,
	OPCUAID_ALARMCONDITIONTYPE_ACTIVESTATE_FALSESTATE := 9168,
	OPCUAID_ALARMCONDITIONTYPE_INPUTNODE := 11120,
	OPCUAID_ALARMCONDITIONTYPE_SUPPRESSEDSTATE := 9169,
	OPCUAID_ALARMCONDITIONTYPE_SUPPRESSEDSTATE_ID := 9170,
	OPCUAID_ALARMCONDITIONTYPE_SUPPRESSEDSTATE_TRANSITIONTIME := 9174,
	OPCUAID_ALARMCONDITIONTYPE_SUPPRESSEDSTATE_TRUESTATE := 9176,
	OPCUAID_ALARMCONDITIONTYPE_SUPPRESSEDSTATE_FALSESTATE := 9177,
	OPCUAID_ALARMCONDITIONTYPE_OUTOFSERVICESTATE := 16371,
	OPCUAID_ALARMCONDITIONTYPE_OUTOFSERVICESTATE_ID := 16372,
	OPCUAID_ALARMCONDITIONTYPE_OUTOFSERVICESTATE_TRANSITIONTIME := 16376,
	OPCUAID_ALARMCONDITIONTYPE_OUTOFSERVICESTATE_TRUESTATE := 16378,
	OPCUAID_ALARMCONDITIONTYPE_OUTOFSERVICESTATE_FALSESTATE := 16379,
	OPCUAID_ALARMCONDITIONTYPE_SHELVINGSTATE_CURRENTSTATE := 9179,
	OPCUAID_ALARMCONDITIONTYPE_SHELVINGSTATE_CURRENTSTATE_ID := 9180,
	OPCUAID_ALARMCONDITIONTYPE_SHELVINGSTATE_LASTTRANSITION := 9184,
	OPCUAID_ALARMCONDITIONTYPE_SHELVINGSTATE_LASTTRANSITION_ID := 9185,
	OPCUAID_ALARMCONDITIONTYPE_SHELVINGSTATE_LASTTRANSITION_TRANSITIONTIME := 9188,
	OPCUAID_ALARMCONDITIONTYPE_SHELVINGSTATE_UNSHELVETIME := 9189,
	OPCUAID_ALARMCONDITIONTYPE_SHELVINGSTATE_TIMEDSHELVE_INPUTARGUMENTS := 9214,
	OPCUAID_ALARMCONDITIONTYPE_SUPPRESSEDORSHELVED := 9215,
	OPCUAID_ALARMCONDITIONTYPE_MAXTIMESHELVED := 9216,
	OPCUAID_ALARMCONDITIONTYPE_AUDIBLEENABLED := 16389,
	OPCUAID_ALARMCONDITIONTYPE_AUDIBLESOUND := 16390,
	OPCUAID_ALARMCONDITIONTYPE_SILENCESTATE := 16380,
	OPCUAID_ALARMCONDITIONTYPE_SILENCESTATE_ID := 16381,
	OPCUAID_ALARMCONDITIONTYPE_SILENCESTATE_TRANSITIONTIME := 16385,
	OPCUAID_ALARMCONDITIONTYPE_SILENCESTATE_TRUESTATE := 16387,
	OPCUAID_ALARMCONDITIONTYPE_SILENCESTATE_FALSESTATE := 16388,
	OPCUAID_ALARMCONDITIONTYPE_ONDELAY := 16395,
	OPCUAID_ALARMCONDITIONTYPE_OFFDELAY := 16396,
	OPCUAID_ALARMCONDITIONTYPE_FIRSTINGROUPFLAG := 16397,
	OPCUAID_ALARMCONDITIONTYPE_LATCHEDSTATE := 18190,
	OPCUAID_ALARMCONDITIONTYPE_LATCHEDSTATE_ID := 18191,
	OPCUAID_ALARMCONDITIONTYPE_LATCHEDSTATE_TRANSITIONTIME := 18195,
	OPCUAID_ALARMCONDITIONTYPE_LATCHEDSTATE_TRUESTATE := 18197,
	OPCUAID_ALARMCONDITIONTYPE_LATCHEDSTATE_FALSESTATE := 18198,
	OPCUAID_ALARMCONDITIONTYPE_REALARMTIME := 16400,
	OPCUAID_ALARMCONDITIONTYPE_REALARMREPEATCOUNT := 16401,
	OPCUAID_ALARMGROUPTYPE_ALARMCONDITIONINSTANCE_PLACEHOLDER_EVENTID := 16407,
	OPCUAID_ALARMGROUPTYPE_ALARMCONDITIONINSTANCE_PLACEHOLDER_EVENTTYPE := 16408,
	OPCUAID_ALARMGROUPTYPE_ALARMCONDITIONINSTANCE_PLACEHOLDER_SOURCENODE := 16409,
	OPCUAID_ALARMGROUPTYPE_ALARMCONDITIONINSTANCE_PLACEHOLDER_SOURCENAME := 16410,
	OPCUAID_ALARMGROUPTYPE_ALARMCONDITIONINSTANCE_PLACEHOLDER_TIME := 16411,
	OPCUAID_ALARMGROUPTYPE_ALARMCONDITIONINSTANCE_PLACEHOLDER_RECEIVETIME := 16412,
	OPCUAID_ALARMGROUPTYPE_ALARMCONDITIONINSTANCE_PLACEHOLDER_LOCALTIME := 16413,
	OPCUAID_ALARMGROUPTYPE_ALARMCONDITIONINSTANCE_PLACEHOLDER_MESSAGE := 16414,
	OPCUAID_ALARMGROUPTYPE_ALARMCONDITIONINSTANCE_PLACEHOLDER_SEVERITY := 16415,
	OPCUAID_ALARMGROUPTYPE_ALARMCONDITIONINSTANCE_PLACEHOLDER_CONDITIONCLASSID := 16416,
	OPCUAID_ALARMGROUPTYPE_ALARMCONDITIONINSTANCE_PLACEHOLDER_CONDITIONCLASSNAME := 16417,
	OPCUAID_ALARMGROUPTYPE_ALARMCONDITIONINSTANCE_PLACEHOLDER_CONDITIONNAME := 16420,
	OPCUAID_ALARMGROUPTYPE_ALARMCONDITIONINSTANCE_PLACEHOLDER_BRANCHID := 16421,
	OPCUAID_ALARMGROUPTYPE_ALARMCONDITIONINSTANCE_PLACEHOLDER_RETAIN := 16422,
	OPCUAID_ALARMGROUPTYPE_ALARMCONDITIONINSTANCE_PLACEHOLDER_ENABLEDSTATE := 16423,
	OPCUAID_ALARMGROUPTYPE_ALARMCONDITIONINSTANCE_PLACEHOLDER_ENABLEDSTATE_ID := 16424,
	OPCUAID_ALARMGROUPTYPE_ALARMCONDITIONINSTANCE_PLACEHOLDER_QUALITY := 16432,
	OPCUAID_ALARMGROUPTYPE_ALARMCONDITIONINSTANCE_PLACEHOLDER_QUALITY_SOURCETIMESTAMP := 16433,
	OPCUAID_ALARMGROUPTYPE_ALARMCONDITIONINSTANCE_PLACEHOLDER_LASTSEVERITY := 16434,
	OPCUAID_ALARMGROUPTYPE_ALARMCONDITIONINSTANCE_PLACEHOLDER_LASTSEVERITY_SOURCETIMESTAMP := 16435,
	OPCUAID_ALARMGROUPTYPE_ALARMCONDITIONINSTANCE_PLACEHOLDER_COMMENT := 16436,
	OPCUAID_ALARMGROUPTYPE_ALARMCONDITIONINSTANCE_PLACEHOLDER_COMMENT_SOURCETIMESTAMP := 16437,
	OPCUAID_ALARMGROUPTYPE_ALARMCONDITIONINSTANCE_PLACEHOLDER_CLIENTUSERID := 16438,
	OPCUAID_ALARMGROUPTYPE_ALARMCONDITIONINSTANCE_PLACEHOLDER_ADDCOMMENT_INPUTARGUMENTS := 16442,
	OPCUAID_ALARMGROUPTYPE_ALARMCONDITIONINSTANCE_PLACEHOLDER_ACKEDSTATE := 16443,
	OPCUAID_ALARMGROUPTYPE_ALARMCONDITIONINSTANCE_PLACEHOLDER_ACKEDSTATE_ID := 16444,
	OPCUAID_ALARMGROUPTYPE_ALARMCONDITIONINSTANCE_PLACEHOLDER_CONFIRMEDSTATE_ID := 16453,
	OPCUAID_ALARMGROUPTYPE_ALARMCONDITIONINSTANCE_PLACEHOLDER_ACKNOWLEDGE_INPUTARGUMENTS := 16462,
	OPCUAID_ALARMGROUPTYPE_ALARMCONDITIONINSTANCE_PLACEHOLDER_CONFIRM_INPUTARGUMENTS := 16464,
	OPCUAID_ALARMGROUPTYPE_ALARMCONDITIONINSTANCE_PLACEHOLDER_ACTIVESTATE := 16465,
	OPCUAID_ALARMGROUPTYPE_ALARMCONDITIONINSTANCE_PLACEHOLDER_ACTIVESTATE_ID := 16466,
	OPCUAID_ALARMGROUPTYPE_ALARMCONDITIONINSTANCE_PLACEHOLDER_INPUTNODE := 16474,
	OPCUAID_ALARMGROUPTYPE_ALARMCONDITIONINSTANCE_PLACEHOLDER_SUPPRESSEDSTATE_ID := 16476,
	OPCUAID_ALARMGROUPTYPE_ALARMCONDITIONINSTANCE_PLACEHOLDER_OUTOFSERVICESTATE_ID := 16485,
	OPCUAID_ALARMGROUPTYPE_ALARMCONDITIONINSTANCE_PLACEHOLDER_SHELVINGSTATE_CURRENTSTATE := 16503,
	OPCUAID_ALARMGROUPTYPE_ALARMCONDITIONINSTANCE_PLACEHOLDER_SHELVINGSTATE_CURRENTSTATE_ID := 16504,
	OPCUAID_ALARMGROUPTYPE_ALARMCONDITIONINSTANCE_PLACEHOLDER_SHELVINGSTATE_LASTTRANSITION_ID := 16509,
	OPCUAID_ALARMGROUPTYPE_ALARMCONDITIONINSTANCE_PLACEHOLDER_SHELVINGSTATE_UNSHELVETIME := 16514,
	OPCUAID_ALARMGROUPTYPE_ALARMCONDITIONINSTANCE_PLACEHOLDER_SHELVINGSTATE_TIMEDSHELVE_INPUTARGUMENTS := 16518,
	OPCUAID_ALARMGROUPTYPE_ALARMCONDITIONINSTANCE_PLACEHOLDER_SUPPRESSEDORSHELVED := 16519,
	OPCUAID_ALARMGROUPTYPE_ALARMCONDITIONINSTANCE_PLACEHOLDER_SILENCESTATE_ID := 16494,
	OPCUAID_ALARMGROUPTYPE_ALARMCONDITIONINSTANCE_PLACEHOLDER_LATCHEDSTATE_ID := 18204,
	OPCUAID_SHELVEDSTATEMACHINETYPE_CURRENTSTATE_ID := 6089,
	OPCUAID_SHELVEDSTATEMACHINETYPE_LASTTRANSITION_ID := 6094,
	OPCUAID_SHELVEDSTATEMACHINETYPE_UNSHELVETIME := 9115,
	OPCUAID_SHELVEDSTATEMACHINETYPE_UNSHELVED_STATENUMBER := 6098,
	OPCUAID_SHELVEDSTATEMACHINETYPE_TIMEDSHELVED_STATENUMBER := 6100,
	OPCUAID_SHELVEDSTATEMACHINETYPE_ONESHOTSHELVED_STATENUMBER := 6101,
	OPCUAID_SHELVEDSTATEMACHINETYPE_UNSHELVEDTOTIMEDSHELVED_TRANSITIONNUMBER := 11322,
	OPCUAID_SHELVEDSTATEMACHINETYPE_UNSHELVEDTOONESHOTSHELVED_TRANSITIONNUMBER := 11323,
	OPCUAID_SHELVEDSTATEMACHINETYPE_TIMEDSHELVEDTOUNSHELVED_TRANSITIONNUMBER := 11324,
	OPCUAID_SHELVEDSTATEMACHINETYPE_TIMEDSHELVEDTOONESHOTSHELVED_TRANSITIONNUMBER := 11325,
	OPCUAID_SHELVEDSTATEMACHINETYPE_ONESHOTSHELVEDTOUNSHELVED_TRANSITIONNUMBER := 11326,
	OPCUAID_SHELVEDSTATEMACHINETYPE_ONESHOTSHELVEDTOTIMEDSHELVED_TRANSITIONNUMBER := 11327,
	OPCUAID_SHELVEDSTATEMACHINETYPE_TIMEDSHELVE_INPUTARGUMENTS := 2991,
	OPCUAID_LIMITALARMTYPE_ENABLEDSTATE_ID := 9220,
	OPCUAID_LIMITALARMTYPE_QUALITY_SOURCETIMESTAMP := 9229,
	OPCUAID_LIMITALARMTYPE_LASTSEVERITY_SOURCETIMESTAMP := 9231,
	OPCUAID_LIMITALARMTYPE_COMMENT_SOURCETIMESTAMP := 9233,
	OPCUAID_LIMITALARMTYPE_ADDCOMMENT_INPUTARGUMENTS := 9238,
	OPCUAID_LIMITALARMTYPE_CONDITIONREFRESH_INPUTARGUMENTS := 6127,
	OPCUAID_LIMITALARMTYPE_CONDITIONREFRESH2_INPUTARGUMENTS := 12987,
	OPCUAID_LIMITALARMTYPE_ACKEDSTATE_ID := 9240,
	OPCUAID_LIMITALARMTYPE_CONFIRMEDSTATE_ID := 9249,
	OPCUAID_LIMITALARMTYPE_ACKNOWLEDGE_INPUTARGUMENTS := 9258,
	OPCUAID_LIMITALARMTYPE_CONFIRM_INPUTARGUMENTS := 9260,
	OPCUAID_LIMITALARMTYPE_ACTIVESTATE_ID := 9262,
	OPCUAID_LIMITALARMTYPE_SUPPRESSEDSTATE_ID := 9271,
	OPCUAID_LIMITALARMTYPE_OUTOFSERVICESTATE_ID := 16539,
	OPCUAID_LIMITALARMTYPE_SHELVINGSTATE_CURRENTSTATE := 9280,
	OPCUAID_LIMITALARMTYPE_SHELVINGSTATE_CURRENTSTATE_ID := 9281,
	OPCUAID_LIMITALARMTYPE_SHELVINGSTATE_LASTTRANSITION_ID := 9286,
	OPCUAID_LIMITALARMTYPE_SHELVINGSTATE_UNSHELVETIME := 9290,
	OPCUAID_LIMITALARMTYPE_SHELVINGSTATE_TIMEDSHELVE_INPUTARGUMENTS := 9315,
	OPCUAID_LIMITALARMTYPE_SILENCESTATE_ID := 16548,
	OPCUAID_LIMITALARMTYPE_LATCHEDSTATE_ID := 18214,
	OPCUAID_LIMITALARMTYPE_HIGHHIGHLIMIT := 11124,
	OPCUAID_LIMITALARMTYPE_HIGHLIMIT := 11125,
	OPCUAID_LIMITALARMTYPE_LOWLIMIT := 11126,
	OPCUAID_LIMITALARMTYPE_LOWLOWLIMIT := 11127,
	OPCUAID_LIMITALARMTYPE_BASEHIGHHIGHLIMIT := 16572,
	OPCUAID_LIMITALARMTYPE_BASEHIGHLIMIT := 16573,
	OPCUAID_LIMITALARMTYPE_BASELOWLIMIT := 16574,
	OPCUAID_LIMITALARMTYPE_BASELOWLOWLIMIT := 16575,
	OPCUAID_EXCLUSIVELIMITSTATEMACHINETYPE_CURRENTSTATE_ID := 9320,
	OPCUAID_EXCLUSIVELIMITSTATEMACHINETYPE_LASTTRANSITION_ID := 9325,
	OPCUAID_EXCLUSIVELIMITSTATEMACHINETYPE_HIGHHIGH_STATENUMBER := 9330,
	OPCUAID_EXCLUSIVELIMITSTATEMACHINETYPE_HIGH_STATENUMBER := 9332,
	OPCUAID_EXCLUSIVELIMITSTATEMACHINETYPE_LOW_STATENUMBER := 9334,
	OPCUAID_EXCLUSIVELIMITSTATEMACHINETYPE_LOWLOW_STATENUMBER := 9336,
	OPCUAID_EXCLUSIVELIMITSTATEMACHINETYPE_LOWLOWTOLOW_TRANSITIONNUMBER := 11340,
	OPCUAID_EXCLUSIVELIMITSTATEMACHINETYPE_LOWTOLOWLOW_TRANSITIONNUMBER := 11341,
	OPCUAID_EXCLUSIVELIMITSTATEMACHINETYPE_HIGHHIGHTOHIGH_TRANSITIONNUMBER := 11342,
	OPCUAID_EXCLUSIVELIMITSTATEMACHINETYPE_HIGHTOHIGHHIGH_TRANSITIONNUMBER := 11343,
	OPCUAID_EXCLUSIVELIMITALARMTYPE_ENABLEDSTATE_ID := 9355,
	OPCUAID_EXCLUSIVELIMITALARMTYPE_QUALITY_SOURCETIMESTAMP := 9364,
	OPCUAID_EXCLUSIVELIMITALARMTYPE_LASTSEVERITY_SOURCETIMESTAMP := 9366,
	OPCUAID_EXCLUSIVELIMITALARMTYPE_COMMENT_SOURCETIMESTAMP := 9368,
	OPCUAID_EXCLUSIVELIMITALARMTYPE_ADDCOMMENT_INPUTARGUMENTS := 9373,
	OPCUAID_EXCLUSIVELIMITALARMTYPE_CONDITIONREFRESH_INPUTARGUMENTS := 9375,
	OPCUAID_EXCLUSIVELIMITALARMTYPE_CONDITIONREFRESH2_INPUTARGUMENTS := 12989,
	OPCUAID_EXCLUSIVELIMITALARMTYPE_ACKEDSTATE_ID := 9377,
	OPCUAID_EXCLUSIVELIMITALARMTYPE_CONFIRMEDSTATE_ID := 9386,
	OPCUAID_EXCLUSIVELIMITALARMTYPE_ACKNOWLEDGE_INPUTARGUMENTS := 9395,
	OPCUAID_EXCLUSIVELIMITALARMTYPE_CONFIRM_INPUTARGUMENTS := 9397,
	OPCUAID_EXCLUSIVELIMITALARMTYPE_ACTIVESTATE := 9398,
	OPCUAID_EXCLUSIVELIMITALARMTYPE_ACTIVESTATE_ID := 9399,
	OPCUAID_EXCLUSIVELIMITALARMTYPE_SUPPRESSEDSTATE_ID := 9408,
	OPCUAID_EXCLUSIVELIMITALARMTYPE_OUTOFSERVICESTATE_ID := 16579,
	OPCUAID_EXCLUSIVELIMITALARMTYPE_SHELVINGSTATE_CURRENTSTATE := 9417,
	OPCUAID_EXCLUSIVELIMITALARMTYPE_SHELVINGSTATE_CURRENTSTATE_ID := 9418,
	OPCUAID_EXCLUSIVELIMITALARMTYPE_SHELVINGSTATE_LASTTRANSITION_ID := 9423,
	OPCUAID_EXCLUSIVELIMITALARMTYPE_SHELVINGSTATE_UNSHELVETIME := 9427,
	OPCUAID_EXCLUSIVELIMITALARMTYPE_SHELVINGSTATE_TIMEDSHELVE_INPUTARGUMENTS := 9452,
	OPCUAID_EXCLUSIVELIMITALARMTYPE_SILENCESTATE_ID := 16588,
	OPCUAID_EXCLUSIVELIMITALARMTYPE_LATCHEDSTATE_ID := 18224,
	OPCUAID_EXCLUSIVELIMITALARMTYPE_LIMITSTATE_CURRENTSTATE := 9456,
	OPCUAID_EXCLUSIVELIMITALARMTYPE_LIMITSTATE_CURRENTSTATE_ID := 9457,
	OPCUAID_EXCLUSIVELIMITALARMTYPE_LIMITSTATE_LASTTRANSITION := 9461,
	OPCUAID_EXCLUSIVELIMITALARMTYPE_LIMITSTATE_LASTTRANSITION_ID := 9462,
	OPCUAID_EXCLUSIVELIMITALARMTYPE_LIMITSTATE_LASTTRANSITION_TRANSITIONTIME := 9465,
	OPCUAID_NONEXCLUSIVELIMITALARMTYPE_ENABLEDSTATE_ID := 9920,
	OPCUAID_NONEXCLUSIVELIMITALARMTYPE_QUALITY_SOURCETIMESTAMP := 9929,
	OPCUAID_NONEXCLUSIVELIMITALARMTYPE_LASTSEVERITY_SOURCETIMESTAMP := 9931,
	OPCUAID_NONEXCLUSIVELIMITALARMTYPE_COMMENT_SOURCETIMESTAMP := 9933,
	OPCUAID_NONEXCLUSIVELIMITALARMTYPE_ADDCOMMENT_INPUTARGUMENTS := 9938,
	OPCUAID_NONEXCLUSIVELIMITALARMTYPE_CONDITIONREFRESH_INPUTARGUMENTS := 9940,
	OPCUAID_NONEXCLUSIVELIMITALARMTYPE_CONDITIONREFRESH2_INPUTARGUMENTS := 12991,
	OPCUAID_NONEXCLUSIVELIMITALARMTYPE_ACKEDSTATE_ID := 9942,
	OPCUAID_NONEXCLUSIVELIMITALARMTYPE_CONFIRMEDSTATE_ID := 9951,
	OPCUAID_NONEXCLUSIVELIMITALARMTYPE_ACKNOWLEDGE_INPUTARGUMENTS := 9960,
	OPCUAID_NONEXCLUSIVELIMITALARMTYPE_CONFIRM_INPUTARGUMENTS := 9962,
	OPCUAID_NONEXCLUSIVELIMITALARMTYPE_ACTIVESTATE := 9963,
	OPCUAID_NONEXCLUSIVELIMITALARMTYPE_ACTIVESTATE_ID := 9964,
	OPCUAID_NONEXCLUSIVELIMITALARMTYPE_SUPPRESSEDSTATE_ID := 9973,
	OPCUAID_NONEXCLUSIVELIMITALARMTYPE_OUTOFSERVICESTATE_ID := 16619,
	OPCUAID_NONEXCLUSIVELIMITALARMTYPE_SHELVINGSTATE_CURRENTSTATE := 9982,
	OPCUAID_NONEXCLUSIVELIMITALARMTYPE_SHELVINGSTATE_CURRENTSTATE_ID := 9983,
	OPCUAID_NONEXCLUSIVELIMITALARMTYPE_SHELVINGSTATE_LASTTRANSITION_ID := 9988,
	OPCUAID_NONEXCLUSIVELIMITALARMTYPE_SHELVINGSTATE_UNSHELVETIME := 9992,
	OPCUAID_NONEXCLUSIVELIMITALARMTYPE_SHELVINGSTATE_TIMEDSHELVE_INPUTARGUMENTS := 10017,
	OPCUAID_NONEXCLUSIVELIMITALARMTYPE_SILENCESTATE_ID := 16628,
	OPCUAID_NONEXCLUSIVELIMITALARMTYPE_LATCHEDSTATE_ID := 18234,
	OPCUAID_NONEXCLUSIVELIMITALARMTYPE_HIGHHIGHSTATE := 10020,
	OPCUAID_NONEXCLUSIVELIMITALARMTYPE_HIGHHIGHSTATE_ID := 10021,
	OPCUAID_NONEXCLUSIVELIMITALARMTYPE_HIGHHIGHSTATE_TRANSITIONTIME := 10025,
	OPCUAID_NONEXCLUSIVELIMITALARMTYPE_HIGHHIGHSTATE_TRUESTATE := 10027,
	OPCUAID_NONEXCLUSIVELIMITALARMTYPE_HIGHHIGHSTATE_FALSESTATE := 10028,
	OPCUAID_NONEXCLUSIVELIMITALARMTYPE_HIGHSTATE := 10029,
	OPCUAID_NONEXCLUSIVELIMITALARMTYPE_HIGHSTATE_ID := 10030,
	OPCUAID_NONEXCLUSIVELIMITALARMTYPE_HIGHSTATE_TRANSITIONTIME := 10034,
	OPCUAID_NONEXCLUSIVELIMITALARMTYPE_HIGHSTATE_TRUESTATE := 10036,
	OPCUAID_NONEXCLUSIVELIMITALARMTYPE_HIGHSTATE_FALSESTATE := 10037,
	OPCUAID_NONEXCLUSIVELIMITALARMTYPE_LOWSTATE := 10038,
	OPCUAID_NONEXCLUSIVELIMITALARMTYPE_LOWSTATE_ID := 10039,
	OPCUAID_NONEXCLUSIVELIMITALARMTYPE_LOWSTATE_TRANSITIONTIME := 10043,
	OPCUAID_NONEXCLUSIVELIMITALARMTYPE_LOWSTATE_TRUESTATE := 10045,
	OPCUAID_NONEXCLUSIVELIMITALARMTYPE_LOWSTATE_FALSESTATE := 10046,
	OPCUAID_NONEXCLUSIVELIMITALARMTYPE_LOWLOWSTATE := 10047,
	OPCUAID_NONEXCLUSIVELIMITALARMTYPE_LOWLOWSTATE_ID := 10048,
	OPCUAID_NONEXCLUSIVELIMITALARMTYPE_LOWLOWSTATE_TRANSITIONTIME := 10052,
	OPCUAID_NONEXCLUSIVELIMITALARMTYPE_LOWLOWSTATE_TRUESTATE := 10054,
	OPCUAID_NONEXCLUSIVELIMITALARMTYPE_LOWLOWSTATE_FALSESTATE := 10055,
	OPCUAID_NONEXCLUSIVELEVELALARMTYPE_ENABLEDSTATE_ID := 10074,
	OPCUAID_NONEXCLUSIVELEVELALARMTYPE_QUALITY_SOURCETIMESTAMP := 10083,
	OPCUAID_NONEXCLUSIVELEVELALARMTYPE_LASTSEVERITY_SOURCETIMESTAMP := 10085,
	OPCUAID_NONEXCLUSIVELEVELALARMTYPE_COMMENT_SOURCETIMESTAMP := 10087,
	OPCUAID_NONEXCLUSIVELEVELALARMTYPE_ADDCOMMENT_INPUTARGUMENTS := 10092,
	OPCUAID_NONEXCLUSIVELEVELALARMTYPE_CONDITIONREFRESH_INPUTARGUMENTS := 10094,
	OPCUAID_NONEXCLUSIVELEVELALARMTYPE_CONDITIONREFRESH2_INPUTARGUMENTS := 12993,
	OPCUAID_NONEXCLUSIVELEVELALARMTYPE_ACKEDSTATE_ID := 10096,
	OPCUAID_NONEXCLUSIVELEVELALARMTYPE_CONFIRMEDSTATE_ID := 10105,
	OPCUAID_NONEXCLUSIVELEVELALARMTYPE_ACKNOWLEDGE_INPUTARGUMENTS := 10114,
	OPCUAID_NONEXCLUSIVELEVELALARMTYPE_CONFIRM_INPUTARGUMENTS := 10116,
	OPCUAID_NONEXCLUSIVELEVELALARMTYPE_ACTIVESTATE_ID := 10118,
	OPCUAID_NONEXCLUSIVELEVELALARMTYPE_SUPPRESSEDSTATE_ID := 10127,
	OPCUAID_NONEXCLUSIVELEVELALARMTYPE_OUTOFSERVICESTATE_ID := 16659,
	OPCUAID_NONEXCLUSIVELEVELALARMTYPE_SHELVINGSTATE_CURRENTSTATE := 10136,
	OPCUAID_NONEXCLUSIVELEVELALARMTYPE_SHELVINGSTATE_CURRENTSTATE_ID := 10137,
	OPCUAID_NONEXCLUSIVELEVELALARMTYPE_SHELVINGSTATE_LASTTRANSITION_ID := 10142,
	OPCUAID_NONEXCLUSIVELEVELALARMTYPE_SHELVINGSTATE_UNSHELVETIME := 10146,
	OPCUAID_NONEXCLUSIVELEVELALARMTYPE_SHELVINGSTATE_TIMEDSHELVE_INPUTARGUMENTS := 10171,
	OPCUAID_NONEXCLUSIVELEVELALARMTYPE_SILENCESTATE_ID := 16668,
	OPCUAID_NONEXCLUSIVELEVELALARMTYPE_LATCHEDSTATE_ID := 18247,
	OPCUAID_NONEXCLUSIVELEVELALARMTYPE_HIGHHIGHSTATE_ID := 10175,
	OPCUAID_NONEXCLUSIVELEVELALARMTYPE_HIGHSTATE_ID := 10184,
	OPCUAID_NONEXCLUSIVELEVELALARMTYPE_LOWSTATE_ID := 10193,
	OPCUAID_NONEXCLUSIVELEVELALARMTYPE_LOWLOWSTATE_ID := 10202,
	OPCUAID_EXCLUSIVELEVELALARMTYPE_ENABLEDSTATE_ID := 9496,
	OPCUAID_EXCLUSIVELEVELALARMTYPE_QUALITY_SOURCETIMESTAMP := 9505,
	OPCUAID_EXCLUSIVELEVELALARMTYPE_LASTSEVERITY_SOURCETIMESTAMP := 9507,
	OPCUAID_EXCLUSIVELEVELALARMTYPE_COMMENT_SOURCETIMESTAMP := 9509,
	OPCUAID_EXCLUSIVELEVELALARMTYPE_ADDCOMMENT_INPUTARGUMENTS := 9514,
	OPCUAID_EXCLUSIVELEVELALARMTYPE_CONDITIONREFRESH_INPUTARGUMENTS := 9516,
	OPCUAID_EXCLUSIVELEVELALARMTYPE_CONDITIONREFRESH2_INPUTARGUMENTS := 12995,
	OPCUAID_EXCLUSIVELEVELALARMTYPE_ACKEDSTATE_ID := 9518,
	OPCUAID_EXCLUSIVELEVELALARMTYPE_CONFIRMEDSTATE_ID := 9527,
	OPCUAID_EXCLUSIVELEVELALARMTYPE_ACKNOWLEDGE_INPUTARGUMENTS := 9536,
	OPCUAID_EXCLUSIVELEVELALARMTYPE_CONFIRM_INPUTARGUMENTS := 9538,
	OPCUAID_EXCLUSIVELEVELALARMTYPE_ACTIVESTATE_ID := 9540,
	OPCUAID_EXCLUSIVELEVELALARMTYPE_SUPPRESSEDSTATE_ID := 9549,
	OPCUAID_EXCLUSIVELEVELALARMTYPE_OUTOFSERVICESTATE_ID := 16699,
	OPCUAID_EXCLUSIVELEVELALARMTYPE_SHELVINGSTATE_CURRENTSTATE := 9558,
	OPCUAID_EXCLUSIVELEVELALARMTYPE_SHELVINGSTATE_CURRENTSTATE_ID := 9559,
	OPCUAID_EXCLUSIVELEVELALARMTYPE_SHELVINGSTATE_LASTTRANSITION_ID := 9564,
	OPCUAID_EXCLUSIVELEVELALARMTYPE_SHELVINGSTATE_UNSHELVETIME := 9568,
	OPCUAID_EXCLUSIVELEVELALARMTYPE_SHELVINGSTATE_TIMEDSHELVE_INPUTARGUMENTS := 9593,
	OPCUAID_EXCLUSIVELEVELALARMTYPE_SILENCESTATE_ID := 16708,
	OPCUAID_EXCLUSIVELEVELALARMTYPE_LATCHEDSTATE_ID := 18258,
	OPCUAID_EXCLUSIVELEVELALARMTYPE_LIMITSTATE_CURRENTSTATE := 9597,
	OPCUAID_EXCLUSIVELEVELALARMTYPE_LIMITSTATE_CURRENTSTATE_ID := 9598,
	OPCUAID_EXCLUSIVELEVELALARMTYPE_LIMITSTATE_LASTTRANSITION_ID := 9603,
	OPCUAID_NONEXCLUSIVEDEVIATIONALARMTYPE_ENABLEDSTATE_ID := 10382,
	OPCUAID_NONEXCLUSIVEDEVIATIONALARMTYPE_QUALITY_SOURCETIMESTAMP := 10391,
	OPCUAID_NONEXCLUSIVEDEVIATIONALARMTYPE_LASTSEVERITY_SOURCETIMESTAMP := 10393,
	OPCUAID_NONEXCLUSIVEDEVIATIONALARMTYPE_COMMENT_SOURCETIMESTAMP := 10395,
	OPCUAID_NONEXCLUSIVEDEVIATIONALARMTYPE_ADDCOMMENT_INPUTARGUMENTS := 10400,
	OPCUAID_NONEXCLUSIVEDEVIATIONALARMTYPE_CONDITIONREFRESH_INPUTARGUMENTS := 10402,
	OPCUAID_NONEXCLUSIVEDEVIATIONALARMTYPE_CONDITIONREFRESH2_INPUTARGUMENTS := 12997,
	OPCUAID_NONEXCLUSIVEDEVIATIONALARMTYPE_ACKEDSTATE_ID := 10404,
	OPCUAID_NONEXCLUSIVEDEVIATIONALARMTYPE_CONFIRMEDSTATE_ID := 10413,
	OPCUAID_NONEXCLUSIVEDEVIATIONALARMTYPE_ACKNOWLEDGE_INPUTARGUMENTS := 10422,
	OPCUAID_NONEXCLUSIVEDEVIATIONALARMTYPE_CONFIRM_INPUTARGUMENTS := 10424,
	OPCUAID_NONEXCLUSIVEDEVIATIONALARMTYPE_ACTIVESTATE_ID := 10426,
	OPCUAID_NONEXCLUSIVEDEVIATIONALARMTYPE_SUPPRESSEDSTATE_ID := 10435,
	OPCUAID_NONEXCLUSIVEDEVIATIONALARMTYPE_OUTOFSERVICESTATE_ID := 16739,
	OPCUAID_NONEXCLUSIVEDEVIATIONALARMTYPE_SHELVINGSTATE_CURRENTSTATE := 10444,
	OPCUAID_NONEXCLUSIVEDEVIATIONALARMTYPE_SHELVINGSTATE_CURRENTSTATE_ID := 10445,
	OPCUAID_NONEXCLUSIVEDEVIATIONALARMTYPE_SHELVINGSTATE_LASTTRANSITION_ID := 10450,
	OPCUAID_NONEXCLUSIVEDEVIATIONALARMTYPE_SHELVINGSTATE_UNSHELVETIME := 10454,
	OPCUAID_NONEXCLUSIVEDEVIATIONALARMTYPE_SHELVINGSTATE_TIMEDSHELVE_INPUTARGUMENTS := 10479,
	OPCUAID_NONEXCLUSIVEDEVIATIONALARMTYPE_SILENCESTATE_ID := 16748,
	OPCUAID_NONEXCLUSIVEDEVIATIONALARMTYPE_LATCHEDSTATE_ID := 18268,
	OPCUAID_NONEXCLUSIVEDEVIATIONALARMTYPE_HIGHHIGHSTATE_ID := 10483,
	OPCUAID_NONEXCLUSIVEDEVIATIONALARMTYPE_HIGHSTATE_ID := 10492,
	OPCUAID_NONEXCLUSIVEDEVIATIONALARMTYPE_LOWSTATE_ID := 10501,
	OPCUAID_NONEXCLUSIVEDEVIATIONALARMTYPE_LOWLOWSTATE_ID := 10510,
	OPCUAID_NONEXCLUSIVEDEVIATIONALARMTYPE_SETPOINTNODE := 10522,
	OPCUAID_NONEXCLUSIVEDEVIATIONALARMTYPE_BASESETPOINTNODE := 16776,
	OPCUAID_NONEXCLUSIVERATEOFCHANGEALARMTYPE_ENABLEDSTATE_ID := 10228,
	OPCUAID_NONEXCLUSIVERATEOFCHANGEALARMTYPE_QUALITY_SOURCETIMESTAMP := 10237,
	OPCUAID_NONEXCLUSIVERATEOFCHANGEALARMTYPE_LASTSEVERITY_SOURCETIMESTAMP := 10239,
	OPCUAID_NONEXCLUSIVERATEOFCHANGEALARMTYPE_COMMENT_SOURCETIMESTAMP := 10241,
	OPCUAID_NONEXCLUSIVERATEOFCHANGEALARMTYPE_ADDCOMMENT_INPUTARGUMENTS := 10246,
	OPCUAID_NONEXCLUSIVERATEOFCHANGEALARMTYPE_CONDITIONREFRESH_INPUTARGUMENTS := 10248,
	OPCUAID_NONEXCLUSIVERATEOFCHANGEALARMTYPE_CONDITIONREFRESH2_INPUTARGUMENTS := 13001,
	OPCUAID_NONEXCLUSIVERATEOFCHANGEALARMTYPE_ACKEDSTATE_ID := 10250,
	OPCUAID_NONEXCLUSIVERATEOFCHANGEALARMTYPE_CONFIRMEDSTATE_ID := 10259,
	OPCUAID_NONEXCLUSIVERATEOFCHANGEALARMTYPE_ACKNOWLEDGE_INPUTARGUMENTS := 10268,
	OPCUAID_NONEXCLUSIVERATEOFCHANGEALARMTYPE_CONFIRM_INPUTARGUMENTS := 10270,
	OPCUAID_NONEXCLUSIVERATEOFCHANGEALARMTYPE_ACTIVESTATE_ID := 10272,
	OPCUAID_NONEXCLUSIVERATEOFCHANGEALARMTYPE_SUPPRESSEDSTATE_ID := 10281,
	OPCUAID_NONEXCLUSIVERATEOFCHANGEALARMTYPE_OUTOFSERVICESTATE_ID := 16821,
	OPCUAID_NONEXCLUSIVERATEOFCHANGEALARMTYPE_SHELVINGSTATE_CURRENTSTATE := 10290,
	OPCUAID_NONEXCLUSIVERATEOFCHANGEALARMTYPE_SHELVINGSTATE_CURRENTSTATE_ID := 10291,
	OPCUAID_NONEXCLUSIVERATEOFCHANGEALARMTYPE_SHELVINGSTATE_LASTTRANSITION_ID := 10296,
	OPCUAID_NONEXCLUSIVERATEOFCHANGEALARMTYPE_SHELVINGSTATE_UNSHELVETIME := 10300,
	OPCUAID_NONEXCLUSIVERATEOFCHANGEALARMTYPE_SHELVINGSTATE_TIMEDSHELVE_INPUTARGUMENTS := 10325,
	OPCUAID_NONEXCLUSIVERATEOFCHANGEALARMTYPE_SILENCESTATE_ID := 16830,
	OPCUAID_NONEXCLUSIVERATEOFCHANGEALARMTYPE_LATCHEDSTATE_ID := 18278,
	OPCUAID_NONEXCLUSIVERATEOFCHANGEALARMTYPE_HIGHHIGHSTATE_ID := 10329,
	OPCUAID_NONEXCLUSIVERATEOFCHANGEALARMTYPE_HIGHSTATE_ID := 10338,
	OPCUAID_NONEXCLUSIVERATEOFCHANGEALARMTYPE_LOWSTATE_ID := 10347,
	OPCUAID_NONEXCLUSIVERATEOFCHANGEALARMTYPE_LOWLOWSTATE_ID := 10356,
	OPCUAID_NONEXCLUSIVERATEOFCHANGEALARMTYPE_ENGINEERINGUNITS := 16858,
	OPCUAID_EXCLUSIVEDEVIATIONALARMTYPE_ENABLEDSTATE_ID := 9778,
	OPCUAID_EXCLUSIVEDEVIATIONALARMTYPE_QUALITY_SOURCETIMESTAMP := 9787,
	OPCUAID_EXCLUSIVEDEVIATIONALARMTYPE_LASTSEVERITY_SOURCETIMESTAMP := 9789,
	OPCUAID_EXCLUSIVEDEVIATIONALARMTYPE_COMMENT_SOURCETIMESTAMP := 9791,
	OPCUAID_EXCLUSIVEDEVIATIONALARMTYPE_ADDCOMMENT_INPUTARGUMENTS := 9796,
	OPCUAID_EXCLUSIVEDEVIATIONALARMTYPE_CONDITIONREFRESH_INPUTARGUMENTS := 9798,
	OPCUAID_EXCLUSIVEDEVIATIONALARMTYPE_CONDITIONREFRESH2_INPUTARGUMENTS := 12999,
	OPCUAID_EXCLUSIVEDEVIATIONALARMTYPE_ACKEDSTATE_ID := 9800,
	OPCUAID_EXCLUSIVEDEVIATIONALARMTYPE_CONFIRMEDSTATE_ID := 9809,
	OPCUAID_EXCLUSIVEDEVIATIONALARMTYPE_ACKNOWLEDGE_INPUTARGUMENTS := 9818,
	OPCUAID_EXCLUSIVEDEVIATIONALARMTYPE_CONFIRM_INPUTARGUMENTS := 9820,
	OPCUAID_EXCLUSIVEDEVIATIONALARMTYPE_ACTIVESTATE_ID := 9822,
	OPCUAID_EXCLUSIVEDEVIATIONALARMTYPE_SUPPRESSEDSTATE_ID := 9831,
	OPCUAID_EXCLUSIVEDEVIATIONALARMTYPE_OUTOFSERVICESTATE_ID := 16780,
	OPCUAID_EXCLUSIVEDEVIATIONALARMTYPE_SHELVINGSTATE_CURRENTSTATE := 9840,
	OPCUAID_EXCLUSIVEDEVIATIONALARMTYPE_SHELVINGSTATE_CURRENTSTATE_ID := 9841,
	OPCUAID_EXCLUSIVEDEVIATIONALARMTYPE_SHELVINGSTATE_LASTTRANSITION_ID := 9846,
	OPCUAID_EXCLUSIVEDEVIATIONALARMTYPE_SHELVINGSTATE_UNSHELVETIME := 9850,
	OPCUAID_EXCLUSIVEDEVIATIONALARMTYPE_SHELVINGSTATE_TIMEDSHELVE_INPUTARGUMENTS := 9875,
	OPCUAID_EXCLUSIVEDEVIATIONALARMTYPE_SILENCESTATE_ID := 16789,
	OPCUAID_EXCLUSIVEDEVIATIONALARMTYPE_LATCHEDSTATE_ID := 18288,
	OPCUAID_EXCLUSIVEDEVIATIONALARMTYPE_LIMITSTATE_CURRENTSTATE := 9879,
	OPCUAID_EXCLUSIVEDEVIATIONALARMTYPE_LIMITSTATE_CURRENTSTATE_ID := 9880,
	OPCUAID_EXCLUSIVEDEVIATIONALARMTYPE_LIMITSTATE_LASTTRANSITION_ID := 9885,
	OPCUAID_EXCLUSIVEDEVIATIONALARMTYPE_SETPOINTNODE := 9905,
	OPCUAID_EXCLUSIVEDEVIATIONALARMTYPE_BASESETPOINTNODE := 16817,
	OPCUAID_EXCLUSIVERATEOFCHANGEALARMTYPE_ENABLEDSTATE_ID := 9637,
	OPCUAID_EXCLUSIVERATEOFCHANGEALARMTYPE_QUALITY_SOURCETIMESTAMP := 9646,
	OPCUAID_EXCLUSIVERATEOFCHANGEALARMTYPE_LASTSEVERITY_SOURCETIMESTAMP := 9648,
	OPCUAID_EXCLUSIVERATEOFCHANGEALARMTYPE_COMMENT_SOURCETIMESTAMP := 9650,
	OPCUAID_EXCLUSIVERATEOFCHANGEALARMTYPE_ADDCOMMENT_INPUTARGUMENTS := 9655,
	OPCUAID_EXCLUSIVERATEOFCHANGEALARMTYPE_CONDITIONREFRESH_INPUTARGUMENTS := 9657,
	OPCUAID_EXCLUSIVERATEOFCHANGEALARMTYPE_CONDITIONREFRESH2_INPUTARGUMENTS := 13003,
	OPCUAID_EXCLUSIVERATEOFCHANGEALARMTYPE_ACKEDSTATE_ID := 9659,
	OPCUAID_EXCLUSIVERATEOFCHANGEALARMTYPE_CONFIRMEDSTATE_ID := 9668,
	OPCUAID_EXCLUSIVERATEOFCHANGEALARMTYPE_ACKNOWLEDGE_INPUTARGUMENTS := 9677,
	OPCUAID_EXCLUSIVERATEOFCHANGEALARMTYPE_CONFIRM_INPUTARGUMENTS := 9679,
	OPCUAID_EXCLUSIVERATEOFCHANGEALARMTYPE_ACTIVESTATE_ID := 9681,
	OPCUAID_EXCLUSIVERATEOFCHANGEALARMTYPE_SUPPRESSEDSTATE_ID := 9690,
	OPCUAID_EXCLUSIVERATEOFCHANGEALARMTYPE_OUTOFSERVICESTATE_ID := 16862,
	OPCUAID_EXCLUSIVERATEOFCHANGEALARMTYPE_SHELVINGSTATE_CURRENTSTATE := 9699,
	OPCUAID_EXCLUSIVERATEOFCHANGEALARMTYPE_SHELVINGSTATE_CURRENTSTATE_ID := 9700,
	OPCUAID_EXCLUSIVERATEOFCHANGEALARMTYPE_SHELVINGSTATE_LASTTRANSITION_ID := 9705,
	OPCUAID_EXCLUSIVERATEOFCHANGEALARMTYPE_SHELVINGSTATE_UNSHELVETIME := 9709,
	OPCUAID_EXCLUSIVERATEOFCHANGEALARMTYPE_SHELVINGSTATE_TIMEDSHELVE_INPUTARGUMENTS := 9734,
	OPCUAID_EXCLUSIVERATEOFCHANGEALARMTYPE_SILENCESTATE_ID := 16871,
	OPCUAID_EXCLUSIVERATEOFCHANGEALARMTYPE_LATCHEDSTATE_ID := 18298,
	OPCUAID_EXCLUSIVERATEOFCHANGEALARMTYPE_LIMITSTATE_CURRENTSTATE := 9738,
	OPCUAID_EXCLUSIVERATEOFCHANGEALARMTYPE_LIMITSTATE_CURRENTSTATE_ID := 9739,
	OPCUAID_EXCLUSIVERATEOFCHANGEALARMTYPE_LIMITSTATE_LASTTRANSITION_ID := 9744,
	OPCUAID_EXCLUSIVERATEOFCHANGEALARMTYPE_ENGINEERINGUNITS := 16899,
	OPCUAID_DISCRETEALARMTYPE_ENABLEDSTATE_ID := 10537,
	OPCUAID_DISCRETEALARMTYPE_QUALITY_SOURCETIMESTAMP := 10546,
	OPCUAID_DISCRETEALARMTYPE_LASTSEVERITY_SOURCETIMESTAMP := 10548,
	OPCUAID_DISCRETEALARMTYPE_COMMENT_SOURCETIMESTAMP := 10550,
	OPCUAID_DISCRETEALARMTYPE_ADDCOMMENT_INPUTARGUMENTS := 10555,
	OPCUAID_DISCRETEALARMTYPE_CONDITIONREFRESH_INPUTARGUMENTS := 10557,
	OPCUAID_DISCRETEALARMTYPE_CONDITIONREFRESH2_INPUTARGUMENTS := 13005,
	OPCUAID_DISCRETEALARMTYPE_ACKEDSTATE_ID := 10559,
	OPCUAID_DISCRETEALARMTYPE_CONFIRMEDSTATE_ID := 10568,
	OPCUAID_DISCRETEALARMTYPE_ACKNOWLEDGE_INPUTARGUMENTS := 10577,
	OPCUAID_DISCRETEALARMTYPE_CONFIRM_INPUTARGUMENTS := 10579,
	OPCUAID_DISCRETEALARMTYPE_ACTIVESTATE_ID := 10581,
	OPCUAID_DISCRETEALARMTYPE_SUPPRESSEDSTATE_ID := 10590,
	OPCUAID_DISCRETEALARMTYPE_OUTOFSERVICESTATE_ID := 16903,
	OPCUAID_DISCRETEALARMTYPE_SHELVINGSTATE_CURRENTSTATE := 10599,
	OPCUAID_DISCRETEALARMTYPE_SHELVINGSTATE_CURRENTSTATE_ID := 10600,
	OPCUAID_DISCRETEALARMTYPE_SHELVINGSTATE_LASTTRANSITION_ID := 10605,
	OPCUAID_DISCRETEALARMTYPE_SHELVINGSTATE_UNSHELVETIME := 10609,
	OPCUAID_DISCRETEALARMTYPE_SHELVINGSTATE_TIMEDSHELVE_INPUTARGUMENTS := 10634,
	OPCUAID_DISCRETEALARMTYPE_SILENCESTATE_ID := 16912,
	OPCUAID_DISCRETEALARMTYPE_LATCHEDSTATE_ID := 18308,
	OPCUAID_OFFNORMALALARMTYPE_ENABLEDSTATE_ID := 10651,
	OPCUAID_OFFNORMALALARMTYPE_QUALITY_SOURCETIMESTAMP := 10660,
	OPCUAID_OFFNORMALALARMTYPE_LASTSEVERITY_SOURCETIMESTAMP := 10662,
	OPCUAID_OFFNORMALALARMTYPE_COMMENT_SOURCETIMESTAMP := 10664,
	OPCUAID_OFFNORMALALARMTYPE_ADDCOMMENT_INPUTARGUMENTS := 10669,
	OPCUAID_OFFNORMALALARMTYPE_CONDITIONREFRESH_INPUTARGUMENTS := 10671,
	OPCUAID_OFFNORMALALARMTYPE_CONDITIONREFRESH2_INPUTARGUMENTS := 13007,
	OPCUAID_OFFNORMALALARMTYPE_ACKEDSTATE_ID := 10673,
	OPCUAID_OFFNORMALALARMTYPE_CONFIRMEDSTATE_ID := 10682,
	OPCUAID_OFFNORMALALARMTYPE_ACKNOWLEDGE_INPUTARGUMENTS := 10691,
	OPCUAID_OFFNORMALALARMTYPE_CONFIRM_INPUTARGUMENTS := 10693,
	OPCUAID_OFFNORMALALARMTYPE_ACTIVESTATE_ID := 10695,
	OPCUAID_OFFNORMALALARMTYPE_SUPPRESSEDSTATE_ID := 10704,
	OPCUAID_OFFNORMALALARMTYPE_OUTOFSERVICESTATE_ID := 16939,
	OPCUAID_OFFNORMALALARMTYPE_SHELVINGSTATE_CURRENTSTATE := 10713,
	OPCUAID_OFFNORMALALARMTYPE_SHELVINGSTATE_CURRENTSTATE_ID := 10714,
	OPCUAID_OFFNORMALALARMTYPE_SHELVINGSTATE_LASTTRANSITION_ID := 10719,
	OPCUAID_OFFNORMALALARMTYPE_SHELVINGSTATE_UNSHELVETIME := 10723,
	OPCUAID_OFFNORMALALARMTYPE_SHELVINGSTATE_TIMEDSHELVE_INPUTARGUMENTS := 10748,
	OPCUAID_OFFNORMALALARMTYPE_SILENCESTATE_ID := 16948,
	OPCUAID_OFFNORMALALARMTYPE_LATCHEDSTATE_ID := 18318,
	OPCUAID_OFFNORMALALARMTYPE_NORMALSTATE := 11158,
	OPCUAID_SYSTEMOFFNORMALALARMTYPE_ENABLEDSTATE_ID := 11769,
	OPCUAID_SYSTEMOFFNORMALALARMTYPE_QUALITY_SOURCETIMESTAMP := 11778,
	OPCUAID_SYSTEMOFFNORMALALARMTYPE_LASTSEVERITY_SOURCETIMESTAMP := 11780,
	OPCUAID_SYSTEMOFFNORMALALARMTYPE_COMMENT_SOURCETIMESTAMP := 11782,
	OPCUAID_SYSTEMOFFNORMALALARMTYPE_ADDCOMMENT_INPUTARGUMENTS := 11787,
	OPCUAID_SYSTEMOFFNORMALALARMTYPE_CONDITIONREFRESH_INPUTARGUMENTS := 11789,
	OPCUAID_SYSTEMOFFNORMALALARMTYPE_CONDITIONREFRESH2_INPUTARGUMENTS := 13009,
	OPCUAID_SYSTEMOFFNORMALALARMTYPE_ACKEDSTATE_ID := 11791,
	OPCUAID_SYSTEMOFFNORMALALARMTYPE_CONFIRMEDSTATE_ID := 11800,
	OPCUAID_SYSTEMOFFNORMALALARMTYPE_ACKNOWLEDGE_INPUTARGUMENTS := 11809,
	OPCUAID_SYSTEMOFFNORMALALARMTYPE_CONFIRM_INPUTARGUMENTS := 11811,
	OPCUAID_SYSTEMOFFNORMALALARMTYPE_ACTIVESTATE_ID := 11813,
	OPCUAID_SYSTEMOFFNORMALALARMTYPE_SUPPRESSEDSTATE_ID := 11823,
	OPCUAID_SYSTEMOFFNORMALALARMTYPE_OUTOFSERVICESTATE_ID := 16975,
	OPCUAID_SYSTEMOFFNORMALALARMTYPE_SHELVINGSTATE_CURRENTSTATE := 11832,
	OPCUAID_SYSTEMOFFNORMALALARMTYPE_SHELVINGSTATE_CURRENTSTATE_ID := 11833,
	OPCUAID_SYSTEMOFFNORMALALARMTYPE_SHELVINGSTATE_LASTTRANSITION_ID := 11838,
	OPCUAID_SYSTEMOFFNORMALALARMTYPE_SHELVINGSTATE_UNSHELVETIME := 11843,
	OPCUAID_SYSTEMOFFNORMALALARMTYPE_SHELVINGSTATE_TIMEDSHELVE_INPUTARGUMENTS := 11847,
	OPCUAID_SYSTEMOFFNORMALALARMTYPE_SILENCESTATE_ID := 16984,
	OPCUAID_SYSTEMOFFNORMALALARMTYPE_LATCHEDSTATE_ID := 18328,
	OPCUAID_TRIPALARMTYPE_ENABLEDSTATE_ID := 10765,
	OPCUAID_TRIPALARMTYPE_QUALITY_SOURCETIMESTAMP := 10774,
	OPCUAID_TRIPALARMTYPE_LASTSEVERITY_SOURCETIMESTAMP := 10776,
	OPCUAID_TRIPALARMTYPE_COMMENT_SOURCETIMESTAMP := 10778,
	OPCUAID_TRIPALARMTYPE_ADDCOMMENT_INPUTARGUMENTS := 10783,
	OPCUAID_TRIPALARMTYPE_CONDITIONREFRESH_INPUTARGUMENTS := 10785,
	OPCUAID_TRIPALARMTYPE_CONDITIONREFRESH2_INPUTARGUMENTS := 13011,
	OPCUAID_TRIPALARMTYPE_ACKEDSTATE_ID := 10787,
	OPCUAID_TRIPALARMTYPE_CONFIRMEDSTATE_ID := 10796,
	OPCUAID_TRIPALARMTYPE_ACKNOWLEDGE_INPUTARGUMENTS := 10805,
	OPCUAID_TRIPALARMTYPE_CONFIRM_INPUTARGUMENTS := 10807,
	OPCUAID_TRIPALARMTYPE_ACTIVESTATE_ID := 10809,
	OPCUAID_TRIPALARMTYPE_SUPPRESSEDSTATE_ID := 10818,
	OPCUAID_TRIPALARMTYPE_OUTOFSERVICESTATE_ID := 17011,
	OPCUAID_TRIPALARMTYPE_SHELVINGSTATE_CURRENTSTATE := 10827,
	OPCUAID_TRIPALARMTYPE_SHELVINGSTATE_CURRENTSTATE_ID := 10828,
	OPCUAID_TRIPALARMTYPE_SHELVINGSTATE_LASTTRANSITION_ID := 10833,
	OPCUAID_TRIPALARMTYPE_SHELVINGSTATE_UNSHELVETIME := 10837,
	OPCUAID_TRIPALARMTYPE_SHELVINGSTATE_TIMEDSHELVE_INPUTARGUMENTS := 10862,
	OPCUAID_TRIPALARMTYPE_SILENCESTATE_ID := 17020,
	OPCUAID_TRIPALARMTYPE_LATCHEDSTATE_ID := 18338,
	OPCUAID_INSTRUMENTDIAGNOSTICALARMTYPE_ENABLEDSTATE_ID := 18365,
	OPCUAID_INSTRUMENTDIAGNOSTICALARMTYPE_QUALITY_SOURCETIMESTAMP := 18374,
	OPCUAID_INSTRUMENTDIAGNOSTICALARMTYPE_LASTSEVERITY_SOURCETIMESTAMP := 18376,
	OPCUAID_INSTRUMENTDIAGNOSTICALARMTYPE_COMMENT_SOURCETIMESTAMP := 18378,
	OPCUAID_INSTRUMENTDIAGNOSTICALARMTYPE_ADDCOMMENT_INPUTARGUMENTS := 18383,
	OPCUAID_INSTRUMENTDIAGNOSTICALARMTYPE_CONDITIONREFRESH_INPUTARGUMENTS := 18385,
	OPCUAID_INSTRUMENTDIAGNOSTICALARMTYPE_CONDITIONREFRESH2_INPUTARGUMENTS := 18387,
	OPCUAID_INSTRUMENTDIAGNOSTICALARMTYPE_ACKEDSTATE_ID := 18389,
	OPCUAID_INSTRUMENTDIAGNOSTICALARMTYPE_CONFIRMEDSTATE_ID := 18398,
	OPCUAID_INSTRUMENTDIAGNOSTICALARMTYPE_ACKNOWLEDGE_INPUTARGUMENTS := 18407,
	OPCUAID_INSTRUMENTDIAGNOSTICALARMTYPE_CONFIRM_INPUTARGUMENTS := 18409,
	OPCUAID_INSTRUMENTDIAGNOSTICALARMTYPE_ACTIVESTATE_ID := 18411,
	OPCUAID_INSTRUMENTDIAGNOSTICALARMTYPE_SUPPRESSEDSTATE_ID := 18421,
	OPCUAID_INSTRUMENTDIAGNOSTICALARMTYPE_OUTOFSERVICESTATE_ID := 18430,
	OPCUAID_INSTRUMENTDIAGNOSTICALARMTYPE_SHELVINGSTATE_CURRENTSTATE := 18439,
	OPCUAID_INSTRUMENTDIAGNOSTICALARMTYPE_SHELVINGSTATE_CURRENTSTATE_ID := 18440,
	OPCUAID_INSTRUMENTDIAGNOSTICALARMTYPE_SHELVINGSTATE_LASTTRANSITION_ID := 18445,
	OPCUAID_INSTRUMENTDIAGNOSTICALARMTYPE_SHELVINGSTATE_UNSHELVETIME := 18452,
	OPCUAID_INSTRUMENTDIAGNOSTICALARMTYPE_SHELVINGSTATE_TIMEDSHELVE_INPUTARGUMENTS := 18454,
	OPCUAID_INSTRUMENTDIAGNOSTICALARMTYPE_SILENCESTATE_ID := 18465,
	OPCUAID_INSTRUMENTDIAGNOSTICALARMTYPE_LATCHEDSTATE_ID := 18478,
	OPCUAID_SYSTEMDIAGNOSTICALARMTYPE_ENABLEDSTATE_ID := 18514,
	OPCUAID_SYSTEMDIAGNOSTICALARMTYPE_QUALITY_SOURCETIMESTAMP := 18523,
	OPCUAID_SYSTEMDIAGNOSTICALARMTYPE_LASTSEVERITY_SOURCETIMESTAMP := 18525,
	OPCUAID_SYSTEMDIAGNOSTICALARMTYPE_COMMENT_SOURCETIMESTAMP := 18527,
	OPCUAID_SYSTEMDIAGNOSTICALARMTYPE_ADDCOMMENT_INPUTARGUMENTS := 18532,
	OPCUAID_SYSTEMDIAGNOSTICALARMTYPE_CONDITIONREFRESH_INPUTARGUMENTS := 18534,
	OPCUAID_SYSTEMDIAGNOSTICALARMTYPE_CONDITIONREFRESH2_INPUTARGUMENTS := 18536,
	OPCUAID_SYSTEMDIAGNOSTICALARMTYPE_ACKEDSTATE_ID := 18538,
	OPCUAID_SYSTEMDIAGNOSTICALARMTYPE_CONFIRMEDSTATE_ID := 18547,
	OPCUAID_SYSTEMDIAGNOSTICALARMTYPE_ACKNOWLEDGE_INPUTARGUMENTS := 18556,
	OPCUAID_SYSTEMDIAGNOSTICALARMTYPE_CONFIRM_INPUTARGUMENTS := 18558,
	OPCUAID_SYSTEMDIAGNOSTICALARMTYPE_ACTIVESTATE_ID := 18560,
	OPCUAID_SYSTEMDIAGNOSTICALARMTYPE_SUPPRESSEDSTATE_ID := 18570,
	OPCUAID_SYSTEMDIAGNOSTICALARMTYPE_OUTOFSERVICESTATE_ID := 18579,
	OPCUAID_SYSTEMDIAGNOSTICALARMTYPE_SHELVINGSTATE_CURRENTSTATE := 18588,
	OPCUAID_SYSTEMDIAGNOSTICALARMTYPE_SHELVINGSTATE_CURRENTSTATE_ID := 18589,
	OPCUAID_SYSTEMDIAGNOSTICALARMTYPE_SHELVINGSTATE_LASTTRANSITION_ID := 18594,
	OPCUAID_SYSTEMDIAGNOSTICALARMTYPE_SHELVINGSTATE_UNSHELVETIME := 18601,
	OPCUAID_SYSTEMDIAGNOSTICALARMTYPE_SHELVINGSTATE_TIMEDSHELVE_INPUTARGUMENTS := 18603,
	OPCUAID_SYSTEMDIAGNOSTICALARMTYPE_SILENCESTATE_ID := 18614,
	OPCUAID_SYSTEMDIAGNOSTICALARMTYPE_LATCHEDSTATE_ID := 18627,
	OPCUAID_CERTIFICATEEXPIRATIONALARMTYPE_ENABLEDSTATE_ID := 13241,
	OPCUAID_CERTIFICATEEXPIRATIONALARMTYPE_QUALITY_SOURCETIMESTAMP := 13250,
	OPCUAID_CERTIFICATEEXPIRATIONALARMTYPE_LASTSEVERITY_SOURCETIMESTAMP := 13252,
	OPCUAID_CERTIFICATEEXPIRATIONALARMTYPE_COMMENT_SOURCETIMESTAMP := 13254,
	OPCUAID_CERTIFICATEEXPIRATIONALARMTYPE_ADDCOMMENT_INPUTARGUMENTS := 13259,
	OPCUAID_CERTIFICATEEXPIRATIONALARMTYPE_CONDITIONREFRESH_INPUTARGUMENTS := 13261,
	OPCUAID_CERTIFICATEEXPIRATIONALARMTYPE_CONDITIONREFRESH2_INPUTARGUMENTS := 13263,
	OPCUAID_CERTIFICATEEXPIRATIONALARMTYPE_ACKEDSTATE_ID := 13265,
	OPCUAID_CERTIFICATEEXPIRATIONALARMTYPE_CONFIRMEDSTATE_ID := 13274,
	OPCUAID_CERTIFICATEEXPIRATIONALARMTYPE_ACKNOWLEDGE_INPUTARGUMENTS := 13283,
	OPCUAID_CERTIFICATEEXPIRATIONALARMTYPE_CONFIRM_INPUTARGUMENTS := 13285,
	OPCUAID_CERTIFICATEEXPIRATIONALARMTYPE_ACTIVESTATE_ID := 13287,
	OPCUAID_CERTIFICATEEXPIRATIONALARMTYPE_SUPPRESSEDSTATE_ID := 13297,
	OPCUAID_CERTIFICATEEXPIRATIONALARMTYPE_OUTOFSERVICESTATE_ID := 17047,
	OPCUAID_CERTIFICATEEXPIRATIONALARMTYPE_SHELVINGSTATE_CURRENTSTATE := 13306,
	OPCUAID_CERTIFICATEEXPIRATIONALARMTYPE_SHELVINGSTATE_CURRENTSTATE_ID := 13307,
	OPCUAID_CERTIFICATEEXPIRATIONALARMTYPE_SHELVINGSTATE_LASTTRANSITION_ID := 13312,
	OPCUAID_CERTIFICATEEXPIRATIONALARMTYPE_SHELVINGSTATE_UNSHELVETIME := 13317,
	OPCUAID_CERTIFICATEEXPIRATIONALARMTYPE_SHELVINGSTATE_TIMEDSHELVE_INPUTARGUMENTS := 13321,
	OPCUAID_CERTIFICATEEXPIRATIONALARMTYPE_SILENCESTATE_ID := 17056,
	OPCUAID_CERTIFICATEEXPIRATIONALARMTYPE_LATCHEDSTATE_ID := 18646,
	OPCUAID_CERTIFICATEEXPIRATIONALARMTYPE_EXPIRATIONDATE := 13325,
	OPCUAID_CERTIFICATEEXPIRATIONALARMTYPE_EXPIRATIONLIMIT := 14900,
	OPCUAID_CERTIFICATEEXPIRATIONALARMTYPE_CERTIFICATETYPE := 13326,
	OPCUAID_CERTIFICATEEXPIRATIONALARMTYPE_CERTIFICATE := 13327,
	OPCUAID_DISCREPANCYALARMTYPE_ENABLEDSTATE_ID := 17098,
	OPCUAID_DISCREPANCYALARMTYPE_QUALITY_SOURCETIMESTAMP := 17107,
	OPCUAID_DISCREPANCYALARMTYPE_LASTSEVERITY_SOURCETIMESTAMP := 17109,
	OPCUAID_DISCREPANCYALARMTYPE_COMMENT_SOURCETIMESTAMP := 17111,
	OPCUAID_DISCREPANCYALARMTYPE_ADDCOMMENT_INPUTARGUMENTS := 17116,
	OPCUAID_DISCREPANCYALARMTYPE_CONDITIONREFRESH_INPUTARGUMENTS := 17118,
	OPCUAID_DISCREPANCYALARMTYPE_CONDITIONREFRESH2_INPUTARGUMENTS := 17120,
	OPCUAID_DISCREPANCYALARMTYPE_ACKEDSTATE_ID := 17122,
	OPCUAID_DISCREPANCYALARMTYPE_CONFIRMEDSTATE_ID := 17131,
	OPCUAID_DISCREPANCYALARMTYPE_ACKNOWLEDGE_INPUTARGUMENTS := 17140,
	OPCUAID_DISCREPANCYALARMTYPE_CONFIRM_INPUTARGUMENTS := 17142,
	OPCUAID_DISCREPANCYALARMTYPE_ACTIVESTATE_ID := 17144,
	OPCUAID_DISCREPANCYALARMTYPE_SUPPRESSEDSTATE_ID := 17154,
	OPCUAID_DISCREPANCYALARMTYPE_OUTOFSERVICESTATE_ID := 17163,
	OPCUAID_DISCREPANCYALARMTYPE_SHELVINGSTATE_CURRENTSTATE := 17181,
	OPCUAID_DISCREPANCYALARMTYPE_SHELVINGSTATE_CURRENTSTATE_ID := 17182,
	OPCUAID_DISCREPANCYALARMTYPE_SHELVINGSTATE_LASTTRANSITION_ID := 17187,
	OPCUAID_DISCREPANCYALARMTYPE_SHELVINGSTATE_UNSHELVETIME := 17192,
	OPCUAID_DISCREPANCYALARMTYPE_SHELVINGSTATE_TIMEDSHELVE_INPUTARGUMENTS := 17196,
	OPCUAID_DISCREPANCYALARMTYPE_SILENCESTATE_ID := 17172,
	OPCUAID_DISCREPANCYALARMTYPE_LATCHEDSTATE_ID := 18656,
	OPCUAID_DISCREPANCYALARMTYPE_TARGETVALUENODE := 17215,
	OPCUAID_DISCREPANCYALARMTYPE_EXPECTEDTIME := 17216,
	OPCUAID_DISCREPANCYALARMTYPE_TOLERANCE := 17217,
	OPCUAID_AUDITCONDITIONCOMMENTEVENTTYPE_CONDITIONEVENTID := 17222,
	OPCUAID_AUDITCONDITIONCOMMENTEVENTTYPE_COMMENT := 11851,
	OPCUAID_AUDITCONDITIONRESPONDEVENTTYPE_SELECTEDRESPONSE := 11852,
	OPCUAID_AUDITCONDITIONACKNOWLEDGEEVENTTYPE_CONDITIONEVENTID := 17223,
	OPCUAID_AUDITCONDITIONACKNOWLEDGEEVENTTYPE_COMMENT := 11853,
	OPCUAID_AUDITCONDITIONCONFIRMEVENTTYPE_CONDITIONEVENTID := 17224,
	OPCUAID_AUDITCONDITIONCONFIRMEVENTTYPE_COMMENT := 11854,
	OPCUAID_AUDITCONDITIONSHELVINGEVENTTYPE_SHELVINGTIME := 11855,
	OPCUAID_ALARMMETRICSTYPE_ALARMCOUNT := 17280,
	OPCUAID_ALARMMETRICSTYPE_STARTTIME := 17991,
	OPCUAID_ALARMMETRICSTYPE_MAXIMUMACTIVESTATE := 17281,
	OPCUAID_ALARMMETRICSTYPE_MAXIMUMUNACK := 17282,
	OPCUAID_ALARMMETRICSTYPE_CURRENTALARMRATE := 17284,
	OPCUAID_ALARMMETRICSTYPE_CURRENTALARMRATE_RATE := 17285,
	OPCUAID_ALARMMETRICSTYPE_MAXIMUMALARMRATE := 17286,
	OPCUAID_ALARMMETRICSTYPE_MAXIMUMALARMRATE_RATE := 17287,
	OPCUAID_ALARMMETRICSTYPE_MAXIMUMREALARMCOUNT := 17283,
	OPCUAID_ALARMMETRICSTYPE_AVERAGEALARMRATE := 17288,
	OPCUAID_ALARMMETRICSTYPE_AVERAGEALARMRATE_RATE := 17289,
	OPCUAID_ALARMRATEVARIABLETYPE_RATE := 17278,
	OPCUAID_PROGRAMSTATEMACHINETYPE_CURRENTSTATE := 3830,
	OPCUAID_PROGRAMSTATEMACHINETYPE_CURRENTSTATE_ID := 3831,
	OPCUAID_PROGRAMSTATEMACHINETYPE_CURRENTSTATE_NUMBER := 3833,
	OPCUAID_PROGRAMSTATEMACHINETYPE_LASTTRANSITION := 3835,
	OPCUAID_PROGRAMSTATEMACHINETYPE_LASTTRANSITION_ID := 3836,
	OPCUAID_PROGRAMSTATEMACHINETYPE_LASTTRANSITION_NUMBER := 3838,
	OPCUAID_PROGRAMSTATEMACHINETYPE_LASTTRANSITION_TRANSITIONTIME := 3839,
	OPCUAID_PROGRAMSTATEMACHINETYPE_CREATABLE := 2392,
	OPCUAID_PROGRAMSTATEMACHINETYPE_DELETABLE := 2393,
	OPCUAID_PROGRAMSTATEMACHINETYPE_AUTODELETE := 2394,
	OPCUAID_PROGRAMSTATEMACHINETYPE_RECYCLECOUNT := 2395,
	OPCUAID_PROGRAMSTATEMACHINETYPE_INSTANCECOUNT := 2396,
	OPCUAID_PROGRAMSTATEMACHINETYPE_MAXINSTANCECOUNT := 2397,
	OPCUAID_PROGRAMSTATEMACHINETYPE_MAXRECYCLECOUNT := 2398,
	OPCUAID_PROGRAMSTATEMACHINETYPE_PROGRAMDIAGNOSTICS := 2399,
	OPCUAID_PROGRAMSTATEMACHINETYPE_PROGRAMDIAGNOSTICS_CREATESESSIONID := 3840,
	OPCUAID_PROGRAMSTATEMACHINETYPE_PROGRAMDIAGNOSTICS_CREATECLIENTNAME := 3841,
	OPCUAID_PROGRAMSTATEMACHINETYPE_PROGRAMDIAGNOSTICS_INVOCATIONCREATIONTIME := 3842,
	OPCUAID_PROGRAMSTATEMACHINETYPE_PROGRAMDIAGNOSTICS_LASTTRANSITIONTIME := 3843,
	OPCUAID_PROGRAMSTATEMACHINETYPE_PROGRAMDIAGNOSTICS_LASTMETHODCALL := 3844,
	OPCUAID_PROGRAMSTATEMACHINETYPE_PROGRAMDIAGNOSTICS_LASTMETHODSESSIONID := 3845,
	OPCUAID_PROGRAMSTATEMACHINETYPE_PROGRAMDIAGNOSTICS_LASTMETHODINPUTARGUMENTS := 3846,
	OPCUAID_PROGRAMSTATEMACHINETYPE_PROGRAMDIAGNOSTICS_LASTMETHODOUTPUTARGUMENTS := 3847,
	OPCUAID_PROGRAMSTATEMACHINETYPE_PROGRAMDIAGNOSTICS_LASTMETHODINPUTVALUES := 15038,
	OPCUAID_PROGRAMSTATEMACHINETYPE_PROGRAMDIAGNOSTICS_LASTMETHODOUTPUTVALUES := 15040,
	OPCUAID_PROGRAMSTATEMACHINETYPE_PROGRAMDIAGNOSTICS_LASTMETHODCALLTIME := 3848,
	OPCUAID_PROGRAMSTATEMACHINETYPE_PROGRAMDIAGNOSTICS_LASTMETHODRETURNSTATUS := 3849,
	OPCUAID_PROGRAMSTATEMACHINETYPE_HALTED_STATENUMBER := 2407,
	OPCUAID_PROGRAMSTATEMACHINETYPE_READY_STATENUMBER := 2401,
	OPCUAID_PROGRAMSTATEMACHINETYPE_RUNNING_STATENUMBER := 2403,
	OPCUAID_PROGRAMSTATEMACHINETYPE_SUSPENDED_STATENUMBER := 2405,
	OPCUAID_PROGRAMSTATEMACHINETYPE_HALTEDTOREADY_TRANSITIONNUMBER := 2409,
	OPCUAID_PROGRAMSTATEMACHINETYPE_READYTORUNNING_TRANSITIONNUMBER := 2411,
	OPCUAID_PROGRAMSTATEMACHINETYPE_RUNNINGTOHALTED_TRANSITIONNUMBER := 2413,
	OPCUAID_PROGRAMSTATEMACHINETYPE_RUNNINGTOREADY_TRANSITIONNUMBER := 2415,
	OPCUAID_PROGRAMSTATEMACHINETYPE_RUNNINGTOSUSPENDED_TRANSITIONNUMBER := 2417,
	OPCUAID_PROGRAMSTATEMACHINETYPE_SUSPENDEDTORUNNING_TRANSITIONNUMBER := 2419,
	OPCUAID_PROGRAMSTATEMACHINETYPE_SUSPENDEDTOHALTED_TRANSITIONNUMBER := 2421,
	OPCUAID_PROGRAMSTATEMACHINETYPE_SUSPENDEDTOREADY_TRANSITIONNUMBER := 2423,
	OPCUAID_PROGRAMSTATEMACHINETYPE_READYTOHALTED_TRANSITIONNUMBER := 2425,
	OPCUAID_PROGRAMTRANSITIONEVENTTYPE_TRANSITION_ID := 3802,
	OPCUAID_PROGRAMTRANSITIONEVENTTYPE_FROMSTATE_ID := 3792,
	OPCUAID_PROGRAMTRANSITIONEVENTTYPE_TOSTATE_ID := 3797,
	OPCUAID_PROGRAMTRANSITIONEVENTTYPE_INTERMEDIATERESULT := 2379,
	OPCUAID_AUDITPROGRAMTRANSITIONEVENTTYPE_TRANSITIONNUMBER := 11875,
	OPCUAID_PROGRAMTRANSITIONAUDITEVENTTYPE_TRANSITION := 3825,
	OPCUAID_PROGRAMTRANSITIONAUDITEVENTTYPE_TRANSITION_ID := 3826,
	OPCUAID_PROGRAMDIAGNOSTICTYPE_CREATESESSIONID := 2381,
	OPCUAID_PROGRAMDIAGNOSTICTYPE_CREATECLIENTNAME := 2382,
	OPCUAID_PROGRAMDIAGNOSTICTYPE_INVOCATIONCREATIONTIME := 2383,
	OPCUAID_PROGRAMDIAGNOSTICTYPE_LASTTRANSITIONTIME := 2384,
	OPCUAID_PROGRAMDIAGNOSTICTYPE_LASTMETHODCALL := 2385,
	OPCUAID_PROGRAMDIAGNOSTICTYPE_LASTMETHODSESSIONID := 2386,
	OPCUAID_PROGRAMDIAGNOSTICTYPE_LASTMETHODINPUTARGUMENTS := 2387,
	OPCUAID_PROGRAMDIAGNOSTICTYPE_LASTMETHODOUTPUTARGUMENTS := 2388,
	OPCUAID_PROGRAMDIAGNOSTICTYPE_LASTMETHODCALLTIME := 2389,
	OPCUAID_PROGRAMDIAGNOSTICTYPE_LASTMETHODRETURNSTATUS := 2390,
	OPCUAID_PROGRAMDIAGNOSTIC2TYPE_CREATESESSIONID := 15384,
	OPCUAID_PROGRAMDIAGNOSTIC2TYPE_CREATECLIENTNAME := 15385,
	OPCUAID_PROGRAMDIAGNOSTIC2TYPE_INVOCATIONCREATIONTIME := 15386,
	OPCUAID_PROGRAMDIAGNOSTIC2TYPE_LASTTRANSITIONTIME := 15387,
	OPCUAID_PROGRAMDIAGNOSTIC2TYPE_LASTMETHODCALL := 15388,
	OPCUAID_PROGRAMDIAGNOSTIC2TYPE_LASTMETHODSESSIONID := 15389,
	OPCUAID_PROGRAMDIAGNOSTIC2TYPE_LASTMETHODINPUTARGUMENTS := 15390,
	OPCUAID_PROGRAMDIAGNOSTIC2TYPE_LASTMETHODOUTPUTARGUMENTS := 15391,
	OPCUAID_PROGRAMDIAGNOSTIC2TYPE_LASTMETHODINPUTVALUES := 15392,
	OPCUAID_PROGRAMDIAGNOSTIC2TYPE_LASTMETHODOUTPUTVALUES := 15393,
	OPCUAID_PROGRAMDIAGNOSTIC2TYPE_LASTMETHODCALLTIME := 15394,
	OPCUAID_PROGRAMDIAGNOSTIC2TYPE_LASTMETHODRETURNSTATUS := 15395,
	OPCUAID_ANNOTATIONS := 11214,
	OPCUAID_HISTORICALDATACONFIGURATIONTYPE_AGGREGATECONFIGURATION_TREATUNCERTAINASBAD := 11168,
	OPCUAID_HISTORICALDATACONFIGURATIONTYPE_AGGREGATECONFIGURATION_PERCENTDATABAD := 11169,
	OPCUAID_HISTORICALDATACONFIGURATIONTYPE_AGGREGATECONFIGURATION_PERCENTDATAGOOD := 11170,
	OPCUAID_HISTORICALDATACONFIGURATIONTYPE_AGGREGATECONFIGURATION_USESLOPEDEXTRAPOLATION := 11171,
	OPCUAID_HISTORICALDATACONFIGURATIONTYPE_STEPPED := 2323,
	OPCUAID_HISTORICALDATACONFIGURATIONTYPE_DEFINITION := 2324,
	OPCUAID_HISTORICALDATACONFIGURATIONTYPE_MAXTIMEINTERVAL := 2325,
	OPCUAID_HISTORICALDATACONFIGURATIONTYPE_MINTIMEINTERVAL := 2326,
	OPCUAID_HISTORICALDATACONFIGURATIONTYPE_EXCEPTIONDEVIATION := 2327,
	OPCUAID_HISTORICALDATACONFIGURATIONTYPE_EXCEPTIONDEVIATIONFORMAT := 2328,
	OPCUAID_HISTORICALDATACONFIGURATIONTYPE_STARTOFARCHIVE := 11499,
	OPCUAID_HISTORICALDATACONFIGURATIONTYPE_STARTOFONLINEARCHIVE := 11500,
	OPCUAID_HACONFIGURATION_AGGREGATECONFIGURATION_TREATUNCERTAINASBAD := 11204,
	OPCUAID_HACONFIGURATION_AGGREGATECONFIGURATION_PERCENTDATABAD := 11205,
	OPCUAID_HACONFIGURATION_AGGREGATECONFIGURATION_PERCENTDATAGOOD := 11206,
	OPCUAID_HACONFIGURATION_AGGREGATECONFIGURATION_USESLOPEDEXTRAPOLATION := 11207,
	OPCUAID_HACONFIGURATION_STEPPED := 11208,
	OPCUAID_HISTORICALEVENTFILTER := 11215,
	OPCUAID_HISTORYSERVERCAPABILITIESTYPE_ACCESSHISTORYDATACAPABILITY := 2331,
	OPCUAID_HISTORYSERVERCAPABILITIESTYPE_ACCESSHISTORYEVENTSCAPABILITY := 2332,
	OPCUAID_HISTORYSERVERCAPABILITIESTYPE_MAXRETURNDATAVALUES := 11268,
	OPCUAID_HISTORYSERVERCAPABILITIESTYPE_MAXRETURNEVENTVALUES := 11269,
	OPCUAID_HISTORYSERVERCAPABILITIESTYPE_INSERTDATACAPABILITY := 2334,
	OPCUAID_HISTORYSERVERCAPABILITIESTYPE_REPLACEDATACAPABILITY := 2335,
	OPCUAID_HISTORYSERVERCAPABILITIESTYPE_UPDATEDATACAPABILITY := 2336,
	OPCUAID_HISTORYSERVERCAPABILITIESTYPE_DELETERAWCAPABILITY := 2337,
	OPCUAID_HISTORYSERVERCAPABILITIESTYPE_DELETEATTIMECAPABILITY := 2338,
	OPCUAID_HISTORYSERVERCAPABILITIESTYPE_INSERTEVENTCAPABILITY := 11278,
	OPCUAID_HISTORYSERVERCAPABILITIESTYPE_REPLACEEVENTCAPABILITY := 11279,
	OPCUAID_HISTORYSERVERCAPABILITIESTYPE_UPDATEEVENTCAPABILITY := 11280,
	OPCUAID_HISTORYSERVERCAPABILITIESTYPE_DELETEEVENTCAPABILITY := 11501,
	OPCUAID_HISTORYSERVERCAPABILITIESTYPE_INSERTANNOTATIONCAPABILITY := 11270,
	OPCUAID_AUDITHISTORYEVENTUPDATEEVENTTYPE_UPDATEDNODE := 3025,
	OPCUAID_AUDITHISTORYEVENTUPDATEEVENTTYPE_PERFORMINSERTREPLACE := 3028,
	OPCUAID_AUDITHISTORYEVENTUPDATEEVENTTYPE_FILTER := 3003,
	OPCUAID_AUDITHISTORYEVENTUPDATEEVENTTYPE_NEWVALUES := 3029,
	OPCUAID_AUDITHISTORYEVENTUPDATEEVENTTYPE_OLDVALUES := 3030,
	OPCUAID_AUDITHISTORYVALUEUPDATEEVENTTYPE_UPDATEDNODE := 3026,
	OPCUAID_AUDITHISTORYVALUEUPDATEEVENTTYPE_PERFORMINSERTREPLACE := 3031,
	OPCUAID_AUDITHISTORYVALUEUPDATEEVENTTYPE_NEWVALUES := 3032,
	OPCUAID_AUDITHISTORYVALUEUPDATEEVENTTYPE_OLDVALUES := 3033,
	OPCUAID_AUDITHISTORYDELETEEVENTTYPE_UPDATEDNODE := 3027,
	OPCUAID_AUDITHISTORYRAWMODIFYDELETEEVENTTYPE_ISDELETEMODIFIED := 3015,
	OPCUAID_AUDITHISTORYRAWMODIFYDELETEEVENTTYPE_STARTTIME := 3016,
	OPCUAID_AUDITHISTORYRAWMODIFYDELETEEVENTTYPE_ENDTIME := 3017,
	OPCUAID_AUDITHISTORYRAWMODIFYDELETEEVENTTYPE_OLDVALUES := 3034,
	OPCUAID_AUDITHISTORYATTIMEDELETEEVENTTYPE_REQTIMES := 3020,
	OPCUAID_AUDITHISTORYATTIMEDELETEEVENTTYPE_OLDVALUES := 3021,
	OPCUAID_AUDITHISTORYEVENTDELETEEVENTTYPE_EVENTIDS := 3023,
	OPCUAID_AUDITHISTORYEVENTDELETEEVENTTYPE_OLDVALUES := 3024,
	OPCUAID_TRUSTLISTTYPE_OPEN_INPUTARGUMENTS := 12528,
	OPCUAID_TRUSTLISTTYPE_OPEN_OUTPUTARGUMENTS := 12529,
	OPCUAID_TRUSTLISTTYPE_CLOSE_INPUTARGUMENTS := 12531,
	OPCUAID_TRUSTLISTTYPE_READ_INPUTARGUMENTS := 12533,
	OPCUAID_TRUSTLISTTYPE_READ_OUTPUTARGUMENTS := 12534,
	OPCUAID_TRUSTLISTTYPE_WRITE_INPUTARGUMENTS := 12536,
	OPCUAID_TRUSTLISTTYPE_GETPOSITION_INPUTARGUMENTS := 12538,
	OPCUAID_TRUSTLISTTYPE_GETPOSITION_OUTPUTARGUMENTS := 12539,
	OPCUAID_TRUSTLISTTYPE_SETPOSITION_INPUTARGUMENTS := 12541,
	OPCUAID_TRUSTLISTTYPE_LASTUPDATETIME := 12542,
	OPCUAID_TRUSTLISTTYPE_OPENWITHMASKS_INPUTARGUMENTS := 12544,
	OPCUAID_TRUSTLISTTYPE_OPENWITHMASKS_OUTPUTARGUMENTS := 12545,
	OPCUAID_TRUSTLISTTYPE_CLOSEANDUPDATE_INPUTARGUMENTS := 12705,
	OPCUAID_TRUSTLISTTYPE_CLOSEANDUPDATE_OUTPUTARGUMENTS := 12547,
	OPCUAID_TRUSTLISTTYPE_ADDCERTIFICATE_INPUTARGUMENTS := 12549,
	OPCUAID_TRUSTLISTTYPE_REMOVECERTIFICATE_INPUTARGUMENTS := 12551,
	OPCUAID_TRUSTLISTMASKS_ENUMVALUES := 12553,
	OPCUAID_CERTIFICATEGROUPTYPE_TRUSTLIST_SIZE := 13600,
	OPCUAID_CERTIFICATEGROUPTYPE_TRUSTLIST_WRITABLE := 13601,
	OPCUAID_CERTIFICATEGROUPTYPE_TRUSTLIST_USERWRITABLE := 13602,
	OPCUAID_CERTIFICATEGROUPTYPE_TRUSTLIST_OPENCOUNT := 13603,
	OPCUAID_CERTIFICATEGROUPTYPE_TRUSTLIST_OPEN_INPUTARGUMENTS := 13606,
	OPCUAID_CERTIFICATEGROUPTYPE_TRUSTLIST_OPEN_OUTPUTARGUMENTS := 13607,
	OPCUAID_CERTIFICATEGROUPTYPE_TRUSTLIST_CLOSE_INPUTARGUMENTS := 13609,
	OPCUAID_CERTIFICATEGROUPTYPE_TRUSTLIST_READ_INPUTARGUMENTS := 13611,
	OPCUAID_CERTIFICATEGROUPTYPE_TRUSTLIST_READ_OUTPUTARGUMENTS := 13612,
	OPCUAID_CERTIFICATEGROUPTYPE_TRUSTLIST_WRITE_INPUTARGUMENTS := 13614,
	OPCUAID_CERTIFICATEGROUPTYPE_TRUSTLIST_GETPOSITION_INPUTARGUMENTS := 13616,
	OPCUAID_CERTIFICATEGROUPTYPE_TRUSTLIST_GETPOSITION_OUTPUTARGUMENTS := 13617,
	OPCUAID_CERTIFICATEGROUPTYPE_TRUSTLIST_SETPOSITION_INPUTARGUMENTS := 13619,
	OPCUAID_CERTIFICATEGROUPTYPE_TRUSTLIST_LASTUPDATETIME := 13620,
	OPCUAID_CERTIFICATEGROUPTYPE_TRUSTLIST_OPENWITHMASKS_INPUTARGUMENTS := 13622,
	OPCUAID_CERTIFICATEGROUPTYPE_TRUSTLIST_OPENWITHMASKS_OUTPUTARGUMENTS := 13623,
	OPCUAID_CERTIFICATEGROUPTYPE_TRUSTLIST_CLOSEANDUPDATE_INPUTARGUMENTS := 13625,
	OPCUAID_CERTIFICATEGROUPTYPE_TRUSTLIST_CLOSEANDUPDATE_OUTPUTARGUMENTS := 13626,
	OPCUAID_CERTIFICATEGROUPTYPE_TRUSTLIST_ADDCERTIFICATE_INPUTARGUMENTS := 13628,
	OPCUAID_CERTIFICATEGROUPTYPE_TRUSTLIST_REMOVECERTIFICATE_INPUTARGUMENTS := 13630,
	OPCUAID_CERTIFICATEGROUPTYPE_CERTIFICATETYPES := 13631,
	OPCUAID_CERTIFICATEGROUPFOLDERTYPE_DEFAULTAPPLICATIONGROUP_TRUSTLIST_SIZE := 13816,
	OPCUAID_CERTIFICATEGROUPFOLDERTYPE_DEFAULTAPPLICATIONGROUP_TRUSTLIST_WRITABLE := 13817,
	OPCUAID_CERTIFICATEGROUPFOLDERTYPE_DEFAULTAPPLICATIONGROUP_TRUSTLIST_USERWRITABLE := 13818,
	OPCUAID_CERTIFICATEGROUPFOLDERTYPE_DEFAULTAPPLICATIONGROUP_TRUSTLIST_OPENCOUNT := 13819,
	OPCUAID_CERTIFICATEGROUPFOLDERTYPE_DEFAULTAPPLICATIONGROUP_TRUSTLIST_OPEN_INPUTARGUMENTS := 13822,
	OPCUAID_CERTIFICATEGROUPFOLDERTYPE_DEFAULTAPPLICATIONGROUP_TRUSTLIST_OPEN_OUTPUTARGUMENTS := 13823,
	OPCUAID_CERTIFICATEGROUPFOLDERTYPE_DEFAULTAPPLICATIONGROUP_TRUSTLIST_CLOSE_INPUTARGUMENTS := 13825,
	OPCUAID_CERTIFICATEGROUPFOLDERTYPE_DEFAULTAPPLICATIONGROUP_TRUSTLIST_READ_INPUTARGUMENTS := 13827,
	OPCUAID_CERTIFICATEGROUPFOLDERTYPE_DEFAULTAPPLICATIONGROUP_TRUSTLIST_READ_OUTPUTARGUMENTS := 13828,
	OPCUAID_CERTIFICATEGROUPFOLDERTYPE_DEFAULTAPPLICATIONGROUP_TRUSTLIST_WRITE_INPUTARGUMENTS := 13830,
	OPCUAID_CERTIFICATEGROUPFOLDERTYPE_DEFAULTAPPLICATIONGROUP_TRUSTLIST_GETPOSITION_INPUTARGUMENTS := 13832,
	OPCUAID_CERTIFICATEGROUPFOLDERTYPE_DEFAULTAPPLICATIONGROUP_TRUSTLIST_GETPOSITION_OUTPUTARGUMENTS := 13833,
	OPCUAID_CERTIFICATEGROUPFOLDERTYPE_DEFAULTAPPLICATIONGROUP_TRUSTLIST_SETPOSITION_INPUTARGUMENTS := 13835,
	OPCUAID_CERTIFICATEGROUPFOLDERTYPE_DEFAULTAPPLICATIONGROUP_TRUSTLIST_LASTUPDATETIME := 13836,
	OPCUAID_CERTIFICATEGROUPFOLDERTYPE_DEFAULTAPPLICATIONGROUP_TRUSTLIST_OPENWITHMASKS_INPUTARGUMENTS := 13838,
	OPCUAID_CERTIFICATEGROUPFOLDERTYPE_DEFAULTAPPLICATIONGROUP_TRUSTLIST_OPENWITHMASKS_OUTPUTARGUMENTS := 13839,
	OPCUAID_CERTIFICATEGROUPFOLDERTYPE_DEFAULTAPPLICATIONGROUP_TRUSTLIST_CLOSEANDUPDATE_INPUTARGUMENTS := 13841,
	OPCUAID_CERTIFICATEGROUPFOLDERTYPE_DEFAULTAPPLICATIONGROUP_TRUSTLIST_CLOSEANDUPDATE_OUTPUTARGUMENTS := 13842,
	OPCUAID_CERTIFICATEGROUPFOLDERTYPE_DEFAULTAPPLICATIONGROUP_TRUSTLIST_ADDCERTIFICATE_INPUTARGUMENTS := 13844,
	OPCUAID_CERTIFICATEGROUPFOLDERTYPE_DEFAULTAPPLICATIONGROUP_TRUSTLIST_REMOVECERTIFICATE_INPUTARGUMENTS := 13846,
	OPCUAID_CERTIFICATEGROUPFOLDERTYPE_DEFAULTAPPLICATIONGROUP_CERTIFICATETYPES := 13847,
	OPCUAID_CERTIFICATEGROUPFOLDERTYPE_DEFAULTHTTPSGROUP_TRUSTLIST_SIZE := 13850,
	OPCUAID_CERTIFICATEGROUPFOLDERTYPE_DEFAULTHTTPSGROUP_TRUSTLIST_WRITABLE := 13851,
	OPCUAID_CERTIFICATEGROUPFOLDERTYPE_DEFAULTHTTPSGROUP_TRUSTLIST_USERWRITABLE := 13852,
	OPCUAID_CERTIFICATEGROUPFOLDERTYPE_DEFAULTHTTPSGROUP_TRUSTLIST_OPENCOUNT := 13853,
	OPCUAID_CERTIFICATEGROUPFOLDERTYPE_DEFAULTHTTPSGROUP_TRUSTLIST_OPEN_INPUTARGUMENTS := 13856,
	OPCUAID_CERTIFICATEGROUPFOLDERTYPE_DEFAULTHTTPSGROUP_TRUSTLIST_OPEN_OUTPUTARGUMENTS := 13857,
	OPCUAID_CERTIFICATEGROUPFOLDERTYPE_DEFAULTHTTPSGROUP_TRUSTLIST_CLOSE_INPUTARGUMENTS := 13859,
	OPCUAID_CERTIFICATEGROUPFOLDERTYPE_DEFAULTHTTPSGROUP_TRUSTLIST_READ_INPUTARGUMENTS := 13861,
	OPCUAID_CERTIFICATEGROUPFOLDERTYPE_DEFAULTHTTPSGROUP_TRUSTLIST_READ_OUTPUTARGUMENTS := 13862,
	OPCUAID_CERTIFICATEGROUPFOLDERTYPE_DEFAULTHTTPSGROUP_TRUSTLIST_WRITE_INPUTARGUMENTS := 13864,
	OPCUAID_CERTIFICATEGROUPFOLDERTYPE_DEFAULTHTTPSGROUP_TRUSTLIST_GETPOSITION_INPUTARGUMENTS := 13866,
	OPCUAID_CERTIFICATEGROUPFOLDERTYPE_DEFAULTHTTPSGROUP_TRUSTLIST_GETPOSITION_OUTPUTARGUMENTS := 13867,
	OPCUAID_CERTIFICATEGROUPFOLDERTYPE_DEFAULTHTTPSGROUP_TRUSTLIST_SETPOSITION_INPUTARGUMENTS := 13869,
	OPCUAID_CERTIFICATEGROUPFOLDERTYPE_DEFAULTHTTPSGROUP_TRUSTLIST_LASTUPDATETIME := 13870,
	OPCUAID_CERTIFICATEGROUPFOLDERTYPE_DEFAULTHTTPSGROUP_TRUSTLIST_OPENWITHMASKS_INPUTARGUMENTS := 13872,
	OPCUAID_CERTIFICATEGROUPFOLDERTYPE_DEFAULTHTTPSGROUP_TRUSTLIST_OPENWITHMASKS_OUTPUTARGUMENTS := 13873,
	OPCUAID_CERTIFICATEGROUPFOLDERTYPE_DEFAULTHTTPSGROUP_TRUSTLIST_CLOSEANDUPDATE_INPUTARGUMENTS := 13875,
	OPCUAID_CERTIFICATEGROUPFOLDERTYPE_DEFAULTHTTPSGROUP_TRUSTLIST_CLOSEANDUPDATE_OUTPUTARGUMENTS := 13876,
	OPCUAID_CERTIFICATEGROUPFOLDERTYPE_DEFAULTHTTPSGROUP_TRUSTLIST_ADDCERTIFICATE_INPUTARGUMENTS := 13878,
	OPCUAID_CERTIFICATEGROUPFOLDERTYPE_DEFAULTHTTPSGROUP_TRUSTLIST_REMOVECERTIFICATE_INPUTARGUMENTS := 13880,
	OPCUAID_CERTIFICATEGROUPFOLDERTYPE_DEFAULTHTTPSGROUP_CERTIFICATETYPES := 13881,
	OPCUAID_CERTIFICATEGROUPFOLDERTYPE_DEFAULTUSERTOKENGROUP_TRUSTLIST_SIZE := 13884,
	OPCUAID_CERTIFICATEGROUPFOLDERTYPE_DEFAULTUSERTOKENGROUP_TRUSTLIST_WRITABLE := 13885,
	OPCUAID_CERTIFICATEGROUPFOLDERTYPE_DEFAULTUSERTOKENGROUP_TRUSTLIST_USERWRITABLE := 13886,
	OPCUAID_CERTIFICATEGROUPFOLDERTYPE_DEFAULTUSERTOKENGROUP_TRUSTLIST_OPENCOUNT := 13887,
	OPCUAID_CERTIFICATEGROUPFOLDERTYPE_DEFAULTUSERTOKENGROUP_TRUSTLIST_OPEN_INPUTARGUMENTS := 13890,
	OPCUAID_CERTIFICATEGROUPFOLDERTYPE_DEFAULTUSERTOKENGROUP_TRUSTLIST_OPEN_OUTPUTARGUMENTS := 13891,
	OPCUAID_CERTIFICATEGROUPFOLDERTYPE_DEFAULTUSERTOKENGROUP_TRUSTLIST_CLOSE_INPUTARGUMENTS := 13893,
	OPCUAID_CERTIFICATEGROUPFOLDERTYPE_DEFAULTUSERTOKENGROUP_TRUSTLIST_READ_INPUTARGUMENTS := 13895,
	OPCUAID_CERTIFICATEGROUPFOLDERTYPE_DEFAULTUSERTOKENGROUP_TRUSTLIST_READ_OUTPUTARGUMENTS := 13896,
	OPCUAID_CERTIFICATEGROUPFOLDERTYPE_DEFAULTUSERTOKENGROUP_TRUSTLIST_WRITE_INPUTARGUMENTS := 13898,
	OPCUAID_CERTIFICATEGROUPFOLDERTYPE_DEFAULTUSERTOKENGROUP_TRUSTLIST_GETPOSITION_INPUTARGUMENTS := 13900,
	OPCUAID_CERTIFICATEGROUPFOLDERTYPE_DEFAULTUSERTOKENGROUP_TRUSTLIST_GETPOSITION_OUTPUTARGUMENTS := 13901,
	OPCUAID_CERTIFICATEGROUPFOLDERTYPE_DEFAULTUSERTOKENGROUP_TRUSTLIST_SETPOSITION_INPUTARGUMENTS := 13903,
	OPCUAID_CERTIFICATEGROUPFOLDERTYPE_DEFAULTUSERTOKENGROUP_TRUSTLIST_LASTUPDATETIME := 13904,
	OPCUAID_CERTIFICATEGROUPFOLDERTYPE_DEFAULTUSERTOKENGROUP_TRUSTLIST_OPENWITHMASKS_INPUTARGUMENTS := 13906,
	OPCUAID_CERTIFICATEGROUPFOLDERTYPE_DEFAULTUSERTOKENGROUP_TRUSTLIST_OPENWITHMASKS_OUTPUTARGUMENTS := 13907,
	OPCUAID_CERTIFICATEGROUPFOLDERTYPE_DEFAULTUSERTOKENGROUP_TRUSTLIST_CLOSEANDUPDATE_INPUTARGUMENTS := 13909,
	OPCUAID_CERTIFICATEGROUPFOLDERTYPE_DEFAULTUSERTOKENGROUP_TRUSTLIST_CLOSEANDUPDATE_OUTPUTARGUMENTS := 13910,
	OPCUAID_CERTIFICATEGROUPFOLDERTYPE_DEFAULTUSERTOKENGROUP_TRUSTLIST_ADDCERTIFICATE_INPUTARGUMENTS := 13912,
	OPCUAID_CERTIFICATEGROUPFOLDERTYPE_DEFAULTUSERTOKENGROUP_TRUSTLIST_REMOVECERTIFICATE_INPUTARGUMENTS := 13914,
	OPCUAID_CERTIFICATEGROUPFOLDERTYPE_DEFAULTUSERTOKENGROUP_CERTIFICATETYPES := 13915,
	OPCUAID_CERTIFICATEGROUPFOLDERTYPE_ADDITIONALGROUP_PLACEHOLDER_TRUSTLIST_SIZE := 13918,
	OPCUAID_CERTIFICATEGROUPFOLDERTYPE_ADDITIONALGROUP_PLACEHOLDER_TRUSTLIST_WRITABLE := 13919,
	OPCUAID_CERTIFICATEGROUPFOLDERTYPE_ADDITIONALGROUP_PLACEHOLDER_TRUSTLIST_USERWRITABLE := 13920,
	OPCUAID_CERTIFICATEGROUPFOLDERTYPE_ADDITIONALGROUP_PLACEHOLDER_TRUSTLIST_OPENCOUNT := 13921,
	OPCUAID_CERTIFICATEGROUPFOLDERTYPE_ADDITIONALGROUP_PLACEHOLDER_TRUSTLIST_OPEN_INPUTARGUMENTS := 13924,
	OPCUAID_CERTIFICATEGROUPFOLDERTYPE_ADDITIONALGROUP_PLACEHOLDER_TRUSTLIST_OPEN_OUTPUTARGUMENTS := 13925,
	OPCUAID_CERTIFICATEGROUPFOLDERTYPE_ADDITIONALGROUP_PLACEHOLDER_TRUSTLIST_CLOSE_INPUTARGUMENTS := 13927,
	OPCUAID_CERTIFICATEGROUPFOLDERTYPE_ADDITIONALGROUP_PLACEHOLDER_TRUSTLIST_READ_INPUTARGUMENTS := 13929,
	OPCUAID_CERTIFICATEGROUPFOLDERTYPE_ADDITIONALGROUP_PLACEHOLDER_TRUSTLIST_READ_OUTPUTARGUMENTS := 13930,
	OPCUAID_CERTIFICATEGROUPFOLDERTYPE_ADDITIONALGROUP_PLACEHOLDER_TRUSTLIST_WRITE_INPUTARGUMENTS := 13932,
	OPCUAID_CERTIFICATEGROUPFOLDERTYPE_ADDITIONALGROUP_PLACEHOLDER_TRUSTLIST_GETPOSITION_INPUTARGUMENTS := 13934,
	OPCUAID_CERTIFICATEGROUPFOLDERTYPE_ADDITIONALGROUP_PLACEHOLDER_TRUSTLIST_GETPOSITION_OUTPUTARGUMENTS := 13935,
	OPCUAID_CERTIFICATEGROUPFOLDERTYPE_ADDITIONALGROUP_PLACEHOLDER_TRUSTLIST_SETPOSITION_INPUTARGUMENTS := 13937,
	OPCUAID_CERTIFICATEGROUPFOLDERTYPE_ADDITIONALGROUP_PLACEHOLDER_TRUSTLIST_LASTUPDATETIME := 13938,
	OPCUAID_CERTIFICATEGROUPFOLDERTYPE_ADDITIONALGROUP_PLACEHOLDER_TRUSTLIST_OPENWITHMASKS_INPUTARGUMENTS := 13940,
	OPCUAID_CERTIFICATEGROUPFOLDERTYPE_ADDITIONALGROUP_PLACEHOLDER_TRUSTLIST_OPENWITHMASKS_OUTPUTARGUMENTS := 13941,
	OPCUAID_CERTIFICATEGROUPFOLDERTYPE_ADDITIONALGROUP_PLACEHOLDER_TRUSTLIST_CLOSEANDUPDATE_INPUTARGUMENTS := 13943,
	OPCUAID_CERTIFICATEGROUPFOLDERTYPE_ADDITIONALGROUP_PLACEHOLDER_TRUSTLIST_CLOSEANDUPDATE_OUTPUTARGUMENTS := 13944,
	OPCUAID_CERTIFICATEGROUPFOLDERTYPE_ADDITIONALGROUP_PLACEHOLDER_TRUSTLIST_ADDCERTIFICATE_INPUTARGUMENTS := 13946,
	OPCUAID_CERTIFICATEGROUPFOLDERTYPE_ADDITIONALGROUP_PLACEHOLDER_TRUSTLIST_REMOVECERTIFICATE_INPUTARGUMENTS := 13948,
	OPCUAID_CERTIFICATEGROUPFOLDERTYPE_ADDITIONALGROUP_PLACEHOLDER_CERTIFICATETYPES := 13949,
	OPCUAID_SERVERCONFIGURATIONTYPE_CERTIFICATEGROUPS_DEFAULTAPPLICATIONGROUP_TRUSTLIST_SIZE := 13953,
	OPCUAID_SERVERCONFIGURATIONTYPE_CERTIFICATEGROUPS_DEFAULTAPPLICATIONGROUP_TRUSTLIST_WRITABLE := 13954,
	OPCUAID_SERVERCONFIGURATIONTYPE_CERTIFICATEGROUPS_DEFAULTAPPLICATIONGROUP_TRUSTLIST_USERWRITABLE := 13955,
	OPCUAID_SERVERCONFIGURATIONTYPE_CERTIFICATEGROUPS_DEFAULTAPPLICATIONGROUP_TRUSTLIST_OPENCOUNT := 13956,
	OPCUAID_SERVERCONFIGURATIONTYPE_CERTIFICATEGROUPS_DEFAULTAPPLICATIONGROUP_TRUSTLIST_OPEN_INPUTARGUMENTS := 13959,
	OPCUAID_SERVERCONFIGURATIONTYPE_CERTIFICATEGROUPS_DEFAULTAPPLICATIONGROUP_TRUSTLIST_OPEN_OUTPUTARGUMENTS := 13960,
	OPCUAID_SERVERCONFIGURATIONTYPE_CERTIFICATEGROUPS_DEFAULTAPPLICATIONGROUP_TRUSTLIST_CLOSE_INPUTARGUMENTS := 13962,
	OPCUAID_SERVERCONFIGURATIONTYPE_CERTIFICATEGROUPS_DEFAULTAPPLICATIONGROUP_TRUSTLIST_READ_INPUTARGUMENTS := 13964,
	OPCUAID_SERVERCONFIGURATIONTYPE_CERTIFICATEGROUPS_DEFAULTAPPLICATIONGROUP_TRUSTLIST_READ_OUTPUTARGUMENTS := 13965,
	OPCUAID_SERVERCONFIGURATIONTYPE_CERTIFICATEGROUPS_DEFAULTAPPLICATIONGROUP_TRUSTLIST_WRITE_INPUTARGUMENTS := 13967,
	OPCUAID_SERVERCONFIGURATIONTYPE_CERTIFICATEGROUPS_DEFAULTAPPLICATIONGROUP_TRUSTLIST_GETPOSITION_INPUTARGUMENTS := 13969,
	OPCUAID_SERVERCONFIGURATIONTYPE_CERTIFICATEGROUPS_DEFAULTAPPLICATIONGROUP_TRUSTLIST_GETPOSITION_OUTPUTARGUMENTS := 13970,
	OPCUAID_SERVERCONFIGURATIONTYPE_CERTIFICATEGROUPS_DEFAULTAPPLICATIONGROUP_TRUSTLIST_SETPOSITION_INPUTARGUMENTS := 13972,
	OPCUAID_SERVERCONFIGURATIONTYPE_CERTIFICATEGROUPS_DEFAULTAPPLICATIONGROUP_TRUSTLIST_LASTUPDATETIME := 13973,
	OPCUAID_SERVERCONFIGURATIONTYPE_CERTIFICATEGROUPS_DEFAULTAPPLICATIONGROUP_TRUSTLIST_OPENWITHMASKS_INPUTARGUMENTS := 13975,
	OPCUAID_SERVERCONFIGURATIONTYPE_CERTIFICATEGROUPS_DEFAULTAPPLICATIONGROUP_TRUSTLIST_OPENWITHMASKS_OUTPUTARGUMENTS := 13976,
	OPCUAID_SERVERCONFIGURATIONTYPE_CERTIFICATEGROUPS_DEFAULTAPPLICATIONGROUP_TRUSTLIST_CLOSEANDUPDATE_INPUTARGUMENTS := 13978,
	OPCUAID_SERVERCONFIGURATIONTYPE_CERTIFICATEGROUPS_DEFAULTAPPLICATIONGROUP_TRUSTLIST_CLOSEANDUPDATE_OUTPUTARGUMENTS := 13979,
	OPCUAID_SERVERCONFIGURATIONTYPE_CERTIFICATEGROUPS_DEFAULTAPPLICATIONGROUP_TRUSTLIST_ADDCERTIFICATE_INPUTARGUMENTS := 13981,
	OPCUAID_SERVERCONFIGURATIONTYPE_CERTIFICATEGROUPS_DEFAULTAPPLICATIONGROUP_TRUSTLIST_REMOVECERTIFICATE_INPUTARGUMENTS := 13983,
	OPCUAID_SERVERCONFIGURATIONTYPE_CERTIFICATEGROUPS_DEFAULTAPPLICATIONGROUP_CERTIFICATETYPES := 13984,
	OPCUAID_SERVERCONFIGURATIONTYPE_CERTIFICATEGROUPS_DEFAULTHTTPSGROUP_TRUSTLIST_SIZE := 13987,
	OPCUAID_SERVERCONFIGURATIONTYPE_CERTIFICATEGROUPS_DEFAULTHTTPSGROUP_TRUSTLIST_WRITABLE := 13988,
	OPCUAID_SERVERCONFIGURATIONTYPE_CERTIFICATEGROUPS_DEFAULTHTTPSGROUP_TRUSTLIST_USERWRITABLE := 13989,
	OPCUAID_SERVERCONFIGURATIONTYPE_CERTIFICATEGROUPS_DEFAULTHTTPSGROUP_TRUSTLIST_OPENCOUNT := 13990,
	OPCUAID_SERVERCONFIGURATIONTYPE_CERTIFICATEGROUPS_DEFAULTHTTPSGROUP_TRUSTLIST_OPEN_INPUTARGUMENTS := 13993,
	OPCUAID_SERVERCONFIGURATIONTYPE_CERTIFICATEGROUPS_DEFAULTHTTPSGROUP_TRUSTLIST_OPEN_OUTPUTARGUMENTS := 13994,
	OPCUAID_SERVERCONFIGURATIONTYPE_CERTIFICATEGROUPS_DEFAULTHTTPSGROUP_TRUSTLIST_CLOSE_INPUTARGUMENTS := 13996,
	OPCUAID_SERVERCONFIGURATIONTYPE_CERTIFICATEGROUPS_DEFAULTHTTPSGROUP_TRUSTLIST_READ_INPUTARGUMENTS := 13998,
	OPCUAID_SERVERCONFIGURATIONTYPE_CERTIFICATEGROUPS_DEFAULTHTTPSGROUP_TRUSTLIST_READ_OUTPUTARGUMENTS := 13999,
	OPCUAID_SERVERCONFIGURATIONTYPE_CERTIFICATEGROUPS_DEFAULTHTTPSGROUP_TRUSTLIST_WRITE_INPUTARGUMENTS := 14001,
	OPCUAID_SERVERCONFIGURATIONTYPE_CERTIFICATEGROUPS_DEFAULTHTTPSGROUP_TRUSTLIST_GETPOSITION_INPUTARGUMENTS := 14003,
	OPCUAID_SERVERCONFIGURATIONTYPE_CERTIFICATEGROUPS_DEFAULTHTTPSGROUP_TRUSTLIST_GETPOSITION_OUTPUTARGUMENTS := 14004,
	OPCUAID_SERVERCONFIGURATIONTYPE_CERTIFICATEGROUPS_DEFAULTHTTPSGROUP_TRUSTLIST_SETPOSITION_INPUTARGUMENTS := 14006,
	OPCUAID_SERVERCONFIGURATIONTYPE_CERTIFICATEGROUPS_DEFAULTHTTPSGROUP_TRUSTLIST_LASTUPDATETIME := 14007,
	OPCUAID_SERVERCONFIGURATIONTYPE_CERTIFICATEGROUPS_DEFAULTHTTPSGROUP_TRUSTLIST_OPENWITHMASKS_INPUTARGUMENTS := 14009,
	OPCUAID_SERVERCONFIGURATIONTYPE_CERTIFICATEGROUPS_DEFAULTHTTPSGROUP_TRUSTLIST_OPENWITHMASKS_OUTPUTARGUMENTS := 14010,
	OPCUAID_SERVERCONFIGURATIONTYPE_CERTIFICATEGROUPS_DEFAULTHTTPSGROUP_TRUSTLIST_CLOSEANDUPDATE_INPUTARGUMENTS := 14012,
	OPCUAID_SERVERCONFIGURATIONTYPE_CERTIFICATEGROUPS_DEFAULTHTTPSGROUP_TRUSTLIST_CLOSEANDUPDATE_OUTPUTARGUMENTS := 14013,
	OPCUAID_SERVERCONFIGURATIONTYPE_CERTIFICATEGROUPS_DEFAULTHTTPSGROUP_TRUSTLIST_ADDCERTIFICATE_INPUTARGUMENTS := 14015,
	OPCUAID_SERVERCONFIGURATIONTYPE_CERTIFICATEGROUPS_DEFAULTHTTPSGROUP_TRUSTLIST_REMOVECERTIFICATE_INPUTARGUMENTS := 14017,
	OPCUAID_SERVERCONFIGURATIONTYPE_CERTIFICATEGROUPS_DEFAULTHTTPSGROUP_CERTIFICATETYPES := 14018,
	OPCUAID_SERVERCONFIGURATIONTYPE_CERTIFICATEGROUPS_DEFAULTUSERTOKENGROUP_TRUSTLIST_SIZE := 14021,
	OPCUAID_SERVERCONFIGURATIONTYPE_CERTIFICATEGROUPS_DEFAULTUSERTOKENGROUP_TRUSTLIST_WRITABLE := 14022,
	OPCUAID_SERVERCONFIGURATIONTYPE_CERTIFICATEGROUPS_DEFAULTUSERTOKENGROUP_TRUSTLIST_USERWRITABLE := 14023,
	OPCUAID_SERVERCONFIGURATIONTYPE_CERTIFICATEGROUPS_DEFAULTUSERTOKENGROUP_TRUSTLIST_OPENCOUNT := 14024,
	OPCUAID_SERVERCONFIGURATIONTYPE_CERTIFICATEGROUPS_DEFAULTUSERTOKENGROUP_TRUSTLIST_OPEN_INPUTARGUMENTS := 14027,
	OPCUAID_SERVERCONFIGURATIONTYPE_CERTIFICATEGROUPS_DEFAULTUSERTOKENGROUP_TRUSTLIST_OPEN_OUTPUTARGUMENTS := 14028,
	OPCUAID_SERVERCONFIGURATIONTYPE_CERTIFICATEGROUPS_DEFAULTUSERTOKENGROUP_TRUSTLIST_CLOSE_INPUTARGUMENTS := 14030,
	OPCUAID_SERVERCONFIGURATIONTYPE_CERTIFICATEGROUPS_DEFAULTUSERTOKENGROUP_TRUSTLIST_READ_INPUTARGUMENTS := 14032,
	OPCUAID_SERVERCONFIGURATIONTYPE_CERTIFICATEGROUPS_DEFAULTUSERTOKENGROUP_TRUSTLIST_READ_OUTPUTARGUMENTS := 14033,
	OPCUAID_SERVERCONFIGURATIONTYPE_CERTIFICATEGROUPS_DEFAULTUSERTOKENGROUP_TRUSTLIST_WRITE_INPUTARGUMENTS := 14035,
	OPCUAID_SERVERCONFIGURATIONTYPE_CERTIFICATEGROUPS_DEFAULTUSERTOKENGROUP_TRUSTLIST_GETPOSITION_INPUTARGUMENTS := 14037,
	OPCUAID_SERVERCONFIGURATIONTYPE_CERTIFICATEGROUPS_DEFAULTUSERTOKENGROUP_TRUSTLIST_GETPOSITION_OUTPUTARGUMENTS := 14038,
	OPCUAID_SERVERCONFIGURATIONTYPE_CERTIFICATEGROUPS_DEFAULTUSERTOKENGROUP_TRUSTLIST_SETPOSITION_INPUTARGUMENTS := 14040,
	OPCUAID_SERVERCONFIGURATIONTYPE_CERTIFICATEGROUPS_DEFAULTUSERTOKENGROUP_TRUSTLIST_LASTUPDATETIME := 14041,
	OPCUAID_SERVERCONFIGURATIONTYPE_CERTIFICATEGROUPS_DEFAULTUSERTOKENGROUP_TRUSTLIST_OPENWITHMASKS_INPUTARGUMENTS := 14043,
	OPCUAID_SERVERCONFIGURATIONTYPE_CERTIFICATEGROUPS_DEFAULTUSERTOKENGROUP_TRUSTLIST_OPENWITHMASKS_OUTPUTARGUMENTS := 14044,
	OPCUAID_SERVERCONFIGURATIONTYPE_CERTIFICATEGROUPS_DEFAULTUSERTOKENGROUP_TRUSTLIST_CLOSEANDUPDATE_INPUTARGUMENTS := 14046,
	OPCUAID_SERVERCONFIGURATIONTYPE_CERTIFICATEGROUPS_DEFAULTUSERTOKENGROUP_TRUSTLIST_CLOSEANDUPDATE_OUTPUTARGUMENTS := 14047,
	OPCUAID_SERVERCONFIGURATIONTYPE_CERTIFICATEGROUPS_DEFAULTUSERTOKENGROUP_TRUSTLIST_ADDCERTIFICATE_INPUTARGUMENTS := 14049,
	OPCUAID_SERVERCONFIGURATIONTYPE_CERTIFICATEGROUPS_DEFAULTUSERTOKENGROUP_TRUSTLIST_REMOVECERTIFICATE_INPUTARGUMENTS := 14051,
	OPCUAID_SERVERCONFIGURATIONTYPE_CERTIFICATEGROUPS_DEFAULTUSERTOKENGROUP_CERTIFICATETYPES := 14052,
	OPCUAID_SERVERCONFIGURATIONTYPE_SERVERCAPABILITIES := 12708,
	OPCUAID_SERVERCONFIGURATIONTYPE_SUPPORTEDPRIVATEKEYFORMATS := 12583,
	OPCUAID_SERVERCONFIGURATIONTYPE_MAXTRUSTLISTSIZE := 12584,
	OPCUAID_SERVERCONFIGURATIONTYPE_MULTICASTDNSENABLED := 12585,
	OPCUAID_SERVERCONFIGURATIONTYPE_UPDATECERTIFICATE_INPUTARGUMENTS := 12617,
	OPCUAID_SERVERCONFIGURATIONTYPE_UPDATECERTIFICATE_OUTPUTARGUMENTS := 12618,
	OPCUAID_SERVERCONFIGURATIONTYPE_CREATESIGNINGREQUEST_INPUTARGUMENTS := 12732,
	OPCUAID_SERVERCONFIGURATIONTYPE_CREATESIGNINGREQUEST_OUTPUTARGUMENTS := 12733,
	OPCUAID_SERVERCONFIGURATIONTYPE_GETREJECTEDLIST_OUTPUTARGUMENTS := 12776,
	OPCUAID_CERTIFICATEUPDATEDAUDITEVENTTYPE_CERTIFICATEGROUP := 13735,
	OPCUAID_CERTIFICATEUPDATEDAUDITEVENTTYPE_CERTIFICATETYPE := 13736,
	OPCUAID_SERVERCONFIGURATION_CERTIFICATEGROUPS_DEFAULTAPPLICATIONGROUP_TRUSTLIST_SIZE := 12643,
	OPCUAID_SERVERCONFIGURATION_CERTIFICATEGROUPS_DEFAULTAPPLICATIONGROUP_TRUSTLIST_WRITABLE := 14157,
	OPCUAID_SERVERCONFIGURATION_CERTIFICATEGROUPS_DEFAULTAPPLICATIONGROUP_TRUSTLIST_USERWRITABLE := 14158,
	OPCUAID_SERVERCONFIGURATION_CERTIFICATEGROUPS_DEFAULTAPPLICATIONGROUP_TRUSTLIST_OPENCOUNT := 12646,
	OPCUAID_SERVERCONFIGURATION_CERTIFICATEGROUPS_DEFAULTAPPLICATIONGROUP_TRUSTLIST_OPEN_INPUTARGUMENTS := 12648,
	OPCUAID_SERVERCONFIGURATION_CERTIFICATEGROUPS_DEFAULTAPPLICATIONGROUP_TRUSTLIST_OPEN_OUTPUTARGUMENTS := 12649,
	OPCUAID_SERVERCONFIGURATION_CERTIFICATEGROUPS_DEFAULTAPPLICATIONGROUP_TRUSTLIST_CLOSE_INPUTARGUMENTS := 12651,
	OPCUAID_SERVERCONFIGURATION_CERTIFICATEGROUPS_DEFAULTAPPLICATIONGROUP_TRUSTLIST_READ_INPUTARGUMENTS := 12653,
	OPCUAID_SERVERCONFIGURATION_CERTIFICATEGROUPS_DEFAULTAPPLICATIONGROUP_TRUSTLIST_READ_OUTPUTARGUMENTS := 12654,
	OPCUAID_SERVERCONFIGURATION_CERTIFICATEGROUPS_DEFAULTAPPLICATIONGROUP_TRUSTLIST_WRITE_INPUTARGUMENTS := 12656,
	OPCUAID_SERVERCONFIGURATION_CERTIFICATEGROUPS_DEFAULTAPPLICATIONGROUP_TRUSTLIST_GETPOSITION_INPUTARGUMENTS := 12658,
	OPCUAID_SERVERCONFIGURATION_CERTIFICATEGROUPS_DEFAULTAPPLICATIONGROUP_TRUSTLIST_GETPOSITION_OUTPUTARGUMENTS := 12659,
	OPCUAID_SERVERCONFIGURATION_CERTIFICATEGROUPS_DEFAULTAPPLICATIONGROUP_TRUSTLIST_SETPOSITION_INPUTARGUMENTS := 12661,
	OPCUAID_SERVERCONFIGURATION_CERTIFICATEGROUPS_DEFAULTAPPLICATIONGROUP_TRUSTLIST_LASTUPDATETIME := 12662,
	OPCUAID_SERVERCONFIGURATION_CERTIFICATEGROUPS_DEFAULTAPPLICATIONGROUP_TRUSTLIST_OPENWITHMASKS_INPUTARGUMENTS := 12664,
	OPCUAID_SERVERCONFIGURATION_CERTIFICATEGROUPS_DEFAULTAPPLICATIONGROUP_TRUSTLIST_OPENWITHMASKS_OUTPUTARGUMENTS := 12665,
	OPCUAID_SERVERCONFIGURATION_CERTIFICATEGROUPS_DEFAULTAPPLICATIONGROUP_TRUSTLIST_CLOSEANDUPDATE_INPUTARGUMENTS := 14160,
	OPCUAID_SERVERCONFIGURATION_CERTIFICATEGROUPS_DEFAULTAPPLICATIONGROUP_TRUSTLIST_CLOSEANDUPDATE_OUTPUTARGUMENTS := 12667,
	OPCUAID_SERVERCONFIGURATION_CERTIFICATEGROUPS_DEFAULTAPPLICATIONGROUP_TRUSTLIST_ADDCERTIFICATE_INPUTARGUMENTS := 12669,
	OPCUAID_SERVERCONFIGURATION_CERTIFICATEGROUPS_DEFAULTAPPLICATIONGROUP_TRUSTLIST_REMOVECERTIFICATE_INPUTARGUMENTS := 12671,
	OPCUAID_SERVERCONFIGURATION_CERTIFICATEGROUPS_DEFAULTAPPLICATIONGROUP_CERTIFICATETYPES := 14161,
	OPCUAID_SERVERCONFIGURATION_CERTIFICATEGROUPS_DEFAULTHTTPSGROUP_TRUSTLIST_SIZE := 14090,
	OPCUAID_SERVERCONFIGURATION_CERTIFICATEGROUPS_DEFAULTHTTPSGROUP_TRUSTLIST_WRITABLE := 14091,
	OPCUAID_SERVERCONFIGURATION_CERTIFICATEGROUPS_DEFAULTHTTPSGROUP_TRUSTLIST_USERWRITABLE := 14092,
	OPCUAID_SERVERCONFIGURATION_CERTIFICATEGROUPS_DEFAULTHTTPSGROUP_TRUSTLIST_OPENCOUNT := 14093,
	OPCUAID_SERVERCONFIGURATION_CERTIFICATEGROUPS_DEFAULTHTTPSGROUP_TRUSTLIST_OPEN_INPUTARGUMENTS := 14096,
	OPCUAID_SERVERCONFIGURATION_CERTIFICATEGROUPS_DEFAULTHTTPSGROUP_TRUSTLIST_OPEN_OUTPUTARGUMENTS := 14097,
	OPCUAID_SERVERCONFIGURATION_CERTIFICATEGROUPS_DEFAULTHTTPSGROUP_TRUSTLIST_CLOSE_INPUTARGUMENTS := 14099,
	OPCUAID_SERVERCONFIGURATION_CERTIFICATEGROUPS_DEFAULTHTTPSGROUP_TRUSTLIST_READ_INPUTARGUMENTS := 14101,
	OPCUAID_SERVERCONFIGURATION_CERTIFICATEGROUPS_DEFAULTHTTPSGROUP_TRUSTLIST_READ_OUTPUTARGUMENTS := 14102,
	OPCUAID_SERVERCONFIGURATION_CERTIFICATEGROUPS_DEFAULTHTTPSGROUP_TRUSTLIST_WRITE_INPUTARGUMENTS := 14104,
	OPCUAID_SERVERCONFIGURATION_CERTIFICATEGROUPS_DEFAULTHTTPSGROUP_TRUSTLIST_GETPOSITION_INPUTARGUMENTS := 14106,
	OPCUAID_SERVERCONFIGURATION_CERTIFICATEGROUPS_DEFAULTHTTPSGROUP_TRUSTLIST_GETPOSITION_OUTPUTARGUMENTS := 14107,
	OPCUAID_SERVERCONFIGURATION_CERTIFICATEGROUPS_DEFAULTHTTPSGROUP_TRUSTLIST_SETPOSITION_INPUTARGUMENTS := 14109,
	OPCUAID_SERVERCONFIGURATION_CERTIFICATEGROUPS_DEFAULTHTTPSGROUP_TRUSTLIST_LASTUPDATETIME := 14110,
	OPCUAID_SERVERCONFIGURATION_CERTIFICATEGROUPS_DEFAULTHTTPSGROUP_TRUSTLIST_OPENWITHMASKS_INPUTARGUMENTS := 14112,
	OPCUAID_SERVERCONFIGURATION_CERTIFICATEGROUPS_DEFAULTHTTPSGROUP_TRUSTLIST_OPENWITHMASKS_OUTPUTARGUMENTS := 14113,
	OPCUAID_SERVERCONFIGURATION_CERTIFICATEGROUPS_DEFAULTHTTPSGROUP_TRUSTLIST_CLOSEANDUPDATE_INPUTARGUMENTS := 14115,
	OPCUAID_SERVERCONFIGURATION_CERTIFICATEGROUPS_DEFAULTHTTPSGROUP_TRUSTLIST_CLOSEANDUPDATE_OUTPUTARGUMENTS := 14116,
	OPCUAID_SERVERCONFIGURATION_CERTIFICATEGROUPS_DEFAULTHTTPSGROUP_TRUSTLIST_ADDCERTIFICATE_INPUTARGUMENTS := 14118,
	OPCUAID_SERVERCONFIGURATION_CERTIFICATEGROUPS_DEFAULTHTTPSGROUP_TRUSTLIST_REMOVECERTIFICATE_INPUTARGUMENTS := 14120,
	OPCUAID_SERVERCONFIGURATION_CERTIFICATEGROUPS_DEFAULTHTTPSGROUP_CERTIFICATETYPES := 14121,
	OPCUAID_SERVERCONFIGURATION_CERTIFICATEGROUPS_DEFAULTUSERTOKENGROUP_TRUSTLIST_SIZE := 14124,
	OPCUAID_SERVERCONFIGURATION_CERTIFICATEGROUPS_DEFAULTUSERTOKENGROUP_TRUSTLIST_WRITABLE := 14125,
	OPCUAID_SERVERCONFIGURATION_CERTIFICATEGROUPS_DEFAULTUSERTOKENGROUP_TRUSTLIST_USERWRITABLE := 14126,
	OPCUAID_SERVERCONFIGURATION_CERTIFICATEGROUPS_DEFAULTUSERTOKENGROUP_TRUSTLIST_OPENCOUNT := 14127,
	OPCUAID_SERVERCONFIGURATION_CERTIFICATEGROUPS_DEFAULTUSERTOKENGROUP_TRUSTLIST_OPEN_INPUTARGUMENTS := 14130,
	OPCUAID_SERVERCONFIGURATION_CERTIFICATEGROUPS_DEFAULTUSERTOKENGROUP_TRUSTLIST_OPEN_OUTPUTARGUMENTS := 14131,
	OPCUAID_SERVERCONFIGURATION_CERTIFICATEGROUPS_DEFAULTUSERTOKENGROUP_TRUSTLIST_CLOSE_INPUTARGUMENTS := 14133,
	OPCUAID_SERVERCONFIGURATION_CERTIFICATEGROUPS_DEFAULTUSERTOKENGROUP_TRUSTLIST_READ_INPUTARGUMENTS := 14135,
	OPCUAID_SERVERCONFIGURATION_CERTIFICATEGROUPS_DEFAULTUSERTOKENGROUP_TRUSTLIST_READ_OUTPUTARGUMENTS := 14136,
	OPCUAID_SERVERCONFIGURATION_CERTIFICATEGROUPS_DEFAULTUSERTOKENGROUP_TRUSTLIST_WRITE_INPUTARGUMENTS := 14138,
	OPCUAID_SERVERCONFIGURATION_CERTIFICATEGROUPS_DEFAULTUSERTOKENGROUP_TRUSTLIST_GETPOSITION_INPUTARGUMENTS := 14140,
	OPCUAID_SERVERCONFIGURATION_CERTIFICATEGROUPS_DEFAULTUSERTOKENGROUP_TRUSTLIST_GETPOSITION_OUTPUTARGUMENTS := 14141,
	OPCUAID_SERVERCONFIGURATION_CERTIFICATEGROUPS_DEFAULTUSERTOKENGROUP_TRUSTLIST_SETPOSITION_INPUTARGUMENTS := 14143,
	OPCUAID_SERVERCONFIGURATION_CERTIFICATEGROUPS_DEFAULTUSERTOKENGROUP_TRUSTLIST_LASTUPDATETIME := 14144,
	OPCUAID_SERVERCONFIGURATION_CERTIFICATEGROUPS_DEFAULTUSERTOKENGROUP_TRUSTLIST_OPENWITHMASKS_INPUTARGUMENTS := 14146,
	OPCUAID_SERVERCONFIGURATION_CERTIFICATEGROUPS_DEFAULTUSERTOKENGROUP_TRUSTLIST_OPENWITHMASKS_OUTPUTARGUMENTS := 14147,
	OPCUAID_SERVERCONFIGURATION_CERTIFICATEGROUPS_DEFAULTUSERTOKENGROUP_TRUSTLIST_CLOSEANDUPDATE_INPUTARGUMENTS := 14149,
	OPCUAID_SERVERCONFIGURATION_CERTIFICATEGROUPS_DEFAULTUSERTOKENGROUP_TRUSTLIST_CLOSEANDUPDATE_OUTPUTARGUMENTS := 14150,
	OPCUAID_SERVERCONFIGURATION_CERTIFICATEGROUPS_DEFAULTUSERTOKENGROUP_TRUSTLIST_ADDCERTIFICATE_INPUTARGUMENTS := 14152,
	OPCUAID_SERVERCONFIGURATION_CERTIFICATEGROUPS_DEFAULTUSERTOKENGROUP_TRUSTLIST_REMOVECERTIFICATE_INPUTARGUMENTS := 14154,
	OPCUAID_SERVERCONFIGURATION_CERTIFICATEGROUPS_DEFAULTUSERTOKENGROUP_CERTIFICATETYPES := 14155,
	OPCUAID_SERVERCONFIGURATION_SERVERCAPABILITIES := 12710,
	OPCUAID_SERVERCONFIGURATION_SUPPORTEDPRIVATEKEYFORMATS := 12639,
	OPCUAID_SERVERCONFIGURATION_MAXTRUSTLISTSIZE := 12640,
	OPCUAID_SERVERCONFIGURATION_MULTICASTDNSENABLED := 12641,
	OPCUAID_SERVERCONFIGURATION_UPDATECERTIFICATE_INPUTARGUMENTS := 13738,
	OPCUAID_SERVERCONFIGURATION_UPDATECERTIFICATE_OUTPUTARGUMENTS := 13739,
	OPCUAID_SERVERCONFIGURATION_CREATESIGNINGREQUEST_INPUTARGUMENTS := 12738,
	OPCUAID_SERVERCONFIGURATION_CREATESIGNINGREQUEST_OUTPUTARGUMENTS := 12739,
	OPCUAID_SERVERCONFIGURATION_GETREJECTEDLIST_OUTPUTARGUMENTS := 12778,
	OPCUAID_KEYCREDENTIALCONFIGURATIONFOLDERTYPE_SERVICENAME_PLACEHOLDER_RESOURCEURI := 17512,
	OPCUAID_KEYCREDENTIALCONFIGURATIONFOLDERTYPE_SERVICENAME_PLACEHOLDER_PROFILEURI := 17513,
	OPCUAID_KEYCREDENTIALCONFIGURATIONFOLDERTYPE_SERVICENAME_PLACEHOLDER_GETENCRYPTINGKEY_INPUTARGUMENTS := 17517,
	OPCUAID_KEYCREDENTIALCONFIGURATIONFOLDERTYPE_SERVICENAME_PLACEHOLDER_GETENCRYPTINGKEY_OUTPUTARGUMENTS := 17518,
	OPCUAID_KEYCREDENTIALCONFIGURATIONFOLDERTYPE_SERVICENAME_PLACEHOLDER_UPDATECREDENTIAL_INPUTARGUMENTS := 17520,
	OPCUAID_KEYCREDENTIALCONFIGURATIONFOLDERTYPE_CREATECREDENTIAL_INPUTARGUMENTS := 17523,
	OPCUAID_KEYCREDENTIALCONFIGURATIONFOLDERTYPE_CREATECREDENTIAL_OUTPUTARGUMENTS := 17524,
	OPCUAID_KEYCREDENTIALCONFIGURATION_SERVICENAME_PLACEHOLDER_RESOURCEURI := 18157,
	OPCUAID_KEYCREDENTIALCONFIGURATION_SERVICENAME_PLACEHOLDER_PROFILEURI := 18164,
	OPCUAID_KEYCREDENTIALCONFIGURATION_SERVICENAME_PLACEHOLDER_GETENCRYPTINGKEY_INPUTARGUMENTS := 17526,
	OPCUAID_KEYCREDENTIALCONFIGURATION_SERVICENAME_PLACEHOLDER_GETENCRYPTINGKEY_OUTPUTARGUMENTS := 17527,
	OPCUAID_KEYCREDENTIALCONFIGURATION_SERVICENAME_PLACEHOLDER_UPDATECREDENTIAL_INPUTARGUMENTS := 18162,
	OPCUAID_KEYCREDENTIALCONFIGURATION_CREATECREDENTIAL_INPUTARGUMENTS := 17529,
	OPCUAID_KEYCREDENTIALCONFIGURATION_CREATECREDENTIAL_OUTPUTARGUMENTS := 17530,
	OPCUAID_KEYCREDENTIALCONFIGURATIONTYPE_RESOURCEURI := 18069,
	OPCUAID_KEYCREDENTIALCONFIGURATIONTYPE_PROFILEURI := 18165,
	OPCUAID_KEYCREDENTIALCONFIGURATIONTYPE_ENDPOINTURLS := 18004,
	OPCUAID_KEYCREDENTIALCONFIGURATIONTYPE_SERVICESTATUS := 18005,
	OPCUAID_KEYCREDENTIALCONFIGURATIONTYPE_GETENCRYPTINGKEY_INPUTARGUMENTS := 17535,
	OPCUAID_KEYCREDENTIALCONFIGURATIONTYPE_GETENCRYPTINGKEY_OUTPUTARGUMENTS := 17536,
	OPCUAID_KEYCREDENTIALCONFIGURATIONTYPE_UPDATECREDENTIAL_INPUTARGUMENTS := 18007,
	OPCUAID_KEYCREDENTIALAUDITEVENTTYPE_RESOURCEURI := 18028,
	OPCUAID_AUTHORIZATIONSERVICES_SERVICENAME_PLACEHOLDER_SERVICEURI := 18070,
	OPCUAID_AUTHORIZATIONSERVICES_SERVICENAME_PLACEHOLDER_SERVICECERTIFICATE := 18066,
	OPCUAID_AUTHORIZATIONSERVICES_SERVICENAME_PLACEHOLDER_ISSUERENDPOINTURL := 18071,
	OPCUAID_AUTHORIZATIONSERVICECONFIGURATIONTYPE_SERVICEURI := 18072,
	OPCUAID_AUTHORIZATIONSERVICECONFIGURATIONTYPE_SERVICECERTIFICATE := 17860,
	OPCUAID_AUTHORIZATIONSERVICECONFIGURATIONTYPE_ISSUERENDPOINTURL := 18073,
	OPCUAID_AGGREGATECONFIGURATIONTYPE_TREATUNCERTAINASBAD := 11188,
	OPCUAID_AGGREGATECONFIGURATIONTYPE_PERCENTDATABAD := 11189,
	OPCUAID_AGGREGATECONFIGURATIONTYPE_PERCENTDATAGOOD := 11190,
	OPCUAID_AGGREGATECONFIGURATIONTYPE_USESLOPEDEXTRAPOLATION := 11191,
	OPCUAID_PUBSUBSTATE_ENUMSTRINGS := 14648,
	OPCUAID_DATASETFIELDFLAGS_OPTIONSETVALUES := 15577,
	OPCUAID_DATASETFIELDCONTENTMASK_OPTIONSETVALUES := 15584,
	OPCUAID_OVERRIDEVALUEHANDLING_ENUMSTRINGS := 15875,
	OPCUAID_DATASETORDERINGTYPE_ENUMSTRINGS := 15641,
	OPCUAID_UADPNETWORKMESSAGECONTENTMASK_OPTIONSETVALUES := 15643,
	OPCUAID_UADPDATASETMESSAGECONTENTMASK_OPTIONSETVALUES := 15647,
	OPCUAID_JSONNETWORKMESSAGECONTENTMASK_OPTIONSETVALUES := 15655,
	OPCUAID_JSONDATASETMESSAGECONTENTMASK_OPTIONSETVALUES := 15659,
	OPCUAID_BROKERTRANSPORTQUALITYOFSERVICE_ENUMSTRINGS := 15009,
	OPCUAID_PUBSUBKEYSERVICETYPE_GETSECURITYKEYS_INPUTARGUMENTS := 15908,
	OPCUAID_PUBSUBKEYSERVICETYPE_GETSECURITYKEYS_OUTPUTARGUMENTS := 15909,
	OPCUAID_PUBSUBKEYSERVICETYPE_GETSECURITYGROUP_INPUTARGUMENTS := 15911,
	OPCUAID_PUBSUBKEYSERVICETYPE_GETSECURITYGROUP_OUTPUTARGUMENTS := 15912,
	OPCUAID_PUBSUBKEYSERVICETYPE_SECURITYGROUPS_ADDSECURITYGROUP_INPUTARGUMENTS := 15915,
	OPCUAID_PUBSUBKEYSERVICETYPE_SECURITYGROUPS_ADDSECURITYGROUP_OUTPUTARGUMENTS := 15916,
	OPCUAID_PUBSUBKEYSERVICETYPE_SECURITYGROUPS_REMOVESECURITYGROUP_INPUTARGUMENTS := 15918,
	OPCUAID_SECURITYGROUPFOLDERTYPE_SECURITYGROUPFOLDERNAME_PLACEHOLDER_ADDSECURITYGROUP_INPUTARGUMENTS := 15455,
	OPCUAID_SECURITYGROUPFOLDERTYPE_SECURITYGROUPFOLDERNAME_PLACEHOLDER_ADDSECURITYGROUP_OUTPUTARGUMENTS := 15456,
	OPCUAID_SECURITYGROUPFOLDERTYPE_SECURITYGROUPFOLDERNAME_PLACEHOLDER_REMOVESECURITYGROUP_INPUTARGUMENTS := 15458,
	OPCUAID_SECURITYGROUPFOLDERTYPE_SECURITYGROUPNAME_PLACEHOLDER_SECURITYGROUPID := 15460,
	OPCUAID_SECURITYGROUPFOLDERTYPE_SECURITYGROUPNAME_PLACEHOLDER_KEYLIFETIME := 15010,
	OPCUAID_SECURITYGROUPFOLDERTYPE_SECURITYGROUPNAME_PLACEHOLDER_SECURITYPOLICYURI := 15011,
	OPCUAID_SECURITYGROUPFOLDERTYPE_SECURITYGROUPNAME_PLACEHOLDER_MAXFUTUREKEYCOUNT := 15012,
	OPCUAID_SECURITYGROUPFOLDERTYPE_SECURITYGROUPNAME_PLACEHOLDER_MAXPASTKEYCOUNT := 15043,
	OPCUAID_SECURITYGROUPFOLDERTYPE_ADDSECURITYGROUP_INPUTARGUMENTS := 15462,
	OPCUAID_SECURITYGROUPFOLDERTYPE_ADDSECURITYGROUP_OUTPUTARGUMENTS := 15463,
	OPCUAID_SECURITYGROUPFOLDERTYPE_REMOVESECURITYGROUP_INPUTARGUMENTS := 15465,
	OPCUAID_SECURITYGROUPTYPE_SECURITYGROUPID := 15472,
	OPCUAID_SECURITYGROUPTYPE_KEYLIFETIME := 15046,
	OPCUAID_SECURITYGROUPTYPE_SECURITYPOLICYURI := 15047,
	OPCUAID_SECURITYGROUPTYPE_MAXFUTUREKEYCOUNT := 15048,
	OPCUAID_SECURITYGROUPTYPE_MAXPASTKEYCOUNT := 15056,
	OPCUAID_PUBLISHSUBSCRIBETYPE_GETSECURITYKEYS_INPUTARGUMENTS := 15213,
	OPCUAID_PUBLISHSUBSCRIBETYPE_GETSECURITYKEYS_OUTPUTARGUMENTS := 15214,
	OPCUAID_PUBLISHSUBSCRIBETYPE_GETSECURITYGROUP_INPUTARGUMENTS := 15432,
	OPCUAID_PUBLISHSUBSCRIBETYPE_GETSECURITYGROUP_OUTPUTARGUMENTS := 15433,
	OPCUAID_PUBLISHSUBSCRIBETYPE_SECURITYGROUPS_ADDSECURITYGROUP_INPUTARGUMENTS := 15436,
	OPCUAID_PUBLISHSUBSCRIBETYPE_SECURITYGROUPS_ADDSECURITYGROUP_OUTPUTARGUMENTS := 15437,
	OPCUAID_PUBLISHSUBSCRIBETYPE_SECURITYGROUPS_REMOVESECURITYGROUP_INPUTARGUMENTS := 15439,
	OPCUAID_PUBLISHSUBSCRIBETYPE_CONNECTIONNAME_PLACEHOLDER_PUBLISHERID := 14418,
	OPCUAID_PUBLISHSUBSCRIBETYPE_CONNECTIONNAME_PLACEHOLDER_TRANSPORTPROFILEURI := 17292,
	OPCUAID_PUBLISHSUBSCRIBETYPE_CONNECTIONNAME_PLACEHOLDER_TRANSPORTPROFILEURI_SELECTIONS := 17706,
	OPCUAID_PUBLISHSUBSCRIBETYPE_CONNECTIONNAME_PLACEHOLDER_CONNECTIONPROPERTIES := 17478,
	OPCUAID_PUBLISHSUBSCRIBETYPE_CONNECTIONNAME_PLACEHOLDER_ADDRESS_NETWORKINTERFACE := 15533,
	OPCUAID_PUBLISHSUBSCRIBETYPE_CONNECTIONNAME_PLACEHOLDER_STATUS_STATE := 14420,
	OPCUAID_PUBLISHSUBSCRIBETYPE_CONNECTIONNAME_PLACEHOLDER_DIAGNOSTICS_DIAGNOSTICSLEVEL := 18668,
	OPCUAID_PUBLISHSUBSCRIBETYPE_CONNECTIONNAME_PLACEHOLDER_DIAGNOSTICS_TOTALINFORMATION := 18669,
	OPCUAID_PUBLISHSUBSCRIBETYPE_CONNECTIONNAME_PLACEHOLDER_DIAGNOSTICS_TOTALINFORMATION_ACTIVE := 18670,
	OPCUAID_PUBLISHSUBSCRIBETYPE_CONNECTIONNAME_PLACEHOLDER_DIAGNOSTICS_TOTALINFORMATION_CLASSIFICATION := 18671,
	OPCUAID_PUBLISHSUBSCRIBETYPE_CONNECTIONNAME_PLACEHOLDER_DIAGNOSTICS_TOTALINFORMATION_DIAGNOSTICSLEVEL := 18672,
	OPCUAID_PUBLISHSUBSCRIBETYPE_CONNECTIONNAME_PLACEHOLDER_DIAGNOSTICS_TOTALINFORMATION_TIMEFIRSTCHANGE := 18673,
	OPCUAID_PUBLISHSUBSCRIBETYPE_CONNECTIONNAME_PLACEHOLDER_DIAGNOSTICS_TOTALERROR := 18674,
	OPCUAID_PUBLISHSUBSCRIBETYPE_CONNECTIONNAME_PLACEHOLDER_DIAGNOSTICS_TOTALERROR_ACTIVE := 18675,
	OPCUAID_PUBLISHSUBSCRIBETYPE_CONNECTIONNAME_PLACEHOLDER_DIAGNOSTICS_TOTALERROR_CLASSIFICATION := 18676,
	OPCUAID_PUBLISHSUBSCRIBETYPE_CONNECTIONNAME_PLACEHOLDER_DIAGNOSTICS_TOTALERROR_DIAGNOSTICSLEVEL := 18677,
	OPCUAID_PUBLISHSUBSCRIBETYPE_CONNECTIONNAME_PLACEHOLDER_DIAGNOSTICS_TOTALERROR_TIMEFIRSTCHANGE := 18678,
	OPCUAID_PUBLISHSUBSCRIBETYPE_CONNECTIONNAME_PLACEHOLDER_DIAGNOSTICS_SUBERROR := 18680,
	OPCUAID_PUBLISHSUBSCRIBETYPE_CONNECTIONNAME_PLACEHOLDER_DIAGNOSTICS_COUNTERS_STATEERROR := 18682,
	OPCUAID_PUBLISHSUBSCRIBETYPE_CONNECTIONNAME_PLACEHOLDER_DIAGNOSTICS_COUNTERS_STATEERROR_ACTIVE := 18683,
	OPCUAID_PUBLISHSUBSCRIBETYPE_CONNECTIONNAME_PLACEHOLDER_DIAGNOSTICS_COUNTERS_STATEERROR_CLASSIFICATION := 18684,
	OPCUAID_PUBLISHSUBSCRIBETYPE_CONNECTIONNAME_PLACEHOLDER_DIAGNOSTICS_COUNTERS_STATEERROR_DIAGNOSTICSLEVEL := 18685,
	OPCUAID_PUBLISHSUBSCRIBETYPE_CONNECTIONNAME_PLACEHOLDER_DIAGNOSTICS_COUNTERS_STATEERROR_TIMEFIRSTCHANGE := 18686,
	OPCUAID_PUBLISHSUBSCRIBETYPE_CONNECTIONNAME_PLACEHOLDER_DIAGNOSTICS_COUNTERS_STATEOPERATIONALBYMETHOD := 18687,
	OPCUAID_PUBLISHSUBSCRIBETYPE_CONNECTIONNAME_PLACEHOLDER_DIAGNOSTICS_COUNTERS_STATEOPERATIONALBYMETHOD_ACTIVE := 18688,
	OPCUAID_PUBLISHSUBSCRIBETYPE_CONNECTIONNAME_PLACEHOLDER_DIAGNOSTICS_COUNTERS_STATEOPERATIONALBYMETHOD_CLASSIFICATION := 18689,
	OPCUAID_PUBLISHSUBSCRIBETYPE_CONNECTIONNAME_PLACEHOLDER_DIAGNOSTICS_COUNTERS_STATEOPERATIONALBYMETHOD_DIAGNOSTICSLEVEL := 18690,
	OPCUAID_PUBLISHSUBSCRIBETYPE_CONNECTIONNAME_PLACEHOLDER_DIAGNOSTICS_COUNTERS_STATEOPERATIONALBYMETHOD_TIMEFIRSTCHANGE := 18691,
	OPCUAID_PUBLISHSUBSCRIBETYPE_CONNECTIONNAME_PLACEHOLDER_DIAGNOSTICS_COUNTERS_STATEOPERATIONALBYPARENT := 18692,
	OPCUAID_PUBLISHSUBSCRIBETYPE_CONNECTIONNAME_PLACEHOLDER_DIAGNOSTICS_COUNTERS_STATEOPERATIONALBYPARENT_ACTIVE := 18693,
	OPCUAID_PUBLISHSUBSCRIBETYPE_CONNECTIONNAME_PLACEHOLDER_DIAGNOSTICS_COUNTERS_STATEOPERATIONALBYPARENT_CLASSIFICATION := 18694,
	OPCUAID_PUBLISHSUBSCRIBETYPE_CONNECTIONNAME_PLACEHOLDER_DIAGNOSTICS_COUNTERS_STATEOPERATIONALBYPARENT_DIAGNOSTICSLEVEL := 18695,
	OPCUAID_PUBLISHSUBSCRIBETYPE_CONNECTIONNAME_PLACEHOLDER_DIAGNOSTICS_COUNTERS_STATEOPERATIONALBYPARENT_TIMEFIRSTCHANGE := 18696,
	OPCUAID_PUBLISHSUBSCRIBETYPE_CONNECTIONNAME_PLACEHOLDER_DIAGNOSTICS_COUNTERS_STATEOPERATIONALFROMERROR := 18697,
	OPCUAID_PUBLISHSUBSCRIBETYPE_CONNECTIONNAME_PLACEHOLDER_DIAGNOSTICS_COUNTERS_STATEOPERATIONALFROMERROR_ACTIVE := 18698,
	OPCUAID_PUBLISHSUBSCRIBETYPE_CONNECTIONNAME_PLACEHOLDER_DIAGNOSTICS_COUNTERS_STATEOPERATIONALFROMERROR_CLASSIFICATION := 18699,
	OPCUAID_PUBLISHSUBSCRIBETYPE_CONNECTIONNAME_PLACEHOLDER_DIAGNOSTICS_COUNTERS_STATEOPERATIONALFROMERROR_DIAGNOSTICSLEVEL := 18700,
	OPCUAID_PUBLISHSUBSCRIBETYPE_CONNECTIONNAME_PLACEHOLDER_DIAGNOSTICS_COUNTERS_STATEOPERATIONALFROMERROR_TIMEFIRSTCHANGE := 18701,
	OPCUAID_PUBLISHSUBSCRIBETYPE_CONNECTIONNAME_PLACEHOLDER_DIAGNOSTICS_COUNTERS_STATEPAUSEDBYPARENT := 18702,
	OPCUAID_PUBLISHSUBSCRIBETYPE_CONNECTIONNAME_PLACEHOLDER_DIAGNOSTICS_COUNTERS_STATEPAUSEDBYPARENT_ACTIVE := 18703,
	OPCUAID_PUBLISHSUBSCRIBETYPE_CONNECTIONNAME_PLACEHOLDER_DIAGNOSTICS_COUNTERS_STATEPAUSEDBYPARENT_CLASSIFICATION := 18704,
	OPCUAID_PUBLISHSUBSCRIBETYPE_CONNECTIONNAME_PLACEHOLDER_DIAGNOSTICS_COUNTERS_STATEPAUSEDBYPARENT_DIAGNOSTICSLEVEL := 18705,
	OPCUAID_PUBLISHSUBSCRIBETYPE_CONNECTIONNAME_PLACEHOLDER_DIAGNOSTICS_COUNTERS_STATEPAUSEDBYPARENT_TIMEFIRSTCHANGE := 18706,
	OPCUAID_PUBLISHSUBSCRIBETYPE_CONNECTIONNAME_PLACEHOLDER_DIAGNOSTICS_COUNTERS_STATEDISABLEDBYMETHOD := 18707,
	OPCUAID_PUBLISHSUBSCRIBETYPE_CONNECTIONNAME_PLACEHOLDER_DIAGNOSTICS_COUNTERS_STATEDISABLEDBYMETHOD_ACTIVE := 18708,
	OPCUAID_PUBLISHSUBSCRIBETYPE_CONNECTIONNAME_PLACEHOLDER_DIAGNOSTICS_COUNTERS_STATEDISABLEDBYMETHOD_CLASSIFICATION := 18709,
	OPCUAID_PUBLISHSUBSCRIBETYPE_CONNECTIONNAME_PLACEHOLDER_DIAGNOSTICS_COUNTERS_STATEDISABLEDBYMETHOD_DIAGNOSTICSLEVEL := 18710,
	OPCUAID_PUBLISHSUBSCRIBETYPE_CONNECTIONNAME_PLACEHOLDER_DIAGNOSTICS_COUNTERS_STATEDISABLEDBYMETHOD_TIMEFIRSTCHANGE := 18711,
	OPCUAID_PUBLISHSUBSCRIBETYPE_CONNECTIONNAME_PLACEHOLDER_DIAGNOSTICS_LIVEVALUES_RESOLVEDADDRESS := 18713,
	OPCUAID_PUBLISHSUBSCRIBETYPE_CONNECTIONNAME_PLACEHOLDER_DIAGNOSTICS_LIVEVALUES_RESOLVEDADDRESS_DIAGNOSTICSLEVEL := 18714,
	OPCUAID_PUBLISHSUBSCRIBETYPE_CONNECTIONNAME_PLACEHOLDER_ADDWRITERGROUP_INPUTARGUMENTS := 16558,
	OPCUAID_PUBLISHSUBSCRIBETYPE_CONNECTIONNAME_PLACEHOLDER_ADDWRITERGROUP_OUTPUTARGUMENTS := 16559,
	OPCUAID_PUBLISHSUBSCRIBETYPE_CONNECTIONNAME_PLACEHOLDER_ADDREADERGROUP_INPUTARGUMENTS := 16561,
	OPCUAID_PUBLISHSUBSCRIBETYPE_CONNECTIONNAME_PLACEHOLDER_ADDREADERGROUP_OUTPUTARGUMENTS := 16571,
	OPCUAID_PUBLISHSUBSCRIBETYPE_CONNECTIONNAME_PLACEHOLDER_REMOVEGROUP_INPUTARGUMENTS := 14425,
	OPCUAID_PUBLISHSUBSCRIBETYPE_SETSECURITYKEYS_INPUTARGUMENTS := 17297,
	OPCUAID_PUBLISHSUBSCRIBETYPE_ADDCONNECTION_INPUTARGUMENTS := 16599,
	OPCUAID_PUBLISHSUBSCRIBETYPE_ADDCONNECTION_OUTPUTARGUMENTS := 16600,
	OPCUAID_PUBLISHSUBSCRIBETYPE_REMOVECONNECTION_INPUTARGUMENTS := 14433,
	OPCUAID_PUBLISHSUBSCRIBETYPE_PUBLISHEDDATASETS_ADDPUBLISHEDDATAITEMS_INPUTARGUMENTS := 14436,
	OPCUAID_PUBLISHSUBSCRIBETYPE_PUBLISHEDDATASETS_ADDPUBLISHEDDATAITEMS_OUTPUTARGUMENTS := 14437,
	OPCUAID_PUBLISHSUBSCRIBETYPE_PUBLISHEDDATASETS_ADDPUBLISHEDEVENTS_INPUTARGUMENTS := 14439,
	OPCUAID_PUBLISHSUBSCRIBETYPE_PUBLISHEDDATASETS_ADDPUBLISHEDEVENTS_OUTPUTARGUMENTS := 14440,
	OPCUAID_PUBLISHSUBSCRIBETYPE_PUBLISHEDDATASETS_ADDPUBLISHEDDATAITEMSTEMPLATE_INPUTARGUMENTS := 16611,
	OPCUAID_PUBLISHSUBSCRIBETYPE_PUBLISHEDDATASETS_ADDPUBLISHEDDATAITEMSTEMPLATE_OUTPUTARGUMENTS := 16638,
	OPCUAID_PUBLISHSUBSCRIBETYPE_PUBLISHEDDATASETS_ADDPUBLISHEDEVENTSTEMPLATE_INPUTARGUMENTS := 16640,
	OPCUAID_PUBLISHSUBSCRIBETYPE_PUBLISHEDDATASETS_ADDPUBLISHEDEVENTSTEMPLATE_OUTPUTARGUMENTS := 16641,
	OPCUAID_PUBLISHSUBSCRIBETYPE_PUBLISHEDDATASETS_REMOVEPUBLISHEDDATASET_INPUTARGUMENTS := 14442,
	OPCUAID_PUBLISHSUBSCRIBETYPE_PUBLISHEDDATASETS_ADDDATASETFOLDER_INPUTARGUMENTS := 16678,
	OPCUAID_PUBLISHSUBSCRIBETYPE_PUBLISHEDDATASETS_ADDDATASETFOLDER_OUTPUTARGUMENTS := 16679,
	OPCUAID_PUBLISHSUBSCRIBETYPE_PUBLISHEDDATASETS_REMOVEDATASETFOLDER_INPUTARGUMENTS := 16681,
	OPCUAID_PUBLISHSUBSCRIBETYPE_STATUS_STATE := 15845,
	OPCUAID_PUBLISHSUBSCRIBETYPE_DIAGNOSTICS_DIAGNOSTICSLEVEL := 18716,
	OPCUAID_PUBLISHSUBSCRIBETYPE_DIAGNOSTICS_TOTALINFORMATION := 18717,
	OPCUAID_PUBLISHSUBSCRIBETYPE_DIAGNOSTICS_TOTALINFORMATION_ACTIVE := 18718,
	OPCUAID_PUBLISHSUBSCRIBETYPE_DIAGNOSTICS_TOTALINFORMATION_CLASSIFICATION := 18719,
	OPCUAID_PUBLISHSUBSCRIBETYPE_DIAGNOSTICS_TOTALINFORMATION_DIAGNOSTICSLEVEL := 18720,
	OPCUAID_PUBLISHSUBSCRIBETYPE_DIAGNOSTICS_TOTALINFORMATION_TIMEFIRSTCHANGE := 18721,
	OPCUAID_PUBLISHSUBSCRIBETYPE_DIAGNOSTICS_TOTALERROR := 18722,
	OPCUAID_PUBLISHSUBSCRIBETYPE_DIAGNOSTICS_TOTALERROR_ACTIVE := 18723,
	OPCUAID_PUBLISHSUBSCRIBETYPE_DIAGNOSTICS_TOTALERROR_CLASSIFICATION := 18724,
	OPCUAID_PUBLISHSUBSCRIBETYPE_DIAGNOSTICS_TOTALERROR_DIAGNOSTICSLEVEL := 18725,
	OPCUAID_PUBLISHSUBSCRIBETYPE_DIAGNOSTICS_TOTALERROR_TIMEFIRSTCHANGE := 18726,
	OPCUAID_PUBLISHSUBSCRIBETYPE_DIAGNOSTICS_SUBERROR := 18728,
	OPCUAID_PUBLISHSUBSCRIBETYPE_DIAGNOSTICS_COUNTERS_STATEERROR := 18730,
	OPCUAID_PUBLISHSUBSCRIBETYPE_DIAGNOSTICS_COUNTERS_STATEERROR_ACTIVE := 18731,
	OPCUAID_PUBLISHSUBSCRIBETYPE_DIAGNOSTICS_COUNTERS_STATEERROR_CLASSIFICATION := 18732,
	OPCUAID_PUBLISHSUBSCRIBETYPE_DIAGNOSTICS_COUNTERS_STATEERROR_DIAGNOSTICSLEVEL := 18733,
	OPCUAID_PUBLISHSUBSCRIBETYPE_DIAGNOSTICS_COUNTERS_STATEERROR_TIMEFIRSTCHANGE := 18734,
	OPCUAID_PUBLISHSUBSCRIBETYPE_DIAGNOSTICS_COUNTERS_STATEOPERATIONALBYMETHOD := 18735,
	OPCUAID_PUBLISHSUBSCRIBETYPE_DIAGNOSTICS_COUNTERS_STATEOPERATIONALBYMETHOD_ACTIVE := 18736,
	OPCUAID_PUBLISHSUBSCRIBETYPE_DIAGNOSTICS_COUNTERS_STATEOPERATIONALBYMETHOD_CLASSIFICATION := 18737,
	OPCUAID_PUBLISHSUBSCRIBETYPE_DIAGNOSTICS_COUNTERS_STATEOPERATIONALBYMETHOD_DIAGNOSTICSLEVEL := 18738,
	OPCUAID_PUBLISHSUBSCRIBETYPE_DIAGNOSTICS_COUNTERS_STATEOPERATIONALBYMETHOD_TIMEFIRSTCHANGE := 18739,
	OPCUAID_PUBLISHSUBSCRIBETYPE_DIAGNOSTICS_COUNTERS_STATEOPERATIONALBYPARENT := 18740,
	OPCUAID_PUBLISHSUBSCRIBETYPE_DIAGNOSTICS_COUNTERS_STATEOPERATIONALBYPARENT_ACTIVE := 18741,
	OPCUAID_PUBLISHSUBSCRIBETYPE_DIAGNOSTICS_COUNTERS_STATEOPERATIONALBYPARENT_CLASSIFICATION := 18742,
	OPCUAID_PUBLISHSUBSCRIBETYPE_DIAGNOSTICS_COUNTERS_STATEOPERATIONALBYPARENT_DIAGNOSTICSLEVEL := 18743,
	OPCUAID_PUBLISHSUBSCRIBETYPE_DIAGNOSTICS_COUNTERS_STATEOPERATIONALBYPARENT_TIMEFIRSTCHANGE := 18744,
	OPCUAID_PUBLISHSUBSCRIBETYPE_DIAGNOSTICS_COUNTERS_STATEOPERATIONALFROMERROR := 18745,
	OPCUAID_PUBLISHSUBSCRIBETYPE_DIAGNOSTICS_COUNTERS_STATEOPERATIONALFROMERROR_ACTIVE := 18746,
	OPCUAID_PUBLISHSUBSCRIBETYPE_DIAGNOSTICS_COUNTERS_STATEOPERATIONALFROMERROR_CLASSIFICATION := 18747,
	OPCUAID_PUBLISHSUBSCRIBETYPE_DIAGNOSTICS_COUNTERS_STATEOPERATIONALFROMERROR_DIAGNOSTICSLEVEL := 18748,
	OPCUAID_PUBLISHSUBSCRIBETYPE_DIAGNOSTICS_COUNTERS_STATEOPERATIONALFROMERROR_TIMEFIRSTCHANGE := 18749,
	OPCUAID_PUBLISHSUBSCRIBETYPE_DIAGNOSTICS_COUNTERS_STATEPAUSEDBYPARENT := 18750,
	OPCUAID_PUBLISHSUBSCRIBETYPE_DIAGNOSTICS_COUNTERS_STATEPAUSEDBYPARENT_ACTIVE := 18751,
	OPCUAID_PUBLISHSUBSCRIBETYPE_DIAGNOSTICS_COUNTERS_STATEPAUSEDBYPARENT_CLASSIFICATION := 18752,
	OPCUAID_PUBLISHSUBSCRIBETYPE_DIAGNOSTICS_COUNTERS_STATEPAUSEDBYPARENT_DIAGNOSTICSLEVEL := 18753,
	OPCUAID_PUBLISHSUBSCRIBETYPE_DIAGNOSTICS_COUNTERS_STATEPAUSEDBYPARENT_TIMEFIRSTCHANGE := 18754,
	OPCUAID_PUBLISHSUBSCRIBETYPE_DIAGNOSTICS_COUNTERS_STATEDISABLEDBYMETHOD := 18755,
	OPCUAID_PUBLISHSUBSCRIBETYPE_DIAGNOSTICS_COUNTERS_STATEDISABLEDBYMETHOD_ACTIVE := 18756,
	OPCUAID_PUBLISHSUBSCRIBETYPE_DIAGNOSTICS_COUNTERS_STATEDISABLEDBYMETHOD_CLASSIFICATION := 18757,
	OPCUAID_PUBLISHSUBSCRIBETYPE_DIAGNOSTICS_COUNTERS_STATEDISABLEDBYMETHOD_DIAGNOSTICSLEVEL := 18758,
	OPCUAID_PUBLISHSUBSCRIBETYPE_DIAGNOSTICS_COUNTERS_STATEDISABLEDBYMETHOD_TIMEFIRSTCHANGE := 18759,
	OPCUAID_PUBLISHSUBSCRIBETYPE_DIAGNOSTICS_LIVEVALUES_CONFIGUREDDATASETWRITERS := 18761,
	OPCUAID_PUBLISHSUBSCRIBETYPE_DIAGNOSTICS_LIVEVALUES_CONFIGUREDDATASETWRITERS_DIAGNOSTICSLEVEL := 18762,
	OPCUAID_PUBLISHSUBSCRIBETYPE_DIAGNOSTICS_LIVEVALUES_CONFIGUREDDATASETREADERS := 18763,
	OPCUAID_PUBLISHSUBSCRIBETYPE_DIAGNOSTICS_LIVEVALUES_CONFIGUREDDATASETREADERS_DIAGNOSTICSLEVEL := 18764,
	OPCUAID_PUBLISHSUBSCRIBETYPE_DIAGNOSTICS_LIVEVALUES_OPERATIONALDATASETWRITERS := 18765,
	OPCUAID_PUBLISHSUBSCRIBETYPE_DIAGNOSTICS_LIVEVALUES_OPERATIONALDATASETWRITERS_DIAGNOSTICSLEVEL := 18766,
	OPCUAID_PUBLISHSUBSCRIBETYPE_DIAGNOSTICS_LIVEVALUES_OPERATIONALDATASETREADERS := 18767,
	OPCUAID_PUBLISHSUBSCRIBETYPE_DIAGNOSTICS_LIVEVALUES_OPERATIONALDATASETREADERS_DIAGNOSTICSLEVEL := 18768,
	OPCUAID_PUBLISHSUBSCRIBETYPE_SUPPORTEDTRANSPORTPROFILES := 17479,
	OPCUAID_PUBLISHSUBSCRIBE_GETSECURITYKEYS_INPUTARGUMENTS := 15216,
	OPCUAID_PUBLISHSUBSCRIBE_GETSECURITYKEYS_OUTPUTARGUMENTS := 15217,
	OPCUAID_PUBLISHSUBSCRIBE_GETSECURITYGROUP_INPUTARGUMENTS := 15441,
	OPCUAID_PUBLISHSUBSCRIBE_GETSECURITYGROUP_OUTPUTARGUMENTS := 15442,
	OPCUAID_PUBLISHSUBSCRIBE_SECURITYGROUPS_ADDSECURITYGROUP_INPUTARGUMENTS := 15445,
	OPCUAID_PUBLISHSUBSCRIBE_SECURITYGROUPS_ADDSECURITYGROUP_OUTPUTARGUMENTS := 15446,
	OPCUAID_PUBLISHSUBSCRIBE_SECURITYGROUPS_REMOVESECURITYGROUP_INPUTARGUMENTS := 15448,
	OPCUAID_PUBLISHSUBSCRIBE_CONNECTIONNAME_PLACEHOLDER_PUBLISHERID := 15791,
	OPCUAID_PUBLISHSUBSCRIBE_CONNECTIONNAME_PLACEHOLDER_TRANSPORTPROFILEURI := 15792,
	OPCUAID_PUBLISHSUBSCRIBE_CONNECTIONNAME_PLACEHOLDER_TRANSPORTPROFILEURI_SELECTIONS := 15848,
	OPCUAID_PUBLISHSUBSCRIBE_CONNECTIONNAME_PLACEHOLDER_CONNECTIONPROPERTIES := 17480,
	OPCUAID_PUBLISHSUBSCRIBE_CONNECTIONNAME_PLACEHOLDER_ADDRESS_NETWORKINTERFACE := 15863,
	OPCUAID_PUBLISHSUBSCRIBE_CONNECTIONNAME_PLACEHOLDER_STATUS_STATE := 15892,
	OPCUAID_PUBLISHSUBSCRIBE_CONNECTIONNAME_PLACEHOLDER_DIAGNOSTICS_DIAGNOSTICSLEVEL := 15938,
	OPCUAID_PUBLISHSUBSCRIBE_CONNECTIONNAME_PLACEHOLDER_DIAGNOSTICS_TOTALINFORMATION := 15939,
	OPCUAID_PUBLISHSUBSCRIBE_CONNECTIONNAME_PLACEHOLDER_DIAGNOSTICS_TOTALINFORMATION_ACTIVE := 15989,
	OPCUAID_PUBLISHSUBSCRIBE_CONNECTIONNAME_PLACEHOLDER_DIAGNOSTICS_TOTALINFORMATION_CLASSIFICATION := 15994,
	OPCUAID_PUBLISHSUBSCRIBE_CONNECTIONNAME_PLACEHOLDER_DIAGNOSTICS_TOTALINFORMATION_DIAGNOSTICSLEVEL := 16013,
	OPCUAID_PUBLISHSUBSCRIBE_CONNECTIONNAME_PLACEHOLDER_DIAGNOSTICS_TOTALINFORMATION_TIMEFIRSTCHANGE := 16020,
	OPCUAID_PUBLISHSUBSCRIBE_CONNECTIONNAME_PLACEHOLDER_DIAGNOSTICS_TOTALERROR := 16059,
	OPCUAID_PUBLISHSUBSCRIBE_CONNECTIONNAME_PLACEHOLDER_DIAGNOSTICS_TOTALERROR_ACTIVE := 16060,
	OPCUAID_PUBLISHSUBSCRIBE_CONNECTIONNAME_PLACEHOLDER_DIAGNOSTICS_TOTALERROR_CLASSIFICATION := 16061,
	OPCUAID_PUBLISHSUBSCRIBE_CONNECTIONNAME_PLACEHOLDER_DIAGNOSTICS_TOTALERROR_DIAGNOSTICSLEVEL := 16074,
	OPCUAID_PUBLISHSUBSCRIBE_CONNECTIONNAME_PLACEHOLDER_DIAGNOSTICS_TOTALERROR_TIMEFIRSTCHANGE := 16075,
	OPCUAID_PUBLISHSUBSCRIBE_CONNECTIONNAME_PLACEHOLDER_DIAGNOSTICS_SUBERROR := 16101,
	OPCUAID_PUBLISHSUBSCRIBE_CONNECTIONNAME_PLACEHOLDER_DIAGNOSTICS_COUNTERS_STATEERROR := 16103,
	OPCUAID_PUBLISHSUBSCRIBE_CONNECTIONNAME_PLACEHOLDER_DIAGNOSTICS_COUNTERS_STATEERROR_ACTIVE := 16122,
	OPCUAID_PUBLISHSUBSCRIBE_CONNECTIONNAME_PLACEHOLDER_DIAGNOSTICS_COUNTERS_STATEERROR_CLASSIFICATION := 16123,
	OPCUAID_PUBLISHSUBSCRIBE_CONNECTIONNAME_PLACEHOLDER_DIAGNOSTICS_COUNTERS_STATEERROR_DIAGNOSTICSLEVEL := 16124,
	OPCUAID_PUBLISHSUBSCRIBE_CONNECTIONNAME_PLACEHOLDER_DIAGNOSTICS_COUNTERS_STATEERROR_TIMEFIRSTCHANGE := 16160,
	OPCUAID_PUBLISHSUBSCRIBE_CONNECTIONNAME_PLACEHOLDER_DIAGNOSTICS_COUNTERS_STATEOPERATIONALBYMETHOD := 16283,
	OPCUAID_PUBLISHSUBSCRIBE_CONNECTIONNAME_PLACEHOLDER_DIAGNOSTICS_COUNTERS_STATEOPERATIONALBYMETHOD_ACTIVE := 16322,
	OPCUAID_PUBLISHSUBSCRIBE_CONNECTIONNAME_PLACEHOLDER_DIAGNOSTICS_COUNTERS_STATEOPERATIONALBYMETHOD_CLASSIFICATION := 16523,
	OPCUAID_PUBLISHSUBSCRIBE_CONNECTIONNAME_PLACEHOLDER_DIAGNOSTICS_COUNTERS_STATEOPERATIONALBYMETHOD_DIAGNOSTICSLEVEL := 17300,
	OPCUAID_PUBLISHSUBSCRIBE_CONNECTIONNAME_PLACEHOLDER_DIAGNOSTICS_COUNTERS_STATEOPERATIONALBYMETHOD_TIMEFIRSTCHANGE := 17303,
	OPCUAID_PUBLISHSUBSCRIBE_CONNECTIONNAME_PLACEHOLDER_DIAGNOSTICS_COUNTERS_STATEOPERATIONALBYPARENT := 17304,
	OPCUAID_PUBLISHSUBSCRIBE_CONNECTIONNAME_PLACEHOLDER_DIAGNOSTICS_COUNTERS_STATEOPERATIONALBYPARENT_ACTIVE := 17305,
	OPCUAID_PUBLISHSUBSCRIBE_CONNECTIONNAME_PLACEHOLDER_DIAGNOSTICS_COUNTERS_STATEOPERATIONALBYPARENT_CLASSIFICATION := 17320,
	OPCUAID_PUBLISHSUBSCRIBE_CONNECTIONNAME_PLACEHOLDER_DIAGNOSTICS_COUNTERS_STATEOPERATIONALBYPARENT_DIAGNOSTICSLEVEL := 17335,
	OPCUAID_PUBLISHSUBSCRIBE_CONNECTIONNAME_PLACEHOLDER_DIAGNOSTICS_COUNTERS_STATEOPERATIONALBYPARENT_TIMEFIRSTCHANGE := 17336,
	OPCUAID_PUBLISHSUBSCRIBE_CONNECTIONNAME_PLACEHOLDER_DIAGNOSTICS_COUNTERS_STATEOPERATIONALFROMERROR := 17337,
	OPCUAID_PUBLISHSUBSCRIBE_CONNECTIONNAME_PLACEHOLDER_DIAGNOSTICS_COUNTERS_STATEOPERATIONALFROMERROR_ACTIVE := 17338,
	OPCUAID_PUBLISHSUBSCRIBE_CONNECTIONNAME_PLACEHOLDER_DIAGNOSTICS_COUNTERS_STATEOPERATIONALFROMERROR_CLASSIFICATION := 17339,
	OPCUAID_PUBLISHSUBSCRIBE_CONNECTIONNAME_PLACEHOLDER_DIAGNOSTICS_COUNTERS_STATEOPERATIONALFROMERROR_DIAGNOSTICSLEVEL := 17340,
	OPCUAID_PUBLISHSUBSCRIBE_CONNECTIONNAME_PLACEHOLDER_DIAGNOSTICS_COUNTERS_STATEOPERATIONALFROMERROR_TIMEFIRSTCHANGE := 17341,
	OPCUAID_PUBLISHSUBSCRIBE_CONNECTIONNAME_PLACEHOLDER_DIAGNOSTICS_COUNTERS_STATEPAUSEDBYPARENT := 17342,
	OPCUAID_PUBLISHSUBSCRIBE_CONNECTIONNAME_PLACEHOLDER_DIAGNOSTICS_COUNTERS_STATEPAUSEDBYPARENT_ACTIVE := 17343,
	OPCUAID_PUBLISHSUBSCRIBE_CONNECTIONNAME_PLACEHOLDER_DIAGNOSTICS_COUNTERS_STATEPAUSEDBYPARENT_CLASSIFICATION := 17344,
	OPCUAID_PUBLISHSUBSCRIBE_CONNECTIONNAME_PLACEHOLDER_DIAGNOSTICS_COUNTERS_STATEPAUSEDBYPARENT_DIAGNOSTICSLEVEL := 17345,
	OPCUAID_PUBLISHSUBSCRIBE_CONNECTIONNAME_PLACEHOLDER_DIAGNOSTICS_COUNTERS_STATEPAUSEDBYPARENT_TIMEFIRSTCHANGE := 17346,
	OPCUAID_PUBLISHSUBSCRIBE_CONNECTIONNAME_PLACEHOLDER_DIAGNOSTICS_COUNTERS_STATEDISABLEDBYMETHOD := 17347,
	OPCUAID_PUBLISHSUBSCRIBE_CONNECTIONNAME_PLACEHOLDER_DIAGNOSTICS_COUNTERS_STATEDISABLEDBYMETHOD_ACTIVE := 17348,
	OPCUAID_PUBLISHSUBSCRIBE_CONNECTIONNAME_PLACEHOLDER_DIAGNOSTICS_COUNTERS_STATEDISABLEDBYMETHOD_CLASSIFICATION := 17349,
	OPCUAID_PUBLISHSUBSCRIBE_CONNECTIONNAME_PLACEHOLDER_DIAGNOSTICS_COUNTERS_STATEDISABLEDBYMETHOD_DIAGNOSTICSLEVEL := 17350,
	OPCUAID_PUBLISHSUBSCRIBE_CONNECTIONNAME_PLACEHOLDER_DIAGNOSTICS_COUNTERS_STATEDISABLEDBYMETHOD_TIMEFIRSTCHANGE := 17351,
	OPCUAID_PUBLISHSUBSCRIBE_CONNECTIONNAME_PLACEHOLDER_DIAGNOSTICS_LIVEVALUES_RESOLVEDADDRESS := 17353,
	OPCUAID_PUBLISHSUBSCRIBE_CONNECTIONNAME_PLACEHOLDER_DIAGNOSTICS_LIVEVALUES_RESOLVEDADDRESS_DIAGNOSTICSLEVEL := 17354,
	OPCUAID_PUBLISHSUBSCRIBE_CONNECTIONNAME_PLACEHOLDER_ADDWRITERGROUP_INPUTARGUMENTS := 17357,
	OPCUAID_PUBLISHSUBSCRIBE_CONNECTIONNAME_PLACEHOLDER_ADDWRITERGROUP_OUTPUTARGUMENTS := 17358,
	OPCUAID_PUBLISHSUBSCRIBE_CONNECTIONNAME_PLACEHOLDER_ADDREADERGROUP_INPUTARGUMENTS := 17360,
	OPCUAID_PUBLISHSUBSCRIBE_CONNECTIONNAME_PLACEHOLDER_ADDREADERGROUP_OUTPUTARGUMENTS := 17361,
	OPCUAID_PUBLISHSUBSCRIBE_CONNECTIONNAME_PLACEHOLDER_REMOVEGROUP_INPUTARGUMENTS := 17363,
	OPCUAID_PUBLISHSUBSCRIBE_SETSECURITYKEYS_INPUTARGUMENTS := 17365,
	OPCUAID_PUBLISHSUBSCRIBE_ADDCONNECTION_INPUTARGUMENTS := 17367,
	OPCUAID_PUBLISHSUBSCRIBE_ADDCONNECTION_OUTPUTARGUMENTS := 17368,
	OPCUAID_PUBLISHSUBSCRIBE_REMOVECONNECTION_INPUTARGUMENTS := 17370,
	OPCUAID_PUBLISHSUBSCRIBE_PUBLISHEDDATASETS_ADDPUBLISHEDDATAITEMS_INPUTARGUMENTS := 17373,
	OPCUAID_PUBLISHSUBSCRIBE_PUBLISHEDDATASETS_ADDPUBLISHEDDATAITEMS_OUTPUTARGUMENTS := 17374,
	OPCUAID_PUBLISHSUBSCRIBE_PUBLISHEDDATASETS_ADDPUBLISHEDEVENTS_INPUTARGUMENTS := 17376,
	OPCUAID_PUBLISHSUBSCRIBE_PUBLISHEDDATASETS_ADDPUBLISHEDEVENTS_OUTPUTARGUMENTS := 17377,
	OPCUAID_PUBLISHSUBSCRIBE_PUBLISHEDDATASETS_ADDPUBLISHEDDATAITEMSTEMPLATE_INPUTARGUMENTS := 17379,
	OPCUAID_PUBLISHSUBSCRIBE_PUBLISHEDDATASETS_ADDPUBLISHEDDATAITEMSTEMPLATE_OUTPUTARGUMENTS := 17380,
	OPCUAID_PUBLISHSUBSCRIBE_PUBLISHEDDATASETS_ADDPUBLISHEDEVENTSTEMPLATE_INPUTARGUMENTS := 17382,
	OPCUAID_PUBLISHSUBSCRIBE_PUBLISHEDDATASETS_ADDPUBLISHEDEVENTSTEMPLATE_OUTPUTARGUMENTS := 17383,
	OPCUAID_PUBLISHSUBSCRIBE_PUBLISHEDDATASETS_REMOVEPUBLISHEDDATASET_INPUTARGUMENTS := 17385,
	OPCUAID_PUBLISHSUBSCRIBE_PUBLISHEDDATASETS_ADDDATASETFOLDER_INPUTARGUMENTS := 17401,
	OPCUAID_PUBLISHSUBSCRIBE_PUBLISHEDDATASETS_ADDDATASETFOLDER_OUTPUTARGUMENTS := 17402,
	OPCUAID_PUBLISHSUBSCRIBE_PUBLISHEDDATASETS_REMOVEDATASETFOLDER_INPUTARGUMENTS := 17404,
	OPCUAID_PUBLISHSUBSCRIBE_STATUS_STATE := 17406,
	OPCUAID_PUBLISHSUBSCRIBE_DIAGNOSTICS_DIAGNOSTICSLEVEL := 17410,
	OPCUAID_PUBLISHSUBSCRIBE_DIAGNOSTICS_TOTALINFORMATION := 17411,
	OPCUAID_PUBLISHSUBSCRIBE_DIAGNOSTICS_TOTALINFORMATION_ACTIVE := 17412,
	OPCUAID_PUBLISHSUBSCRIBE_DIAGNOSTICS_TOTALINFORMATION_CLASSIFICATION := 17413,
	OPCUAID_PUBLISHSUBSCRIBE_DIAGNOSTICS_TOTALINFORMATION_DIAGNOSTICSLEVEL := 17414,
	OPCUAID_PUBLISHSUBSCRIBE_DIAGNOSTICS_TOTALINFORMATION_TIMEFIRSTCHANGE := 17415,
	OPCUAID_PUBLISHSUBSCRIBE_DIAGNOSTICS_TOTALERROR := 17416,
	OPCUAID_PUBLISHSUBSCRIBE_DIAGNOSTICS_TOTALERROR_ACTIVE := 17417,
	OPCUAID_PUBLISHSUBSCRIBE_DIAGNOSTICS_TOTALERROR_CLASSIFICATION := 17418,
	OPCUAID_PUBLISHSUBSCRIBE_DIAGNOSTICS_TOTALERROR_DIAGNOSTICSLEVEL := 17419,
	OPCUAID_PUBLISHSUBSCRIBE_DIAGNOSTICS_TOTALERROR_TIMEFIRSTCHANGE := 17420,
	OPCUAID_PUBLISHSUBSCRIBE_DIAGNOSTICS_SUBERROR := 17422,
	OPCUAID_PUBLISHSUBSCRIBE_DIAGNOSTICS_COUNTERS_STATEERROR := 17424,
	OPCUAID_PUBLISHSUBSCRIBE_DIAGNOSTICS_COUNTERS_STATEERROR_ACTIVE := 17425,
	OPCUAID_PUBLISHSUBSCRIBE_DIAGNOSTICS_COUNTERS_STATEERROR_CLASSIFICATION := 17426,
	OPCUAID_PUBLISHSUBSCRIBE_DIAGNOSTICS_COUNTERS_STATEERROR_DIAGNOSTICSLEVEL := 17429,
	OPCUAID_PUBLISHSUBSCRIBE_DIAGNOSTICS_COUNTERS_STATEERROR_TIMEFIRSTCHANGE := 17430,
	OPCUAID_PUBLISHSUBSCRIBE_DIAGNOSTICS_COUNTERS_STATEOPERATIONALBYMETHOD := 17431,
	OPCUAID_PUBLISHSUBSCRIBE_DIAGNOSTICS_COUNTERS_STATEOPERATIONALBYMETHOD_ACTIVE := 17432,
	OPCUAID_PUBLISHSUBSCRIBE_DIAGNOSTICS_COUNTERS_STATEOPERATIONALBYMETHOD_CLASSIFICATION := 17433,
	OPCUAID_PUBLISHSUBSCRIBE_DIAGNOSTICS_COUNTERS_STATEOPERATIONALBYMETHOD_DIAGNOSTICSLEVEL := 17434,
	OPCUAID_PUBLISHSUBSCRIBE_DIAGNOSTICS_COUNTERS_STATEOPERATIONALBYMETHOD_TIMEFIRSTCHANGE := 17435,
	OPCUAID_PUBLISHSUBSCRIBE_DIAGNOSTICS_COUNTERS_STATEOPERATIONALBYPARENT := 17436,
	OPCUAID_PUBLISHSUBSCRIBE_DIAGNOSTICS_COUNTERS_STATEOPERATIONALBYPARENT_ACTIVE := 17437,
	OPCUAID_PUBLISHSUBSCRIBE_DIAGNOSTICS_COUNTERS_STATEOPERATIONALBYPARENT_CLASSIFICATION := 17438,
	OPCUAID_PUBLISHSUBSCRIBE_DIAGNOSTICS_COUNTERS_STATEOPERATIONALBYPARENT_DIAGNOSTICSLEVEL := 17439,
	OPCUAID_PUBLISHSUBSCRIBE_DIAGNOSTICS_COUNTERS_STATEOPERATIONALBYPARENT_TIMEFIRSTCHANGE := 17440,
	OPCUAID_PUBLISHSUBSCRIBE_DIAGNOSTICS_COUNTERS_STATEOPERATIONALFROMERROR := 17441,
	OPCUAID_PUBLISHSUBSCRIBE_DIAGNOSTICS_COUNTERS_STATEOPERATIONALFROMERROR_ACTIVE := 17442,
	OPCUAID_PUBLISHSUBSCRIBE_DIAGNOSTICS_COUNTERS_STATEOPERATIONALFROMERROR_CLASSIFICATION := 17443,
	OPCUAID_PUBLISHSUBSCRIBE_DIAGNOSTICS_COUNTERS_STATEOPERATIONALFROMERROR_DIAGNOSTICSLEVEL := 17444,
	OPCUAID_PUBLISHSUBSCRIBE_DIAGNOSTICS_COUNTERS_STATEOPERATIONALFROMERROR_TIMEFIRSTCHANGE := 17445,
	OPCUAID_PUBLISHSUBSCRIBE_DIAGNOSTICS_COUNTERS_STATEPAUSEDBYPARENT := 17446,
	OPCUAID_PUBLISHSUBSCRIBE_DIAGNOSTICS_COUNTERS_STATEPAUSEDBYPARENT_ACTIVE := 17447,
	OPCUAID_PUBLISHSUBSCRIBE_DIAGNOSTICS_COUNTERS_STATEPAUSEDBYPARENT_CLASSIFICATION := 17448,
	OPCUAID_PUBLISHSUBSCRIBE_DIAGNOSTICS_COUNTERS_STATEPAUSEDBYPARENT_DIAGNOSTICSLEVEL := 17449,
	OPCUAID_PUBLISHSUBSCRIBE_DIAGNOSTICS_COUNTERS_STATEPAUSEDBYPARENT_TIMEFIRSTCHANGE := 17450,
	OPCUAID_PUBLISHSUBSCRIBE_DIAGNOSTICS_COUNTERS_STATEDISABLEDBYMETHOD := 17451,
	OPCUAID_PUBLISHSUBSCRIBE_DIAGNOSTICS_COUNTERS_STATEDISABLEDBYMETHOD_ACTIVE := 17452,
	OPCUAID_PUBLISHSUBSCRIBE_DIAGNOSTICS_COUNTERS_STATEDISABLEDBYMETHOD_CLASSIFICATION := 17453,
	OPCUAID_PUBLISHSUBSCRIBE_DIAGNOSTICS_COUNTERS_STATEDISABLEDBYMETHOD_DIAGNOSTICSLEVEL := 17454,
	OPCUAID_PUBLISHSUBSCRIBE_DIAGNOSTICS_COUNTERS_STATEDISABLEDBYMETHOD_TIMEFIRSTCHANGE := 17455,
	OPCUAID_PUBLISHSUBSCRIBE_DIAGNOSTICS_LIVEVALUES_CONFIGUREDDATASETWRITERS := 17458,
	OPCUAID_PUBLISHSUBSCRIBE_DIAGNOSTICS_LIVEVALUES_CONFIGUREDDATASETWRITERS_DIAGNOSTICSLEVEL := 17459,
	OPCUAID_PUBLISHSUBSCRIBE_DIAGNOSTICS_LIVEVALUES_CONFIGUREDDATASETREADERS := 17460,
	OPCUAID_PUBLISHSUBSCRIBE_DIAGNOSTICS_LIVEVALUES_CONFIGUREDDATASETREADERS_DIAGNOSTICSLEVEL := 17461,
	OPCUAID_PUBLISHSUBSCRIBE_DIAGNOSTICS_LIVEVALUES_OPERATIONALDATASETWRITERS := 17462,
	OPCUAID_PUBLISHSUBSCRIBE_DIAGNOSTICS_LIVEVALUES_OPERATIONALDATASETWRITERS_DIAGNOSTICSLEVEL := 17463,
	OPCUAID_PUBLISHSUBSCRIBE_DIAGNOSTICS_LIVEVALUES_OPERATIONALDATASETREADERS := 17464,
	OPCUAID_PUBLISHSUBSCRIBE_DIAGNOSTICS_LIVEVALUES_OPERATIONALDATASETREADERS_DIAGNOSTICSLEVEL := 17466,
	OPCUAID_PUBLISHSUBSCRIBE_SUPPORTEDTRANSPORTPROFILES := 17481,
	OPCUAID_PUBLISHEDDATASETTYPE_DATASETWRITERNAME_PLACEHOLDER_DATASETWRITERID := 16720,
	OPCUAID_PUBLISHEDDATASETTYPE_DATASETWRITERNAME_PLACEHOLDER_DATASETFIELDCONTENTMASK := 16721,
	OPCUAID_PUBLISHEDDATASETTYPE_DATASETWRITERNAME_PLACEHOLDER_DATASETWRITERPROPERTIES := 17482,
	OPCUAID_PUBLISHEDDATASETTYPE_DATASETWRITERNAME_PLACEHOLDER_STATUS_STATE := 15224,
	OPCUAID_PUBLISHEDDATASETTYPE_DATASETWRITERNAME_PLACEHOLDER_DIAGNOSTICS_DIAGNOSTICSLEVEL := 18872,
	OPCUAID_PUBLISHEDDATASETTYPE_DATASETWRITERNAME_PLACEHOLDER_DIAGNOSTICS_TOTALINFORMATION := 18873,
	OPCUAID_PUBLISHEDDATASETTYPE_DATASETWRITERNAME_PLACEHOLDER_DIAGNOSTICS_TOTALINFORMATION_ACTIVE := 18874,
	OPCUAID_PUBLISHEDDATASETTYPE_DATASETWRITERNAME_PLACEHOLDER_DIAGNOSTICS_TOTALINFORMATION_CLASSIFICATION := 18875,
	OPCUAID_PUBLISHEDDATASETTYPE_DATASETWRITERNAME_PLACEHOLDER_DIAGNOSTICS_TOTALINFORMATION_DIAGNOSTICSLEVEL := 18876,
	OPCUAID_PUBLISHEDDATASETTYPE_DATASETWRITERNAME_PLACEHOLDER_DIAGNOSTICS_TOTALINFORMATION_TIMEFIRSTCHANGE := 18877,
	OPCUAID_PUBLISHEDDATASETTYPE_DATASETWRITERNAME_PLACEHOLDER_DIAGNOSTICS_TOTALERROR := 18878,
	OPCUAID_PUBLISHEDDATASETTYPE_DATASETWRITERNAME_PLACEHOLDER_DIAGNOSTICS_TOTALERROR_ACTIVE := 18879,
	OPCUAID_PUBLISHEDDATASETTYPE_DATASETWRITERNAME_PLACEHOLDER_DIAGNOSTICS_TOTALERROR_CLASSIFICATION := 18880,
	OPCUAID_PUBLISHEDDATASETTYPE_DATASETWRITERNAME_PLACEHOLDER_DIAGNOSTICS_TOTALERROR_DIAGNOSTICSLEVEL := 18881,
	OPCUAID_PUBLISHEDDATASETTYPE_DATASETWRITERNAME_PLACEHOLDER_DIAGNOSTICS_TOTALERROR_TIMEFIRSTCHANGE := 18882,
	OPCUAID_PUBLISHEDDATASETTYPE_DATASETWRITERNAME_PLACEHOLDER_DIAGNOSTICS_SUBERROR := 18884,
	OPCUAID_PUBLISHEDDATASETTYPE_DATASETWRITERNAME_PLACEHOLDER_DIAGNOSTICS_COUNTERS_STATEERROR := 18886,
	OPCUAID_PUBLISHEDDATASETTYPE_DATASETWRITERNAME_PLACEHOLDER_DIAGNOSTICS_COUNTERS_STATEERROR_ACTIVE := 18887,
	OPCUAID_PUBLISHEDDATASETTYPE_DATASETWRITERNAME_PLACEHOLDER_DIAGNOSTICS_COUNTERS_STATEERROR_CLASSIFICATION := 18888,
	OPCUAID_PUBLISHEDDATASETTYPE_DATASETWRITERNAME_PLACEHOLDER_DIAGNOSTICS_COUNTERS_STATEERROR_DIAGNOSTICSLEVEL := 18889,
	OPCUAID_PUBLISHEDDATASETTYPE_DATASETWRITERNAME_PLACEHOLDER_DIAGNOSTICS_COUNTERS_STATEERROR_TIMEFIRSTCHANGE := 18890,
	OPCUAID_PUBLISHEDDATASETTYPE_DATASETWRITERNAME_PLACEHOLDER_DIAGNOSTICS_COUNTERS_STATEOPERATIONALBYMETHOD := 18891,
	OPCUAID_PUBLISHEDDATASETTYPE_DATASETWRITERNAME_PLACEHOLDER_DIAGNOSTICS_COUNTERS_STATEOPERATIONALBYMETHOD_ACTIVE := 18892,
	OPCUAID_PUBLISHEDDATASETTYPE_DATASETWRITERNAME_PLACEHOLDER_DIAGNOSTICS_COUNTERS_STATEOPERATIONALBYMETHOD_CLASSIFICATION := 18893,
	OPCUAID_PUBLISHEDDATASETTYPE_DATASETWRITERNAME_PLACEHOLDER_DIAGNOSTICS_COUNTERS_STATEOPERATIONALBYMETHOD_DIAGNOSTICSLEVEL := 18894,
	OPCUAID_PUBLISHEDDATASETTYPE_DATASETWRITERNAME_PLACEHOLDER_DIAGNOSTICS_COUNTERS_STATEOPERATIONALBYMETHOD_TIMEFIRSTCHANGE := 18895,
	OPCUAID_PUBLISHEDDATASETTYPE_DATASETWRITERNAME_PLACEHOLDER_DIAGNOSTICS_COUNTERS_STATEOPERATIONALBYPARENT := 18896,
	OPCUAID_PUBLISHEDDATASETTYPE_DATASETWRITERNAME_PLACEHOLDER_DIAGNOSTICS_COUNTERS_STATEOPERATIONALBYPARENT_ACTIVE := 18897,
	OPCUAID_PUBLISHEDDATASETTYPE_DATASETWRITERNAME_PLACEHOLDER_DIAGNOSTICS_COUNTERS_STATEOPERATIONALBYPARENT_CLASSIFICATION := 18898,
	OPCUAID_PUBLISHEDDATASETTYPE_DATASETWRITERNAME_PLACEHOLDER_DIAGNOSTICS_COUNTERS_STATEOPERATIONALBYPARENT_DIAGNOSTICSLEVEL := 18899,
	OPCUAID_PUBLISHEDDATASETTYPE_DATASETWRITERNAME_PLACEHOLDER_DIAGNOSTICS_COUNTERS_STATEOPERATIONALBYPARENT_TIMEFIRSTCHANGE := 18900,
	OPCUAID_PUBLISHEDDATASETTYPE_DATASETWRITERNAME_PLACEHOLDER_DIAGNOSTICS_COUNTERS_STATEOPERATIONALFROMERROR := 18901,
	OPCUAID_PUBLISHEDDATASETTYPE_DATASETWRITERNAME_PLACEHOLDER_DIAGNOSTICS_COUNTERS_STATEOPERATIONALFROMERROR_ACTIVE := 18902,
	OPCUAID_PUBLISHEDDATASETTYPE_DATASETWRITERNAME_PLACEHOLDER_DIAGNOSTICS_COUNTERS_STATEOPERATIONALFROMERROR_CLASSIFICATION := 18903,
	OPCUAID_PUBLISHEDDATASETTYPE_DATASETWRITERNAME_PLACEHOLDER_DIAGNOSTICS_COUNTERS_STATEOPERATIONALFROMERROR_DIAGNOSTICSLEVEL := 18904,
	OPCUAID_PUBLISHEDDATASETTYPE_DATASETWRITERNAME_PLACEHOLDER_DIAGNOSTICS_COUNTERS_STATEOPERATIONALFROMERROR_TIMEFIRSTCHANGE := 18905,
	OPCUAID_PUBLISHEDDATASETTYPE_DATASETWRITERNAME_PLACEHOLDER_DIAGNOSTICS_COUNTERS_STATEPAUSEDBYPARENT := 18906,
	OPCUAID_PUBLISHEDDATASETTYPE_DATASETWRITERNAME_PLACEHOLDER_DIAGNOSTICS_COUNTERS_STATEPAUSEDBYPARENT_ACTIVE := 18907,
	OPCUAID_PUBLISHEDDATASETTYPE_DATASETWRITERNAME_PLACEHOLDER_DIAGNOSTICS_COUNTERS_STATEPAUSEDBYPARENT_CLASSIFICATION := 18908,
	OPCUAID_PUBLISHEDDATASETTYPE_DATASETWRITERNAME_PLACEHOLDER_DIAGNOSTICS_COUNTERS_STATEPAUSEDBYPARENT_DIAGNOSTICSLEVEL := 18909,
	OPCUAID_PUBLISHEDDATASETTYPE_DATASETWRITERNAME_PLACEHOLDER_DIAGNOSTICS_COUNTERS_STATEPAUSEDBYPARENT_TIMEFIRSTCHANGE := 18910,
	OPCUAID_PUBLISHEDDATASETTYPE_DATASETWRITERNAME_PLACEHOLDER_DIAGNOSTICS_COUNTERS_STATEDISABLEDBYMETHOD := 18911,
	OPCUAID_PUBLISHEDDATASETTYPE_DATASETWRITERNAME_PLACEHOLDER_DIAGNOSTICS_COUNTERS_STATEDISABLEDBYMETHOD_ACTIVE := 18912,
	OPCUAID_PUBLISHEDDATASETTYPE_DATASETWRITERNAME_PLACEHOLDER_DIAGNOSTICS_COUNTERS_STATEDISABLEDBYMETHOD_CLASSIFICATION := 18913,
	OPCUAID_PUBLISHEDDATASETTYPE_DATASETWRITERNAME_PLACEHOLDER_DIAGNOSTICS_COUNTERS_STATEDISABLEDBYMETHOD_DIAGNOSTICSLEVEL := 18914,
	OPCUAID_PUBLISHEDDATASETTYPE_DATASETWRITERNAME_PLACEHOLDER_DIAGNOSTICS_COUNTERS_STATEDISABLEDBYMETHOD_TIMEFIRSTCHANGE := 18915,
	OPCUAID_PUBLISHEDDATASETTYPE_DATASETWRITERNAME_PLACEHOLDER_DIAGNOSTICS_COUNTERS_FAILEDDATASETMESSAGES := 18917,
	OPCUAID_PUBLISHEDDATASETTYPE_DATASETWRITERNAME_PLACEHOLDER_DIAGNOSTICS_COUNTERS_FAILEDDATASETMESSAGES_ACTIVE := 18918,
	OPCUAID_PUBLISHEDDATASETTYPE_DATASETWRITERNAME_PLACEHOLDER_DIAGNOSTICS_COUNTERS_FAILEDDATASETMESSAGES_CLASSIFICATION := 18919,
	OPCUAID_PUBLISHEDDATASETTYPE_DATASETWRITERNAME_PLACEHOLDER_DIAGNOSTICS_COUNTERS_FAILEDDATASETMESSAGES_DIAGNOSTICSLEVEL := 18920,
	OPCUAID_PUBLISHEDDATASETTYPE_DATASETWRITERNAME_PLACEHOLDER_DIAGNOSTICS_COUNTERS_FAILEDDATASETMESSAGES_TIMEFIRSTCHANGE := 18921,
	OPCUAID_PUBLISHEDDATASETTYPE_DATASETWRITERNAME_PLACEHOLDER_DIAGNOSTICS_LIVEVALUES_MESSAGESEQUENCENUMBER_DIAGNOSTICSLEVEL := 18923,
	OPCUAID_PUBLISHEDDATASETTYPE_DATASETWRITERNAME_PLACEHOLDER_DIAGNOSTICS_LIVEVALUES_STATUSCODE_DIAGNOSTICSLEVEL := 18925,
	OPCUAID_PUBLISHEDDATASETTYPE_DATASETWRITERNAME_PLACEHOLDER_DIAGNOSTICS_LIVEVALUES_MAJORVERSION_DIAGNOSTICSLEVEL := 18927,
	OPCUAID_PUBLISHEDDATASETTYPE_DATASETWRITERNAME_PLACEHOLDER_DIAGNOSTICS_LIVEVALUES_MINORVERSION_DIAGNOSTICSLEVEL := 18929,
	OPCUAID_PUBLISHEDDATASETTYPE_CONFIGURATIONVERSION := 14519,
	OPCUAID_PUBLISHEDDATASETTYPE_DATASETMETADATA := 15229,
	OPCUAID_PUBLISHEDDATASETTYPE_DATASETCLASSID := 16759,
	OPCUAID_PUBLISHEDDATASETTYPE_EXTENSIONFIELDS_ADDEXTENSIONFIELD_INPUTARGUMENTS := 15483,
	OPCUAID_PUBLISHEDDATASETTYPE_EXTENSIONFIELDS_ADDEXTENSIONFIELD_OUTPUTARGUMENTS := 15484,
	OPCUAID_PUBLISHEDDATASETTYPE_EXTENSIONFIELDS_REMOVEEXTENSIONFIELD_INPUTARGUMENTS := 15486,
	OPCUAID_EXTENSIONFIELDSTYPE_EXTENSIONFIELDNAME_PLACEHOLDER := 15490,
	OPCUAID_EXTENSIONFIELDSTYPE_ADDEXTENSIONFIELD_INPUTARGUMENTS := 15492,
	OPCUAID_EXTENSIONFIELDSTYPE_ADDEXTENSIONFIELD_OUTPUTARGUMENTS := 15493,
	OPCUAID_EXTENSIONFIELDSTYPE_REMOVEEXTENSIONFIELD_INPUTARGUMENTS := 15495,
	OPCUAID_PUBLISHEDDATAITEMSTYPE_DATASETWRITERNAME_PLACEHOLDER_DATASETWRITERID := 16760,
	OPCUAID_PUBLISHEDDATAITEMSTYPE_DATASETWRITERNAME_PLACEHOLDER_DATASETFIELDCONTENTMASK := 16761,
	OPCUAID_PUBLISHEDDATAITEMSTYPE_DATASETWRITERNAME_PLACEHOLDER_DATASETWRITERPROPERTIES := 17483,
	OPCUAID_PUBLISHEDDATAITEMSTYPE_DATASETWRITERNAME_PLACEHOLDER_STATUS_STATE := 15232,
	OPCUAID_PUBLISHEDDATAITEMSTYPE_DATASETWRITERNAME_PLACEHOLDER_DIAGNOSTICS_DIAGNOSTICSLEVEL := 18931,
	OPCUAID_PUBLISHEDDATAITEMSTYPE_DATASETWRITERNAME_PLACEHOLDER_DIAGNOSTICS_TOTALINFORMATION := 18932,
	OPCUAID_PUBLISHEDDATAITEMSTYPE_DATASETWRITERNAME_PLACEHOLDER_DIAGNOSTICS_TOTALINFORMATION_ACTIVE := 18933,
	OPCUAID_PUBLISHEDDATAITEMSTYPE_DATASETWRITERNAME_PLACEHOLDER_DIAGNOSTICS_TOTALINFORMATION_CLASSIFICATION := 18934,
	OPCUAID_PUBLISHEDDATAITEMSTYPE_DATASETWRITERNAME_PLACEHOLDER_DIAGNOSTICS_TOTALINFORMATION_DIAGNOSTICSLEVEL := 18935,
	OPCUAID_PUBLISHEDDATAITEMSTYPE_DATASETWRITERNAME_PLACEHOLDER_DIAGNOSTICS_TOTALINFORMATION_TIMEFIRSTCHANGE := 18936,
	OPCUAID_PUBLISHEDDATAITEMSTYPE_DATASETWRITERNAME_PLACEHOLDER_DIAGNOSTICS_TOTALERROR := 18937,
	OPCUAID_PUBLISHEDDATAITEMSTYPE_DATASETWRITERNAME_PLACEHOLDER_DIAGNOSTICS_TOTALERROR_ACTIVE := 18938,
	OPCUAID_PUBLISHEDDATAITEMSTYPE_DATASETWRITERNAME_PLACEHOLDER_DIAGNOSTICS_TOTALERROR_CLASSIFICATION := 18939,
	OPCUAID_PUBLISHEDDATAITEMSTYPE_DATASETWRITERNAME_PLACEHOLDER_DIAGNOSTICS_TOTALERROR_DIAGNOSTICSLEVEL := 18940,
	OPCUAID_PUBLISHEDDATAITEMSTYPE_DATASETWRITERNAME_PLACEHOLDER_DIAGNOSTICS_TOTALERROR_TIMEFIRSTCHANGE := 18941,
	OPCUAID_PUBLISHEDDATAITEMSTYPE_DATASETWRITERNAME_PLACEHOLDER_DIAGNOSTICS_SUBERROR := 18943,
	OPCUAID_PUBLISHEDDATAITEMSTYPE_DATASETWRITERNAME_PLACEHOLDER_DIAGNOSTICS_COUNTERS_STATEERROR := 18945,
	OPCUAID_PUBLISHEDDATAITEMSTYPE_DATASETWRITERNAME_PLACEHOLDER_DIAGNOSTICS_COUNTERS_STATEERROR_ACTIVE := 18946,
	OPCUAID_PUBLISHEDDATAITEMSTYPE_DATASETWRITERNAME_PLACEHOLDER_DIAGNOSTICS_COUNTERS_STATEERROR_CLASSIFICATION := 18947,
	OPCUAID_PUBLISHEDDATAITEMSTYPE_DATASETWRITERNAME_PLACEHOLDER_DIAGNOSTICS_COUNTERS_STATEERROR_DIAGNOSTICSLEVEL := 18948,
	OPCUAID_PUBLISHEDDATAITEMSTYPE_DATASETWRITERNAME_PLACEHOLDER_DIAGNOSTICS_COUNTERS_STATEERROR_TIMEFIRSTCHANGE := 18949,
	OPCUAID_PUBLISHEDDATAITEMSTYPE_DATASETWRITERNAME_PLACEHOLDER_DIAGNOSTICS_COUNTERS_STATEOPERATIONALBYMETHOD := 18950,
	OPCUAID_PUBLISHEDDATAITEMSTYPE_DATASETWRITERNAME_PLACEHOLDER_DIAGNOSTICS_COUNTERS_STATEOPERATIONALBYMETHOD_ACTIVE := 18951,
	OPCUAID_PUBLISHEDDATAITEMSTYPE_DATASETWRITERNAME_PLACEHOLDER_DIAGNOSTICS_COUNTERS_STATEOPERATIONALBYMETHOD_CLASSIFICATION := 18952,
	OPCUAID_PUBLISHEDDATAITEMSTYPE_DATASETWRITERNAME_PLACEHOLDER_DIAGNOSTICS_COUNTERS_STATEOPERATIONALBYMETHOD_DIAGNOSTICSLEVEL := 18953,
	OPCUAID_PUBLISHEDDATAITEMSTYPE_DATASETWRITERNAME_PLACEHOLDER_DIAGNOSTICS_COUNTERS_STATEOPERATIONALBYMETHOD_TIMEFIRSTCHANGE := 18954,
	OPCUAID_PUBLISHEDDATAITEMSTYPE_DATASETWRITERNAME_PLACEHOLDER_DIAGNOSTICS_COUNTERS_STATEOPERATIONALBYPARENT := 18955,
	OPCUAID_PUBLISHEDDATAITEMSTYPE_DATASETWRITERNAME_PLACEHOLDER_DIAGNOSTICS_COUNTERS_STATEOPERATIONALBYPARENT_ACTIVE := 18956,
	OPCUAID_PUBLISHEDDATAITEMSTYPE_DATASETWRITERNAME_PLACEHOLDER_DIAGNOSTICS_COUNTERS_STATEOPERATIONALBYPARENT_CLASSIFICATION := 18957,
	OPCUAID_PUBLISHEDDATAITEMSTYPE_DATASETWRITERNAME_PLACEHOLDER_DIAGNOSTICS_COUNTERS_STATEOPERATIONALBYPARENT_DIAGNOSTICSLEVEL := 18958,
	OPCUAID_PUBLISHEDDATAITEMSTYPE_DATASETWRITERNAME_PLACEHOLDER_DIAGNOSTICS_COUNTERS_STATEOPERATIONALBYPARENT_TIMEFIRSTCHANGE := 18959,
	OPCUAID_PUBLISHEDDATAITEMSTYPE_DATASETWRITERNAME_PLACEHOLDER_DIAGNOSTICS_COUNTERS_STATEOPERATIONALFROMERROR := 18960,
	OPCUAID_PUBLISHEDDATAITEMSTYPE_DATASETWRITERNAME_PLACEHOLDER_DIAGNOSTICS_COUNTERS_STATEOPERATIONALFROMERROR_ACTIVE := 18961,
	OPCUAID_PUBLISHEDDATAITEMSTYPE_DATASETWRITERNAME_PLACEHOLDER_DIAGNOSTICS_COUNTERS_STATEOPERATIONALFROMERROR_CLASSIFICATION := 18962,
	OPCUAID_PUBLISHEDDATAITEMSTYPE_DATASETWRITERNAME_PLACEHOLDER_DIAGNOSTICS_COUNTERS_STATEOPERATIONALFROMERROR_DIAGNOSTICSLEVEL := 18963,
	OPCUAID_PUBLISHEDDATAITEMSTYPE_DATASETWRITERNAME_PLACEHOLDER_DIAGNOSTICS_COUNTERS_STATEOPERATIONALFROMERROR_TIMEFIRSTCHANGE := 18964,
	OPCUAID_PUBLISHEDDATAITEMSTYPE_DATASETWRITERNAME_PLACEHOLDER_DIAGNOSTICS_COUNTERS_STATEPAUSEDBYPARENT := 18965,
	OPCUAID_PUBLISHEDDATAITEMSTYPE_DATASETWRITERNAME_PLACEHOLDER_DIAGNOSTICS_COUNTERS_STATEPAUSEDBYPARENT_ACTIVE := 18966,
	OPCUAID_PUBLISHEDDATAITEMSTYPE_DATASETWRITERNAME_PLACEHOLDER_DIAGNOSTICS_COUNTERS_STATEPAUSEDBYPARENT_CLASSIFICATION := 18967,
	OPCUAID_PUBLISHEDDATAITEMSTYPE_DATASETWRITERNAME_PLACEHOLDER_DIAGNOSTICS_COUNTERS_STATEPAUSEDBYPARENT_DIAGNOSTICSLEVEL := 18968,
	OPCUAID_PUBLISHEDDATAITEMSTYPE_DATASETWRITERNAME_PLACEHOLDER_DIAGNOSTICS_COUNTERS_STATEPAUSEDBYPARENT_TIMEFIRSTCHANGE := 18969,
	OPCUAID_PUBLISHEDDATAITEMSTYPE_DATASETWRITERNAME_PLACEHOLDER_DIAGNOSTICS_COUNTERS_STATEDISABLEDBYMETHOD := 18970,
	OPCUAID_PUBLISHEDDATAITEMSTYPE_DATASETWRITERNAME_PLACEHOLDER_DIAGNOSTICS_COUNTERS_STATEDISABLEDBYMETHOD_ACTIVE := 18971,
	OPCUAID_PUBLISHEDDATAITEMSTYPE_DATASETWRITERNAME_PLACEHOLDER_DIAGNOSTICS_COUNTERS_STATEDISABLEDBYMETHOD_CLASSIFICATION := 18972,
	OPCUAID_PUBLISHEDDATAITEMSTYPE_DATASETWRITERNAME_PLACEHOLDER_DIAGNOSTICS_COUNTERS_STATEDISABLEDBYMETHOD_DIAGNOSTICSLEVEL := 18973,
	OPCUAID_PUBLISHEDDATAITEMSTYPE_DATASETWRITERNAME_PLACEHOLDER_DIAGNOSTICS_COUNTERS_STATEDISABLEDBYMETHOD_TIMEFIRSTCHANGE := 18974,
	OPCUAID_PUBLISHEDDATAITEMSTYPE_DATASETWRITERNAME_PLACEHOLDER_DIAGNOSTICS_COUNTERS_FAILEDDATASETMESSAGES := 18976,
	OPCUAID_PUBLISHEDDATAITEMSTYPE_DATASETWRITERNAME_PLACEHOLDER_DIAGNOSTICS_COUNTERS_FAILEDDATASETMESSAGES_ACTIVE := 18977,
	OPCUAID_PUBLISHEDDATAITEMSTYPE_DATASETWRITERNAME_PLACEHOLDER_DIAGNOSTICS_COUNTERS_FAILEDDATASETMESSAGES_CLASSIFICATION := 18978,
	OPCUAID_PUBLISHEDDATAITEMSTYPE_DATASETWRITERNAME_PLACEHOLDER_DIAGNOSTICS_COUNTERS_FAILEDDATASETMESSAGES_DIAGNOSTICSLEVEL := 18979,
	OPCUAID_PUBLISHEDDATAITEMSTYPE_DATASETWRITERNAME_PLACEHOLDER_DIAGNOSTICS_COUNTERS_FAILEDDATASETMESSAGES_TIMEFIRSTCHANGE := 18980,
	OPCUAID_PUBLISHEDDATAITEMSTYPE_DATASETWRITERNAME_PLACEHOLDER_DIAGNOSTICS_LIVEVALUES_MESSAGESEQUENCENUMBER_DIAGNOSTICSLEVEL := 18982,
	OPCUAID_PUBLISHEDDATAITEMSTYPE_DATASETWRITERNAME_PLACEHOLDER_DIAGNOSTICS_LIVEVALUES_STATUSCODE_DIAGNOSTICSLEVEL := 18984,
	OPCUAID_PUBLISHEDDATAITEMSTYPE_DATASETWRITERNAME_PLACEHOLDER_DIAGNOSTICS_LIVEVALUES_MAJORVERSION_DIAGNOSTICSLEVEL := 18986,
	OPCUAID_PUBLISHEDDATAITEMSTYPE_DATASETWRITERNAME_PLACEHOLDER_DIAGNOSTICS_LIVEVALUES_MINORVERSION_DIAGNOSTICSLEVEL := 18988,
	OPCUAID_PUBLISHEDDATAITEMSTYPE_EXTENSIONFIELDS_ADDEXTENSIONFIELD_INPUTARGUMENTS := 15505,
	OPCUAID_PUBLISHEDDATAITEMSTYPE_EXTENSIONFIELDS_ADDEXTENSIONFIELD_OUTPUTARGUMENTS := 15506,
	OPCUAID_PUBLISHEDDATAITEMSTYPE_EXTENSIONFIELDS_REMOVEEXTENSIONFIELD_INPUTARGUMENTS := 15508,
	OPCUAID_PUBLISHEDDATAITEMSTYPE_PUBLISHEDDATA := 14548,
	OPCUAID_PUBLISHEDDATAITEMSTYPE_ADDVARIABLES_INPUTARGUMENTS := 14556,
	OPCUAID_PUBLISHEDDATAITEMSTYPE_ADDVARIABLES_OUTPUTARGUMENTS := 14557,
	OPCUAID_PUBLISHEDDATAITEMSTYPE_REMOVEVARIABLES_INPUTARGUMENTS := 14559,
	OPCUAID_PUBLISHEDDATAITEMSTYPE_REMOVEVARIABLES_OUTPUTARGUMENTS := 14560,
	OPCUAID_PUBLISHEDEVENTSTYPE_DATASETWRITERNAME_PLACEHOLDER_DATASETWRITERID := 16801,
	OPCUAID_PUBLISHEDEVENTSTYPE_DATASETWRITERNAME_PLACEHOLDER_DATASETFIELDCONTENTMASK := 16802,
	OPCUAID_PUBLISHEDEVENTSTYPE_DATASETWRITERNAME_PLACEHOLDER_DATASETWRITERPROPERTIES := 17484,
	OPCUAID_PUBLISHEDEVENTSTYPE_DATASETWRITERNAME_PLACEHOLDER_STATUS_STATE := 15240,
	OPCUAID_PUBLISHEDEVENTSTYPE_DATASETWRITERNAME_PLACEHOLDER_DIAGNOSTICS_DIAGNOSTICSLEVEL := 18990,
	OPCUAID_PUBLISHEDEVENTSTYPE_DATASETWRITERNAME_PLACEHOLDER_DIAGNOSTICS_TOTALINFORMATION := 18991,
	OPCUAID_PUBLISHEDEVENTSTYPE_DATASETWRITERNAME_PLACEHOLDER_DIAGNOSTICS_TOTALINFORMATION_ACTIVE := 18992,
	OPCUAID_PUBLISHEDEVENTSTYPE_DATASETWRITERNAME_PLACEHOLDER_DIAGNOSTICS_TOTALINFORMATION_CLASSIFICATION := 18993,
	OPCUAID_PUBLISHEDEVENTSTYPE_DATASETWRITERNAME_PLACEHOLDER_DIAGNOSTICS_TOTALINFORMATION_DIAGNOSTICSLEVEL := 18994,
	OPCUAID_PUBLISHEDEVENTSTYPE_DATASETWRITERNAME_PLACEHOLDER_DIAGNOSTICS_TOTALINFORMATION_TIMEFIRSTCHANGE := 18995,
	OPCUAID_PUBLISHEDEVENTSTYPE_DATASETWRITERNAME_PLACEHOLDER_DIAGNOSTICS_TOTALERROR := 18996,
	OPCUAID_PUBLISHEDEVENTSTYPE_DATASETWRITERNAME_PLACEHOLDER_DIAGNOSTICS_TOTALERROR_ACTIVE := 18997,
	OPCUAID_PUBLISHEDEVENTSTYPE_DATASETWRITERNAME_PLACEHOLDER_DIAGNOSTICS_TOTALERROR_CLASSIFICATION := 18998,
	OPCUAID_PUBLISHEDEVENTSTYPE_DATASETWRITERNAME_PLACEHOLDER_DIAGNOSTICS_TOTALERROR_DIAGNOSTICSLEVEL := 18999,
	OPCUAID_PUBLISHEDEVENTSTYPE_DATASETWRITERNAME_PLACEHOLDER_DIAGNOSTICS_TOTALERROR_TIMEFIRSTCHANGE := 19000,
	OPCUAID_PUBLISHEDEVENTSTYPE_DATASETWRITERNAME_PLACEHOLDER_DIAGNOSTICS_SUBERROR := 19002,
	OPCUAID_PUBLISHEDEVENTSTYPE_DATASETWRITERNAME_PLACEHOLDER_DIAGNOSTICS_COUNTERS_STATEERROR := 19004,
	OPCUAID_PUBLISHEDEVENTSTYPE_DATASETWRITERNAME_PLACEHOLDER_DIAGNOSTICS_COUNTERS_STATEERROR_ACTIVE := 19005,
	OPCUAID_PUBLISHEDEVENTSTYPE_DATASETWRITERNAME_PLACEHOLDER_DIAGNOSTICS_COUNTERS_STATEERROR_CLASSIFICATION := 19006,
	OPCUAID_PUBLISHEDEVENTSTYPE_DATASETWRITERNAME_PLACEHOLDER_DIAGNOSTICS_COUNTERS_STATEERROR_DIAGNOSTICSLEVEL := 19007,
	OPCUAID_PUBLISHEDEVENTSTYPE_DATASETWRITERNAME_PLACEHOLDER_DIAGNOSTICS_COUNTERS_STATEERROR_TIMEFIRSTCHANGE := 19008,
	OPCUAID_PUBLISHEDEVENTSTYPE_DATASETWRITERNAME_PLACEHOLDER_DIAGNOSTICS_COUNTERS_STATEOPERATIONALBYMETHOD := 19009,
	OPCUAID_PUBLISHEDEVENTSTYPE_DATASETWRITERNAME_PLACEHOLDER_DIAGNOSTICS_COUNTERS_STATEOPERATIONALBYMETHOD_ACTIVE := 19010,
	OPCUAID_PUBLISHEDEVENTSTYPE_DATASETWRITERNAME_PLACEHOLDER_DIAGNOSTICS_COUNTERS_STATEOPERATIONALBYMETHOD_CLASSIFICATION := 19011,
	OPCUAID_PUBLISHEDEVENTSTYPE_DATASETWRITERNAME_PLACEHOLDER_DIAGNOSTICS_COUNTERS_STATEOPERATIONALBYMETHOD_DIAGNOSTICSLEVEL := 19012,
	OPCUAID_PUBLISHEDEVENTSTYPE_DATASETWRITERNAME_PLACEHOLDER_DIAGNOSTICS_COUNTERS_STATEOPERATIONALBYMETHOD_TIMEFIRSTCHANGE := 19013,
	OPCUAID_PUBLISHEDEVENTSTYPE_DATASETWRITERNAME_PLACEHOLDER_DIAGNOSTICS_COUNTERS_STATEOPERATIONALBYPARENT := 19014,
	OPCUAID_PUBLISHEDEVENTSTYPE_DATASETWRITERNAME_PLACEHOLDER_DIAGNOSTICS_COUNTERS_STATEOPERATIONALBYPARENT_ACTIVE := 19015,
	OPCUAID_PUBLISHEDEVENTSTYPE_DATASETWRITERNAME_PLACEHOLDER_DIAGNOSTICS_COUNTERS_STATEOPERATIONALBYPARENT_CLASSIFICATION := 19016,
	OPCUAID_PUBLISHEDEVENTSTYPE_DATASETWRITERNAME_PLACEHOLDER_DIAGNOSTICS_COUNTERS_STATEOPERATIONALBYPARENT_DIAGNOSTICSLEVEL := 19017,
	OPCUAID_PUBLISHEDEVENTSTYPE_DATASETWRITERNAME_PLACEHOLDER_DIAGNOSTICS_COUNTERS_STATEOPERATIONALBYPARENT_TIMEFIRSTCHANGE := 19018,
	OPCUAID_PUBLISHEDEVENTSTYPE_DATASETWRITERNAME_PLACEHOLDER_DIAGNOSTICS_COUNTERS_STATEOPERATIONALFROMERROR := 19019,
	OPCUAID_PUBLISHEDEVENTSTYPE_DATASETWRITERNAME_PLACEHOLDER_DIAGNOSTICS_COUNTERS_STATEOPERATIONALFROMERROR_ACTIVE := 19020,
	OPCUAID_PUBLISHEDEVENTSTYPE_DATASETWRITERNAME_PLACEHOLDER_DIAGNOSTICS_COUNTERS_STATEOPERATIONALFROMERROR_CLASSIFICATION := 19021,
	OPCUAID_PUBLISHEDEVENTSTYPE_DATASETWRITERNAME_PLACEHOLDER_DIAGNOSTICS_COUNTERS_STATEOPERATIONALFROMERROR_DIAGNOSTICSLEVEL := 19022,
	OPCUAID_PUBLISHEDEVENTSTYPE_DATASETWRITERNAME_PLACEHOLDER_DIAGNOSTICS_COUNTERS_STATEOPERATIONALFROMERROR_TIMEFIRSTCHANGE := 19023,
	OPCUAID_PUBLISHEDEVENTSTYPE_DATASETWRITERNAME_PLACEHOLDER_DIAGNOSTICS_COUNTERS_STATEPAUSEDBYPARENT := 19024,
	OPCUAID_PUBLISHEDEVENTSTYPE_DATASETWRITERNAME_PLACEHOLDER_DIAGNOSTICS_COUNTERS_STATEPAUSEDBYPARENT_ACTIVE := 19025,
	OPCUAID_PUBLISHEDEVENTSTYPE_DATASETWRITERNAME_PLACEHOLDER_DIAGNOSTICS_COUNTERS_STATEPAUSEDBYPARENT_CLASSIFICATION := 19026,
	OPCUAID_PUBLISHEDEVENTSTYPE_DATASETWRITERNAME_PLACEHOLDER_DIAGNOSTICS_COUNTERS_STATEPAUSEDBYPARENT_DIAGNOSTICSLEVEL := 19027,
	OPCUAID_PUBLISHEDEVENTSTYPE_DATASETWRITERNAME_PLACEHOLDER_DIAGNOSTICS_COUNTERS_STATEPAUSEDBYPARENT_TIMEFIRSTCHANGE := 19028,
	OPCUAID_PUBLISHEDEVENTSTYPE_DATASETWRITERNAME_PLACEHOLDER_DIAGNOSTICS_COUNTERS_STATEDISABLEDBYMETHOD := 19029,
	OPCUAID_PUBLISHEDEVENTSTYPE_DATASETWRITERNAME_PLACEHOLDER_DIAGNOSTICS_COUNTERS_STATEDISABLEDBYMETHOD_ACTIVE := 19030,
	OPCUAID_PUBLISHEDEVENTSTYPE_DATASETWRITERNAME_PLACEHOLDER_DIAGNOSTICS_COUNTERS_STATEDISABLEDBYMETHOD_CLASSIFICATION := 19031,
	OPCUAID_PUBLISHEDEVENTSTYPE_DATASETWRITERNAME_PLACEHOLDER_DIAGNOSTICS_COUNTERS_STATEDISABLEDBYMETHOD_DIAGNOSTICSLEVEL := 19032,
	OPCUAID_PUBLISHEDEVENTSTYPE_DATASETWRITERNAME_PLACEHOLDER_DIAGNOSTICS_COUNTERS_STATEDISABLEDBYMETHOD_TIMEFIRSTCHANGE := 19033,
	OPCUAID_PUBLISHEDEVENTSTYPE_DATASETWRITERNAME_PLACEHOLDER_DIAGNOSTICS_COUNTERS_FAILEDDATASETMESSAGES := 19035,
	OPCUAID_PUBLISHEDEVENTSTYPE_DATASETWRITERNAME_PLACEHOLDER_DIAGNOSTICS_COUNTERS_FAILEDDATASETMESSAGES_ACTIVE := 19036,
	OPCUAID_PUBLISHEDEVENTSTYPE_DATASETWRITERNAME_PLACEHOLDER_DIAGNOSTICS_COUNTERS_FAILEDDATASETMESSAGES_CLASSIFICATION := 19037,
	OPCUAID_PUBLISHEDEVENTSTYPE_DATASETWRITERNAME_PLACEHOLDER_DIAGNOSTICS_COUNTERS_FAILEDDATASETMESSAGES_DIAGNOSTICSLEVEL := 19038,
	OPCUAID_PUBLISHEDEVENTSTYPE_DATASETWRITERNAME_PLACEHOLDER_DIAGNOSTICS_COUNTERS_FAILEDDATASETMESSAGES_TIMEFIRSTCHANGE := 19039,
	OPCUAID_PUBLISHEDEVENTSTYPE_DATASETWRITERNAME_PLACEHOLDER_DIAGNOSTICS_LIVEVALUES_MESSAGESEQUENCENUMBER_DIAGNOSTICSLEVEL := 19041,
	OPCUAID_PUBLISHEDEVENTSTYPE_DATASETWRITERNAME_PLACEHOLDER_DIAGNOSTICS_LIVEVALUES_STATUSCODE_DIAGNOSTICSLEVEL := 19043,
	OPCUAID_PUBLISHEDEVENTSTYPE_DATASETWRITERNAME_PLACEHOLDER_DIAGNOSTICS_LIVEVALUES_MAJORVERSION_DIAGNOSTICSLEVEL := 19045,
	OPCUAID_PUBLISHEDEVENTSTYPE_DATASETWRITERNAME_PLACEHOLDER_DIAGNOSTICS_LIVEVALUES_MINORVERSION_DIAGNOSTICSLEVEL := 19047,
	OPCUAID_PUBLISHEDEVENTSTYPE_EXTENSIONFIELDS_ADDEXTENSIONFIELD_INPUTARGUMENTS := 15513,
	OPCUAID_PUBLISHEDEVENTSTYPE_EXTENSIONFIELDS_ADDEXTENSIONFIELD_OUTPUTARGUMENTS := 15514,
	OPCUAID_PUBLISHEDEVENTSTYPE_EXTENSIONFIELDS_REMOVEEXTENSIONFIELD_INPUTARGUMENTS := 15516,
	OPCUAID_PUBLISHEDEVENTSTYPE_PUBSUBEVENTNOTIFIER := 14586,
	OPCUAID_PUBLISHEDEVENTSTYPE_SELECTEDFIELDS := 14587,
	OPCUAID_PUBLISHEDEVENTSTYPE_FILTER := 14588,
	OPCUAID_PUBLISHEDEVENTSTYPE_MODIFYFIELDSELECTION_INPUTARGUMENTS := 15053,
	OPCUAID_PUBLISHEDEVENTSTYPE_MODIFYFIELDSELECTION_OUTPUTARGUMENTS := 15517,
	OPCUAID_DATASETFOLDERTYPE_DATASETFOLDERNAME_PLACEHOLDER_ADDPUBLISHEDDATAITEMS_INPUTARGUMENTS := 14480,
	OPCUAID_DATASETFOLDERTYPE_DATASETFOLDERNAME_PLACEHOLDER_ADDPUBLISHEDDATAITEMS_OUTPUTARGUMENTS := 14481,
	OPCUAID_DATASETFOLDERTYPE_DATASETFOLDERNAME_PLACEHOLDER_ADDPUBLISHEDEVENTS_INPUTARGUMENTS := 14483,
	OPCUAID_DATASETFOLDERTYPE_DATASETFOLDERNAME_PLACEHOLDER_ADDPUBLISHEDEVENTS_OUTPUTARGUMENTS := 14484,
	OPCUAID_DATASETFOLDERTYPE_DATASETFOLDERNAME_PLACEHOLDER_ADDPUBLISHEDDATAITEMSTEMPLATE_INPUTARGUMENTS := 16843,
	OPCUAID_DATASETFOLDERTYPE_DATASETFOLDERNAME_PLACEHOLDER_ADDPUBLISHEDDATAITEMSTEMPLATE_OUTPUTARGUMENTS := 16853,
	OPCUAID_DATASETFOLDERTYPE_DATASETFOLDERNAME_PLACEHOLDER_ADDPUBLISHEDEVENTSTEMPLATE_INPUTARGUMENTS := 16882,
	OPCUAID_DATASETFOLDERTYPE_DATASETFOLDERNAME_PLACEHOLDER_ADDPUBLISHEDEVENTSTEMPLATE_OUTPUTARGUMENTS := 16883,
	OPCUAID_DATASETFOLDERTYPE_DATASETFOLDERNAME_PLACEHOLDER_REMOVEPUBLISHEDDATASET_INPUTARGUMENTS := 14486,
	OPCUAID_DATASETFOLDERTYPE_DATASETFOLDERNAME_PLACEHOLDER_ADDDATASETFOLDER_INPUTARGUMENTS := 16894,
	OPCUAID_DATASETFOLDERTYPE_DATASETFOLDERNAME_PLACEHOLDER_ADDDATASETFOLDER_OUTPUTARGUMENTS := 16922,
	OPCUAID_DATASETFOLDERTYPE_DATASETFOLDERNAME_PLACEHOLDER_REMOVEDATASETFOLDER_INPUTARGUMENTS := 16924,
	OPCUAID_DATASETFOLDERTYPE_PUBLISHEDDATASETNAME_PLACEHOLDER_CONFIGURATIONVERSION := 14489,
	OPCUAID_DATASETFOLDERTYPE_PUBLISHEDDATASETNAME_PLACEHOLDER_DATASETMETADATA := 15221,
	OPCUAID_DATASETFOLDERTYPE_PUBLISHEDDATASETNAME_PLACEHOLDER_EXTENSIONFIELDS_ADDEXTENSIONFIELD_INPUTARGUMENTS := 15475,
	OPCUAID_DATASETFOLDERTYPE_PUBLISHEDDATASETNAME_PLACEHOLDER_EXTENSIONFIELDS_ADDEXTENSIONFIELD_OUTPUTARGUMENTS := 15476,
	OPCUAID_DATASETFOLDERTYPE_PUBLISHEDDATASETNAME_PLACEHOLDER_EXTENSIONFIELDS_REMOVEEXTENSIONFIELD_INPUTARGUMENTS := 15478,
	OPCUAID_DATASETFOLDERTYPE_ADDPUBLISHEDDATAITEMS_INPUTARGUMENTS := 14494,
	OPCUAID_DATASETFOLDERTYPE_ADDPUBLISHEDDATAITEMS_OUTPUTARGUMENTS := 14495,
	OPCUAID_DATASETFOLDERTYPE_ADDPUBLISHEDEVENTS_INPUTARGUMENTS := 14497,
	OPCUAID_DATASETFOLDERTYPE_ADDPUBLISHEDEVENTS_OUTPUTARGUMENTS := 14498,
	OPCUAID_DATASETFOLDERTYPE_ADDPUBLISHEDDATAITEMSTEMPLATE_INPUTARGUMENTS := 16958,
	OPCUAID_DATASETFOLDERTYPE_ADDPUBLISHEDDATAITEMSTEMPLATE_OUTPUTARGUMENTS := 16959,
	OPCUAID_DATASETFOLDERTYPE_ADDPUBLISHEDEVENTSTEMPLATE_INPUTARGUMENTS := 16961,
	OPCUAID_DATASETFOLDERTYPE_ADDPUBLISHEDEVENTSTEMPLATE_OUTPUTARGUMENTS := 16971,
	OPCUAID_DATASETFOLDERTYPE_REMOVEPUBLISHEDDATASET_INPUTARGUMENTS := 14500,
	OPCUAID_DATASETFOLDERTYPE_ADDDATASETFOLDER_INPUTARGUMENTS := 16995,
	OPCUAID_DATASETFOLDERTYPE_ADDDATASETFOLDER_OUTPUTARGUMENTS := 16996,
	OPCUAID_DATASETFOLDERTYPE_REMOVEDATASETFOLDER_INPUTARGUMENTS := 17007,
	OPCUAID_PUBSUBCONNECTIONTYPE_PUBLISHERID := 14595,
	OPCUAID_PUBSUBCONNECTIONTYPE_TRANSPORTPROFILEURI := 17306,
	OPCUAID_PUBSUBCONNECTIONTYPE_TRANSPORTPROFILEURI_SELECTIONS := 17710,
	OPCUAID_PUBSUBCONNECTIONTYPE_CONNECTIONPROPERTIES := 17485,
	OPCUAID_PUBSUBCONNECTIONTYPE_ADDRESS_NETWORKINTERFACE := 17202,
	OPCUAID_PUBSUBCONNECTIONTYPE_WRITERGROUPNAME_PLACEHOLDER_SECURITYMODE := 17311,
	OPCUAID_PUBSUBCONNECTIONTYPE_WRITERGROUPNAME_PLACEHOLDER_MAXNETWORKMESSAGESIZE := 17204,
	OPCUAID_PUBSUBCONNECTIONTYPE_WRITERGROUPNAME_PLACEHOLDER_GROUPPROPERTIES := 17486,
	OPCUAID_PUBSUBCONNECTIONTYPE_WRITERGROUPNAME_PLACEHOLDER_STATUS_STATE := 17315,
	OPCUAID_PUBSUBCONNECTIONTYPE_WRITERGROUPNAME_PLACEHOLDER_WRITERGROUPID := 17214,
	OPCUAID_PUBSUBCONNECTIONTYPE_WRITERGROUPNAME_PLACEHOLDER_PUBLISHINGINTERVAL := 17318,
	OPCUAID_PUBSUBCONNECTIONTYPE_WRITERGROUPNAME_PLACEHOLDER_KEEPALIVETIME := 17319,
	OPCUAID_PUBSUBCONNECTIONTYPE_WRITERGROUPNAME_PLACEHOLDER_PRIORITY := 17321,
	OPCUAID_PUBSUBCONNECTIONTYPE_WRITERGROUPNAME_PLACEHOLDER_LOCALEIDS := 17322,
	OPCUAID_PUBSUBCONNECTIONTYPE_WRITERGROUPNAME_PLACEHOLDER_DIAGNOSTICS_DIAGNOSTICSLEVEL := 19108,
	OPCUAID_PUBSUBCONNECTIONTYPE_WRITERGROUPNAME_PLACEHOLDER_DIAGNOSTICS_TOTALINFORMATION := 19109,
	OPCUAID_PUBSUBCONNECTIONTYPE_WRITERGROUPNAME_PLACEHOLDER_DIAGNOSTICS_TOTALINFORMATION_ACTIVE := 19110,
	OPCUAID_PUBSUBCONNECTIONTYPE_WRITERGROUPNAME_PLACEHOLDER_DIAGNOSTICS_TOTALINFORMATION_CLASSIFICATION := 19111,
	OPCUAID_PUBSUBCONNECTIONTYPE_WRITERGROUPNAME_PLACEHOLDER_DIAGNOSTICS_TOTALINFORMATION_DIAGNOSTICSLEVEL := 19112,
	OPCUAID_PUBSUBCONNECTIONTYPE_WRITERGROUPNAME_PLACEHOLDER_DIAGNOSTICS_TOTALINFORMATION_TIMEFIRSTCHANGE := 19113,
	OPCUAID_PUBSUBCONNECTIONTYPE_WRITERGROUPNAME_PLACEHOLDER_DIAGNOSTICS_TOTALERROR := 19114,
	OPCUAID_PUBSUBCONNECTIONTYPE_WRITERGROUPNAME_PLACEHOLDER_DIAGNOSTICS_TOTALERROR_ACTIVE := 19115,
	OPCUAID_PUBSUBCONNECTIONTYPE_WRITERGROUPNAME_PLACEHOLDER_DIAGNOSTICS_TOTALERROR_CLASSIFICATION := 19116,
	OPCUAID_PUBSUBCONNECTIONTYPE_WRITERGROUPNAME_PLACEHOLDER_DIAGNOSTICS_TOTALERROR_DIAGNOSTICSLEVEL := 19117,
	OPCUAID_PUBSUBCONNECTIONTYPE_WRITERGROUPNAME_PLACEHOLDER_DIAGNOSTICS_TOTALERROR_TIMEFIRSTCHANGE := 19118,
	OPCUAID_PUBSUBCONNECTIONTYPE_WRITERGROUPNAME_PLACEHOLDER_DIAGNOSTICS_SUBERROR := 19120,
	OPCUAID_PUBSUBCONNECTIONTYPE_WRITERGROUPNAME_PLACEHOLDER_DIAGNOSTICS_COUNTERS_STATEERROR := 19122,
	OPCUAID_PUBSUBCONNECTIONTYPE_WRITERGROUPNAME_PLACEHOLDER_DIAGNOSTICS_COUNTERS_STATEERROR_ACTIVE := 19123,
	OPCUAID_PUBSUBCONNECTIONTYPE_WRITERGROUPNAME_PLACEHOLDER_DIAGNOSTICS_COUNTERS_STATEERROR_CLASSIFICATION := 19124,
	OPCUAID_PUBSUBCONNECTIONTYPE_WRITERGROUPNAME_PLACEHOLDER_DIAGNOSTICS_COUNTERS_STATEERROR_DIAGNOSTICSLEVEL := 19125,
	OPCUAID_PUBSUBCONNECTIONTYPE_WRITERGROUPNAME_PLACEHOLDER_DIAGNOSTICS_COUNTERS_STATEERROR_TIMEFIRSTCHANGE := 19126,
	OPCUAID_PUBSUBCONNECTIONTYPE_WRITERGROUPNAME_PLACEHOLDER_DIAGNOSTICS_COUNTERS_STATEOPERATIONALBYMETHOD := 19127,
	OPCUAID_PUBSUBCONNECTIONTYPE_WRITERGROUPNAME_PLACEHOLDER_DIAGNOSTICS_COUNTERS_STATEOPERATIONALBYMETHOD_ACTIVE := 19128,
	OPCUAID_PUBSUBCONNECTIONTYPE_WRITERGROUPNAME_PLACEHOLDER_DIAGNOSTICS_COUNTERS_STATEOPERATIONALBYMETHOD_CLASSIFICATION := 19129,
	OPCUAID_PUBSUBCONNECTIONTYPE_WRITERGROUPNAME_PLACEHOLDER_DIAGNOSTICS_COUNTERS_STATEOPERATIONALBYMETHOD_DIAGNOSTICSLEVEL := 19130,
	OPCUAID_PUBSUBCONNECTIONTYPE_WRITERGROUPNAME_PLACEHOLDER_DIAGNOSTICS_COUNTERS_STATEOPERATIONALBYMETHOD_TIMEFIRSTCHANGE := 19131,
	OPCUAID_PUBSUBCONNECTIONTYPE_WRITERGROUPNAME_PLACEHOLDER_DIAGNOSTICS_COUNTERS_STATEOPERATIONALBYPARENT := 19132,
	OPCUAID_PUBSUBCONNECTIONTYPE_WRITERGROUPNAME_PLACEHOLDER_DIAGNOSTICS_COUNTERS_STATEOPERATIONALBYPARENT_ACTIVE := 19133,
	OPCUAID_PUBSUBCONNECTIONTYPE_WRITERGROUPNAME_PLACEHOLDER_DIAGNOSTICS_COUNTERS_STATEOPERATIONALBYPARENT_CLASSIFICATION := 19134,
	OPCUAID_PUBSUBCONNECTIONTYPE_WRITERGROUPNAME_PLACEHOLDER_DIAGNOSTICS_COUNTERS_STATEOPERATIONALBYPARENT_DIAGNOSTICSLEVEL := 19135,
	OPCUAID_PUBSUBCONNECTIONTYPE_WRITERGROUPNAME_PLACEHOLDER_DIAGNOSTICS_COUNTERS_STATEOPERATIONALBYPARENT_TIMEFIRSTCHANGE := 19136,
	OPCUAID_PUBSUBCONNECTIONTYPE_WRITERGROUPNAME_PLACEHOLDER_DIAGNOSTICS_COUNTERS_STATEOPERATIONALFROMERROR := 19137,
	OPCUAID_PUBSUBCONNECTIONTYPE_WRITERGROUPNAME_PLACEHOLDER_DIAGNOSTICS_COUNTERS_STATEOPERATIONALFROMERROR_ACTIVE := 19138,
	OPCUAID_PUBSUBCONNECTIONTYPE_WRITERGROUPNAME_PLACEHOLDER_DIAGNOSTICS_COUNTERS_STATEOPERATIONALFROMERROR_CLASSIFICATION := 19139,
	OPCUAID_PUBSUBCONNECTIONTYPE_WRITERGROUPNAME_PLACEHOLDER_DIAGNOSTICS_COUNTERS_STATEOPERATIONALFROMERROR_DIAGNOSTICSLEVEL := 19140,
	OPCUAID_PUBSUBCONNECTIONTYPE_WRITERGROUPNAME_PLACEHOLDER_DIAGNOSTICS_COUNTERS_STATEOPERATIONALFROMERROR_TIMEFIRSTCHANGE := 19141,
	OPCUAID_PUBSUBCONNECTIONTYPE_WRITERGROUPNAME_PLACEHOLDER_DIAGNOSTICS_COUNTERS_STATEPAUSEDBYPARENT := 19142,
	OPCUAID_PUBSUBCONNECTIONTYPE_WRITERGROUPNAME_PLACEHOLDER_DIAGNOSTICS_COUNTERS_STATEPAUSEDBYPARENT_ACTIVE := 19143,
	OPCUAID_PUBSUBCONNECTIONTYPE_WRITERGROUPNAME_PLACEHOLDER_DIAGNOSTICS_COUNTERS_STATEPAUSEDBYPARENT_CLASSIFICATION := 19144,
	OPCUAID_PUBSUBCONNECTIONTYPE_WRITERGROUPNAME_PLACEHOLDER_DIAGNOSTICS_COUNTERS_STATEPAUSEDBYPARENT_DIAGNOSTICSLEVEL := 19145,
	OPCUAID_PUBSUBCONNECTIONTYPE_WRITERGROUPNAME_PLACEHOLDER_DIAGNOSTICS_COUNTERS_STATEPAUSEDBYPARENT_TIMEFIRSTCHANGE := 19146,
	OPCUAID_PUBSUBCONNECTIONTYPE_WRITERGROUPNAME_PLACEHOLDER_DIAGNOSTICS_COUNTERS_STATEDISABLEDBYMETHOD := 19147,
	OPCUAID_PUBSUBCONNECTIONTYPE_WRITERGROUPNAME_PLACEHOLDER_DIAGNOSTICS_COUNTERS_STATEDISABLEDBYMETHOD_ACTIVE := 19148,
	OPCUAID_PUBSUBCONNECTIONTYPE_WRITERGROUPNAME_PLACEHOLDER_DIAGNOSTICS_COUNTERS_STATEDISABLEDBYMETHOD_CLASSIFICATION := 19149,
	OPCUAID_PUBSUBCONNECTIONTYPE_WRITERGROUPNAME_PLACEHOLDER_DIAGNOSTICS_COUNTERS_STATEDISABLEDBYMETHOD_DIAGNOSTICSLEVEL := 19150,
	OPCUAID_PUBSUBCONNECTIONTYPE_WRITERGROUPNAME_PLACEHOLDER_DIAGNOSTICS_COUNTERS_STATEDISABLEDBYMETHOD_TIMEFIRSTCHANGE := 19151,
	OPCUAID_PUBSUBCONNECTIONTYPE_WRITERGROUPNAME_PLACEHOLDER_DIAGNOSTICS_COUNTERS_SENTNETWORKMESSAGES := 19153,
	OPCUAID_PUBSUBCONNECTIONTYPE_WRITERGROUPNAME_PLACEHOLDER_DIAGNOSTICS_COUNTERS_SENTNETWORKMESSAGES_ACTIVE := 19154,
	OPCUAID_PUBSUBCONNECTIONTYPE_WRITERGROUPNAME_PLACEHOLDER_DIAGNOSTICS_COUNTERS_SENTNETWORKMESSAGES_CLASSIFICATION := 19155,
	OPCUAID_PUBSUBCONNECTIONTYPE_WRITERGROUPNAME_PLACEHOLDER_DIAGNOSTICS_COUNTERS_SENTNETWORKMESSAGES_DIAGNOSTICSLEVEL := 19156,
	OPCUAID_PUBSUBCONNECTIONTYPE_WRITERGROUPNAME_PLACEHOLDER_DIAGNOSTICS_COUNTERS_SENTNETWORKMESSAGES_TIMEFIRSTCHANGE := 19157,
	OPCUAID_PUBSUBCONNECTIONTYPE_WRITERGROUPNAME_PLACEHOLDER_DIAGNOSTICS_COUNTERS_FAILEDTRANSMISSIONS := 19158,
	OPCUAID_PUBSUBCONNECTIONTYPE_WRITERGROUPNAME_PLACEHOLDER_DIAGNOSTICS_COUNTERS_FAILEDTRANSMISSIONS_ACTIVE := 19159,
	OPCUAID_PUBSUBCONNECTIONTYPE_WRITERGROUPNAME_PLACEHOLDER_DIAGNOSTICS_COUNTERS_FAILEDTRANSMISSIONS_CLASSIFICATION := 19160,
	OPCUAID_PUBSUBCONNECTIONTYPE_WRITERGROUPNAME_PLACEHOLDER_DIAGNOSTICS_COUNTERS_FAILEDTRANSMISSIONS_DIAGNOSTICSLEVEL := 19161,
	OPCUAID_PUBSUBCONNECTIONTYPE_WRITERGROUPNAME_PLACEHOLDER_DIAGNOSTICS_COUNTERS_FAILEDTRANSMISSIONS_TIMEFIRSTCHANGE := 19162,
	OPCUAID_PUBSUBCONNECTIONTYPE_WRITERGROUPNAME_PLACEHOLDER_DIAGNOSTICS_COUNTERS_ENCRYPTIONERRORS := 19163,
	OPCUAID_PUBSUBCONNECTIONTYPE_WRITERGROUPNAME_PLACEHOLDER_DIAGNOSTICS_COUNTERS_ENCRYPTIONERRORS_ACTIVE := 19164,
	OPCUAID_PUBSUBCONNECTIONTYPE_WRITERGROUPNAME_PLACEHOLDER_DIAGNOSTICS_COUNTERS_ENCRYPTIONERRORS_CLASSIFICATION := 19165,
	OPCUAID_PUBSUBCONNECTIONTYPE_WRITERGROUPNAME_PLACEHOLDER_DIAGNOSTICS_COUNTERS_ENCRYPTIONERRORS_DIAGNOSTICSLEVEL := 19166,
	OPCUAID_PUBSUBCONNECTIONTYPE_WRITERGROUPNAME_PLACEHOLDER_DIAGNOSTICS_COUNTERS_ENCRYPTIONERRORS_TIMEFIRSTCHANGE := 19167,
	OPCUAID_PUBSUBCONNECTIONTYPE_WRITERGROUPNAME_PLACEHOLDER_DIAGNOSTICS_LIVEVALUES_CONFIGUREDDATASETWRITERS := 19168,
	OPCUAID_PUBSUBCONNECTIONTYPE_WRITERGROUPNAME_PLACEHOLDER_DIAGNOSTICS_LIVEVALUES_CONFIGUREDDATASETWRITERS_DIAGNOSTICSLEVEL := 19169,
	OPCUAID_PUBSUBCONNECTIONTYPE_WRITERGROUPNAME_PLACEHOLDER_DIAGNOSTICS_LIVEVALUES_OPERATIONALDATASETWRITERS := 19170,
	OPCUAID_PUBSUBCONNECTIONTYPE_WRITERGROUPNAME_PLACEHOLDER_DIAGNOSTICS_LIVEVALUES_OPERATIONALDATASETWRITERS_DIAGNOSTICSLEVEL := 19171,
	OPCUAID_PUBSUBCONNECTIONTYPE_WRITERGROUPNAME_PLACEHOLDER_DIAGNOSTICS_LIVEVALUES_SECURITYTOKENID_DIAGNOSTICSLEVEL := 19173,
	OPCUAID_PUBSUBCONNECTIONTYPE_WRITERGROUPNAME_PLACEHOLDER_DIAGNOSTICS_LIVEVALUES_TIMETONEXTTOKENID_DIAGNOSTICSLEVEL := 19175,
	OPCUAID_PUBSUBCONNECTIONTYPE_WRITERGROUPNAME_PLACEHOLDER_ADDDATASETWRITER_INPUTARGUMENTS := 17294,
	OPCUAID_PUBSUBCONNECTIONTYPE_WRITERGROUPNAME_PLACEHOLDER_ADDDATASETWRITER_OUTPUTARGUMENTS := 17301,
	OPCUAID_PUBSUBCONNECTIONTYPE_WRITERGROUPNAME_PLACEHOLDER_REMOVEDATASETWRITER_INPUTARGUMENTS := 17324,
	OPCUAID_PUBSUBCONNECTIONTYPE_READERGROUPNAME_PLACEHOLDER_SECURITYMODE := 17326,
	OPCUAID_PUBSUBCONNECTIONTYPE_READERGROUPNAME_PLACEHOLDER_MAXNETWORKMESSAGESIZE := 17302,
	OPCUAID_PUBSUBCONNECTIONTYPE_READERGROUPNAME_PLACEHOLDER_GROUPPROPERTIES := 17487,
	OPCUAID_PUBSUBCONNECTIONTYPE_READERGROUPNAME_PLACEHOLDER_STATUS_STATE := 17330,
	OPCUAID_PUBSUBCONNECTIONTYPE_READERGROUPNAME_PLACEHOLDER_DIAGNOSTICS_DIAGNOSTICSLEVEL := 19177,
	OPCUAID_PUBSUBCONNECTIONTYPE_READERGROUPNAME_PLACEHOLDER_DIAGNOSTICS_TOTALINFORMATION := 19178,
	OPCUAID_PUBSUBCONNECTIONTYPE_READERGROUPNAME_PLACEHOLDER_DIAGNOSTICS_TOTALINFORMATION_ACTIVE := 19179,
	OPCUAID_PUBSUBCONNECTIONTYPE_READERGROUPNAME_PLACEHOLDER_DIAGNOSTICS_TOTALINFORMATION_CLASSIFICATION := 19180,
	OPCUAID_PUBSUBCONNECTIONTYPE_READERGROUPNAME_PLACEHOLDER_DIAGNOSTICS_TOTALINFORMATION_DIAGNOSTICSLEVEL := 19181,
	OPCUAID_PUBSUBCONNECTIONTYPE_READERGROUPNAME_PLACEHOLDER_DIAGNOSTICS_TOTALINFORMATION_TIMEFIRSTCHANGE := 19182,
	OPCUAID_PUBSUBCONNECTIONTYPE_READERGROUPNAME_PLACEHOLDER_DIAGNOSTICS_TOTALERROR := 19183,
	OPCUAID_PUBSUBCONNECTIONTYPE_READERGROUPNAME_PLACEHOLDER_DIAGNOSTICS_TOTALERROR_ACTIVE := 19184,
	OPCUAID_PUBSUBCONNECTIONTYPE_READERGROUPNAME_PLACEHOLDER_DIAGNOSTICS_TOTALERROR_CLASSIFICATION := 19185,
	OPCUAID_PUBSUBCONNECTIONTYPE_READERGROUPNAME_PLACEHOLDER_DIAGNOSTICS_TOTALERROR_DIAGNOSTICSLEVEL := 19186,
	OPCUAID_PUBSUBCONNECTIONTYPE_READERGROUPNAME_PLACEHOLDER_DIAGNOSTICS_TOTALERROR_TIMEFIRSTCHANGE := 19187,
	OPCUAID_PUBSUBCONNECTIONTYPE_READERGROUPNAME_PLACEHOLDER_DIAGNOSTICS_SUBERROR := 19189,
	OPCUAID_PUBSUBCONNECTIONTYPE_READERGROUPNAME_PLACEHOLDER_DIAGNOSTICS_COUNTERS_STATEERROR := 19191,
	OPCUAID_PUBSUBCONNECTIONTYPE_READERGROUPNAME_PLACEHOLDER_DIAGNOSTICS_COUNTERS_STATEERROR_ACTIVE := 19192,
	OPCUAID_PUBSUBCONNECTIONTYPE_READERGROUPNAME_PLACEHOLDER_DIAGNOSTICS_COUNTERS_STATEERROR_CLASSIFICATION := 19193,
	OPCUAID_PUBSUBCONNECTIONTYPE_READERGROUPNAME_PLACEHOLDER_DIAGNOSTICS_COUNTERS_STATEERROR_DIAGNOSTICSLEVEL := 19194,
	OPCUAID_PUBSUBCONNECTIONTYPE_READERGROUPNAME_PLACEHOLDER_DIAGNOSTICS_COUNTERS_STATEERROR_TIMEFIRSTCHANGE := 19195,
	OPCUAID_PUBSUBCONNECTIONTYPE_READERGROUPNAME_PLACEHOLDER_DIAGNOSTICS_COUNTERS_STATEOPERATIONALBYMETHOD := 19196,
	OPCUAID_PUBSUBCONNECTIONTYPE_READERGROUPNAME_PLACEHOLDER_DIAGNOSTICS_COUNTERS_STATEOPERATIONALBYMETHOD_ACTIVE := 19197,
	OPCUAID_PUBSUBCONNECTIONTYPE_READERGROUPNAME_PLACEHOLDER_DIAGNOSTICS_COUNTERS_STATEOPERATIONALBYMETHOD_CLASSIFICATION := 19198,
	OPCUAID_PUBSUBCONNECTIONTYPE_READERGROUPNAME_PLACEHOLDER_DIAGNOSTICS_COUNTERS_STATEOPERATIONALBYMETHOD_DIAGNOSTICSLEVEL := 19199,
	OPCUAID_PUBSUBCONNECTIONTYPE_READERGROUPNAME_PLACEHOLDER_DIAGNOSTICS_COUNTERS_STATEOPERATIONALBYMETHOD_TIMEFIRSTCHANGE := 19200,
	OPCUAID_PUBSUBCONNECTIONTYPE_READERGROUPNAME_PLACEHOLDER_DIAGNOSTICS_COUNTERS_STATEOPERATIONALBYPARENT := 19201,
	OPCUAID_PUBSUBCONNECTIONTYPE_READERGROUPNAME_PLACEHOLDER_DIAGNOSTICS_COUNTERS_STATEOPERATIONALBYPARENT_ACTIVE := 19202,
	OPCUAID_PUBSUBCONNECTIONTYPE_READERGROUPNAME_PLACEHOLDER_DIAGNOSTICS_COUNTERS_STATEOPERATIONALBYPARENT_CLASSIFICATION := 19203,
	OPCUAID_PUBSUBCONNECTIONTYPE_READERGROUPNAME_PLACEHOLDER_DIAGNOSTICS_COUNTERS_STATEOPERATIONALBYPARENT_DIAGNOSTICSLEVEL := 19204,
	OPCUAID_PUBSUBCONNECTIONTYPE_READERGROUPNAME_PLACEHOLDER_DIAGNOSTICS_COUNTERS_STATEOPERATIONALBYPARENT_TIMEFIRSTCHANGE := 19205,
	OPCUAID_PUBSUBCONNECTIONTYPE_READERGROUPNAME_PLACEHOLDER_DIAGNOSTICS_COUNTERS_STATEOPERATIONALFROMERROR := 19206,
	OPCUAID_PUBSUBCONNECTIONTYPE_READERGROUPNAME_PLACEHOLDER_DIAGNOSTICS_COUNTERS_STATEOPERATIONALFROMERROR_ACTIVE := 19207,
	OPCUAID_PUBSUBCONNECTIONTYPE_READERGROUPNAME_PLACEHOLDER_DIAGNOSTICS_COUNTERS_STATEOPERATIONALFROMERROR_CLASSIFICATION := 19208,
	OPCUAID_PUBSUBCONNECTIONTYPE_READERGROUPNAME_PLACEHOLDER_DIAGNOSTICS_COUNTERS_STATEOPERATIONALFROMERROR_DIAGNOSTICSLEVEL := 19209,
	OPCUAID_PUBSUBCONNECTIONTYPE_READERGROUPNAME_PLACEHOLDER_DIAGNOSTICS_COUNTERS_STATEOPERATIONALFROMERROR_TIMEFIRSTCHANGE := 19210,
	OPCUAID_PUBSUBCONNECTIONTYPE_READERGROUPNAME_PLACEHOLDER_DIAGNOSTICS_COUNTERS_STATEPAUSEDBYPARENT := 19211,
	OPCUAID_PUBSUBCONNECTIONTYPE_READERGROUPNAME_PLACEHOLDER_DIAGNOSTICS_COUNTERS_STATEPAUSEDBYPARENT_ACTIVE := 19212,
	OPCUAID_PUBSUBCONNECTIONTYPE_READERGROUPNAME_PLACEHOLDER_DIAGNOSTICS_COUNTERS_STATEPAUSEDBYPARENT_CLASSIFICATION := 19213,
	OPCUAID_PUBSUBCONNECTIONTYPE_READERGROUPNAME_PLACEHOLDER_DIAGNOSTICS_COUNTERS_STATEPAUSEDBYPARENT_DIAGNOSTICSLEVEL := 19214,
	OPCUAID_PUBSUBCONNECTIONTYPE_READERGROUPNAME_PLACEHOLDER_DIAGNOSTICS_COUNTERS_STATEPAUSEDBYPARENT_TIMEFIRSTCHANGE := 19215,
	OPCUAID_PUBSUBCONNECTIONTYPE_READERGROUPNAME_PLACEHOLDER_DIAGNOSTICS_COUNTERS_STATEDISABLEDBYMETHOD := 19216,
	OPCUAID_PUBSUBCONNECTIONTYPE_READERGROUPNAME_PLACEHOLDER_DIAGNOSTICS_COUNTERS_STATEDISABLEDBYMETHOD_ACTIVE := 19217,
	OPCUAID_PUBSUBCONNECTIONTYPE_READERGROUPNAME_PLACEHOLDER_DIAGNOSTICS_COUNTERS_STATEDISABLEDBYMETHOD_CLASSIFICATION := 19218,
	OPCUAID_PUBSUBCONNECTIONTYPE_READERGROUPNAME_PLACEHOLDER_DIAGNOSTICS_COUNTERS_STATEDISABLEDBYMETHOD_DIAGNOSTICSLEVEL := 19219,
	OPCUAID_PUBSUBCONNECTIONTYPE_READERGROUPNAME_PLACEHOLDER_DIAGNOSTICS_COUNTERS_STATEDISABLEDBYMETHOD_TIMEFIRSTCHANGE := 19220,
	OPCUAID_PUBSUBCONNECTIONTYPE_READERGROUPNAME_PLACEHOLDER_DIAGNOSTICS_COUNTERS_RECEIVEDNETWORKMESSAGES := 19222,
	OPCUAID_PUBSUBCONNECTIONTYPE_READERGROUPNAME_PLACEHOLDER_DIAGNOSTICS_COUNTERS_RECEIVEDNETWORKMESSAGES_ACTIVE := 19223,
	OPCUAID_PUBSUBCONNECTIONTYPE_READERGROUPNAME_PLACEHOLDER_DIAGNOSTICS_COUNTERS_RECEIVEDNETWORKMESSAGES_CLASSIFICATION := 19224,
	OPCUAID_PUBSUBCONNECTIONTYPE_READERGROUPNAME_PLACEHOLDER_DIAGNOSTICS_COUNTERS_RECEIVEDNETWORKMESSAGES_DIAGNOSTICSLEVEL := 19225,
	OPCUAID_PUBSUBCONNECTIONTYPE_READERGROUPNAME_PLACEHOLDER_DIAGNOSTICS_COUNTERS_RECEIVEDNETWORKMESSAGES_TIMEFIRSTCHANGE := 19226,
	OPCUAID_PUBSUBCONNECTIONTYPE_READERGROUPNAME_PLACEHOLDER_DIAGNOSTICS_COUNTERS_RECEIVEDINVALIDNETWORKMESSAGES_ACTIVE := 19228,
	OPCUAID_PUBSUBCONNECTIONTYPE_READERGROUPNAME_PLACEHOLDER_DIAGNOSTICS_COUNTERS_RECEIVEDINVALIDNETWORKMESSAGES_CLASSIFICATION := 19229,
	OPCUAID_PUBSUBCONNECTIONTYPE_READERGROUPNAME_PLACEHOLDER_DIAGNOSTICS_COUNTERS_RECEIVEDINVALIDNETWORKMESSAGES_DIAGNOSTICSLEVEL := 19230,
	OPCUAID_PUBSUBCONNECTIONTYPE_READERGROUPNAME_PLACEHOLDER_DIAGNOSTICS_COUNTERS_RECEIVEDINVALIDNETWORKMESSAGES_TIMEFIRSTCHANGE := 19231,
	OPCUAID_PUBSUBCONNECTIONTYPE_READERGROUPNAME_PLACEHOLDER_DIAGNOSTICS_COUNTERS_DECRYPTIONERRORS_ACTIVE := 19233,
	OPCUAID_PUBSUBCONNECTIONTYPE_READERGROUPNAME_PLACEHOLDER_DIAGNOSTICS_COUNTERS_DECRYPTIONERRORS_CLASSIFICATION := 19234,
	OPCUAID_PUBSUBCONNECTIONTYPE_READERGROUPNAME_PLACEHOLDER_DIAGNOSTICS_COUNTERS_DECRYPTIONERRORS_DIAGNOSTICSLEVEL := 19235,
	OPCUAID_PUBSUBCONNECTIONTYPE_READERGROUPNAME_PLACEHOLDER_DIAGNOSTICS_COUNTERS_DECRYPTIONERRORS_TIMEFIRSTCHANGE := 19236,
	OPCUAID_PUBSUBCONNECTIONTYPE_READERGROUPNAME_PLACEHOLDER_DIAGNOSTICS_LIVEVALUES_CONFIGUREDDATASETREADERS := 19237,
	OPCUAID_PUBSUBCONNECTIONTYPE_READERGROUPNAME_PLACEHOLDER_DIAGNOSTICS_LIVEVALUES_CONFIGUREDDATASETREADERS_DIAGNOSTICSLEVEL := 19238,
	OPCUAID_PUBSUBCONNECTIONTYPE_READERGROUPNAME_PLACEHOLDER_DIAGNOSTICS_LIVEVALUES_OPERATIONALDATASETREADERS := 19239,
	OPCUAID_PUBSUBCONNECTIONTYPE_READERGROUPNAME_PLACEHOLDER_DIAGNOSTICS_LIVEVALUES_OPERATIONALDATASETREADERS_DIAGNOSTICSLEVEL := 19240,
	OPCUAID_PUBSUBCONNECTIONTYPE_READERGROUPNAME_PLACEHOLDER_ADDDATASETREADER_INPUTARGUMENTS := 17399,
	OPCUAID_PUBSUBCONNECTIONTYPE_READERGROUPNAME_PLACEHOLDER_ADDDATASETREADER_OUTPUTARGUMENTS := 17400,
	OPCUAID_PUBSUBCONNECTIONTYPE_READERGROUPNAME_PLACEHOLDER_REMOVEDATASETREADER_INPUTARGUMENTS := 17334,
	OPCUAID_PUBSUBCONNECTIONTYPE_STATUS_STATE := 14601,
	OPCUAID_PUBSUBCONNECTIONTYPE_DIAGNOSTICS_DIAGNOSTICSLEVEL := 19242,
	OPCUAID_PUBSUBCONNECTIONTYPE_DIAGNOSTICS_TOTALINFORMATION := 19243,
	OPCUAID_PUBSUBCONNECTIONTYPE_DIAGNOSTICS_TOTALINFORMATION_ACTIVE := 19244,
	OPCUAID_PUBSUBCONNECTIONTYPE_DIAGNOSTICS_TOTALINFORMATION_CLASSIFICATION := 19245,
	OPCUAID_PUBSUBCONNECTIONTYPE_DIAGNOSTICS_TOTALINFORMATION_DIAGNOSTICSLEVEL := 19246,
	OPCUAID_PUBSUBCONNECTIONTYPE_DIAGNOSTICS_TOTALINFORMATION_TIMEFIRSTCHANGE := 19247,
	OPCUAID_PUBSUBCONNECTIONTYPE_DIAGNOSTICS_TOTALERROR := 19248,
	OPCUAID_PUBSUBCONNECTIONTYPE_DIAGNOSTICS_TOTALERROR_ACTIVE := 19249,
	OPCUAID_PUBSUBCONNECTIONTYPE_DIAGNOSTICS_TOTALERROR_CLASSIFICATION := 19250,
	OPCUAID_PUBSUBCONNECTIONTYPE_DIAGNOSTICS_TOTALERROR_DIAGNOSTICSLEVEL := 19251,
	OPCUAID_PUBSUBCONNECTIONTYPE_DIAGNOSTICS_TOTALERROR_TIMEFIRSTCHANGE := 19252,
	OPCUAID_PUBSUBCONNECTIONTYPE_DIAGNOSTICS_SUBERROR := 19254,
	OPCUAID_PUBSUBCONNECTIONTYPE_DIAGNOSTICS_COUNTERS_STATEERROR := 19256,
	OPCUAID_PUBSUBCONNECTIONTYPE_DIAGNOSTICS_COUNTERS_STATEERROR_ACTIVE := 19257,
	OPCUAID_PUBSUBCONNECTIONTYPE_DIAGNOSTICS_COUNTERS_STATEERROR_CLASSIFICATION := 19258,
	OPCUAID_PUBSUBCONNECTIONTYPE_DIAGNOSTICS_COUNTERS_STATEERROR_DIAGNOSTICSLEVEL := 19259,
	OPCUAID_PUBSUBCONNECTIONTYPE_DIAGNOSTICS_COUNTERS_STATEERROR_TIMEFIRSTCHANGE := 19260,
	OPCUAID_PUBSUBCONNECTIONTYPE_DIAGNOSTICS_COUNTERS_STATEOPERATIONALBYMETHOD := 19261,
	OPCUAID_PUBSUBCONNECTIONTYPE_DIAGNOSTICS_COUNTERS_STATEOPERATIONALBYMETHOD_ACTIVE := 19262,
	OPCUAID_PUBSUBCONNECTIONTYPE_DIAGNOSTICS_COUNTERS_STATEOPERATIONALBYMETHOD_CLASSIFICATION := 19263,
	OPCUAID_PUBSUBCONNECTIONTYPE_DIAGNOSTICS_COUNTERS_STATEOPERATIONALBYMETHOD_DIAGNOSTICSLEVEL := 19264,
	OPCUAID_PUBSUBCONNECTIONTYPE_DIAGNOSTICS_COUNTERS_STATEOPERATIONALBYMETHOD_TIMEFIRSTCHANGE := 19265,
	OPCUAID_PUBSUBCONNECTIONTYPE_DIAGNOSTICS_COUNTERS_STATEOPERATIONALBYPARENT := 19266,
	OPCUAID_PUBSUBCONNECTIONTYPE_DIAGNOSTICS_COUNTERS_STATEOPERATIONALBYPARENT_ACTIVE := 19267,
	OPCUAID_PUBSUBCONNECTIONTYPE_DIAGNOSTICS_COUNTERS_STATEOPERATIONALBYPARENT_CLASSIFICATION := 19268,
	OPCUAID_PUBSUBCONNECTIONTYPE_DIAGNOSTICS_COUNTERS_STATEOPERATIONALBYPARENT_DIAGNOSTICSLEVEL := 19269,
	OPCUAID_PUBSUBCONNECTIONTYPE_DIAGNOSTICS_COUNTERS_STATEOPERATIONALBYPARENT_TIMEFIRSTCHANGE := 19270,
	OPCUAID_PUBSUBCONNECTIONTYPE_DIAGNOSTICS_COUNTERS_STATEOPERATIONALFROMERROR := 19271,
	OPCUAID_PUBSUBCONNECTIONTYPE_DIAGNOSTICS_COUNTERS_STATEOPERATIONALFROMERROR_ACTIVE := 19272,
	OPCUAID_PUBSUBCONNECTIONTYPE_DIAGNOSTICS_COUNTERS_STATEOPERATIONALFROMERROR_CLASSIFICATION := 19273,
	OPCUAID_PUBSUBCONNECTIONTYPE_DIAGNOSTICS_COUNTERS_STATEOPERATIONALFROMERROR_DIAGNOSTICSLEVEL := 19274,
	OPCUAID_PUBSUBCONNECTIONTYPE_DIAGNOSTICS_COUNTERS_STATEOPERATIONALFROMERROR_TIMEFIRSTCHANGE := 19275,
	OPCUAID_PUBSUBCONNECTIONTYPE_DIAGNOSTICS_COUNTERS_STATEPAUSEDBYPARENT := 19276,
	OPCUAID_PUBSUBCONNECTIONTYPE_DIAGNOSTICS_COUNTERS_STATEPAUSEDBYPARENT_ACTIVE := 19277,
	OPCUAID_PUBSUBCONNECTIONTYPE_DIAGNOSTICS_COUNTERS_STATEPAUSEDBYPARENT_CLASSIFICATION := 19278,
	OPCUAID_PUBSUBCONNECTIONTYPE_DIAGNOSTICS_COUNTERS_STATEPAUSEDBYPARENT_DIAGNOSTICSLEVEL := 19279,
	OPCUAID_PUBSUBCONNECTIONTYPE_DIAGNOSTICS_COUNTERS_STATEPAUSEDBYPARENT_TIMEFIRSTCHANGE := 19280,
	OPCUAID_PUBSUBCONNECTIONTYPE_DIAGNOSTICS_COUNTERS_STATEDISABLEDBYMETHOD := 19281,
	OPCUAID_PUBSUBCONNECTIONTYPE_DIAGNOSTICS_COUNTERS_STATEDISABLEDBYMETHOD_ACTIVE := 19282,
	OPCUAID_PUBSUBCONNECTIONTYPE_DIAGNOSTICS_COUNTERS_STATEDISABLEDBYMETHOD_CLASSIFICATION := 19283,
	OPCUAID_PUBSUBCONNECTIONTYPE_DIAGNOSTICS_COUNTERS_STATEDISABLEDBYMETHOD_DIAGNOSTICSLEVEL := 19284,
	OPCUAID_PUBSUBCONNECTIONTYPE_DIAGNOSTICS_COUNTERS_STATEDISABLEDBYMETHOD_TIMEFIRSTCHANGE := 19285,
	OPCUAID_PUBSUBCONNECTIONTYPE_DIAGNOSTICS_LIVEVALUES_RESOLVEDADDRESS := 19287,
	OPCUAID_PUBSUBCONNECTIONTYPE_DIAGNOSTICS_LIVEVALUES_RESOLVEDADDRESS_DIAGNOSTICSLEVEL := 19288,
	OPCUAID_PUBSUBCONNECTIONTYPE_ADDWRITERGROUP_INPUTARGUMENTS := 17428,
	OPCUAID_PUBSUBCONNECTIONTYPE_ADDWRITERGROUP_OUTPUTARGUMENTS := 17456,
	OPCUAID_PUBSUBCONNECTIONTYPE_ADDREADERGROUP_INPUTARGUMENTS := 17507,
	OPCUAID_PUBSUBCONNECTIONTYPE_ADDREADERGROUP_OUTPUTARGUMENTS := 17508,
	OPCUAID_PUBSUBCONNECTIONTYPE_REMOVEGROUP_INPUTARGUMENTS := 14226,
	OPCUAID_PUBSUBGROUPTYPE_SECURITYMODE := 15926,
	OPCUAID_PUBSUBGROUPTYPE_SECURITYGROUPID := 15927,
	OPCUAID_PUBSUBGROUPTYPE_SECURITYKEYSERVICES := 15928,
	OPCUAID_PUBSUBGROUPTYPE_MAXNETWORKMESSAGESIZE := 17724,
	OPCUAID_PUBSUBGROUPTYPE_GROUPPROPERTIES := 17488,
	OPCUAID_PUBSUBGROUPTYPE_STATUS_STATE := 15266,
	OPCUAID_WRITERGROUPTYPE_STATUS_STATE := 17731,
	OPCUAID_WRITERGROUPTYPE_WRITERGROUPID := 17736,
	OPCUAID_WRITERGROUPTYPE_PUBLISHINGINTERVAL := 17737,
	OPCUAID_WRITERGROUPTYPE_KEEPALIVETIME := 17738,
	OPCUAID_WRITERGROUPTYPE_PRIORITY := 17739,
	OPCUAID_WRITERGROUPTYPE_LOCALEIDS := 17740,
	OPCUAID_WRITERGROUPTYPE_DATASETWRITERNAME_PLACEHOLDER_DATASETWRITERID := 17744,
	OPCUAID_WRITERGROUPTYPE_DATASETWRITERNAME_PLACEHOLDER_DATASETFIELDCONTENTMASK := 17745,
	OPCUAID_WRITERGROUPTYPE_DATASETWRITERNAME_PLACEHOLDER_DATASETWRITERPROPERTIES := 17490,
	OPCUAID_WRITERGROUPTYPE_DATASETWRITERNAME_PLACEHOLDER_STATUS_STATE := 17750,
	OPCUAID_WRITERGROUPTYPE_DATASETWRITERNAME_PLACEHOLDER_DIAGNOSTICS_DIAGNOSTICSLEVEL := 17754,
	OPCUAID_WRITERGROUPTYPE_DATASETWRITERNAME_PLACEHOLDER_DIAGNOSTICS_TOTALINFORMATION := 17755,
	OPCUAID_WRITERGROUPTYPE_DATASETWRITERNAME_PLACEHOLDER_DIAGNOSTICS_TOTALINFORMATION_ACTIVE := 17756,
	OPCUAID_WRITERGROUPTYPE_DATASETWRITERNAME_PLACEHOLDER_DIAGNOSTICS_TOTALINFORMATION_CLASSIFICATION := 17757,
	OPCUAID_WRITERGROUPTYPE_DATASETWRITERNAME_PLACEHOLDER_DIAGNOSTICS_TOTALINFORMATION_DIAGNOSTICSLEVEL := 17758,
	OPCUAID_WRITERGROUPTYPE_DATASETWRITERNAME_PLACEHOLDER_DIAGNOSTICS_TOTALINFORMATION_TIMEFIRSTCHANGE := 17759,
	OPCUAID_WRITERGROUPTYPE_DATASETWRITERNAME_PLACEHOLDER_DIAGNOSTICS_TOTALERROR := 17760,
	OPCUAID_WRITERGROUPTYPE_DATASETWRITERNAME_PLACEHOLDER_DIAGNOSTICS_TOTALERROR_ACTIVE := 17761,
	OPCUAID_WRITERGROUPTYPE_DATASETWRITERNAME_PLACEHOLDER_DIAGNOSTICS_TOTALERROR_CLASSIFICATION := 17762,
	OPCUAID_WRITERGROUPTYPE_DATASETWRITERNAME_PLACEHOLDER_DIAGNOSTICS_TOTALERROR_DIAGNOSTICSLEVEL := 17763,
	OPCUAID_WRITERGROUPTYPE_DATASETWRITERNAME_PLACEHOLDER_DIAGNOSTICS_TOTALERROR_TIMEFIRSTCHANGE := 17764,
	OPCUAID_WRITERGROUPTYPE_DATASETWRITERNAME_PLACEHOLDER_DIAGNOSTICS_SUBERROR := 17766,
	OPCUAID_WRITERGROUPTYPE_DATASETWRITERNAME_PLACEHOLDER_DIAGNOSTICS_COUNTERS_STATEERROR := 17768,
	OPCUAID_WRITERGROUPTYPE_DATASETWRITERNAME_PLACEHOLDER_DIAGNOSTICS_COUNTERS_STATEERROR_ACTIVE := 17769,
	OPCUAID_WRITERGROUPTYPE_DATASETWRITERNAME_PLACEHOLDER_DIAGNOSTICS_COUNTERS_STATEERROR_CLASSIFICATION := 17770,
	OPCUAID_WRITERGROUPTYPE_DATASETWRITERNAME_PLACEHOLDER_DIAGNOSTICS_COUNTERS_STATEERROR_DIAGNOSTICSLEVEL := 17771,
	OPCUAID_WRITERGROUPTYPE_DATASETWRITERNAME_PLACEHOLDER_DIAGNOSTICS_COUNTERS_STATEERROR_TIMEFIRSTCHANGE := 17772,
	OPCUAID_WRITERGROUPTYPE_DATASETWRITERNAME_PLACEHOLDER_DIAGNOSTICS_COUNTERS_STATEOPERATIONALBYMETHOD := 17773,
	OPCUAID_WRITERGROUPTYPE_DATASETWRITERNAME_PLACEHOLDER_DIAGNOSTICS_COUNTERS_STATEOPERATIONALBYMETHOD_ACTIVE := 17774,
	OPCUAID_WRITERGROUPTYPE_DATASETWRITERNAME_PLACEHOLDER_DIAGNOSTICS_COUNTERS_STATEOPERATIONALBYMETHOD_CLASSIFICATION := 17775,
	OPCUAID_WRITERGROUPTYPE_DATASETWRITERNAME_PLACEHOLDER_DIAGNOSTICS_COUNTERS_STATEOPERATIONALBYMETHOD_DIAGNOSTICSLEVEL := 17776,
	OPCUAID_WRITERGROUPTYPE_DATASETWRITERNAME_PLACEHOLDER_DIAGNOSTICS_COUNTERS_STATEOPERATIONALBYMETHOD_TIMEFIRSTCHANGE := 17777,
	OPCUAID_WRITERGROUPTYPE_DATASETWRITERNAME_PLACEHOLDER_DIAGNOSTICS_COUNTERS_STATEOPERATIONALBYPARENT := 17778,
	OPCUAID_WRITERGROUPTYPE_DATASETWRITERNAME_PLACEHOLDER_DIAGNOSTICS_COUNTERS_STATEOPERATIONALBYPARENT_ACTIVE := 17779,
	OPCUAID_WRITERGROUPTYPE_DATASETWRITERNAME_PLACEHOLDER_DIAGNOSTICS_COUNTERS_STATEOPERATIONALBYPARENT_CLASSIFICATION := 17780,
	OPCUAID_WRITERGROUPTYPE_DATASETWRITERNAME_PLACEHOLDER_DIAGNOSTICS_COUNTERS_STATEOPERATIONALBYPARENT_DIAGNOSTICSLEVEL := 17781,
	OPCUAID_WRITERGROUPTYPE_DATASETWRITERNAME_PLACEHOLDER_DIAGNOSTICS_COUNTERS_STATEOPERATIONALBYPARENT_TIMEFIRSTCHANGE := 17782,
	OPCUAID_WRITERGROUPTYPE_DATASETWRITERNAME_PLACEHOLDER_DIAGNOSTICS_COUNTERS_STATEOPERATIONALFROMERROR := 17783,
	OPCUAID_WRITERGROUPTYPE_DATASETWRITERNAME_PLACEHOLDER_DIAGNOSTICS_COUNTERS_STATEOPERATIONALFROMERROR_ACTIVE := 17784,
	OPCUAID_WRITERGROUPTYPE_DATASETWRITERNAME_PLACEHOLDER_DIAGNOSTICS_COUNTERS_STATEOPERATIONALFROMERROR_CLASSIFICATION := 17785,
	OPCUAID_WRITERGROUPTYPE_DATASETWRITERNAME_PLACEHOLDER_DIAGNOSTICS_COUNTERS_STATEOPERATIONALFROMERROR_DIAGNOSTICSLEVEL := 17786,
	OPCUAID_WRITERGROUPTYPE_DATASETWRITERNAME_PLACEHOLDER_DIAGNOSTICS_COUNTERS_STATEOPERATIONALFROMERROR_TIMEFIRSTCHANGE := 17787,
	OPCUAID_WRITERGROUPTYPE_DATASETWRITERNAME_PLACEHOLDER_DIAGNOSTICS_COUNTERS_STATEPAUSEDBYPARENT := 17788,
	OPCUAID_WRITERGROUPTYPE_DATASETWRITERNAME_PLACEHOLDER_DIAGNOSTICS_COUNTERS_STATEPAUSEDBYPARENT_ACTIVE := 17789,
	OPCUAID_WRITERGROUPTYPE_DATASETWRITERNAME_PLACEHOLDER_DIAGNOSTICS_COUNTERS_STATEPAUSEDBYPARENT_CLASSIFICATION := 17790,
	OPCUAID_WRITERGROUPTYPE_DATASETWRITERNAME_PLACEHOLDER_DIAGNOSTICS_COUNTERS_STATEPAUSEDBYPARENT_DIAGNOSTICSLEVEL := 17791,
	OPCUAID_WRITERGROUPTYPE_DATASETWRITERNAME_PLACEHOLDER_DIAGNOSTICS_COUNTERS_STATEPAUSEDBYPARENT_TIMEFIRSTCHANGE := 17792,
	OPCUAID_WRITERGROUPTYPE_DATASETWRITERNAME_PLACEHOLDER_DIAGNOSTICS_COUNTERS_STATEDISABLEDBYMETHOD := 17793,
	OPCUAID_WRITERGROUPTYPE_DATASETWRITERNAME_PLACEHOLDER_DIAGNOSTICS_COUNTERS_STATEDISABLEDBYMETHOD_ACTIVE := 17794,
	OPCUAID_WRITERGROUPTYPE_DATASETWRITERNAME_PLACEHOLDER_DIAGNOSTICS_COUNTERS_STATEDISABLEDBYMETHOD_CLASSIFICATION := 17795,
	OPCUAID_WRITERGROUPTYPE_DATASETWRITERNAME_PLACEHOLDER_DIAGNOSTICS_COUNTERS_STATEDISABLEDBYMETHOD_DIAGNOSTICSLEVEL := 17796,
	OPCUAID_WRITERGROUPTYPE_DATASETWRITERNAME_PLACEHOLDER_DIAGNOSTICS_COUNTERS_STATEDISABLEDBYMETHOD_TIMEFIRSTCHANGE := 17797,
	OPCUAID_WRITERGROUPTYPE_DATASETWRITERNAME_PLACEHOLDER_DIAGNOSTICS_COUNTERS_FAILEDDATASETMESSAGES := 17799,
	OPCUAID_WRITERGROUPTYPE_DATASETWRITERNAME_PLACEHOLDER_DIAGNOSTICS_COUNTERS_FAILEDDATASETMESSAGES_ACTIVE := 17800,
	OPCUAID_WRITERGROUPTYPE_DATASETWRITERNAME_PLACEHOLDER_DIAGNOSTICS_COUNTERS_FAILEDDATASETMESSAGES_CLASSIFICATION := 17801,
	OPCUAID_WRITERGROUPTYPE_DATASETWRITERNAME_PLACEHOLDER_DIAGNOSTICS_COUNTERS_FAILEDDATASETMESSAGES_DIAGNOSTICSLEVEL := 17802,
	OPCUAID_WRITERGROUPTYPE_DATASETWRITERNAME_PLACEHOLDER_DIAGNOSTICS_COUNTERS_FAILEDDATASETMESSAGES_TIMEFIRSTCHANGE := 17803,
	OPCUAID_WRITERGROUPTYPE_DATASETWRITERNAME_PLACEHOLDER_DIAGNOSTICS_LIVEVALUES_MESSAGESEQUENCENUMBER_DIAGNOSTICSLEVEL := 17805,
	OPCUAID_WRITERGROUPTYPE_DATASETWRITERNAME_PLACEHOLDER_DIAGNOSTICS_LIVEVALUES_STATUSCODE_DIAGNOSTICSLEVEL := 17807,
	OPCUAID_WRITERGROUPTYPE_DATASETWRITERNAME_PLACEHOLDER_DIAGNOSTICS_LIVEVALUES_MAJORVERSION_DIAGNOSTICSLEVEL := 17809,
	OPCUAID_WRITERGROUPTYPE_DATASETWRITERNAME_PLACEHOLDER_DIAGNOSTICS_LIVEVALUES_MINORVERSION_DIAGNOSTICSLEVEL := 17811,
	OPCUAID_WRITERGROUPTYPE_DIAGNOSTICS_DIAGNOSTICSLEVEL := 17813,
	OPCUAID_WRITERGROUPTYPE_DIAGNOSTICS_TOTALINFORMATION := 17814,
	OPCUAID_WRITERGROUPTYPE_DIAGNOSTICS_TOTALINFORMATION_ACTIVE := 17815,
	OPCUAID_WRITERGROUPTYPE_DIAGNOSTICS_TOTALINFORMATION_CLASSIFICATION := 17816,
	OPCUAID_WRITERGROUPTYPE_DIAGNOSTICS_TOTALINFORMATION_DIAGNOSTICSLEVEL := 17817,
	OPCUAID_WRITERGROUPTYPE_DIAGNOSTICS_TOTALINFORMATION_TIMEFIRSTCHANGE := 17818,
	OPCUAID_WRITERGROUPTYPE_DIAGNOSTICS_TOTALERROR := 17819,
	OPCUAID_WRITERGROUPTYPE_DIAGNOSTICS_TOTALERROR_ACTIVE := 17820,
	OPCUAID_WRITERGROUPTYPE_DIAGNOSTICS_TOTALERROR_CLASSIFICATION := 17821,
	OPCUAID_WRITERGROUPTYPE_DIAGNOSTICS_TOTALERROR_DIAGNOSTICSLEVEL := 17822,
	OPCUAID_WRITERGROUPTYPE_DIAGNOSTICS_TOTALERROR_TIMEFIRSTCHANGE := 17823,
	OPCUAID_WRITERGROUPTYPE_DIAGNOSTICS_SUBERROR := 17825,
	OPCUAID_WRITERGROUPTYPE_DIAGNOSTICS_COUNTERS_STATEERROR := 17827,
	OPCUAID_WRITERGROUPTYPE_DIAGNOSTICS_COUNTERS_STATEERROR_ACTIVE := 17828,
	OPCUAID_WRITERGROUPTYPE_DIAGNOSTICS_COUNTERS_STATEERROR_CLASSIFICATION := 17829,
	OPCUAID_WRITERGROUPTYPE_DIAGNOSTICS_COUNTERS_STATEERROR_DIAGNOSTICSLEVEL := 17830,
	OPCUAID_WRITERGROUPTYPE_DIAGNOSTICS_COUNTERS_STATEERROR_TIMEFIRSTCHANGE := 17831,
	OPCUAID_WRITERGROUPTYPE_DIAGNOSTICS_COUNTERS_STATEOPERATIONALBYMETHOD := 17832,
	OPCUAID_WRITERGROUPTYPE_DIAGNOSTICS_COUNTERS_STATEOPERATIONALBYMETHOD_ACTIVE := 17833,
	OPCUAID_WRITERGROUPTYPE_DIAGNOSTICS_COUNTERS_STATEOPERATIONALBYMETHOD_CLASSIFICATION := 17834,
	OPCUAID_WRITERGROUPTYPE_DIAGNOSTICS_COUNTERS_STATEOPERATIONALBYMETHOD_DIAGNOSTICSLEVEL := 17835,
	OPCUAID_WRITERGROUPTYPE_DIAGNOSTICS_COUNTERS_STATEOPERATIONALBYMETHOD_TIMEFIRSTCHANGE := 17836,
	OPCUAID_WRITERGROUPTYPE_DIAGNOSTICS_COUNTERS_STATEOPERATIONALBYPARENT := 17837,
	OPCUAID_WRITERGROUPTYPE_DIAGNOSTICS_COUNTERS_STATEOPERATIONALBYPARENT_ACTIVE := 17838,
	OPCUAID_WRITERGROUPTYPE_DIAGNOSTICS_COUNTERS_STATEOPERATIONALBYPARENT_CLASSIFICATION := 17839,
	OPCUAID_WRITERGROUPTYPE_DIAGNOSTICS_COUNTERS_STATEOPERATIONALBYPARENT_DIAGNOSTICSLEVEL := 17840,
	OPCUAID_WRITERGROUPTYPE_DIAGNOSTICS_COUNTERS_STATEOPERATIONALBYPARENT_TIMEFIRSTCHANGE := 17841,
	OPCUAID_WRITERGROUPTYPE_DIAGNOSTICS_COUNTERS_STATEOPERATIONALFROMERROR := 17842,
	OPCUAID_WRITERGROUPTYPE_DIAGNOSTICS_COUNTERS_STATEOPERATIONALFROMERROR_ACTIVE := 17843,
	OPCUAID_WRITERGROUPTYPE_DIAGNOSTICS_COUNTERS_STATEOPERATIONALFROMERROR_CLASSIFICATION := 17844,
	OPCUAID_WRITERGROUPTYPE_DIAGNOSTICS_COUNTERS_STATEOPERATIONALFROMERROR_DIAGNOSTICSLEVEL := 17845,
	OPCUAID_WRITERGROUPTYPE_DIAGNOSTICS_COUNTERS_STATEOPERATIONALFROMERROR_TIMEFIRSTCHANGE := 17846,
	OPCUAID_WRITERGROUPTYPE_DIAGNOSTICS_COUNTERS_STATEPAUSEDBYPARENT := 17847,
	OPCUAID_WRITERGROUPTYPE_DIAGNOSTICS_COUNTERS_STATEPAUSEDBYPARENT_ACTIVE := 17848,
	OPCUAID_WRITERGROUPTYPE_DIAGNOSTICS_COUNTERS_STATEPAUSEDBYPARENT_CLASSIFICATION := 17849,
	OPCUAID_WRITERGROUPTYPE_DIAGNOSTICS_COUNTERS_STATEPAUSEDBYPARENT_DIAGNOSTICSLEVEL := 17850,
	OPCUAID_WRITERGROUPTYPE_DIAGNOSTICS_COUNTERS_STATEPAUSEDBYPARENT_TIMEFIRSTCHANGE := 17851,
	OPCUAID_WRITERGROUPTYPE_DIAGNOSTICS_COUNTERS_STATEDISABLEDBYMETHOD := 17853,
	OPCUAID_WRITERGROUPTYPE_DIAGNOSTICS_COUNTERS_STATEDISABLEDBYMETHOD_ACTIVE := 17854,
	OPCUAID_WRITERGROUPTYPE_DIAGNOSTICS_COUNTERS_STATEDISABLEDBYMETHOD_CLASSIFICATION := 17855,
	OPCUAID_WRITERGROUPTYPE_DIAGNOSTICS_COUNTERS_STATEDISABLEDBYMETHOD_DIAGNOSTICSLEVEL := 17856,
	OPCUAID_WRITERGROUPTYPE_DIAGNOSTICS_COUNTERS_STATEDISABLEDBYMETHOD_TIMEFIRSTCHANGE := 17857,
	OPCUAID_WRITERGROUPTYPE_DIAGNOSTICS_COUNTERS_SENTNETWORKMESSAGES := 17859,
	OPCUAID_WRITERGROUPTYPE_DIAGNOSTICS_COUNTERS_SENTNETWORKMESSAGES_ACTIVE := 17864,
	OPCUAID_WRITERGROUPTYPE_DIAGNOSTICS_COUNTERS_SENTNETWORKMESSAGES_CLASSIFICATION := 17871,
	OPCUAID_WRITERGROUPTYPE_DIAGNOSTICS_COUNTERS_SENTNETWORKMESSAGES_DIAGNOSTICSLEVEL := 17872,
	OPCUAID_WRITERGROUPTYPE_DIAGNOSTICS_COUNTERS_SENTNETWORKMESSAGES_TIMEFIRSTCHANGE := 17873,
	OPCUAID_WRITERGROUPTYPE_DIAGNOSTICS_COUNTERS_FAILEDTRANSMISSIONS := 17874,
	OPCUAID_WRITERGROUPTYPE_DIAGNOSTICS_COUNTERS_FAILEDTRANSMISSIONS_ACTIVE := 17878,
	OPCUAID_WRITERGROUPTYPE_DIAGNOSTICS_COUNTERS_FAILEDTRANSMISSIONS_CLASSIFICATION := 17885,
	OPCUAID_WRITERGROUPTYPE_DIAGNOSTICS_COUNTERS_FAILEDTRANSMISSIONS_DIAGNOSTICSLEVEL := 17892,
	OPCUAID_WRITERGROUPTYPE_DIAGNOSTICS_COUNTERS_FAILEDTRANSMISSIONS_TIMEFIRSTCHANGE := 17899,
	OPCUAID_WRITERGROUPTYPE_DIAGNOSTICS_COUNTERS_ENCRYPTIONERRORS := 17900,
	OPCUAID_WRITERGROUPTYPE_DIAGNOSTICS_COUNTERS_ENCRYPTIONERRORS_ACTIVE := 17901,
	OPCUAID_WRITERGROUPTYPE_DIAGNOSTICS_COUNTERS_ENCRYPTIONERRORS_CLASSIFICATION := 17902,
	OPCUAID_WRITERGROUPTYPE_DIAGNOSTICS_COUNTERS_ENCRYPTIONERRORS_DIAGNOSTICSLEVEL := 17903,
	OPCUAID_WRITERGROUPTYPE_DIAGNOSTICS_COUNTERS_ENCRYPTIONERRORS_TIMEFIRSTCHANGE := 17906,
	OPCUAID_WRITERGROUPTYPE_DIAGNOSTICS_LIVEVALUES_CONFIGUREDDATASETWRITERS := 17913,
	OPCUAID_WRITERGROUPTYPE_DIAGNOSTICS_LIVEVALUES_CONFIGUREDDATASETWRITERS_DIAGNOSTICSLEVEL := 17920,
	OPCUAID_WRITERGROUPTYPE_DIAGNOSTICS_LIVEVALUES_OPERATIONALDATASETWRITERS := 17927,
	OPCUAID_WRITERGROUPTYPE_DIAGNOSTICS_LIVEVALUES_OPERATIONALDATASETWRITERS_DIAGNOSTICSLEVEL := 17934,
	OPCUAID_WRITERGROUPTYPE_DIAGNOSTICS_LIVEVALUES_SECURITYTOKENID_DIAGNOSTICSLEVEL := 17948,
	OPCUAID_WRITERGROUPTYPE_DIAGNOSTICS_LIVEVALUES_TIMETONEXTTOKENID_DIAGNOSTICSLEVEL := 17962,
	OPCUAID_WRITERGROUPTYPE_ADDDATASETWRITER_INPUTARGUMENTS := 17976,
	OPCUAID_WRITERGROUPTYPE_ADDDATASETWRITER_OUTPUTARGUMENTS := 17987,
	OPCUAID_WRITERGROUPTYPE_REMOVEDATASETWRITER_INPUTARGUMENTS := 17993,
	OPCUAID_READERGROUPTYPE_STATUS_STATE := 18068,
	OPCUAID_READERGROUPTYPE_DATASETREADERNAME_PLACEHOLDER_PUBLISHERID := 18077,
	OPCUAID_READERGROUPTYPE_DATASETREADERNAME_PLACEHOLDER_WRITERGROUPID := 18078,
	OPCUAID_READERGROUPTYPE_DATASETREADERNAME_PLACEHOLDER_DATASETWRITERID := 18079,
	OPCUAID_READERGROUPTYPE_DATASETREADERNAME_PLACEHOLDER_DATASETMETADATA := 18080,
	OPCUAID_READERGROUPTYPE_DATASETREADERNAME_PLACEHOLDER_DATASETFIELDCONTENTMASK := 18081,
	OPCUAID_READERGROUPTYPE_DATASETREADERNAME_PLACEHOLDER_MESSAGERECEIVETIMEOUT := 18082,
	OPCUAID_READERGROUPTYPE_DATASETREADERNAME_PLACEHOLDER_DATASETREADERPROPERTIES := 17492,
	OPCUAID_READERGROUPTYPE_DATASETREADERNAME_PLACEHOLDER_STATUS_STATE := 18089,
	OPCUAID_READERGROUPTYPE_DATASETREADERNAME_PLACEHOLDER_DIAGNOSTICS_DIAGNOSTICSLEVEL := 18093,
	OPCUAID_READERGROUPTYPE_DATASETREADERNAME_PLACEHOLDER_DIAGNOSTICS_TOTALINFORMATION := 18094,
	OPCUAID_READERGROUPTYPE_DATASETREADERNAME_PLACEHOLDER_DIAGNOSTICS_TOTALINFORMATION_ACTIVE := 18095,
	OPCUAID_READERGROUPTYPE_DATASETREADERNAME_PLACEHOLDER_DIAGNOSTICS_TOTALINFORMATION_CLASSIFICATION := 18096,
	OPCUAID_READERGROUPTYPE_DATASETREADERNAME_PLACEHOLDER_DIAGNOSTICS_TOTALINFORMATION_DIAGNOSTICSLEVEL := 18097,
	OPCUAID_READERGROUPTYPE_DATASETREADERNAME_PLACEHOLDER_DIAGNOSTICS_TOTALINFORMATION_TIMEFIRSTCHANGE := 18098,
	OPCUAID_READERGROUPTYPE_DATASETREADERNAME_PLACEHOLDER_DIAGNOSTICS_TOTALERROR := 18099,
	OPCUAID_READERGROUPTYPE_DATASETREADERNAME_PLACEHOLDER_DIAGNOSTICS_TOTALERROR_ACTIVE := 18100,
	OPCUAID_READERGROUPTYPE_DATASETREADERNAME_PLACEHOLDER_DIAGNOSTICS_TOTALERROR_CLASSIFICATION := 18101,
	OPCUAID_READERGROUPTYPE_DATASETREADERNAME_PLACEHOLDER_DIAGNOSTICS_TOTALERROR_DIAGNOSTICSLEVEL := 18102,
	OPCUAID_READERGROUPTYPE_DATASETREADERNAME_PLACEHOLDER_DIAGNOSTICS_TOTALERROR_TIMEFIRSTCHANGE := 18103,
	OPCUAID_READERGROUPTYPE_DATASETREADERNAME_PLACEHOLDER_DIAGNOSTICS_SUBERROR := 18105,
	OPCUAID_READERGROUPTYPE_DATASETREADERNAME_PLACEHOLDER_DIAGNOSTICS_COUNTERS_STATEERROR := 18107,
	OPCUAID_READERGROUPTYPE_DATASETREADERNAME_PLACEHOLDER_DIAGNOSTICS_COUNTERS_STATEERROR_ACTIVE := 18108,
	OPCUAID_READERGROUPTYPE_DATASETREADERNAME_PLACEHOLDER_DIAGNOSTICS_COUNTERS_STATEERROR_CLASSIFICATION := 18109,
	OPCUAID_READERGROUPTYPE_DATASETREADERNAME_PLACEHOLDER_DIAGNOSTICS_COUNTERS_STATEERROR_DIAGNOSTICSLEVEL := 18110,
	OPCUAID_READERGROUPTYPE_DATASETREADERNAME_PLACEHOLDER_DIAGNOSTICS_COUNTERS_STATEERROR_TIMEFIRSTCHANGE := 18111,
	OPCUAID_READERGROUPTYPE_DATASETREADERNAME_PLACEHOLDER_DIAGNOSTICS_COUNTERS_STATEOPERATIONALBYMETHOD := 18112,
	OPCUAID_READERGROUPTYPE_DATASETREADERNAME_PLACEHOLDER_DIAGNOSTICS_COUNTERS_STATEOPERATIONALBYMETHOD_ACTIVE := 18113,
	OPCUAID_READERGROUPTYPE_DATASETREADERNAME_PLACEHOLDER_DIAGNOSTICS_COUNTERS_STATEOPERATIONALBYMETHOD_CLASSIFICATION := 18114,
	OPCUAID_READERGROUPTYPE_DATASETREADERNAME_PLACEHOLDER_DIAGNOSTICS_COUNTERS_STATEOPERATIONALBYMETHOD_DIAGNOSTICSLEVEL := 18115,
	OPCUAID_READERGROUPTYPE_DATASETREADERNAME_PLACEHOLDER_DIAGNOSTICS_COUNTERS_STATEOPERATIONALBYMETHOD_TIMEFIRSTCHANGE := 18116,
	OPCUAID_READERGROUPTYPE_DATASETREADERNAME_PLACEHOLDER_DIAGNOSTICS_COUNTERS_STATEOPERATIONALBYPARENT := 18117,
	OPCUAID_READERGROUPTYPE_DATASETREADERNAME_PLACEHOLDER_DIAGNOSTICS_COUNTERS_STATEOPERATIONALBYPARENT_ACTIVE := 18118,
	OPCUAID_READERGROUPTYPE_DATASETREADERNAME_PLACEHOLDER_DIAGNOSTICS_COUNTERS_STATEOPERATIONALBYPARENT_CLASSIFICATION := 18119,
	OPCUAID_READERGROUPTYPE_DATASETREADERNAME_PLACEHOLDER_DIAGNOSTICS_COUNTERS_STATEOPERATIONALBYPARENT_DIAGNOSTICSLEVEL := 18120,
	OPCUAID_READERGROUPTYPE_DATASETREADERNAME_PLACEHOLDER_DIAGNOSTICS_COUNTERS_STATEOPERATIONALBYPARENT_TIMEFIRSTCHANGE := 18121,
	OPCUAID_READERGROUPTYPE_DATASETREADERNAME_PLACEHOLDER_DIAGNOSTICS_COUNTERS_STATEOPERATIONALFROMERROR := 18122,
	OPCUAID_READERGROUPTYPE_DATASETREADERNAME_PLACEHOLDER_DIAGNOSTICS_COUNTERS_STATEOPERATIONALFROMERROR_ACTIVE := 18123,
	OPCUAID_READERGROUPTYPE_DATASETREADERNAME_PLACEHOLDER_DIAGNOSTICS_COUNTERS_STATEOPERATIONALFROMERROR_CLASSIFICATION := 18124,
	OPCUAID_READERGROUPTYPE_DATASETREADERNAME_PLACEHOLDER_DIAGNOSTICS_COUNTERS_STATEOPERATIONALFROMERROR_DIAGNOSTICSLEVEL := 18125,
	OPCUAID_READERGROUPTYPE_DATASETREADERNAME_PLACEHOLDER_DIAGNOSTICS_COUNTERS_STATEOPERATIONALFROMERROR_TIMEFIRSTCHANGE := 18126,
	OPCUAID_READERGROUPTYPE_DATASETREADERNAME_PLACEHOLDER_DIAGNOSTICS_COUNTERS_STATEPAUSEDBYPARENT := 18127,
	OPCUAID_READERGROUPTYPE_DATASETREADERNAME_PLACEHOLDER_DIAGNOSTICS_COUNTERS_STATEPAUSEDBYPARENT_ACTIVE := 18128,
	OPCUAID_READERGROUPTYPE_DATASETREADERNAME_PLACEHOLDER_DIAGNOSTICS_COUNTERS_STATEPAUSEDBYPARENT_CLASSIFICATION := 18129,
	OPCUAID_READERGROUPTYPE_DATASETREADERNAME_PLACEHOLDER_DIAGNOSTICS_COUNTERS_STATEPAUSEDBYPARENT_DIAGNOSTICSLEVEL := 18130,
	OPCUAID_READERGROUPTYPE_DATASETREADERNAME_PLACEHOLDER_DIAGNOSTICS_COUNTERS_STATEPAUSEDBYPARENT_TIMEFIRSTCHANGE := 18131,
	OPCUAID_READERGROUPTYPE_DATASETREADERNAME_PLACEHOLDER_DIAGNOSTICS_COUNTERS_STATEDISABLEDBYMETHOD := 18132,
	OPCUAID_READERGROUPTYPE_DATASETREADERNAME_PLACEHOLDER_DIAGNOSTICS_COUNTERS_STATEDISABLEDBYMETHOD_ACTIVE := 18133,
	OPCUAID_READERGROUPTYPE_DATASETREADERNAME_PLACEHOLDER_DIAGNOSTICS_COUNTERS_STATEDISABLEDBYMETHOD_CLASSIFICATION := 18134,
	OPCUAID_READERGROUPTYPE_DATASETREADERNAME_PLACEHOLDER_DIAGNOSTICS_COUNTERS_STATEDISABLEDBYMETHOD_DIAGNOSTICSLEVEL := 18135,
	OPCUAID_READERGROUPTYPE_DATASETREADERNAME_PLACEHOLDER_DIAGNOSTICS_COUNTERS_STATEDISABLEDBYMETHOD_TIMEFIRSTCHANGE := 18136,
	OPCUAID_READERGROUPTYPE_DATASETREADERNAME_PLACEHOLDER_DIAGNOSTICS_COUNTERS_FAILEDDATASETMESSAGES := 18138,
	OPCUAID_READERGROUPTYPE_DATASETREADERNAME_PLACEHOLDER_DIAGNOSTICS_COUNTERS_FAILEDDATASETMESSAGES_ACTIVE := 18139,
	OPCUAID_READERGROUPTYPE_DATASETREADERNAME_PLACEHOLDER_DIAGNOSTICS_COUNTERS_FAILEDDATASETMESSAGES_CLASSIFICATION := 18140,
	OPCUAID_READERGROUPTYPE_DATASETREADERNAME_PLACEHOLDER_DIAGNOSTICS_COUNTERS_FAILEDDATASETMESSAGES_DIAGNOSTICSLEVEL := 18141,
	OPCUAID_READERGROUPTYPE_DATASETREADERNAME_PLACEHOLDER_DIAGNOSTICS_COUNTERS_FAILEDDATASETMESSAGES_TIMEFIRSTCHANGE := 18142,
	OPCUAID_READERGROUPTYPE_DATASETREADERNAME_PLACEHOLDER_DIAGNOSTICS_COUNTERS_DECRYPTIONERRORS_ACTIVE := 18144,
	OPCUAID_READERGROUPTYPE_DATASETREADERNAME_PLACEHOLDER_DIAGNOSTICS_COUNTERS_DECRYPTIONERRORS_CLASSIFICATION := 18145,
	OPCUAID_READERGROUPTYPE_DATASETREADERNAME_PLACEHOLDER_DIAGNOSTICS_COUNTERS_DECRYPTIONERRORS_DIAGNOSTICSLEVEL := 18146,
	OPCUAID_READERGROUPTYPE_DATASETREADERNAME_PLACEHOLDER_DIAGNOSTICS_COUNTERS_DECRYPTIONERRORS_TIMEFIRSTCHANGE := 18147,
	OPCUAID_READERGROUPTYPE_DATASETREADERNAME_PLACEHOLDER_DIAGNOSTICS_LIVEVALUES_MESSAGESEQUENCENUMBER_DIAGNOSTICSLEVEL := 18149,
	OPCUAID_READERGROUPTYPE_DATASETREADERNAME_PLACEHOLDER_DIAGNOSTICS_LIVEVALUES_STATUSCODE_DIAGNOSTICSLEVEL := 18151,
	OPCUAID_READERGROUPTYPE_DATASETREADERNAME_PLACEHOLDER_DIAGNOSTICS_LIVEVALUES_MAJORVERSION_DIAGNOSTICSLEVEL := 18153,
	OPCUAID_READERGROUPTYPE_DATASETREADERNAME_PLACEHOLDER_DIAGNOSTICS_LIVEVALUES_MINORVERSION_DIAGNOSTICSLEVEL := 18158,
	OPCUAID_READERGROUPTYPE_DATASETREADERNAME_PLACEHOLDER_DIAGNOSTICS_LIVEVALUES_SECURITYTOKENID_DIAGNOSTICSLEVEL := 21003,
	OPCUAID_READERGROUPTYPE_DATASETREADERNAME_PLACEHOLDER_DIAGNOSTICS_LIVEVALUES_TIMETONEXTTOKENID_DIAGNOSTICSLEVEL := 21005,
	OPCUAID_READERGROUPTYPE_DATASETREADERNAME_PLACEHOLDER_SUBSCRIBEDDATASET_DATASETMETADATA := 21007,
	OPCUAID_READERGROUPTYPE_DATASETREADERNAME_PLACEHOLDER_SUBSCRIBEDDATASET_MESSAGERECEIVETIMEOUT := 21008,
	OPCUAID_READERGROUPTYPE_DATASETREADERNAME_PLACEHOLDER_CREATETARGETVARIABLES_INPUTARGUMENTS := 21010,
	OPCUAID_READERGROUPTYPE_DATASETREADERNAME_PLACEHOLDER_CREATETARGETVARIABLES_OUTPUTARGUMENTS := 21011,
	OPCUAID_READERGROUPTYPE_DATASETREADERNAME_PLACEHOLDER_CREATEDATASETMIRROR_INPUTARGUMENTS := 21013,
	OPCUAID_READERGROUPTYPE_DATASETREADERNAME_PLACEHOLDER_CREATEDATASETMIRROR_OUTPUTARGUMENTS := 21014,
	OPCUAID_READERGROUPTYPE_DIAGNOSTICS_DIAGNOSTICSLEVEL := 21016,
	OPCUAID_READERGROUPTYPE_DIAGNOSTICS_TOTALINFORMATION := 21017,
	OPCUAID_READERGROUPTYPE_DIAGNOSTICS_TOTALINFORMATION_ACTIVE := 21018,
	OPCUAID_READERGROUPTYPE_DIAGNOSTICS_TOTALINFORMATION_CLASSIFICATION := 21019,
	OPCUAID_READERGROUPTYPE_DIAGNOSTICS_TOTALINFORMATION_DIAGNOSTICSLEVEL := 21020,
	OPCUAID_READERGROUPTYPE_DIAGNOSTICS_TOTALINFORMATION_TIMEFIRSTCHANGE := 21021,
	OPCUAID_READERGROUPTYPE_DIAGNOSTICS_TOTALERROR := 21022,
	OPCUAID_READERGROUPTYPE_DIAGNOSTICS_TOTALERROR_ACTIVE := 21023,
	OPCUAID_READERGROUPTYPE_DIAGNOSTICS_TOTALERROR_CLASSIFICATION := 21024,
	OPCUAID_READERGROUPTYPE_DIAGNOSTICS_TOTALERROR_DIAGNOSTICSLEVEL := 21025,
	OPCUAID_READERGROUPTYPE_DIAGNOSTICS_TOTALERROR_TIMEFIRSTCHANGE := 21026,
	OPCUAID_READERGROUPTYPE_DIAGNOSTICS_SUBERROR := 21028,
	OPCUAID_READERGROUPTYPE_DIAGNOSTICS_COUNTERS_STATEERROR := 21030,
	OPCUAID_READERGROUPTYPE_DIAGNOSTICS_COUNTERS_STATEERROR_ACTIVE := 21031,
	OPCUAID_READERGROUPTYPE_DIAGNOSTICS_COUNTERS_STATEERROR_CLASSIFICATION := 21032,
	OPCUAID_READERGROUPTYPE_DIAGNOSTICS_COUNTERS_STATEERROR_DIAGNOSTICSLEVEL := 21033,
	OPCUAID_READERGROUPTYPE_DIAGNOSTICS_COUNTERS_STATEERROR_TIMEFIRSTCHANGE := 21034,
	OPCUAID_READERGROUPTYPE_DIAGNOSTICS_COUNTERS_STATEOPERATIONALBYMETHOD := 21035,
	OPCUAID_READERGROUPTYPE_DIAGNOSTICS_COUNTERS_STATEOPERATIONALBYMETHOD_ACTIVE := 21036,
	OPCUAID_READERGROUPTYPE_DIAGNOSTICS_COUNTERS_STATEOPERATIONALBYMETHOD_CLASSIFICATION := 21037,
	OPCUAID_READERGROUPTYPE_DIAGNOSTICS_COUNTERS_STATEOPERATIONALBYMETHOD_DIAGNOSTICSLEVEL := 21038,
	OPCUAID_READERGROUPTYPE_DIAGNOSTICS_COUNTERS_STATEOPERATIONALBYMETHOD_TIMEFIRSTCHANGE := 21039,
	OPCUAID_READERGROUPTYPE_DIAGNOSTICS_COUNTERS_STATEOPERATIONALBYPARENT := 21040,
	OPCUAID_READERGROUPTYPE_DIAGNOSTICS_COUNTERS_STATEOPERATIONALBYPARENT_ACTIVE := 21041,
	OPCUAID_READERGROUPTYPE_DIAGNOSTICS_COUNTERS_STATEOPERATIONALBYPARENT_CLASSIFICATION := 21042,
	OPCUAID_READERGROUPTYPE_DIAGNOSTICS_COUNTERS_STATEOPERATIONALBYPARENT_DIAGNOSTICSLEVEL := 21043,
	OPCUAID_READERGROUPTYPE_DIAGNOSTICS_COUNTERS_STATEOPERATIONALBYPARENT_TIMEFIRSTCHANGE := 21044,
	OPCUAID_READERGROUPTYPE_DIAGNOSTICS_COUNTERS_STATEOPERATIONALFROMERROR := 21045,
	OPCUAID_READERGROUPTYPE_DIAGNOSTICS_COUNTERS_STATEOPERATIONALFROMERROR_ACTIVE := 21046,
	OPCUAID_READERGROUPTYPE_DIAGNOSTICS_COUNTERS_STATEOPERATIONALFROMERROR_CLASSIFICATION := 21047,
	OPCUAID_READERGROUPTYPE_DIAGNOSTICS_COUNTERS_STATEOPERATIONALFROMERROR_DIAGNOSTICSLEVEL := 21048,
	OPCUAID_READERGROUPTYPE_DIAGNOSTICS_COUNTERS_STATEOPERATIONALFROMERROR_TIMEFIRSTCHANGE := 21049,
	OPCUAID_READERGROUPTYPE_DIAGNOSTICS_COUNTERS_STATEPAUSEDBYPARENT := 21050,
	OPCUAID_READERGROUPTYPE_DIAGNOSTICS_COUNTERS_STATEPAUSEDBYPARENT_ACTIVE := 21051,
	OPCUAID_READERGROUPTYPE_DIAGNOSTICS_COUNTERS_STATEPAUSEDBYPARENT_CLASSIFICATION := 21052,
	OPCUAID_READERGROUPTYPE_DIAGNOSTICS_COUNTERS_STATEPAUSEDBYPARENT_DIAGNOSTICSLEVEL := 21053,
	OPCUAID_READERGROUPTYPE_DIAGNOSTICS_COUNTERS_STATEPAUSEDBYPARENT_TIMEFIRSTCHANGE := 21054,
	OPCUAID_READERGROUPTYPE_DIAGNOSTICS_COUNTERS_STATEDISABLEDBYMETHOD := 21055,
	OPCUAID_READERGROUPTYPE_DIAGNOSTICS_COUNTERS_STATEDISABLEDBYMETHOD_ACTIVE := 21056,
	OPCUAID_READERGROUPTYPE_DIAGNOSTICS_COUNTERS_STATEDISABLEDBYMETHOD_CLASSIFICATION := 21057,
	OPCUAID_READERGROUPTYPE_DIAGNOSTICS_COUNTERS_STATEDISABLEDBYMETHOD_DIAGNOSTICSLEVEL := 21058,
	OPCUAID_READERGROUPTYPE_DIAGNOSTICS_COUNTERS_STATEDISABLEDBYMETHOD_TIMEFIRSTCHANGE := 21059,
	OPCUAID_READERGROUPTYPE_DIAGNOSTICS_COUNTERS_RECEIVEDNETWORKMESSAGES := 21061,
	OPCUAID_READERGROUPTYPE_DIAGNOSTICS_COUNTERS_RECEIVEDNETWORKMESSAGES_ACTIVE := 21062,
	OPCUAID_READERGROUPTYPE_DIAGNOSTICS_COUNTERS_RECEIVEDNETWORKMESSAGES_CLASSIFICATION := 21063,
	OPCUAID_READERGROUPTYPE_DIAGNOSTICS_COUNTERS_RECEIVEDNETWORKMESSAGES_DIAGNOSTICSLEVEL := 21064,
	OPCUAID_READERGROUPTYPE_DIAGNOSTICS_COUNTERS_RECEIVEDNETWORKMESSAGES_TIMEFIRSTCHANGE := 21065,
	OPCUAID_READERGROUPTYPE_DIAGNOSTICS_COUNTERS_RECEIVEDINVALIDNETWORKMESSAGES_ACTIVE := 21067,
	OPCUAID_READERGROUPTYPE_DIAGNOSTICS_COUNTERS_RECEIVEDINVALIDNETWORKMESSAGES_CLASSIFICATION := 21068,
	OPCUAID_READERGROUPTYPE_DIAGNOSTICS_COUNTERS_RECEIVEDINVALIDNETWORKMESSAGES_DIAGNOSTICSLEVEL := 21069,
	OPCUAID_READERGROUPTYPE_DIAGNOSTICS_COUNTERS_RECEIVEDINVALIDNETWORKMESSAGES_TIMEFIRSTCHANGE := 21070,
	OPCUAID_READERGROUPTYPE_DIAGNOSTICS_COUNTERS_DECRYPTIONERRORS_ACTIVE := 21072,
	OPCUAID_READERGROUPTYPE_DIAGNOSTICS_COUNTERS_DECRYPTIONERRORS_CLASSIFICATION := 21073,
	OPCUAID_READERGROUPTYPE_DIAGNOSTICS_COUNTERS_DECRYPTIONERRORS_DIAGNOSTICSLEVEL := 21074,
	OPCUAID_READERGROUPTYPE_DIAGNOSTICS_COUNTERS_DECRYPTIONERRORS_TIMEFIRSTCHANGE := 21075,
	OPCUAID_READERGROUPTYPE_DIAGNOSTICS_LIVEVALUES_CONFIGUREDDATASETREADERS := 21076,
	OPCUAID_READERGROUPTYPE_DIAGNOSTICS_LIVEVALUES_CONFIGUREDDATASETREADERS_DIAGNOSTICSLEVEL := 21077,
	OPCUAID_READERGROUPTYPE_DIAGNOSTICS_LIVEVALUES_OPERATIONALDATASETREADERS := 21078,
	OPCUAID_READERGROUPTYPE_DIAGNOSTICS_LIVEVALUES_OPERATIONALDATASETREADERS_DIAGNOSTICSLEVEL := 21079,
	OPCUAID_READERGROUPTYPE_ADDDATASETREADER_INPUTARGUMENTS := 21083,
	OPCUAID_READERGROUPTYPE_ADDDATASETREADER_OUTPUTARGUMENTS := 21084,
	OPCUAID_READERGROUPTYPE_REMOVEDATASETREADER_INPUTARGUMENTS := 21086,
	OPCUAID_DATASETWRITERTYPE_DATASETWRITERID := 21092,
	OPCUAID_DATASETWRITERTYPE_DATASETFIELDCONTENTMASK := 21093,
	OPCUAID_DATASETWRITERTYPE_KEYFRAMECOUNT := 21094,
	OPCUAID_DATASETWRITERTYPE_DATASETWRITERPROPERTIES := 17493,
	OPCUAID_DATASETWRITERTYPE_STATUS_STATE := 15300,
	OPCUAID_DATASETWRITERTYPE_DIAGNOSTICS_DIAGNOSTICSLEVEL := 19551,
	OPCUAID_DATASETWRITERTYPE_DIAGNOSTICS_TOTALINFORMATION := 19552,
	OPCUAID_DATASETWRITERTYPE_DIAGNOSTICS_TOTALINFORMATION_ACTIVE := 19553,
	OPCUAID_DATASETWRITERTYPE_DIAGNOSTICS_TOTALINFORMATION_CLASSIFICATION := 19554,
	OPCUAID_DATASETWRITERTYPE_DIAGNOSTICS_TOTALINFORMATION_DIAGNOSTICSLEVEL := 19555,
	OPCUAID_DATASETWRITERTYPE_DIAGNOSTICS_TOTALINFORMATION_TIMEFIRSTCHANGE := 19556,
	OPCUAID_DATASETWRITERTYPE_DIAGNOSTICS_TOTALERROR := 19557,
	OPCUAID_DATASETWRITERTYPE_DIAGNOSTICS_TOTALERROR_ACTIVE := 19558,
	OPCUAID_DATASETWRITERTYPE_DIAGNOSTICS_TOTALERROR_CLASSIFICATION := 19559,
	OPCUAID_DATASETWRITERTYPE_DIAGNOSTICS_TOTALERROR_DIAGNOSTICSLEVEL := 19560,
	OPCUAID_DATASETWRITERTYPE_DIAGNOSTICS_TOTALERROR_TIMEFIRSTCHANGE := 19561,
	OPCUAID_DATASETWRITERTYPE_DIAGNOSTICS_SUBERROR := 19563,
	OPCUAID_DATASETWRITERTYPE_DIAGNOSTICS_COUNTERS_STATEERROR := 19565,
	OPCUAID_DATASETWRITERTYPE_DIAGNOSTICS_COUNTERS_STATEERROR_ACTIVE := 19566,
	OPCUAID_DATASETWRITERTYPE_DIAGNOSTICS_COUNTERS_STATEERROR_CLASSIFICATION := 19567,
	OPCUAID_DATASETWRITERTYPE_DIAGNOSTICS_COUNTERS_STATEERROR_DIAGNOSTICSLEVEL := 19568,
	OPCUAID_DATASETWRITERTYPE_DIAGNOSTICS_COUNTERS_STATEERROR_TIMEFIRSTCHANGE := 19569,
	OPCUAID_DATASETWRITERTYPE_DIAGNOSTICS_COUNTERS_STATEOPERATIONALBYMETHOD := 19570,
	OPCUAID_DATASETWRITERTYPE_DIAGNOSTICS_COUNTERS_STATEOPERATIONALBYMETHOD_ACTIVE := 19571,
	OPCUAID_DATASETWRITERTYPE_DIAGNOSTICS_COUNTERS_STATEOPERATIONALBYMETHOD_CLASSIFICATION := 19572,
	OPCUAID_DATASETWRITERTYPE_DIAGNOSTICS_COUNTERS_STATEOPERATIONALBYMETHOD_DIAGNOSTICSLEVEL := 19573,
	OPCUAID_DATASETWRITERTYPE_DIAGNOSTICS_COUNTERS_STATEOPERATIONALBYMETHOD_TIMEFIRSTCHANGE := 19574,
	OPCUAID_DATASETWRITERTYPE_DIAGNOSTICS_COUNTERS_STATEOPERATIONALBYPARENT := 19575,
	OPCUAID_DATASETWRITERTYPE_DIAGNOSTICS_COUNTERS_STATEOPERATIONALBYPARENT_ACTIVE := 19576,
	OPCUAID_DATASETWRITERTYPE_DIAGNOSTICS_COUNTERS_STATEOPERATIONALBYPARENT_CLASSIFICATION := 19577,
	OPCUAID_DATASETWRITERTYPE_DIAGNOSTICS_COUNTERS_STATEOPERATIONALBYPARENT_DIAGNOSTICSLEVEL := 19578,
	OPCUAID_DATASETWRITERTYPE_DIAGNOSTICS_COUNTERS_STATEOPERATIONALBYPARENT_TIMEFIRSTCHANGE := 19579,
	OPCUAID_DATASETWRITERTYPE_DIAGNOSTICS_COUNTERS_STATEOPERATIONALFROMERROR := 19580,
	OPCUAID_DATASETWRITERTYPE_DIAGNOSTICS_COUNTERS_STATEOPERATIONALFROMERROR_ACTIVE := 19581,
	OPCUAID_DATASETWRITERTYPE_DIAGNOSTICS_COUNTERS_STATEOPERATIONALFROMERROR_CLASSIFICATION := 19582,
	OPCUAID_DATASETWRITERTYPE_DIAGNOSTICS_COUNTERS_STATEOPERATIONALFROMERROR_DIAGNOSTICSLEVEL := 19583,
	OPCUAID_DATASETWRITERTYPE_DIAGNOSTICS_COUNTERS_STATEOPERATIONALFROMERROR_TIMEFIRSTCHANGE := 19584,
	OPCUAID_DATASETWRITERTYPE_DIAGNOSTICS_COUNTERS_STATEPAUSEDBYPARENT := 19585,
	OPCUAID_DATASETWRITERTYPE_DIAGNOSTICS_COUNTERS_STATEPAUSEDBYPARENT_ACTIVE := 19586,
	OPCUAID_DATASETWRITERTYPE_DIAGNOSTICS_COUNTERS_STATEPAUSEDBYPARENT_CLASSIFICATION := 19587,
	OPCUAID_DATASETWRITERTYPE_DIAGNOSTICS_COUNTERS_STATEPAUSEDBYPARENT_DIAGNOSTICSLEVEL := 19588,
	OPCUAID_DATASETWRITERTYPE_DIAGNOSTICS_COUNTERS_STATEPAUSEDBYPARENT_TIMEFIRSTCHANGE := 19589,
	OPCUAID_DATASETWRITERTYPE_DIAGNOSTICS_COUNTERS_STATEDISABLEDBYMETHOD := 19590,
	OPCUAID_DATASETWRITERTYPE_DIAGNOSTICS_COUNTERS_STATEDISABLEDBYMETHOD_ACTIVE := 19591,
	OPCUAID_DATASETWRITERTYPE_DIAGNOSTICS_COUNTERS_STATEDISABLEDBYMETHOD_CLASSIFICATION := 19592,
	OPCUAID_DATASETWRITERTYPE_DIAGNOSTICS_COUNTERS_STATEDISABLEDBYMETHOD_DIAGNOSTICSLEVEL := 19593,
	OPCUAID_DATASETWRITERTYPE_DIAGNOSTICS_COUNTERS_STATEDISABLEDBYMETHOD_TIMEFIRSTCHANGE := 19594,
	OPCUAID_DATASETWRITERTYPE_DIAGNOSTICS_COUNTERS_FAILEDDATASETMESSAGES := 19596,
	OPCUAID_DATASETWRITERTYPE_DIAGNOSTICS_COUNTERS_FAILEDDATASETMESSAGES_ACTIVE := 19597,
	OPCUAID_DATASETWRITERTYPE_DIAGNOSTICS_COUNTERS_FAILEDDATASETMESSAGES_CLASSIFICATION := 19598,
	OPCUAID_DATASETWRITERTYPE_DIAGNOSTICS_COUNTERS_FAILEDDATASETMESSAGES_DIAGNOSTICSLEVEL := 19599,
	OPCUAID_DATASETWRITERTYPE_DIAGNOSTICS_COUNTERS_FAILEDDATASETMESSAGES_TIMEFIRSTCHANGE := 19600,
	OPCUAID_DATASETWRITERTYPE_DIAGNOSTICS_LIVEVALUES_MESSAGESEQUENCENUMBER_DIAGNOSTICSLEVEL := 19602,
	OPCUAID_DATASETWRITERTYPE_DIAGNOSTICS_LIVEVALUES_STATUSCODE_DIAGNOSTICSLEVEL := 19604,
	OPCUAID_DATASETWRITERTYPE_DIAGNOSTICS_LIVEVALUES_MAJORVERSION_DIAGNOSTICSLEVEL := 19606,
	OPCUAID_DATASETWRITERTYPE_DIAGNOSTICS_LIVEVALUES_MINORVERSION_DIAGNOSTICSLEVEL := 19608,
	OPCUAID_DATASETREADERTYPE_PUBLISHERID := 21097,
	OPCUAID_DATASETREADERTYPE_WRITERGROUPID := 21098,
	OPCUAID_DATASETREADERTYPE_DATASETWRITERID := 21099,
	OPCUAID_DATASETREADERTYPE_DATASETMETADATA := 21100,
	OPCUAID_DATASETREADERTYPE_DATASETFIELDCONTENTMASK := 21101,
	OPCUAID_DATASETREADERTYPE_MESSAGERECEIVETIMEOUT := 21102,
	OPCUAID_DATASETREADERTYPE_SECURITYMODE := 15932,
	OPCUAID_DATASETREADERTYPE_SECURITYGROUPID := 15933,
	OPCUAID_DATASETREADERTYPE_SECURITYKEYSERVICES := 15934,
	OPCUAID_DATASETREADERTYPE_DATASETREADERPROPERTIES := 17494,
	OPCUAID_DATASETREADERTYPE_STATUS_STATE := 15308,
	OPCUAID_DATASETREADERTYPE_DIAGNOSTICS_DIAGNOSTICSLEVEL := 19610,
	OPCUAID_DATASETREADERTYPE_DIAGNOSTICS_TOTALINFORMATION := 19611,
	OPCUAID_DATASETREADERTYPE_DIAGNOSTICS_TOTALINFORMATION_ACTIVE := 19612,
	OPCUAID_DATASETREADERTYPE_DIAGNOSTICS_TOTALINFORMATION_CLASSIFICATION := 19613,
	OPCUAID_DATASETREADERTYPE_DIAGNOSTICS_TOTALINFORMATION_DIAGNOSTICSLEVEL := 19614,
	OPCUAID_DATASETREADERTYPE_DIAGNOSTICS_TOTALINFORMATION_TIMEFIRSTCHANGE := 19615,
	OPCUAID_DATASETREADERTYPE_DIAGNOSTICS_TOTALERROR := 19616,
	OPCUAID_DATASETREADERTYPE_DIAGNOSTICS_TOTALERROR_ACTIVE := 19617,
	OPCUAID_DATASETREADERTYPE_DIAGNOSTICS_TOTALERROR_CLASSIFICATION := 19618,
	OPCUAID_DATASETREADERTYPE_DIAGNOSTICS_TOTALERROR_DIAGNOSTICSLEVEL := 19619,
	OPCUAID_DATASETREADERTYPE_DIAGNOSTICS_TOTALERROR_TIMEFIRSTCHANGE := 19620,
	OPCUAID_DATASETREADERTYPE_DIAGNOSTICS_SUBERROR := 19622,
	OPCUAID_DATASETREADERTYPE_DIAGNOSTICS_COUNTERS_STATEERROR := 19624,
	OPCUAID_DATASETREADERTYPE_DIAGNOSTICS_COUNTERS_STATEERROR_ACTIVE := 19625,
	OPCUAID_DATASETREADERTYPE_DIAGNOSTICS_COUNTERS_STATEERROR_CLASSIFICATION := 19626,
	OPCUAID_DATASETREADERTYPE_DIAGNOSTICS_COUNTERS_STATEERROR_DIAGNOSTICSLEVEL := 19627,
	OPCUAID_DATASETREADERTYPE_DIAGNOSTICS_COUNTERS_STATEERROR_TIMEFIRSTCHANGE := 19628,
	OPCUAID_DATASETREADERTYPE_DIAGNOSTICS_COUNTERS_STATEOPERATIONALBYMETHOD := 19629,
	OPCUAID_DATASETREADERTYPE_DIAGNOSTICS_COUNTERS_STATEOPERATIONALBYMETHOD_ACTIVE := 19630,
	OPCUAID_DATASETREADERTYPE_DIAGNOSTICS_COUNTERS_STATEOPERATIONALBYMETHOD_CLASSIFICATION := 19631,
	OPCUAID_DATASETREADERTYPE_DIAGNOSTICS_COUNTERS_STATEOPERATIONALBYMETHOD_DIAGNOSTICSLEVEL := 19632,
	OPCUAID_DATASETREADERTYPE_DIAGNOSTICS_COUNTERS_STATEOPERATIONALBYMETHOD_TIMEFIRSTCHANGE := 19633,
	OPCUAID_DATASETREADERTYPE_DIAGNOSTICS_COUNTERS_STATEOPERATIONALBYPARENT := 19634,
	OPCUAID_DATASETREADERTYPE_DIAGNOSTICS_COUNTERS_STATEOPERATIONALBYPARENT_ACTIVE := 19635,
	OPCUAID_DATASETREADERTYPE_DIAGNOSTICS_COUNTERS_STATEOPERATIONALBYPARENT_CLASSIFICATION := 19636,
	OPCUAID_DATASETREADERTYPE_DIAGNOSTICS_COUNTERS_STATEOPERATIONALBYPARENT_DIAGNOSTICSLEVEL := 19637,
	OPCUAID_DATASETREADERTYPE_DIAGNOSTICS_COUNTERS_STATEOPERATIONALBYPARENT_TIMEFIRSTCHANGE := 19638,
	OPCUAID_DATASETREADERTYPE_DIAGNOSTICS_COUNTERS_STATEOPERATIONALFROMERROR := 19639,
	OPCUAID_DATASETREADERTYPE_DIAGNOSTICS_COUNTERS_STATEOPERATIONALFROMERROR_ACTIVE := 19640,
	OPCUAID_DATASETREADERTYPE_DIAGNOSTICS_COUNTERS_STATEOPERATIONALFROMERROR_CLASSIFICATION := 19641,
	OPCUAID_DATASETREADERTYPE_DIAGNOSTICS_COUNTERS_STATEOPERATIONALFROMERROR_DIAGNOSTICSLEVEL := 19642,
	OPCUAID_DATASETREADERTYPE_DIAGNOSTICS_COUNTERS_STATEOPERATIONALFROMERROR_TIMEFIRSTCHANGE := 19643,
	OPCUAID_DATASETREADERTYPE_DIAGNOSTICS_COUNTERS_STATEPAUSEDBYPARENT := 19644,
	OPCUAID_DATASETREADERTYPE_DIAGNOSTICS_COUNTERS_STATEPAUSEDBYPARENT_ACTIVE := 19645,
	OPCUAID_DATASETREADERTYPE_DIAGNOSTICS_COUNTERS_STATEPAUSEDBYPARENT_CLASSIFICATION := 19646,
	OPCUAID_DATASETREADERTYPE_DIAGNOSTICS_COUNTERS_STATEPAUSEDBYPARENT_DIAGNOSTICSLEVEL := 19647,
	OPCUAID_DATASETREADERTYPE_DIAGNOSTICS_COUNTERS_STATEPAUSEDBYPARENT_TIMEFIRSTCHANGE := 19648,
	OPCUAID_DATASETREADERTYPE_DIAGNOSTICS_COUNTERS_STATEDISABLEDBYMETHOD := 19649,
	OPCUAID_DATASETREADERTYPE_DIAGNOSTICS_COUNTERS_STATEDISABLEDBYMETHOD_ACTIVE := 19650,
	OPCUAID_DATASETREADERTYPE_DIAGNOSTICS_COUNTERS_STATEDISABLEDBYMETHOD_CLASSIFICATION := 19651,
	OPCUAID_DATASETREADERTYPE_DIAGNOSTICS_COUNTERS_STATEDISABLEDBYMETHOD_DIAGNOSTICSLEVEL := 19652,
	OPCUAID_DATASETREADERTYPE_DIAGNOSTICS_COUNTERS_STATEDISABLEDBYMETHOD_TIMEFIRSTCHANGE := 19653,
	OPCUAID_DATASETREADERTYPE_DIAGNOSTICS_COUNTERS_FAILEDDATASETMESSAGES := 19655,
	OPCUAID_DATASETREADERTYPE_DIAGNOSTICS_COUNTERS_FAILEDDATASETMESSAGES_ACTIVE := 19656,
	OPCUAID_DATASETREADERTYPE_DIAGNOSTICS_COUNTERS_FAILEDDATASETMESSAGES_CLASSIFICATION := 19657,
	OPCUAID_DATASETREADERTYPE_DIAGNOSTICS_COUNTERS_FAILEDDATASETMESSAGES_DIAGNOSTICSLEVEL := 19658,
	OPCUAID_DATASETREADERTYPE_DIAGNOSTICS_COUNTERS_FAILEDDATASETMESSAGES_TIMEFIRSTCHANGE := 19659,
	OPCUAID_DATASETREADERTYPE_DIAGNOSTICS_COUNTERS_DECRYPTIONERRORS_ACTIVE := 19661,
	OPCUAID_DATASETREADERTYPE_DIAGNOSTICS_COUNTERS_DECRYPTIONERRORS_CLASSIFICATION := 19662,
	OPCUAID_DATASETREADERTYPE_DIAGNOSTICS_COUNTERS_DECRYPTIONERRORS_DIAGNOSTICSLEVEL := 19663,
	OPCUAID_DATASETREADERTYPE_DIAGNOSTICS_COUNTERS_DECRYPTIONERRORS_TIMEFIRSTCHANGE := 19664,
	OPCUAID_DATASETREADERTYPE_DIAGNOSTICS_LIVEVALUES_MESSAGESEQUENCENUMBER_DIAGNOSTICSLEVEL := 19666,
	OPCUAID_DATASETREADERTYPE_DIAGNOSTICS_LIVEVALUES_STATUSCODE_DIAGNOSTICSLEVEL := 19668,
	OPCUAID_DATASETREADERTYPE_DIAGNOSTICS_LIVEVALUES_MAJORVERSION_DIAGNOSTICSLEVEL := 19670,
	OPCUAID_DATASETREADERTYPE_DIAGNOSTICS_LIVEVALUES_MINORVERSION_DIAGNOSTICSLEVEL := 19672,
	OPCUAID_DATASETREADERTYPE_DIAGNOSTICS_LIVEVALUES_SECURITYTOKENID_DIAGNOSTICSLEVEL := 19674,
	OPCUAID_DATASETREADERTYPE_DIAGNOSTICS_LIVEVALUES_TIMETONEXTTOKENID_DIAGNOSTICSLEVEL := 19676,
	OPCUAID_DATASETREADERTYPE_SUBSCRIBEDDATASET_DATASETMETADATA := 15317,
	OPCUAID_DATASETREADERTYPE_SUBSCRIBEDDATASET_MESSAGERECEIVETIMEOUT := 15318,
	OPCUAID_DATASETREADERTYPE_CREATETARGETVARIABLES_INPUTARGUMENTS := 17387,
	OPCUAID_DATASETREADERTYPE_CREATETARGETVARIABLES_OUTPUTARGUMENTS := 17388,
	OPCUAID_DATASETREADERTYPE_CREATEDATASETMIRROR_INPUTARGUMENTS := 17390,
	OPCUAID_DATASETREADERTYPE_CREATEDATASETMIRROR_OUTPUTARGUMENTS := 17391,
	OPCUAID_SUBSCRIBEDDATASETTYPE_DATASETMETADATA := 15109,
	OPCUAID_SUBSCRIBEDDATASETTYPE_MESSAGERECEIVETIMEOUT := 15110,
	OPCUAID_TARGETVARIABLESTYPE_TARGETVARIABLES := 15114,
	OPCUAID_TARGETVARIABLESTYPE_ADDTARGETVARIABLES_INPUTARGUMENTS := 15116,
	OPCUAID_TARGETVARIABLESTYPE_ADDTARGETVARIABLES_OUTPUTARGUMENTS := 15117,
	OPCUAID_TARGETVARIABLESTYPE_REMOVETARGETVARIABLES_INPUTARGUMENTS := 15119,
	OPCUAID_TARGETVARIABLESTYPE_REMOVETARGETVARIABLES_OUTPUTARGUMENTS := 15120,
	OPCUAID_PUBSUBSTATUSTYPE_STATE := 14644,
	OPCUAID_PUBSUBDIAGNOSTICSTYPE_DIAGNOSTICSLEVEL := 19678,
	OPCUAID_PUBSUBDIAGNOSTICSTYPE_TOTALINFORMATION := 19679,
	OPCUAID_PUBSUBDIAGNOSTICSTYPE_TOTALINFORMATION_ACTIVE := 19680,
	OPCUAID_PUBSUBDIAGNOSTICSTYPE_TOTALINFORMATION_CLASSIFICATION := 19681,
	OPCUAID_PUBSUBDIAGNOSTICSTYPE_TOTALINFORMATION_DIAGNOSTICSLEVEL := 19682,
	OPCUAID_PUBSUBDIAGNOSTICSTYPE_TOTALINFORMATION_TIMEFIRSTCHANGE := 19683,
	OPCUAID_PUBSUBDIAGNOSTICSTYPE_TOTALERROR := 19684,
	OPCUAID_PUBSUBDIAGNOSTICSTYPE_TOTALERROR_ACTIVE := 19685,
	OPCUAID_PUBSUBDIAGNOSTICSTYPE_TOTALERROR_CLASSIFICATION := 19686,
	OPCUAID_PUBSUBDIAGNOSTICSTYPE_TOTALERROR_DIAGNOSTICSLEVEL := 19687,
	OPCUAID_PUBSUBDIAGNOSTICSTYPE_TOTALERROR_TIMEFIRSTCHANGE := 19688,
	OPCUAID_PUBSUBDIAGNOSTICSTYPE_SUBERROR := 19690,
	OPCUAID_PUBSUBDIAGNOSTICSTYPE_COUNTERS_STATEERROR := 19692,
	OPCUAID_PUBSUBDIAGNOSTICSTYPE_COUNTERS_STATEERROR_ACTIVE := 19693,
	OPCUAID_PUBSUBDIAGNOSTICSTYPE_COUNTERS_STATEERROR_CLASSIFICATION := 19694,
	OPCUAID_PUBSUBDIAGNOSTICSTYPE_COUNTERS_STATEERROR_DIAGNOSTICSLEVEL := 19695,
	OPCUAID_PUBSUBDIAGNOSTICSTYPE_COUNTERS_STATEERROR_TIMEFIRSTCHANGE := 19696,
	OPCUAID_PUBSUBDIAGNOSTICSTYPE_COUNTERS_STATEOPERATIONALBYMETHOD := 19697,
	OPCUAID_PUBSUBDIAGNOSTICSTYPE_COUNTERS_STATEOPERATIONALBYMETHOD_ACTIVE := 19698,
	OPCUAID_PUBSUBDIAGNOSTICSTYPE_COUNTERS_STATEOPERATIONALBYMETHOD_CLASSIFICATION := 19699,
	OPCUAID_PUBSUBDIAGNOSTICSTYPE_COUNTERS_STATEOPERATIONALBYMETHOD_DIAGNOSTICSLEVEL := 19700,
	OPCUAID_PUBSUBDIAGNOSTICSTYPE_COUNTERS_STATEOPERATIONALBYMETHOD_TIMEFIRSTCHANGE := 19701,
	OPCUAID_PUBSUBDIAGNOSTICSTYPE_COUNTERS_STATEOPERATIONALBYPARENT := 19702,
	OPCUAID_PUBSUBDIAGNOSTICSTYPE_COUNTERS_STATEOPERATIONALBYPARENT_ACTIVE := 19703,
	OPCUAID_PUBSUBDIAGNOSTICSTYPE_COUNTERS_STATEOPERATIONALBYPARENT_CLASSIFICATION := 19704,
	OPCUAID_PUBSUBDIAGNOSTICSTYPE_COUNTERS_STATEOPERATIONALBYPARENT_DIAGNOSTICSLEVEL := 19705,
	OPCUAID_PUBSUBDIAGNOSTICSTYPE_COUNTERS_STATEOPERATIONALBYPARENT_TIMEFIRSTCHANGE := 19706,
	OPCUAID_PUBSUBDIAGNOSTICSTYPE_COUNTERS_STATEOPERATIONALFROMERROR := 19707,
	OPCUAID_PUBSUBDIAGNOSTICSTYPE_COUNTERS_STATEOPERATIONALFROMERROR_ACTIVE := 19708,
	OPCUAID_PUBSUBDIAGNOSTICSTYPE_COUNTERS_STATEOPERATIONALFROMERROR_CLASSIFICATION := 19709,
	OPCUAID_PUBSUBDIAGNOSTICSTYPE_COUNTERS_STATEOPERATIONALFROMERROR_DIAGNOSTICSLEVEL := 19710,
	OPCUAID_PUBSUBDIAGNOSTICSTYPE_COUNTERS_STATEOPERATIONALFROMERROR_TIMEFIRSTCHANGE := 19711,
	OPCUAID_PUBSUBDIAGNOSTICSTYPE_COUNTERS_STATEPAUSEDBYPARENT := 19712,
	OPCUAID_PUBSUBDIAGNOSTICSTYPE_COUNTERS_STATEPAUSEDBYPARENT_ACTIVE := 19713,
	OPCUAID_PUBSUBDIAGNOSTICSTYPE_COUNTERS_STATEPAUSEDBYPARENT_CLASSIFICATION := 19714,
	OPCUAID_PUBSUBDIAGNOSTICSTYPE_COUNTERS_STATEPAUSEDBYPARENT_DIAGNOSTICSLEVEL := 19715,
	OPCUAID_PUBSUBDIAGNOSTICSTYPE_COUNTERS_STATEPAUSEDBYPARENT_TIMEFIRSTCHANGE := 19716,
	OPCUAID_PUBSUBDIAGNOSTICSTYPE_COUNTERS_STATEDISABLEDBYMETHOD := 19717,
	OPCUAID_PUBSUBDIAGNOSTICSTYPE_COUNTERS_STATEDISABLEDBYMETHOD_ACTIVE := 19718,
	OPCUAID_PUBSUBDIAGNOSTICSTYPE_COUNTERS_STATEDISABLEDBYMETHOD_CLASSIFICATION := 19719,
	OPCUAID_PUBSUBDIAGNOSTICSTYPE_COUNTERS_STATEDISABLEDBYMETHOD_DIAGNOSTICSLEVEL := 19720,
	OPCUAID_PUBSUBDIAGNOSTICSTYPE_COUNTERS_STATEDISABLEDBYMETHOD_TIMEFIRSTCHANGE := 19721,
	OPCUAID_DIAGNOSTICSLEVEL_ENUMSTRINGS := 19724,
	OPCUAID_PUBSUBDIAGNOSTICSCOUNTERTYPE_ACTIVE := 19726,
	OPCUAID_PUBSUBDIAGNOSTICSCOUNTERTYPE_CLASSIFICATION := 19727,
	OPCUAID_PUBSUBDIAGNOSTICSCOUNTERTYPE_DIAGNOSTICSLEVEL := 19728,
	OPCUAID_PUBSUBDIAGNOSTICSCOUNTERTYPE_TIMEFIRSTCHANGE := 19729,
	OPCUAID_PUBSUBDIAGNOSTICSCOUNTERCLASSIFICATION_ENUMSTRINGS := 19731,
	OPCUAID_PUBSUBDIAGNOSTICSROOTTYPE_TOTALINFORMATION_ACTIVE := 19735,
	OPCUAID_PUBSUBDIAGNOSTICSROOTTYPE_TOTALINFORMATION_CLASSIFICATION := 19736,
	OPCUAID_PUBSUBDIAGNOSTICSROOTTYPE_TOTALINFORMATION_DIAGNOSTICSLEVEL := 19737,
	OPCUAID_PUBSUBDIAGNOSTICSROOTTYPE_TOTALINFORMATION_TIMEFIRSTCHANGE := 19738,
	OPCUAID_PUBSUBDIAGNOSTICSROOTTYPE_TOTALERROR_ACTIVE := 19740,
	OPCUAID_PUBSUBDIAGNOSTICSROOTTYPE_TOTALERROR_CLASSIFICATION := 19741,
	OPCUAID_PUBSUBDIAGNOSTICSROOTTYPE_TOTALERROR_DIAGNOSTICSLEVEL := 19742,
	OPCUAID_PUBSUBDIAGNOSTICSROOTTYPE_TOTALERROR_TIMEFIRSTCHANGE := 19743,
	OPCUAID_PUBSUBDIAGNOSTICSROOTTYPE_COUNTERS_STATEERROR := 19747,
	OPCUAID_PUBSUBDIAGNOSTICSROOTTYPE_COUNTERS_STATEERROR_ACTIVE := 19748,
	OPCUAID_PUBSUBDIAGNOSTICSROOTTYPE_COUNTERS_STATEERROR_CLASSIFICATION := 19749,
	OPCUAID_PUBSUBDIAGNOSTICSROOTTYPE_COUNTERS_STATEERROR_DIAGNOSTICSLEVEL := 19750,
	OPCUAID_PUBSUBDIAGNOSTICSROOTTYPE_COUNTERS_STATEERROR_TIMEFIRSTCHANGE := 19751,
	OPCUAID_PUBSUBDIAGNOSTICSROOTTYPE_COUNTERS_STATEOPERATIONALBYMETHOD := 19752,
	OPCUAID_PUBSUBDIAGNOSTICSROOTTYPE_COUNTERS_STATEOPERATIONALBYMETHOD_ACTIVE := 19753,
	OPCUAID_PUBSUBDIAGNOSTICSROOTTYPE_COUNTERS_STATEOPERATIONALBYMETHOD_CLASSIFICATION := 19754,
	OPCUAID_PUBSUBDIAGNOSTICSROOTTYPE_COUNTERS_STATEOPERATIONALBYMETHOD_DIAGNOSTICSLEVEL := 19755,
	OPCUAID_PUBSUBDIAGNOSTICSROOTTYPE_COUNTERS_STATEOPERATIONALBYMETHOD_TIMEFIRSTCHANGE := 19756,
	OPCUAID_PUBSUBDIAGNOSTICSROOTTYPE_COUNTERS_STATEOPERATIONALBYPARENT := 19757,
	OPCUAID_PUBSUBDIAGNOSTICSROOTTYPE_COUNTERS_STATEOPERATIONALBYPARENT_ACTIVE := 19758,
	OPCUAID_PUBSUBDIAGNOSTICSROOTTYPE_COUNTERS_STATEOPERATIONALBYPARENT_CLASSIFICATION := 19759,
	OPCUAID_PUBSUBDIAGNOSTICSROOTTYPE_COUNTERS_STATEOPERATIONALBYPARENT_DIAGNOSTICSLEVEL := 19760,
	OPCUAID_PUBSUBDIAGNOSTICSROOTTYPE_COUNTERS_STATEOPERATIONALBYPARENT_TIMEFIRSTCHANGE := 19761,
	OPCUAID_PUBSUBDIAGNOSTICSROOTTYPE_COUNTERS_STATEOPERATIONALFROMERROR := 19762,
	OPCUAID_PUBSUBDIAGNOSTICSROOTTYPE_COUNTERS_STATEOPERATIONALFROMERROR_ACTIVE := 19763,
	OPCUAID_PUBSUBDIAGNOSTICSROOTTYPE_COUNTERS_STATEOPERATIONALFROMERROR_CLASSIFICATION := 19764,
	OPCUAID_PUBSUBDIAGNOSTICSROOTTYPE_COUNTERS_STATEOPERATIONALFROMERROR_DIAGNOSTICSLEVEL := 19765,
	OPCUAID_PUBSUBDIAGNOSTICSROOTTYPE_COUNTERS_STATEOPERATIONALFROMERROR_TIMEFIRSTCHANGE := 19766,
	OPCUAID_PUBSUBDIAGNOSTICSROOTTYPE_COUNTERS_STATEPAUSEDBYPARENT := 19767,
	OPCUAID_PUBSUBDIAGNOSTICSROOTTYPE_COUNTERS_STATEPAUSEDBYPARENT_ACTIVE := 19768,
	OPCUAID_PUBSUBDIAGNOSTICSROOTTYPE_COUNTERS_STATEPAUSEDBYPARENT_CLASSIFICATION := 19769,
	OPCUAID_PUBSUBDIAGNOSTICSROOTTYPE_COUNTERS_STATEPAUSEDBYPARENT_DIAGNOSTICSLEVEL := 19770,
	OPCUAID_PUBSUBDIAGNOSTICSROOTTYPE_COUNTERS_STATEPAUSEDBYPARENT_TIMEFIRSTCHANGE := 19771,
	OPCUAID_PUBSUBDIAGNOSTICSROOTTYPE_COUNTERS_STATEDISABLEDBYMETHOD := 19772,
	OPCUAID_PUBSUBDIAGNOSTICSROOTTYPE_COUNTERS_STATEDISABLEDBYMETHOD_ACTIVE := 19773,
	OPCUAID_PUBSUBDIAGNOSTICSROOTTYPE_COUNTERS_STATEDISABLEDBYMETHOD_CLASSIFICATION := 19774,
	OPCUAID_PUBSUBDIAGNOSTICSROOTTYPE_COUNTERS_STATEDISABLEDBYMETHOD_DIAGNOSTICSLEVEL := 19775,
	OPCUAID_PUBSUBDIAGNOSTICSROOTTYPE_COUNTERS_STATEDISABLEDBYMETHOD_TIMEFIRSTCHANGE := 19776,
	OPCUAID_PUBSUBDIAGNOSTICSROOTTYPE_LIVEVALUES_CONFIGUREDDATASETWRITERS := 19778,
	OPCUAID_PUBSUBDIAGNOSTICSROOTTYPE_LIVEVALUES_CONFIGUREDDATASETWRITERS_DIAGNOSTICSLEVEL := 19779,
	OPCUAID_PUBSUBDIAGNOSTICSROOTTYPE_LIVEVALUES_CONFIGUREDDATASETREADERS := 19780,
	OPCUAID_PUBSUBDIAGNOSTICSROOTTYPE_LIVEVALUES_CONFIGUREDDATASETREADERS_DIAGNOSTICSLEVEL := 19781,
	OPCUAID_PUBSUBDIAGNOSTICSROOTTYPE_LIVEVALUES_OPERATIONALDATASETWRITERS := 19782,
	OPCUAID_PUBSUBDIAGNOSTICSROOTTYPE_LIVEVALUES_OPERATIONALDATASETWRITERS_DIAGNOSTICSLEVEL := 19783,
	OPCUAID_PUBSUBDIAGNOSTICSROOTTYPE_LIVEVALUES_OPERATIONALDATASETREADERS := 19784,
	OPCUAID_PUBSUBDIAGNOSTICSROOTTYPE_LIVEVALUES_OPERATIONALDATASETREADERS_DIAGNOSTICSLEVEL := 19785,
	OPCUAID_PUBSUBDIAGNOSTICSCONNECTIONTYPE_TOTALINFORMATION_ACTIVE := 19789,
	OPCUAID_PUBSUBDIAGNOSTICSCONNECTIONTYPE_TOTALINFORMATION_CLASSIFICATION := 19790,
	OPCUAID_PUBSUBDIAGNOSTICSCONNECTIONTYPE_TOTALINFORMATION_DIAGNOSTICSLEVEL := 19791,
	OPCUAID_PUBSUBDIAGNOSTICSCONNECTIONTYPE_TOTALINFORMATION_TIMEFIRSTCHANGE := 19792,
	OPCUAID_PUBSUBDIAGNOSTICSCONNECTIONTYPE_TOTALERROR_ACTIVE := 19794,
	OPCUAID_PUBSUBDIAGNOSTICSCONNECTIONTYPE_TOTALERROR_CLASSIFICATION := 19795,
	OPCUAID_PUBSUBDIAGNOSTICSCONNECTIONTYPE_TOTALERROR_DIAGNOSTICSLEVEL := 19796,
	OPCUAID_PUBSUBDIAGNOSTICSCONNECTIONTYPE_TOTALERROR_TIMEFIRSTCHANGE := 19797,
	OPCUAID_PUBSUBDIAGNOSTICSCONNECTIONTYPE_COUNTERS_STATEERROR := 19801,
	OPCUAID_PUBSUBDIAGNOSTICSCONNECTIONTYPE_COUNTERS_STATEERROR_ACTIVE := 19802,
	OPCUAID_PUBSUBDIAGNOSTICSCONNECTIONTYPE_COUNTERS_STATEERROR_CLASSIFICATION := 19803,
	OPCUAID_PUBSUBDIAGNOSTICSCONNECTIONTYPE_COUNTERS_STATEERROR_DIAGNOSTICSLEVEL := 19804,
	OPCUAID_PUBSUBDIAGNOSTICSCONNECTIONTYPE_COUNTERS_STATEERROR_TIMEFIRSTCHANGE := 19805,
	OPCUAID_PUBSUBDIAGNOSTICSCONNECTIONTYPE_COUNTERS_STATEOPERATIONALBYMETHOD := 19806,
	OPCUAID_PUBSUBDIAGNOSTICSCONNECTIONTYPE_COUNTERS_STATEOPERATIONALBYMETHOD_ACTIVE := 19807,
	OPCUAID_PUBSUBDIAGNOSTICSCONNECTIONTYPE_COUNTERS_STATEOPERATIONALBYMETHOD_CLASSIFICATION := 19808,
	OPCUAID_PUBSUBDIAGNOSTICSCONNECTIONTYPE_COUNTERS_STATEOPERATIONALBYMETHOD_DIAGNOSTICSLEVEL := 19809,
	OPCUAID_PUBSUBDIAGNOSTICSCONNECTIONTYPE_COUNTERS_STATEOPERATIONALBYMETHOD_TIMEFIRSTCHANGE := 19810,
	OPCUAID_PUBSUBDIAGNOSTICSCONNECTIONTYPE_COUNTERS_STATEOPERATIONALBYPARENT := 19811,
	OPCUAID_PUBSUBDIAGNOSTICSCONNECTIONTYPE_COUNTERS_STATEOPERATIONALBYPARENT_ACTIVE := 19812,
	OPCUAID_PUBSUBDIAGNOSTICSCONNECTIONTYPE_COUNTERS_STATEOPERATIONALBYPARENT_CLASSIFICATION := 19813,
	OPCUAID_PUBSUBDIAGNOSTICSCONNECTIONTYPE_COUNTERS_STATEOPERATIONALBYPARENT_DIAGNOSTICSLEVEL := 19814,
	OPCUAID_PUBSUBDIAGNOSTICSCONNECTIONTYPE_COUNTERS_STATEOPERATIONALBYPARENT_TIMEFIRSTCHANGE := 19815,
	OPCUAID_PUBSUBDIAGNOSTICSCONNECTIONTYPE_COUNTERS_STATEOPERATIONALFROMERROR := 19816,
	OPCUAID_PUBSUBDIAGNOSTICSCONNECTIONTYPE_COUNTERS_STATEOPERATIONALFROMERROR_ACTIVE := 19817,
	OPCUAID_PUBSUBDIAGNOSTICSCONNECTIONTYPE_COUNTERS_STATEOPERATIONALFROMERROR_CLASSIFICATION := 19818,
	OPCUAID_PUBSUBDIAGNOSTICSCONNECTIONTYPE_COUNTERS_STATEOPERATIONALFROMERROR_DIAGNOSTICSLEVEL := 19819,
	OPCUAID_PUBSUBDIAGNOSTICSCONNECTIONTYPE_COUNTERS_STATEOPERATIONALFROMERROR_TIMEFIRSTCHANGE := 19820,
	OPCUAID_PUBSUBDIAGNOSTICSCONNECTIONTYPE_COUNTERS_STATEPAUSEDBYPARENT := 19821,
	OPCUAID_PUBSUBDIAGNOSTICSCONNECTIONTYPE_COUNTERS_STATEPAUSEDBYPARENT_ACTIVE := 19822,
	OPCUAID_PUBSUBDIAGNOSTICSCONNECTIONTYPE_COUNTERS_STATEPAUSEDBYPARENT_CLASSIFICATION := 19823,
	OPCUAID_PUBSUBDIAGNOSTICSCONNECTIONTYPE_COUNTERS_STATEPAUSEDBYPARENT_DIAGNOSTICSLEVEL := 19824,
	OPCUAID_PUBSUBDIAGNOSTICSCONNECTIONTYPE_COUNTERS_STATEPAUSEDBYPARENT_TIMEFIRSTCHANGE := 19825,
	OPCUAID_PUBSUBDIAGNOSTICSCONNECTIONTYPE_COUNTERS_STATEDISABLEDBYMETHOD := 19826,
	OPCUAID_PUBSUBDIAGNOSTICSCONNECTIONTYPE_COUNTERS_STATEDISABLEDBYMETHOD_ACTIVE := 19827,
	OPCUAID_PUBSUBDIAGNOSTICSCONNECTIONTYPE_COUNTERS_STATEDISABLEDBYMETHOD_CLASSIFICATION := 19828,
	OPCUAID_PUBSUBDIAGNOSTICSCONNECTIONTYPE_COUNTERS_STATEDISABLEDBYMETHOD_DIAGNOSTICSLEVEL := 19829,
	OPCUAID_PUBSUBDIAGNOSTICSCONNECTIONTYPE_COUNTERS_STATEDISABLEDBYMETHOD_TIMEFIRSTCHANGE := 19830,
	OPCUAID_PUBSUBDIAGNOSTICSCONNECTIONTYPE_LIVEVALUES_RESOLVEDADDRESS := 19832,
	OPCUAID_PUBSUBDIAGNOSTICSCONNECTIONTYPE_LIVEVALUES_RESOLVEDADDRESS_DIAGNOSTICSLEVEL := 19833,
	OPCUAID_PUBSUBDIAGNOSTICSWRITERGROUPTYPE_TOTALINFORMATION_ACTIVE := 19837,
	OPCUAID_PUBSUBDIAGNOSTICSWRITERGROUPTYPE_TOTALINFORMATION_CLASSIFICATION := 19838,
	OPCUAID_PUBSUBDIAGNOSTICSWRITERGROUPTYPE_TOTALINFORMATION_DIAGNOSTICSLEVEL := 19839,
	OPCUAID_PUBSUBDIAGNOSTICSWRITERGROUPTYPE_TOTALINFORMATION_TIMEFIRSTCHANGE := 19840,
	OPCUAID_PUBSUBDIAGNOSTICSWRITERGROUPTYPE_TOTALERROR_ACTIVE := 19842,
	OPCUAID_PUBSUBDIAGNOSTICSWRITERGROUPTYPE_TOTALERROR_CLASSIFICATION := 19843,
	OPCUAID_PUBSUBDIAGNOSTICSWRITERGROUPTYPE_TOTALERROR_DIAGNOSTICSLEVEL := 19844,
	OPCUAID_PUBSUBDIAGNOSTICSWRITERGROUPTYPE_TOTALERROR_TIMEFIRSTCHANGE := 19845,
	OPCUAID_PUBSUBDIAGNOSTICSWRITERGROUPTYPE_COUNTERS_STATEERROR := 19849,
	OPCUAID_PUBSUBDIAGNOSTICSWRITERGROUPTYPE_COUNTERS_STATEERROR_ACTIVE := 19850,
	OPCUAID_PUBSUBDIAGNOSTICSWRITERGROUPTYPE_COUNTERS_STATEERROR_CLASSIFICATION := 19851,
	OPCUAID_PUBSUBDIAGNOSTICSWRITERGROUPTYPE_COUNTERS_STATEERROR_DIAGNOSTICSLEVEL := 19852,
	OPCUAID_PUBSUBDIAGNOSTICSWRITERGROUPTYPE_COUNTERS_STATEERROR_TIMEFIRSTCHANGE := 19853,
	OPCUAID_PUBSUBDIAGNOSTICSWRITERGROUPTYPE_COUNTERS_STATEOPERATIONALBYMETHOD := 19854,
	OPCUAID_PUBSUBDIAGNOSTICSWRITERGROUPTYPE_COUNTERS_STATEOPERATIONALBYMETHOD_ACTIVE := 19855,
	OPCUAID_PUBSUBDIAGNOSTICSWRITERGROUPTYPE_COUNTERS_STATEOPERATIONALBYMETHOD_CLASSIFICATION := 19856,
	OPCUAID_PUBSUBDIAGNOSTICSWRITERGROUPTYPE_COUNTERS_STATEOPERATIONALBYMETHOD_DIAGNOSTICSLEVEL := 19857,
	OPCUAID_PUBSUBDIAGNOSTICSWRITERGROUPTYPE_COUNTERS_STATEOPERATIONALBYMETHOD_TIMEFIRSTCHANGE := 19858,
	OPCUAID_PUBSUBDIAGNOSTICSWRITERGROUPTYPE_COUNTERS_STATEOPERATIONALBYPARENT := 19859,
	OPCUAID_PUBSUBDIAGNOSTICSWRITERGROUPTYPE_COUNTERS_STATEOPERATIONALBYPARENT_ACTIVE := 19860,
	OPCUAID_PUBSUBDIAGNOSTICSWRITERGROUPTYPE_COUNTERS_STATEOPERATIONALBYPARENT_CLASSIFICATION := 19861,
	OPCUAID_PUBSUBDIAGNOSTICSWRITERGROUPTYPE_COUNTERS_STATEOPERATIONALBYPARENT_DIAGNOSTICSLEVEL := 19862,
	OPCUAID_PUBSUBDIAGNOSTICSWRITERGROUPTYPE_COUNTERS_STATEOPERATIONALBYPARENT_TIMEFIRSTCHANGE := 19863,
	OPCUAID_PUBSUBDIAGNOSTICSWRITERGROUPTYPE_COUNTERS_STATEOPERATIONALFROMERROR := 19864,
	OPCUAID_PUBSUBDIAGNOSTICSWRITERGROUPTYPE_COUNTERS_STATEOPERATIONALFROMERROR_ACTIVE := 19865,
	OPCUAID_PUBSUBDIAGNOSTICSWRITERGROUPTYPE_COUNTERS_STATEOPERATIONALFROMERROR_CLASSIFICATION := 19866,
	OPCUAID_PUBSUBDIAGNOSTICSWRITERGROUPTYPE_COUNTERS_STATEOPERATIONALFROMERROR_DIAGNOSTICSLEVEL := 19867,
	OPCUAID_PUBSUBDIAGNOSTICSWRITERGROUPTYPE_COUNTERS_STATEOPERATIONALFROMERROR_TIMEFIRSTCHANGE := 19868,
	OPCUAID_PUBSUBDIAGNOSTICSWRITERGROUPTYPE_COUNTERS_STATEPAUSEDBYPARENT := 19869,
	OPCUAID_PUBSUBDIAGNOSTICSWRITERGROUPTYPE_COUNTERS_STATEPAUSEDBYPARENT_ACTIVE := 19870,
	OPCUAID_PUBSUBDIAGNOSTICSWRITERGROUPTYPE_COUNTERS_STATEPAUSEDBYPARENT_CLASSIFICATION := 19871,
	OPCUAID_PUBSUBDIAGNOSTICSWRITERGROUPTYPE_COUNTERS_STATEPAUSEDBYPARENT_DIAGNOSTICSLEVEL := 19872,
	OPCUAID_PUBSUBDIAGNOSTICSWRITERGROUPTYPE_COUNTERS_STATEPAUSEDBYPARENT_TIMEFIRSTCHANGE := 19873,
	OPCUAID_PUBSUBDIAGNOSTICSWRITERGROUPTYPE_COUNTERS_STATEDISABLEDBYMETHOD := 19874,
	OPCUAID_PUBSUBDIAGNOSTICSWRITERGROUPTYPE_COUNTERS_STATEDISABLEDBYMETHOD_ACTIVE := 19875,
	OPCUAID_PUBSUBDIAGNOSTICSWRITERGROUPTYPE_COUNTERS_STATEDISABLEDBYMETHOD_CLASSIFICATION := 19876,
	OPCUAID_PUBSUBDIAGNOSTICSWRITERGROUPTYPE_COUNTERS_STATEDISABLEDBYMETHOD_DIAGNOSTICSLEVEL := 19877,
	OPCUAID_PUBSUBDIAGNOSTICSWRITERGROUPTYPE_COUNTERS_STATEDISABLEDBYMETHOD_TIMEFIRSTCHANGE := 19878,
	OPCUAID_PUBSUBDIAGNOSTICSWRITERGROUPTYPE_COUNTERS_SENTNETWORKMESSAGES := 19880,
	OPCUAID_PUBSUBDIAGNOSTICSWRITERGROUPTYPE_COUNTERS_SENTNETWORKMESSAGES_ACTIVE := 19881,
	OPCUAID_PUBSUBDIAGNOSTICSWRITERGROUPTYPE_COUNTERS_SENTNETWORKMESSAGES_CLASSIFICATION := 19882,
	OPCUAID_PUBSUBDIAGNOSTICSWRITERGROUPTYPE_COUNTERS_SENTNETWORKMESSAGES_DIAGNOSTICSLEVEL := 19883,
	OPCUAID_PUBSUBDIAGNOSTICSWRITERGROUPTYPE_COUNTERS_SENTNETWORKMESSAGES_TIMEFIRSTCHANGE := 19884,
	OPCUAID_PUBSUBDIAGNOSTICSWRITERGROUPTYPE_COUNTERS_FAILEDTRANSMISSIONS := 19885,
	OPCUAID_PUBSUBDIAGNOSTICSWRITERGROUPTYPE_COUNTERS_FAILEDTRANSMISSIONS_ACTIVE := 19886,
	OPCUAID_PUBSUBDIAGNOSTICSWRITERGROUPTYPE_COUNTERS_FAILEDTRANSMISSIONS_CLASSIFICATION := 19887,
	OPCUAID_PUBSUBDIAGNOSTICSWRITERGROUPTYPE_COUNTERS_FAILEDTRANSMISSIONS_DIAGNOSTICSLEVEL := 19888,
	OPCUAID_PUBSUBDIAGNOSTICSWRITERGROUPTYPE_COUNTERS_FAILEDTRANSMISSIONS_TIMEFIRSTCHANGE := 19889,
	OPCUAID_PUBSUBDIAGNOSTICSWRITERGROUPTYPE_COUNTERS_ENCRYPTIONERRORS := 19890,
	OPCUAID_PUBSUBDIAGNOSTICSWRITERGROUPTYPE_COUNTERS_ENCRYPTIONERRORS_ACTIVE := 19891,
	OPCUAID_PUBSUBDIAGNOSTICSWRITERGROUPTYPE_COUNTERS_ENCRYPTIONERRORS_CLASSIFICATION := 19892,
	OPCUAID_PUBSUBDIAGNOSTICSWRITERGROUPTYPE_COUNTERS_ENCRYPTIONERRORS_DIAGNOSTICSLEVEL := 19893,
	OPCUAID_PUBSUBDIAGNOSTICSWRITERGROUPTYPE_COUNTERS_ENCRYPTIONERRORS_TIMEFIRSTCHANGE := 19894,
	OPCUAID_PUBSUBDIAGNOSTICSWRITERGROUPTYPE_LIVEVALUES_CONFIGUREDDATASETWRITERS := 19895,
	OPCUAID_PUBSUBDIAGNOSTICSWRITERGROUPTYPE_LIVEVALUES_CONFIGUREDDATASETWRITERS_DIAGNOSTICSLEVEL := 19896,
	OPCUAID_PUBSUBDIAGNOSTICSWRITERGROUPTYPE_LIVEVALUES_OPERATIONALDATASETWRITERS := 19897,
	OPCUAID_PUBSUBDIAGNOSTICSWRITERGROUPTYPE_LIVEVALUES_OPERATIONALDATASETWRITERS_DIAGNOSTICSLEVEL := 19898,
	OPCUAID_PUBSUBDIAGNOSTICSWRITERGROUPTYPE_LIVEVALUES_SECURITYTOKENID := 19899,
	OPCUAID_PUBSUBDIAGNOSTICSWRITERGROUPTYPE_LIVEVALUES_SECURITYTOKENID_DIAGNOSTICSLEVEL := 19900,
	OPCUAID_PUBSUBDIAGNOSTICSWRITERGROUPTYPE_LIVEVALUES_TIMETONEXTTOKENID := 19901,
	OPCUAID_PUBSUBDIAGNOSTICSWRITERGROUPTYPE_LIVEVALUES_TIMETONEXTTOKENID_DIAGNOSTICSLEVEL := 19902,
	OPCUAID_PUBSUBDIAGNOSTICSREADERGROUPTYPE_TOTALINFORMATION_ACTIVE := 19906,
	OPCUAID_PUBSUBDIAGNOSTICSREADERGROUPTYPE_TOTALINFORMATION_CLASSIFICATION := 19907,
	OPCUAID_PUBSUBDIAGNOSTICSREADERGROUPTYPE_TOTALINFORMATION_DIAGNOSTICSLEVEL := 19908,
	OPCUAID_PUBSUBDIAGNOSTICSREADERGROUPTYPE_TOTALINFORMATION_TIMEFIRSTCHANGE := 19909,
	OPCUAID_PUBSUBDIAGNOSTICSREADERGROUPTYPE_TOTALERROR_ACTIVE := 19911,
	OPCUAID_PUBSUBDIAGNOSTICSREADERGROUPTYPE_TOTALERROR_CLASSIFICATION := 19912,
	OPCUAID_PUBSUBDIAGNOSTICSREADERGROUPTYPE_TOTALERROR_DIAGNOSTICSLEVEL := 19913,
	OPCUAID_PUBSUBDIAGNOSTICSREADERGROUPTYPE_TOTALERROR_TIMEFIRSTCHANGE := 19914,
	OPCUAID_PUBSUBDIAGNOSTICSREADERGROUPTYPE_COUNTERS_STATEERROR := 19918,
	OPCUAID_PUBSUBDIAGNOSTICSREADERGROUPTYPE_COUNTERS_STATEERROR_ACTIVE := 19919,
	OPCUAID_PUBSUBDIAGNOSTICSREADERGROUPTYPE_COUNTERS_STATEERROR_CLASSIFICATION := 19920,
	OPCUAID_PUBSUBDIAGNOSTICSREADERGROUPTYPE_COUNTERS_STATEERROR_DIAGNOSTICSLEVEL := 19921,
	OPCUAID_PUBSUBDIAGNOSTICSREADERGROUPTYPE_COUNTERS_STATEERROR_TIMEFIRSTCHANGE := 19922,
	OPCUAID_PUBSUBDIAGNOSTICSREADERGROUPTYPE_COUNTERS_STATEOPERATIONALBYMETHOD := 19923,
	OPCUAID_PUBSUBDIAGNOSTICSREADERGROUPTYPE_COUNTERS_STATEOPERATIONALBYMETHOD_ACTIVE := 19924,
	OPCUAID_PUBSUBDIAGNOSTICSREADERGROUPTYPE_COUNTERS_STATEOPERATIONALBYMETHOD_CLASSIFICATION := 19925,
	OPCUAID_PUBSUBDIAGNOSTICSREADERGROUPTYPE_COUNTERS_STATEOPERATIONALBYMETHOD_DIAGNOSTICSLEVEL := 19926,
	OPCUAID_PUBSUBDIAGNOSTICSREADERGROUPTYPE_COUNTERS_STATEOPERATIONALBYMETHOD_TIMEFIRSTCHANGE := 19927,
	OPCUAID_PUBSUBDIAGNOSTICSREADERGROUPTYPE_COUNTERS_STATEOPERATIONALBYPARENT := 19928,
	OPCUAID_PUBSUBDIAGNOSTICSREADERGROUPTYPE_COUNTERS_STATEOPERATIONALBYPARENT_ACTIVE := 19929,
	OPCUAID_PUBSUBDIAGNOSTICSREADERGROUPTYPE_COUNTERS_STATEOPERATIONALBYPARENT_CLASSIFICATION := 19930,
	OPCUAID_PUBSUBDIAGNOSTICSREADERGROUPTYPE_COUNTERS_STATEOPERATIONALBYPARENT_DIAGNOSTICSLEVEL := 19931,
	OPCUAID_PUBSUBDIAGNOSTICSREADERGROUPTYPE_COUNTERS_STATEOPERATIONALBYPARENT_TIMEFIRSTCHANGE := 19932,
	OPCUAID_PUBSUBDIAGNOSTICSREADERGROUPTYPE_COUNTERS_STATEOPERATIONALFROMERROR := 19933,
	OPCUAID_PUBSUBDIAGNOSTICSREADERGROUPTYPE_COUNTERS_STATEOPERATIONALFROMERROR_ACTIVE := 19934,
	OPCUAID_PUBSUBDIAGNOSTICSREADERGROUPTYPE_COUNTERS_STATEOPERATIONALFROMERROR_CLASSIFICATION := 19935,
	OPCUAID_PUBSUBDIAGNOSTICSREADERGROUPTYPE_COUNTERS_STATEOPERATIONALFROMERROR_DIAGNOSTICSLEVEL := 19936,
	OPCUAID_PUBSUBDIAGNOSTICSREADERGROUPTYPE_COUNTERS_STATEOPERATIONALFROMERROR_TIMEFIRSTCHANGE := 19937,
	OPCUAID_PUBSUBDIAGNOSTICSREADERGROUPTYPE_COUNTERS_STATEPAUSEDBYPARENT := 19938,
	OPCUAID_PUBSUBDIAGNOSTICSREADERGROUPTYPE_COUNTERS_STATEPAUSEDBYPARENT_ACTIVE := 19939,
	OPCUAID_PUBSUBDIAGNOSTICSREADERGROUPTYPE_COUNTERS_STATEPAUSEDBYPARENT_CLASSIFICATION := 19940,
	OPCUAID_PUBSUBDIAGNOSTICSREADERGROUPTYPE_COUNTERS_STATEPAUSEDBYPARENT_DIAGNOSTICSLEVEL := 19941,
	OPCUAID_PUBSUBDIAGNOSTICSREADERGROUPTYPE_COUNTERS_STATEPAUSEDBYPARENT_TIMEFIRSTCHANGE := 19942,
	OPCUAID_PUBSUBDIAGNOSTICSREADERGROUPTYPE_COUNTERS_STATEDISABLEDBYMETHOD := 19943,
	OPCUAID_PUBSUBDIAGNOSTICSREADERGROUPTYPE_COUNTERS_STATEDISABLEDBYMETHOD_ACTIVE := 19944,
	OPCUAID_PUBSUBDIAGNOSTICSREADERGROUPTYPE_COUNTERS_STATEDISABLEDBYMETHOD_CLASSIFICATION := 19945,
	OPCUAID_PUBSUBDIAGNOSTICSREADERGROUPTYPE_COUNTERS_STATEDISABLEDBYMETHOD_DIAGNOSTICSLEVEL := 19946,
	OPCUAID_PUBSUBDIAGNOSTICSREADERGROUPTYPE_COUNTERS_STATEDISABLEDBYMETHOD_TIMEFIRSTCHANGE := 19947,
	OPCUAID_PUBSUBDIAGNOSTICSREADERGROUPTYPE_COUNTERS_RECEIVEDNETWORKMESSAGES := 19949,
	OPCUAID_PUBSUBDIAGNOSTICSREADERGROUPTYPE_COUNTERS_RECEIVEDNETWORKMESSAGES_ACTIVE := 19950,
	OPCUAID_PUBSUBDIAGNOSTICSREADERGROUPTYPE_COUNTERS_RECEIVEDNETWORKMESSAGES_CLASSIFICATION := 19951,
	OPCUAID_PUBSUBDIAGNOSTICSREADERGROUPTYPE_COUNTERS_RECEIVEDNETWORKMESSAGES_DIAGNOSTICSLEVEL := 19952,
	OPCUAID_PUBSUBDIAGNOSTICSREADERGROUPTYPE_COUNTERS_RECEIVEDNETWORKMESSAGES_TIMEFIRSTCHANGE := 19953,
	OPCUAID_PUBSUBDIAGNOSTICSREADERGROUPTYPE_COUNTERS_RECEIVEDINVALIDNETWORKMESSAGES := 19954,
	OPCUAID_PUBSUBDIAGNOSTICSREADERGROUPTYPE_COUNTERS_RECEIVEDINVALIDNETWORKMESSAGES_ACTIVE := 19955,
	OPCUAID_PUBSUBDIAGNOSTICSREADERGROUPTYPE_COUNTERS_RECEIVEDINVALIDNETWORKMESSAGES_CLASSIFICATION := 19956,
	OPCUAID_PUBSUBDIAGNOSTICSREADERGROUPTYPE_COUNTERS_RECEIVEDINVALIDNETWORKMESSAGES_DIAGNOSTICSLEVEL := 19957,
	OPCUAID_PUBSUBDIAGNOSTICSREADERGROUPTYPE_COUNTERS_RECEIVEDINVALIDNETWORKMESSAGES_TIMEFIRSTCHANGE := 19958,
	OPCUAID_PUBSUBDIAGNOSTICSREADERGROUPTYPE_COUNTERS_DECRYPTIONERRORS := 19959,
	OPCUAID_PUBSUBDIAGNOSTICSREADERGROUPTYPE_COUNTERS_DECRYPTIONERRORS_ACTIVE := 19960,
	OPCUAID_PUBSUBDIAGNOSTICSREADERGROUPTYPE_COUNTERS_DECRYPTIONERRORS_CLASSIFICATION := 19961,
	OPCUAID_PUBSUBDIAGNOSTICSREADERGROUPTYPE_COUNTERS_DECRYPTIONERRORS_DIAGNOSTICSLEVEL := 19962,
	OPCUAID_PUBSUBDIAGNOSTICSREADERGROUPTYPE_COUNTERS_DECRYPTIONERRORS_TIMEFIRSTCHANGE := 19963,
	OPCUAID_PUBSUBDIAGNOSTICSREADERGROUPTYPE_LIVEVALUES_CONFIGUREDDATASETREADERS := 19964,
	OPCUAID_PUBSUBDIAGNOSTICSREADERGROUPTYPE_LIVEVALUES_CONFIGUREDDATASETREADERS_DIAGNOSTICSLEVEL := 19965,
	OPCUAID_PUBSUBDIAGNOSTICSREADERGROUPTYPE_LIVEVALUES_OPERATIONALDATASETREADERS := 19966,
	OPCUAID_PUBSUBDIAGNOSTICSREADERGROUPTYPE_LIVEVALUES_OPERATIONALDATASETREADERS_DIAGNOSTICSLEVEL := 19967,
	OPCUAID_PUBSUBDIAGNOSTICSDATASETWRITERTYPE_TOTALINFORMATION_ACTIVE := 19971,
	OPCUAID_PUBSUBDIAGNOSTICSDATASETWRITERTYPE_TOTALINFORMATION_CLASSIFICATION := 19972,
	OPCUAID_PUBSUBDIAGNOSTICSDATASETWRITERTYPE_TOTALINFORMATION_DIAGNOSTICSLEVEL := 19973,
	OPCUAID_PUBSUBDIAGNOSTICSDATASETWRITERTYPE_TOTALINFORMATION_TIMEFIRSTCHANGE := 19974,
	OPCUAID_PUBSUBDIAGNOSTICSDATASETWRITERTYPE_TOTALERROR_ACTIVE := 19976,
	OPCUAID_PUBSUBDIAGNOSTICSDATASETWRITERTYPE_TOTALERROR_CLASSIFICATION := 19977,
	OPCUAID_PUBSUBDIAGNOSTICSDATASETWRITERTYPE_TOTALERROR_DIAGNOSTICSLEVEL := 19978,
	OPCUAID_PUBSUBDIAGNOSTICSDATASETWRITERTYPE_TOTALERROR_TIMEFIRSTCHANGE := 19979,
	OPCUAID_PUBSUBDIAGNOSTICSDATASETWRITERTYPE_COUNTERS_STATEERROR := 19983,
	OPCUAID_PUBSUBDIAGNOSTICSDATASETWRITERTYPE_COUNTERS_STATEERROR_ACTIVE := 19984,
	OPCUAID_PUBSUBDIAGNOSTICSDATASETWRITERTYPE_COUNTERS_STATEERROR_CLASSIFICATION := 19985,
	OPCUAID_PUBSUBDIAGNOSTICSDATASETWRITERTYPE_COUNTERS_STATEERROR_DIAGNOSTICSLEVEL := 19986,
	OPCUAID_PUBSUBDIAGNOSTICSDATASETWRITERTYPE_COUNTERS_STATEERROR_TIMEFIRSTCHANGE := 19987,
	OPCUAID_PUBSUBDIAGNOSTICSDATASETWRITERTYPE_COUNTERS_STATEOPERATIONALBYMETHOD := 19988,
	OPCUAID_PUBSUBDIAGNOSTICSDATASETWRITERTYPE_COUNTERS_STATEOPERATIONALBYMETHOD_ACTIVE := 19989,
	OPCUAID_PUBSUBDIAGNOSTICSDATASETWRITERTYPE_COUNTERS_STATEOPERATIONALBYMETHOD_CLASSIFICATION := 19990,
	OPCUAID_PUBSUBDIAGNOSTICSDATASETWRITERTYPE_COUNTERS_STATEOPERATIONALBYMETHOD_DIAGNOSTICSLEVEL := 19991,
	OPCUAID_PUBSUBDIAGNOSTICSDATASETWRITERTYPE_COUNTERS_STATEOPERATIONALBYMETHOD_TIMEFIRSTCHANGE := 19992,
	OPCUAID_PUBSUBDIAGNOSTICSDATASETWRITERTYPE_COUNTERS_STATEOPERATIONALBYPARENT := 19993,
	OPCUAID_PUBSUBDIAGNOSTICSDATASETWRITERTYPE_COUNTERS_STATEOPERATIONALBYPARENT_ACTIVE := 19994,
	OPCUAID_PUBSUBDIAGNOSTICSDATASETWRITERTYPE_COUNTERS_STATEOPERATIONALBYPARENT_CLASSIFICATION := 19995,
	OPCUAID_PUBSUBDIAGNOSTICSDATASETWRITERTYPE_COUNTERS_STATEOPERATIONALBYPARENT_DIAGNOSTICSLEVEL := 19996,
	OPCUAID_PUBSUBDIAGNOSTICSDATASETWRITERTYPE_COUNTERS_STATEOPERATIONALBYPARENT_TIMEFIRSTCHANGE := 19997,
	OPCUAID_PUBSUBDIAGNOSTICSDATASETWRITERTYPE_COUNTERS_STATEOPERATIONALFROMERROR := 19998,
	OPCUAID_PUBSUBDIAGNOSTICSDATASETWRITERTYPE_COUNTERS_STATEOPERATIONALFROMERROR_ACTIVE := 19999,
	OPCUAID_PUBSUBDIAGNOSTICSDATASETWRITERTYPE_COUNTERS_STATEOPERATIONALFROMERROR_CLASSIFICATION := 20000,
	OPCUAID_PUBSUBDIAGNOSTICSDATASETWRITERTYPE_COUNTERS_STATEOPERATIONALFROMERROR_DIAGNOSTICSLEVEL := 20001,
	OPCUAID_PUBSUBDIAGNOSTICSDATASETWRITERTYPE_COUNTERS_STATEOPERATIONALFROMERROR_TIMEFIRSTCHANGE := 20002,
	OPCUAID_PUBSUBDIAGNOSTICSDATASETWRITERTYPE_COUNTERS_STATEPAUSEDBYPARENT := 20003,
	OPCUAID_PUBSUBDIAGNOSTICSDATASETWRITERTYPE_COUNTERS_STATEPAUSEDBYPARENT_ACTIVE := 20004,
	OPCUAID_PUBSUBDIAGNOSTICSDATASETWRITERTYPE_COUNTERS_STATEPAUSEDBYPARENT_CLASSIFICATION := 20005,
	OPCUAID_PUBSUBDIAGNOSTICSDATASETWRITERTYPE_COUNTERS_STATEPAUSEDBYPARENT_DIAGNOSTICSLEVEL := 20006,
	OPCUAID_PUBSUBDIAGNOSTICSDATASETWRITERTYPE_COUNTERS_STATEPAUSEDBYPARENT_TIMEFIRSTCHANGE := 20007,
	OPCUAID_PUBSUBDIAGNOSTICSDATASETWRITERTYPE_COUNTERS_STATEDISABLEDBYMETHOD := 20008,
	OPCUAID_PUBSUBDIAGNOSTICSDATASETWRITERTYPE_COUNTERS_STATEDISABLEDBYMETHOD_ACTIVE := 20009,
	OPCUAID_PUBSUBDIAGNOSTICSDATASETWRITERTYPE_COUNTERS_STATEDISABLEDBYMETHOD_CLASSIFICATION := 20010,
	OPCUAID_PUBSUBDIAGNOSTICSDATASETWRITERTYPE_COUNTERS_STATEDISABLEDBYMETHOD_DIAGNOSTICSLEVEL := 20011,
	OPCUAID_PUBSUBDIAGNOSTICSDATASETWRITERTYPE_COUNTERS_STATEDISABLEDBYM